(* IEC 61131-3 sources: ml2plc/benchmarks/st (part 25) *)

    bias_13 : ARRAY[0..63] OF REAL := [-0.0404071435, 0.0927777886, -0.0413042903, -0.0902542397, -0.0367607661, 0.0712136403, -0.00892876834, -0.0667051747, 0.00637631165, 0.0437391289, -0.0124141583, 0.0894438922, -0.0595212504, 0.0899347588, 0.0368472114, -0.000366137043, -0.0369593501, 0.0098438086, -0.00942459609, 0.0903767124, -0.0075942101, 0.046375595, -0.0592727698, 0.0528409891, -0.0216910169, -0.00787346996, 0.0314517543, 0.0737932697, -0.0810395479, 0.0906123891, 0.0820333436, 0.0979426578, -0.0194323044, -0.0938704684, -0.0664548054, 0.0229378678, -0.0287175067, 0.0409495458, -0.0543716773, 0.0378184244, -0.0231971722, -0.0583018064, -0.064960219, 0.00983823184, -0.0784399733, 0.0101949805, -0.0290268082, 0.0763350129, -0.0110898362, -0.00504951039, 0.0234738979, -0.0619560853, 3.6623473e-07, -0.0102051999, -0.0874569118, 0.0950193256, 0.011268124, 0.0887499079, 0.0580152497, 0.0789389834, -0.0176048651, -0.00555823185, -0.0167076774, -0.0683557615];

    weights_16 : ARRAY[0..191] OF REAL := [-0.204218104, 0.0100585446, 0.124642573, 0.249767885, 0.192972004, -0.114489801, 0.0213469081, -0.192255303, 0.0687296614, -0.116273321, -0.168248311, 0.100407079, -0.0835328773, 0.238771692, -0.1582672, -0.20680669, 0.199099779, -0.355317205, -0.275946528, 0.259559304, -0.152421042, -0.193678349, -0.0476079546, 0.168583572, 0.137155071, -0.424926966, 0.0668462142, 0.121788457, 0.166179895, 0.155418351, -0.239607006, 0.159718022, 0.181392595, 0.012098941, 0.29212448, -0.30051899, -0.042393513, -0.302967817, 0.0276647583, -0.0162179675, -0.0362443365, -0.131818026, 0.0652571768, -0.251479208, -0.163796052, 0.246231601, -0.0993305817, -0.214045271, -0.259664625, 0.121991962, 0.328099579, -0.36496222, 0.286016166, 0.174832657, -0.115100093, 0.240771398, -0.219685465, -0.0312652551, 0.361102194, -0.322652519, 0.172960237, -0.0672435984, -0.196433365, -0.310510099, 0.180873245, -0.229489714, -0.0438734591, -0.0316266902, 0.106365554, -0.354469597, 0.104236148, 0.0969249979, 0.0453101136, 0.189823419, -0.119062148, 0.0151938582, 0.05480076, -0.137107879, 0.231374756, -0.184149876, -0.152093366, 0.298650056, -0.120534711, -0.440170765, -0.291449726, -0.185382351, 0.240590215, 0.0743931085, 0.00839448255, -0.324791044, 0.0127115622, 0.201346219, -0.129334167, 0.217511401, 0.249150231, -0.227794915, -0.152671486, 0.225536987, -0.10112305, -0.260705948, -0.309738696, 0.234022498, 0.247884244, -0.138457581, 0.287121534, 0.107613027, 0.369097799, 0.20829244, -0.189594626, -0.168206543, 0.127910152, 0.117524289, -0.267760575, -0.273475945, -0.0782620981, -0.369871527, 0.318286926, 0.380977005, -0.372844636, -0.159075871, -0.35559544, -0.15261285, 0.021852307, -0.177226037, -0.057486631, 0.270852298, 0.160473123, -0.251653463, 0.100419275, -0.136632696, -0.287902951, -0.344732016, 0.126178026, -0.177843302, 0.339493781, -0.099222295, 0.0892207772, 0.163005397, 0.215954706, -0.0692603961, 0.0789305717, 0.37051788, 0.124587342, -0.095472239, 0.128479376, -0.0207961947, -0.257337809, 0.0661524683, 0.132446691, -0.221712723, -0.32083869, 0.195067048, 0.161428511, -0.336975783, -0.0876864642, 0.283737957, 0.175905675, -0.186329022, -0.0834812075, -0.0544198342, -0.247233495, -0.240931347, -0.316858917, -0.324440151, 0.33110112, 0.302384734, 0.294178426, 0.0780448988, -0.218289346, 0.095910117, 0.0984309539, -0.335624874, 0.34094283, -0.192400947, -0.337153077, 0.305544972, -0.302600533, -0.0743493959, 0.340184033, -0.0958573595, -0.265512377, 0.0674359873, 0.0557227954, -0.208096027, 0.112970375, -0.241400406, -0.123275287, -0.175267965, 0.0384325348, 0.0348930582, -0.135870203, -0.0273135975];
    bias_16 : ARRAY[0..2] OF REAL := [0.0433644801, 0.055319678, -0.0903941169];

END_VAR

VAR
    (* Merged variables from all regions *)
    buffer_0 : ARRAY[0..63] OF REAL;
    buffer_1 : ARRAY[0..63] OF REAL;
    buffer_2 : ARRAY[0..63] OF REAL;

    (* Temporary computation variables *)
    i : DINT;
    j : DINT;
    t : DINT;
    sum : REAL;
    (* Computation helpers *)
    max_val : REAL;
    exp_val : REAL;
    exp_sum : REAL;
    (* Spatial loop variables *)
    oc : DINT;
    oh : DINT;
    ow : DINT;
    ic : DINT;
    kh : DINT;
    kw : DINT;
    ih : DINT;
    iw : DINT;
END_VAR

(* Forward pass execution *)

(* Region: r0 [ACYCLIC] *)
(* Acyclic Region r0 *)
(* Layer 0: Fused Linear + RELU *)
FOR j := 0 TO 63 DO
    sum := 0.0;
    FOR i := 0 TO 0 DO
        sum := sum + input_data * weights_0[i * 64 + j];
    END_FOR;
buffer_0[j] := MAX(sum + bias_0[j], 0.0);
END_FOR;

(* Layer 1: Fused Linear + RELU *)
FOR j := 0 TO 63 DO
    sum := 0.0;
    FOR i := 0 TO 63 DO
        sum := sum + buffer_0[i] * weights_1[i * 64 + j];
    END_FOR;
buffer_2[j] := MAX(sum + bias_1[j], 0.0);
END_FOR;

(* Layer 2: MatMul *)
FOR j := 0 TO 63 DO
    sum := 0.0;
    FOR i := 0 TO 63 DO
        sum := sum + buffer_2[i] * weights_2[i * 64 + j];
    END_FOR;
buffer_1[j] := sum;
END_FOR;

(* Layer 3: Add (Bias) *)
FOR i := 0 TO 63 DO
    buffer_2[i] := buffer_1[i] + bias_3[i];
END_FOR;

(* Layer 4: Add (Element-wise) *)
FOR i := 0 TO 63 DO
    buffer_1[i] := buffer_2[i] + buffer_0[i];
END_FOR;

(* Layer 5: Activation (RELU) *)
FOR i := 0 TO 63 DO
    buffer_0[i] := MAX(buffer_1[i], 0.0);
END_FOR;

(* Layer 6: Fused Linear + RELU *)
FOR j := 0 TO 63 DO
    sum := 0.0;
    FOR i := 0 TO 63 DO
        sum := sum + buffer_0[i] * weights_6[i * 64 + j];
    END_FOR;
buffer_2[j] := MAX(sum + bias_6[j], 0.0);
END_FOR;

(* Layer 7: MatMul *)
FOR j := 0 TO 63 DO
    sum := 0.0;
    FOR i := 0 TO 63 DO
        sum := sum + buffer_2[i] * weights_7[i * 64 + j];
    END_FOR;
buffer_1[j] := sum;
END_FOR;

(* Layer 8: Add (Bias) *)
FOR i := 0 TO 63 DO
    buffer_2[i] := buffer_1[i] + bias_8[i];
END_FOR;

(* Layer 9: Add (Element-wise) *)
FOR i := 0 TO 63 DO
    buffer_1[i] := buffer_2[i] + buffer_0[i];
END_FOR;

(* Layer 10: Activation (RELU) *)
FOR i := 0 TO 63 DO
    buffer_0[i] := MAX(buffer_1[i], 0.0);
END_FOR;

(* Layer 11: Fused Linear + RELU *)
FOR j := 0 TO 63 DO
    sum := 0.0;
    FOR i := 0 TO 63 DO
        sum := sum + buffer_0[i] * weights_11[i * 64 + j];
    END_FOR;
buffer_2[j] := MAX(sum + bias_11[j], 0.0);
END_FOR;

(* Layer 12: MatMul *)
FOR j := 0 TO 63 DO
    sum := 0.0;
    FOR i := 0 TO 63 DO
        sum := sum + buffer_2[i] * weights_12[i * 64 + j];
    END_FOR;
buffer_1[j] := sum;
END_FOR;

(* Layer 13: Add (Bias) *)
FOR i := 0 TO 63 DO
    buffer_2[i] := buffer_1[i] + bias_13[i];
END_FOR;

(* Layer 14: Add (Element-wise) *)
FOR i := 0 TO 63 DO
    buffer_1[i] := buffer_2[i] + buffer_0[i];
END_FOR;

(* Layer 15: Activation (RELU) *)
FOR i := 0 TO 63 DO
    buffer_0[i] := MAX(buffer_1[i], 0.0);
END_FOR;

(* Layer 16: Fused Linear + SOFTMAX *)
FOR j := 0 TO 2 DO
    sum := 0.0;
    FOR i := 0 TO 63 DO
        sum := sum + buffer_0[i] * weights_16[i * 3 + j];
    END_FOR;
output_data[j] := sum + bias_16[j];
END_FOR;

(* Softmax: find max *)
max_val := output_data[0];
FOR i := 1 TO 2 DO
    IF output_data[i] > max_val THEN
        max_val := output_data[i];
    END_IF;
END_FOR;

(* Softmax: compute exponentials and sum *)
exp_sum := 0.0;
FOR i := 0 TO 2 DO
    output_data[i] := EXP(output_data[i] - max_val);
    exp_sum := exp_sum + output_data[i];
END_FOR;

(* Softmax: normalize *)
FOR i := 0 TO 2 DO
    output_data[i] := output_data[i] / exp_sum;
END_FOR;

END_FUNCTION_BLOCK

(* ---- ResNet3_straton.st ---- *)
FUNCTION_BLOCK ResNet3_FB

    (* Model Inputs/Outputs *)
VAR_INPUT
    input_data : REAL;
END_VAR

VAR_OUTPUT
    output_data : ARRAY[0..2] OF REAL;
END_VAR

VAR
    CONSTANT weights_0 : ARRAY[0..63] OF REAL := [-0.190466672, -0.289495766, 0.36445868, 0.11001166, -0.202885658, -0.247976601, -0.217859656, 0.152941793, -0.210685372, 0.322490484, -0.300406843, -0.0737419277, 0.271309823, 0.34986949, -0.269151628, 0.101570874, -0.0975821763, -0.0239237547, -0.28141278, -0.260361493, 0.220720425, 0.342909008, -0.106619239, 0.192217126, -0.139923915, -0.00473925471, 0.256588012, 0.106521919, -0.015166074, -0.237258494, -0.295479923, 0.237283707, -0.111313865, -0.119793385, -0.189164549, 0.109231912, 0.147311017, -0.0809866935, -0.174528345, -0.015255332, 0.110069647, 0.205406636, 0.233189464, 0.175904229, 0.192441761, -0.257080823, 0.113344185, -0.222640619, 0.0253927261, -0.0698330998, 0.304976135, 0.13343668, -0.229343772, 0.317507595, -0.0133918505, 0.251467377, -0.131539866, -0.128968731, 0.204563618, -0.234828115, 0.109687969, 0.0967651531, -0.128085941, 0.0570141077];
    CONSTANT bias_0 : ARRAY[0..63] OF REAL := [0, 0, -0.0451503769, -0.000170675936, 0, 0, 0, -0.0306519736, 0, -0.043658372, 0, 0, -0.0452437028, -0.0463685207, 0, -0.0237470753, 0, 0, 0, 0, -0.0306253415, -0.0182554778, 0, -0.0286273304, 0, 0, -0.0439416394, 0.0359471515, 0, 0, 0, -0.0393987, 0, 0, 0, -0.025377661, 0.0258860644, 0, 0, 0, -0.0256011337, -0.040137399, -0.0210138671, -0.0197667424, -0.0420954861, 0, -0.0343104228, 0, -0.0101194074, 0, -0.0385119878, -0.0309600942, 0, -0.0221530851, 0.0427107885, -0.0482655875, 0, 0, -0.0332414694, 0, -0.0204843841, -0.0293239169, 0, -0.0204854961];
    CONSTANT weights_1 : ARRAY[0..4095] OF REAL := [-0.0287969261, 0.201637134, -0.193626225, -0.0838745981, -0.179824859, -0.158866256, -0.0519343764, 0.0553617924, -0.0298234671, 0.199577436, -0.0565214604, -0.135609776, 0.19474043, -0.0305772722, 0.047594741, 0.174586251, -0.131670237, -0.0606977493, -0.00999130309, 0.160562769, 0.114603773, 0.198183253, -0.0226515681, -0.174445733, 0.0844327062, -0.0653743893, 0.166338369, 0.178600982, -0.179540232, -0.104543671, -0.04106462, 0.0376635343, -0.0928359851, 0.0239627361, -0.0751802325, -0.131423861, 0.107191309, 0.0680955499, -0.134543836, 0.162752822, -0.119452722, -0.118079856, -0.111446388, 0.103158936, -0.0164598525, -0.143377468, 0.0849187821, -0.0122491121, -0.152280733, -0.120597631, -0.0606369525, -0.0807449222, 0.147399679, 0.0629173666, -0.130655468, -0.21262382, -0.169020504, 0.105712339, 0.11746116, 0.0592246503, -0.0597587526, -0.143656209, 0.0653275698, -0.0477767587, -0.154527515, 0.0485876948, -0.0317480415, -0.000382602215, -0.0967821628, 0.0423714072, -0.0512648225, 0.0312831551, -0.17014426, 0.160105124, 0.109350279, -0.0217197388, -0.0921072736, 0.0853802711, -0.0300633907, 0.135347292, -0.0391751528, -0.199345261, -0.195168182, 0.0560685545, 0.215828583, -0.0923638716, 0.192498907, 0.178375289, -0.183688045, 0.116588429, 0.0289125443, 0.0778251439, 0.0613025278, 0.0142809004, 0.0337732583, 0.0574108511, 0.189165697, 0.196946517, 0.107737496, -0.129702166, -0.107477285, -0.107738689, -0.177952528, -0.0559140593, 0.169283316, -0.0538910031, -0.104346119, -0.127213195, -0.0331750959, 0.127317414, 0.0515208095, 0.0195653588, 0.0769012719, -0.124866173, 0.177239373, 0.0280220658, 0.0963039249, -0.0652452409, 0.105720118, 0.15663074, -0.136386782, -0.123085879, 0.0827278346, 0.21160166, -0.16991207, -0.0768297166, 0.120611772, 0.134732291, -0.139711812, -0.184518486, -0.184835598, 0.00858225208, 0.113042273, -0.102391459, -0.0780269504, -0.165388852, -0.140612379, 0.223779544, 0.162238076, -0.00674940646, 0.0487292968, 0.0836367309, -0.19456315, 0.171644017, -0.0955267325, 0.0997560844, -0.0601457544, -0.198954478, -0.00482972385, -0.079228431, -0.127536789, 0.190665379, -0.0999609306, 0.0110752583, -4.10255961e-05, 0.118868679, 0.138081178, -0.0528386459, -0.114722773, 0.170001924, 0.137378082, -0.196978897, -0.15748626, 0.0825704783, -0.033234071, -0.101335384, 0.0289265234, -0.15857622, -0.0556612536, 0.213226333, 0.00719815027, 0.223965615, -0.0638628826, 0.148281991, 0.0975444093, -0.0259753708, 0.0262751374, 0.0979252607, -0.0863377675, 0.0899253041, 0.239503771, 0.289376885, -0.204818711, 0.105383582, 0.293127954, 0.203753337, -0.119700439, -0.16846402, 0.191751063, 0.0327624083, -0.0386312976, -0.264414817, 0.153028056, 0.154591411, 0.124344207, -0.107223384, -0.137165904, 0.0300747007, 0.183606654, 0.198948666, 0.0499654785, 0.144469813, -0.210293442, -0.0324280113, 0.0683567002, -0.04100243, -0.0126516968, 0.164788797, 0.237893194, -0.0847178176, 0.0626023933, 0.155760348, 0.185824335, 0.00780587131, 0.199899733, 0.035005752, -0.0749012083, 0.067025587, 0.141089186, -0.0444214866, -0.0607198402, 0.0990498737, -0.0620695017, 0.0086689936, -0.114031576, -0.111011893, -0.204213917, -0.198096737, 0.138905957, 0.159203395, 0.12167336, 0.0172255039, 0.15101482, 0.131718054, -0.0235928968, 0.200807258, 0.209497362, 0.170748204, -0.231670231, 0.143206522, 0.225486189, 0.104716703, -0.177130625, -0.133289889, -0.0483859442, 0.107198499, -0.0196592454, -0.0476846471, -0.0815907568, -0.135093376, 0.12207596, 0.00658966927, -0.0573140644, 0.0118645504, 0.226763472, 0.178059682, -0.0891532153, 0.0825275332, 0.163484469, -0.0550447851, -0.0375959724, -0.00878846645, 0.0168165267, 0.150091812, 0.084491238, 0.174592748, 0.0785937458, 0.163301513, -0.0316622555, 0.0597050637, 0.157956466, -0.0453870595, 0.101291135, -0.0735865831, 0.0523432046, 0.00310024619, -0.111143999, -0.176621795, 0.0883997232, -0.00594709814, -0.0267459899, 0.164880231, 0.0904007405, -0.00336711109, 0.025017634, -0.136061743, -0.0808758289, 0.139091626, 0.0775778443, -0.155642897, 0.0725118369, -0.0960384831, 0.135437921, -0.188861921, 0.0681308657, 0.121807054, -0.0181216151, 0.126562431, 0.0201322883, 0.0685440749, 0.0470108241, 0.206563786, 0.167886898, -0.182285488, -0.166398615, 0.200898841, 0.191317186, 0.190035328, -0.175405696, 0.124712333, 0.052170679, 0.184364364, -0.0736751109, 0.0639937371, -0.168305129, 0.00677789748, -0.148140043, 0.10284771, -0.13430731, 0.139501527, 0.0359104425, 0.0577303618, -0.188823983, -0.174651235, 0.0696652383, -0.183670074, -0.00257234275, -0.193130046, -0.203748837, -0.153786868, 0.202487156, -0.0460375547, 0.109957233, 0.00299288332, -0.162598059, 0.210710511, -0.194323435, -0.210184813, 0.0554226786, -0.142163336, -0.152110279, -0.0163246542, -0.166943565, 0.175032482, -0.215747178, 0.171988502, 0.132436678, 0.172353908, 0.121031687, 0.186095968, -0.0588158816, -0.0108129233, -0.0942323804, -0.09778703, -0.109081298, -0.106757924, 0.172346756, 0.025905624, 0.0740813166, 0.189657524, 0.148814008, 0.197771326, 0.201267496, -0.068178758, 0.1481594, 0.184583381, -0.014007479, 0.0497234613, -0.0900920182, -0.151112944, -0.154349625, 0.155235782, -0.183371142, -0.164333746, 0.110023871, 0.0927015692, 0.194937959, 0.208203807, -0.00641842186, -0.135277599, -0.0120722651, 0.0209348053, -0.163213924, 0.183399543, 0.00101952255, -0.094531931, -0.0417330861, 0.125320569, 0.140007362, -0.0551816374, -0.0750101358, -0.184187144, 0.0996663719, 0.1298704, -0.00832244754, -0.00248210132, 0.0548401624, -0.0217346549, -0.040534541, 0.0774618536, 0.0789829642, -0.213013336, 0.00969907641, 0.131764188, -0.134339929, -0.16999869, -0.150505453, -0.203993306, 0.133900389, 0.210885063, 0.0592023879, 0.119564161, 0.129766181, -0.116630182, 0.0890186876, 0.0916796774, -0.125102013, 0.144167438, 0.190863922, 0.0828631073, 0.110106811, -0.0818011016, 0.0638723224, 0.0225199312, -0.0798923373, -0.106765099, -0.103232488, -0.0746515393, 0.214082971, -0.139221311, 0.0676382631, 0.20862554, 0.185882255, -0.0279404521, 0.0581518859, -0.0932726786, -0.0684341788, -0.148790196, -0.167229846, 0.160150275, -0.125400275, -0.0166903287, -0.0369179547, 0.0845469385, -0.191490114, -0.161978155, -0.023997426, 0.040678516, 0.14639619, 0.0431083404, 0.0106931906, 0.139329195, -0.149284765, -0.0467167646, -0.0767225027, -0.0320999771, -0.23229675, -0.0372863598, 0.128295347, -0.160325885, -0.148059294, -0.00792731252, 0.0252128541, -0.0963003412, -0.0197790675, -0.0523058102, -0.0141548719, -0.168405354, 0.093509756, -0.0733992159, -0.174149796, 0.0823272243, 0.0543129146, 0.00202205591, 0.112447657, -0.189444944, 0.0949934795, 0.133855537, 0.138600275, -0.170810059, -0.0500965714, -0.186440244, 0.0285257101, -0.000778779387, -0.128126383, -0.0261946935, -0.201500729, 0.11489366, 0.0997269675, -0.138657212, -0.256732196, 0.0291550159, -0.302546233, -0.178278208, -0.234763011, -0.0388856418, 0.0533248745, -0.146624878, -0.0823597312, -0.230229869, 0.0182416849, -0.118736058, 0.0481926613, 0.133541629, -0.114781246, 0.10070549, 0.109701976, 0.0569074266, 0.26510939, 0.00950349867, 0.0546200871, 0.151336238, 0.0048430115, 0.0378029197, 0.144169971, 0.0863773972, 0.200766638, 0.212797061, 0.138086304, -0.182377681, 0.213811055, 0.161403164, 0.124502376, 0.0246564448, -0.196184307, -0.196561068, 0.0875730366, 0.0948206931, -0.149286091, 0.0323978215, 0.0455216914, 0.151648596, -0.127112329, -0.111039624, 0.0246137083, 0.016291365, -0.00267861784, 0.0558695644, 0.201473311, -0.178703129, -0.103530645, 0.173463836, 0.157130465, 0.182277635, 0.0760518163, 0.215445682, -0.106563114, -0.196684077, -0.094135493, 0.10404627, 0.0962792784, -0.0124557465, -0.15429759, -0.0716400295, 0.11189805, 0.0764795393, 0.0549422354, -0.0472201556, -0.00484439731, 0.0528673977, 0.190446272, 0.0174336433, -0.0469030589, -0.0549324602, 0.102302983, -4.00096178e-05, 0.147421315, 0.193782583, -0.0265746713, 0.0705426186, 0.0295248479, -0.134114474, 0.0562623292, 0.172508165, 0.175126389, -0.161904559, -0.0162163712, 0.208393365, -0.100752503, 0.0273437109, -0.153811902, -0.193232462, -0.16940017, 0.188474581, -0.0369768888, 0.0354307853, -0.0991368741, -0.196591377, -0.233054638, -0.118758805, -0.0622535497, 0.0394661725, 0.267733514, 0.107220888, -0.252435923, 0.112368457, 0.166412622, 0.192772374, -0.218732044, 0.126407787, 0.0919501036, 0.00824039057, -0.0796734989, 0.182596043, 0.131103203, -0.109326825, 0.125145733, 0.122357175, 0.0696524829, -0.0965674892, 0.0579061955, -0.200026214, -0.185237691, -0.189040273, -0.224097118, 0.103700139, 0.109744169, 0.283211142, -0.108721465, 0.126635522, -0.0494364649, -0.224469841, 0.151249424, -0.162036136, 0.030354334, -0.00598688424, -0.143472508, -0.047887668, 0.0439753979, 0.0527719408, -0.152598977, 0.110804304, 0.257972151, -0.138091505, -0.110594928, 0.100734361, -0.0214415565, 0.0449742526, 0.22822006, -0.240381643, -0.128085867, -0.0693219751, -0.0846015364, -0.17030485, 0.130928531, 0.00229240954, -0.194736332, -0.0391959101, 0.0145413131, -0.144774944, -0.181710035, 0.032208994, -0.206829414, -0.0198655725, 0.0611966401, 0.00840911269, 0.158986792, 0.126695439, -0.157956257, -0.20029664, -0.104722835, -0.144183606, 0.00487022102, 0.0939430147, -0.0584943891, 0.0557004064, 0.00045491755, 0.114710584, 0.0546646267, 0.20419623, 0.0921241492, 0.0991390496, 0.176430956, -0.158750683, -0.0890071839, -0.179640472, 0.162403598, -0.0909959227, 0.0409451872, -0.0232819319, 0.165903732, 0.069598332, 0.175637826, -0.179648638, -0.00545862317, 0.00749818981, 0.0323755145, -0.158800021, 0.180631563, -0.053162545, -0.014888972, -0.188607126, -0.0488055795, 0.20547007, -0.0377693027, 0.0997820646, -0.124526724, -0.0918210968, -0.167447731, -0.188922942, 0.0540182441, 0.122466967, -0.0612903982, 0.173171565, 0.187880501, 0.0320709199, -0.0716537684, -0.146939963, 0.00549939275, 0.0170418024, -0.156284317, -0.158158392, -0.0161726922, -0.117838174, 0.0458692163, 0.0690316111, -0.102591947, -0.0113369077, -0.0506339818, 0.186475053, 0.10736011, -0.0328097939, -0.13072902, -0.14560762, 0.0873160809, 0.204848334, 0.079661116, -0.018868804, -0.018476963, 0.148941293, 0.0539769381, -0.00221420825, -0.108419128, -0.0766489506, -0.189365566, 0.0919391662, -0.212484032, -0.172094896, 0.0239589214, -0.211048037, 0.189641103, 0.0730664879, 0.206356838, -0.135675371, -0.000756576657, 0.0285059959, 0.209358588, 0.192232445, 0.11306645, -0.115133278, 0.175952092, 0.0211753547, 0.0506318063, -0.19809112, 0.0197272301, 0.054157868, 0.0254253149, -0.155184671, -0.0454918444, -0.196502686, -0.0158347338, -0.135656744, -0.211595923, -0.020885095, -0.00690788031, 0.0370714217, -0.172456279, -0.185076281, 0.160629585, 0.0181837529, -0.0211855043, 0.120963901, -0.00527728582, -0.0352699608, -0.19402647, 0.132209137, 0.0396415927, -0.118135475, 0.00657442212, -0.208759815, -0.0303688291, -0.00777827017, -0.0915059149, 0.11210835, 0.294361055, -0.142053381, -0.0571834072, -0.0146589978, -0.0864291564, -0.101504333, 0.12920031, 0.182926923, 0.192566365, 0.106406614, 0.214629248, 0.06889496, -0.11516425, -0.259321928, 0.184162751, -0.272702873, -0.117973782, 0.0606180206, 0.0292263925, 0.0766455382, -0.120667271, -0.201999113, -0.0266232025, -0.00732299685, -0.0519965291, 0.156876504, 0.123033859, 0.267217845, -0.0109749781, -0.272964209, -0.129237577, 0.053774897, 0.141416252, -0.199857935, 0.0538020581, -0.230259433, -0.0451727808, 0.258897543, 0.148216307, -0.053409934, 0.31615606, 0.0147380829, -0.202499956, 0.110624768, 0.1696845, -0.0922751948, 0.0798982531, 0.0207011886, -0.142718717, 0.0519616678, -0.127546012, 0.126492023, 0.0723542273, 0.147747502, 0.126169741, 0.0813353807, -0.1203655, -0.153749913, -0.0919978395, -0.139003664, 0.0844179541, 0.054092221, 0.110275611, -0.200139761, 0.110008813, -0.126036033, -0.166970596, -0.233972371, 0.0890860558, -0.20025298, -0.230093077, 0.0173213258, 0.275560528, 0.151483357, 0.276097506, 0.00718977815, -0.0111169517, 0.168895632, 0.10235633, -0.240326077, -0.0821303874, -0.00890312064, -0.171553358, -0.00546233356, 0.101003714, 0.0433369204, -0.187788144, -0.103547342, 0.00432489906, -0.109544538, 0.012347714, 0.0869178474, -0.257481515, -0.0600075051, -0.264836371, -0.171154037, 0.0307734851, -0.129194021, -0.199388355, 0.0987441167, -0.0623329841, 0.249395654, -0.034193743, 0.0902072638, 0.203402102, -0.0227374583, 0.0134097785, -0.0912396759, 0.0864051133, 0.0865284353, 0.228083283, 0.126239121, -0.109470509, -0.188946784, 0.00514312088, 0.181860104, 0.0482862443, 0.0316015482, 0.208089277, 0.175173715, 0.157937661, -0.175959155, -0.15175122, 0.0449968129, -0.0724449754, 0.131373897, 0.081098035, 0.0556937009, -0.127380341, 0.131804869, -0.182943538, -0.163977832, -0.00456343591, 0.0986122638, -0.0509269685, 0.144946262, 0.152006164, -0.195760101, -0.158920705, -0.0407915562, 0.0382466763, 0.120302364, 0.163731501, 0.0790192336, 0.0871210247, -0.0502094626, -0.193163037, 0.0618805438, -0.0852957666, 0.124724433, 0.0312432498, 0.114015713, 0.150832668, 0.00696192682, -0.020202592, 0.0919532925, 0.0599388927, -0.155759037, -0.0923569575, -0.0696199685, -0.127464831, -0.187969327, -0.187459841, 0.143950805, -0.0970960557, 0.154307649, -0.05652605, 0.156533435, -0.183348998, 0.139695272, 0.124307856, -0.0476845652, 0.0955802649, -0.0311176628, 0.163419768, 0.113613471, 0.182277307, -0.202524781, 0.0122317718, 0.186174095, -0.113051899, 0.208240613, -0.158425584, 0.0850085169, -0.0775510222, -0.0645689219, -0.0517540723, -0.17061533, 0.0819323882, 0.121917769, -0.119305968, -0.0747042894, 0.0523318127, -0.152910829, 0.100246899, 0.0908019319, 0.066256009, -0.0805988908, 0.0907654166, 0.0451934189, -0.0514816083, 0.192991301, 0.180941716, -0.197929591, -0.0896847397, -0.218640536, 0.058635354, -0.112284772, -0.0678162426, -0.0591657534, 0.190862313, -0.0746522695, -0.0959051773, -0.0859087706, 0.0146463895, 0.127395496, 0.0643470958, 0.222248226, -0.222716317, -0.0038960767, 0.0420699306, -0.189540833, 0.151158154, 0.174533531, 0.0537843928, 0.0724432617, -0.0636890829, -0.0554191582, 0.0796529651, 0.220607117, -0.152003556, 0.0678689852, 0.189509705, 0.196022376, 0.112115934, -0.103596382, 0.0718052611, -0.139615148, 0.17220287, -0.108806856, -0.0700540841, -0.126261801, -0.0981526002, -0.0755177587, 0.112252161, 0.196778193, -0.00826221704, -0.185675785, -0.057513833, -0.101335384, 0.0925282687, -0.0817712694, -0.131041422, -0.0185560435, -0.125542641, 0.191311106, 0.183952644, 0.13196452, -0.153428495, -0.117309444, -0.0829459131, -0.110064179, 0.198635712, -0.171391279, 0.111330763, -0.148759633, 0.0993963033, 0.0926398188, 0.208881006, 0.106514856, 0.205308661, 0.0648586303, 0.000817343593, -0.0404887646, 0.129113868, -0.0304635465, 0.057734862, -0.0244514644, 0.102735177, 0.120236859, -0.138929337, 0.0624369532, -0.155432343, -0.15313834, 0.0859217495, -0.00519438088, 0.126614913, -0.21491994, 0.0207336992, 0.175207987, 0.109249786, -0.054661721, 0.0479473621, 0.00943541527, -0.142473519, 0.116482362, 0.0937203616, -0.0977497622, 0.183454707, 0.126636133, 0.132889017, -0.179818153, -0.00318422914, -0.114538781, 0.190620884, -0.0922307968, 0.171573177, -0.113899581, 0.0264129937, -0.117907241, 0.0159941912, 0.056949541, -0.165546909, -0.079548344, 0.155183807, 0.167912915, -0.12471018, -0.0227756053, 0.195206597, 0.155959591, -0.113060772, 0.0471404046, -0.0937578529, -0.0744760931, 0.0718369633, -0.194636658, 0.0701943189, 0.00457412004, -0.0688510537, -0.159001023, 0.119077131, 0.0420625359, -0.101866595, -0.0260792822, -0.213209078, -0.0761060715, 0.0378767401, -0.0494340956, 0.0950354189, -0.119263433, -0.187393367, -0.19390738, -0.115837008, -0.11679624, 0.0311641246, -0.0763715953, 0.00562612712, 0.104230031, -0.0938740447, -0.158894032, -0.186505824, 0.123571053, 0.0021596998, -0.124141335, 0.0726272911, 0.0728365034, 0.048231259, 0.167245731, 0.173797145, -0.133879036, 0.123410001, 0.0136341602, 0.211613938, 0.0339705497, -0.0568555892, -0.0638442487, -0.165108442, 0.113140717, -0.114156596, 0.0502677411, 0.105490163, 0.154489145, 0.0633081943, 0.0605547279, -0.168472469, -0.174018279, -0.178102687, -0.0923157632, 0.0868086368, 0.142751232, 0.0472065359, -0.0355895907, -0.070602119, 0.0226132125, 0.111900166, 0.072677359, 0.126415685, -0.147081137, -0.145128071, 0.119609222, -0.149196088, -0.0602950752, 0.198493585, 0.137908891, 0.0641960949, 0.200968578, -0.0566390008, -0.1688862, 0.172993645, -0.144077167, -0.197343826, -0.0247414112, 0.199622199, -0.1655339, -0.0133733898, 0.134934023, 0.0719420165, 0.000706866384, 0.149509206, -0.156804532, -0.0837745517, -0.037465632, -0.157091066, 0.107307032, -0.00644093752, 0.0704480559, -0.183203697, -0.196138009, -0.117853299, -0.12040215, -0.11014574, -0.116727851, 0.026737988, -0.0404386818, 0.0639270395, 0.104571596, 0.0609508008, -0.0830935389, -0.20587337, 0.0998597592, 0.0920080096, -0.113937676, -0.0127168447, 0.130367443, -0.162072524, 0.206473872, -0.0470631719, 0.202682182, -0.0224076658, -0.0183282048, -0.0392407626, 0.13104786, 0.0124193132, -0.155867845, 0.187796101, 0.12736474, 0.183426574, 0.0451046377, 0.0507078916, 0.122980073, -0.21496205, 0.0355659574, -0.0358312726, -0.136690676, -0.167069823, 0.0553592891, 0.212405875, 0.186634675, 0.140052691, 0.0532232374, -0.132964134, 0.199990019, 0.129920498, -0.0277204067, 0.162883624, 0.197279349, -0.0547595471, -0.169750974, -0.0363512784, -0.0266377479, 0.122363672, 0.0337654799, -0.199149102, 0.207519457, 0.142926887, 0.215468749, -0.0605023801, -0.0568595082, 0.0636674613, 0.106427982, -0.139160648, -0.11427062, 0.189653918, 0.135131165, -0.0713291317, 0.103454813, 0.115515873, 0.0241415501, -0.141884476, 0.0647414476, 0.1221935, 0.187437966, -0.0765461177, 0.130906656, 0.209548905, 0.198075101, -0.0151947271, 0.106877655, 0.122374028, 0.0876808092, -0.0646020845, 0.179015324, 0.137440547, -0.111645944, -0.0637109131, 0.264909327, -0.00986942649, 0.19460775, -0.215875, -0.216673881, -0.195247158, 0.0369132459, 0.22958532, -0.0758189484, 0.161118656, -0.0532057211, -0.111272402, 0.0191001799, 0.154950529, 0.184459001, -0.0586241372, 0.211076126, 0.0385005176, 0.0375854224, 0.185866401, -0.0925790668, 0.0594946295, -0.199379593, 0.160706773, -0.0215413142, 0.0920865387, -0.0727619678, -0.0503336526, 0.144037127, 0.0390647538, -0.176736578, 0.218084648, 0.282077163, 0.0684015825, -0.0997406542, 0.0936136246, -0.0177756548, -0.116294734, -0.21881853, 0.0861533135, -0.144913971, -0.116913833, -0.228465006, 0.243279889, 0.289645553, -0.157389015, 0.0694431514, -0.0845005885, -0.169205248, 0.0732500702, -0.140289873, 0.217532694, -0.153820172, 0.165036872, -0.0370052084, -0.0649239048, 0.00705603603, 0.00300642545, -0.147408083, -0.0400309153, -0.0219824761, 0.021092033, -0.0739108026, 0.0152327912, 0.16345866, -0.169258162, -0.171906739, -0.0344251506, 0.0626144186, 0.0827743858, 0.0153012248, 0.214705959, 0.149533838, -0.0852295235, 0.108769022, -0.125927284, 0.0506657287, -0.0685000271, 0.132542357, 0.189130142, -0.107204311, 0.208437741, -0.0613691844, -0.15225552, 0.0756992996, -0.0966535062, -0.198031753, 0.0743363649, 0.0633449629, -0.129061252, 0.122365281, -0.130634353, 0.0883900598, 0.0156343877, -0.135135397, 0.198845685, 0.2392952, -0.145629406, 0.188295275, -0.13789998, 0.132967234, 0.132922307, -0.17668727, 0.245915323, -0.141065955, 0.192191795, -0.157576233, -0.085805878, -0.0276803467, -0.095566079, 0.219359696, 0.202878788, -0.0802682042, -0.176504254, 0.023325054, 0.0037062054, -0.138832927, 0.053536851, 0.127934501, -0.168392971, 0.0300281346, 0.0400527865, -0.206524342, -0.081766516, 0.104110494, 0.00106944144, -0.120554268, -0.0580964088, 0.109146222, -0.000105708838, 0.182546988, -0.148469537, -0.148119092, 0.149815395, 0.205082461, -0.0108131766, 0.179644182, -0.192448467, -0.0218183249, 0.112928316, 0.173357442, 0.0719634742, 0.20145084, 0.0719409138, -0.164568782, -0.130916566, -0.202400431, 0.0947056264, -0.192789838, 0.0868111402, -0.00978286564, 0.196489051, -0.0734990388, -0.146960199, -0.000552743673, 0.0167299211, -0.199335337, -0.158682853, 0.0911645144, 0.180834278, -0.122386955, 0.00548417866, -0.187905684, -0.107697234, -0.084947437, 0.0716611892, 0.132587507, 0.13105391, 0.0321043134, 0.0708666295, 0.136131003, 0.0918786675, 0.0526147634, 0.14389886, -0.0311155468, -0.188370556, -0.212843508, 0.0522523373, 0.167048857, -0.206337899, 0.072918728, 0.120494351, -0.190175474, -0.154683962, -0.000773754495, -0.186758995, 0.25392881, 0.165069968, -0.174278378, -0.0480074361, 0.0444551259, -0.0307127461, 0.197782025, 0.127323076, -0.19140029, -0.17637898, -0.0651647598, -0.0631855875, -0.170364678, 0.128072217, 0.142127141, 0.0896252617, -0.168872684, 0.0608825311, -0.199593708, 0.0163794793, -0.111544512, -0.0925613791, 0.0456584245, 0.273554981, 0.0908730105, -0.121767685, 0.133312061, -0.0430089869, 0.048706051, -0.106118105, 0.156891361, 0.199550763, 0.0661296993, 0.190545216, 0.0400548801, 0.0303085539, -0.0425427854, 0.0662297159, 0.266184568, 0.028025724, -0.122740746, 0.0264457632, 0.00358478306, 0.129521757, 0.162871301, 0.26886633, -0.0782814473, -0.0386863798, -0.0817479417, 0.0508834422, 0.212506562, -0.104619637, 0.0130023751, 0.0292652808, -0.08503066, 0.158758327, 0.0168799069, -0.0856374726, -0.150301456, -0.0860033929, -0.118447781, -0.179989219, -0.0929494426, -0.0466621518, -0.0659421533, 0.121023342, 0.105154112, -0.0455614179, -0.203972697, 0.173838392, -0.0386415124, -0.0278328806, 0.178764507, 0.104911312, 0.108715996, -0.0253986865, -0.168122798, -0.114805967, -0.0621888191, -0.0132009238, 0.0253832936, -0.0265160799, 0.0423865467, -0.100953348, 0.172172591, 0.201425806, 0.141991392, 0.0940631181, 0.194293097, 0.0401813537, 0.12128751, 0.196684197, -0.0543928444, 0.0463825911, 0.0403407067, -0.21529898, 0.00518736243, -0.0455965251, 0.0162204355, -0.183138445, -0.193831608, 0.187192395, 0.00752931833, 0.157815233, 0.141796991, -0.0405156463, 0.198203638, 0.00560341775, -0.0508095473, -0.0763344318, -0.0735320747, -0.0695720166, 0.148685709, 0.0700013191, 0.182473376, -0.1108841, -0.0968367755, 0.0362190455, 0.036774829, 0.0170685947, -0.0752303004, -0.0852943808, -0.206426427, -0.149846435, -0.155158252, 0.119575307, 0.0180834234, 0.146422639, -0.101406202, 0.0536810011, 0.0994656831, -0.0630992353, 0.0158559978, -0.0455258042, -0.21185334, -0.118426792, 0.159210399, -0.116417825, 0.0386347026, 0.159501418, 0.033601746, -0.0757299215, 0.00185963511, 0.085397765, 0.083639726, 0.178043649, 0.190545216, -0.0945898443, 0.0499521047, 0.0201606303, 0.106833711, -0.0188183188, 0.177461788, -0.100810207, -0.0469589531, -0.0987466872, 0.177121416, 0.1593398, 0.0223871171, -0.208162114, 0.062356934, -0.125736207, 0.096315518, 0.0971169025, 0.0245347768, -0.020675838, -0.111754142, 0.212888882, -0.170801476, 0.0786470622, -0.0122303218, 0.162038699, -0.199096397, 0.170362726, 0.0747093409, 0.111208364, -0.0473197848, -0.0435504466, -0.0453317761, -0.110917084, -0.0126232058, -0.177978754, -0.0992414504, 0.130278543, 0.018110469, -0.0700823665, -0.114136361, 0.0361899287, -0.18268013, 0.0165710393, 0.0793500915, -0.00841967668, 0.125138253, 0.0887469351, -0.107942894, -0.239920467, 0.201740548, 0.149393812, 0.203771755, 0.0577221662, -0.00337263942, -0.146427289, -0.257600576, 0.119674787, 0.194880754, 0.245413616, 0.0804518312, -0.166380689, -0.000451727072, 0.0460289009, 0.132229939, -0.1964733, 0.187092066, -0.0433319323, -0.0352629423, 0.137847543, 0.182559997, 0.0790997595, 0.114835717, -0.0771531537, -0.0737332329, 0.0758020729, -0.0452585854, 0.145568117, -0.1918246, -0.0583546832, -0.0145606585, 0.129812345, -0.0127620762, -0.0558166765, 0.16816707, -0.0112826349, -0.0819175765, -0.239855021, 0.103059068, -0.215481281, 0.116379917, 0.0303741544, -0.0232816786, -0.142835721, -0.178205758, 0.208591044, 0.288504571, 0.160375908, -0.10488455, -0.0112059414, 0.149956122, 0.0636754483, -0.195255071, 0.108991124, 0.206127957, 0.259172261, -0.150578156, -0.0045624678, -0.199588045, -0.115991615, 0.0703731775, -0.22166048, 0.115133122, 0.07192339, -0.00083938241, 0.0757085681, 0.160763949, -0.0662796795, -0.172549099, 0.0753220916, 0.121819116, -0.186484084, -0.165406242, -0.0917130634, -0.127552748, 0.209713519, 0.00541543402, 0.108752683, -0.048205357, 0.210129693, 0.0972502008, 0.211364299, 0.0602482185, 0.123633213, -0.154390544, -0.117387019, 0.105454966, -0.0183485299, 0.154096812, -0.168688595, 0.0630255491, -0.190940425, 0.13162984, 0.201842621, -0.189648613, -0.0979222134, 0.0130105121, 0.00230050553, -0.157333851, 0.13677448, 0.0410381854, 0.0108493455, -0.126054719, 0.0934812054, -0.0121305455, 0.150938109, -0.197522938, -0.216986924, 0.12068636, 0.100021429, -0.0908799618, 0.168728262, 0.0442929193, 0.139804959, 0.00512484135, -0.041490376, 0.163413405, 0.122350357, 0.0158086959, -0.161861941, -0.0287991706, -0.0309194028, 0.180298939, -0.0883494616, 0.163443282, 0.213652179, -0.0104613453, -0.0396695137, 0.153360203, -0.148807853, 0.00914561749, -0.165651739, -0.1075399, 0.120668754, 0.15019466, -0.168916598, -0.159659475, 0.134091392, 0.13391538, 0.0127349049, -0.148728609, 9.60677862e-05, 0.0587041825, -0.114760749, 0.076023981, -0.198310554, -0.122234218, -0.00825509429, -0.196786553, -0.111470282, 0.0473584384, 0.0859691352, -0.0197229534, -0.139441609, -0.195919603, 0.214953706, -0.211334214, 0.0864942521, 0.149090514, -0.0995983481, 0.14995639, -0.211273924, -0.128281027, 0.134673044, 0.206308767, 0.173526242, 0.00177001953, 0.178798303, -0.186740786, -0.125183105, 0.190860763, -0.15597181, 0.104340389, 0.0919784755, -0.109020695, 0.123255745, 0.160754845, -0.0181522816, 0.00826106966, -0.108122781, -0.118333563, 0.0240668505, 0.0728541166, -0.0888753533, 0.0701249689, -0.0911424607, -0.035492748, -0.0625108778, -0.201834172, -0.00986467302, -0.171905458, -0.198220938, -0.125818759, -0.0823892057, 0.124080285, 0.133759275, -0.0294942409, -0.023840189, -0.166492149, 0.0786484629, -0.0805669874, -0.202838793, -0.0324053615, 0.161780253, 0.125890866, 0.162339553, -0.184726253, 0.0838932842, -0.0687282532, 0.192603484, -0.0388252288, -0.127744973, -0.213563338, -0.101094738, -0.00717841089, -0.0166087151, -0.203627214, 0.183910921, 0.00717809796, 0.12827535, 0.0516086072, -0.162369341, 0.120600984, 0.186384007, 0.0617960542, 0.115706041, 0.115686163, -0.0111425072, 0.120042011, -0.0624903291, 0.010419935, -0.0645890683, 0.128529057, -0.0571770221, -0.175542116, -0.0534045845, 0.154075637, 0.0780510157, 0.0838643163, -0.127966419, -0.0523578525, -0.163016126, 0.00269818306, -0.0729043931, 0.213392332, -0.0667243898, -0.00207157433, -0.0347132534, 0.0671278983, 0.0825990885, -0.176288694, 0.115147576, 0.144309029, -0.0388330817, 0.0370965153, -0.145275503, 0.115442678, 0.137224212, -0.0672999918, -0.0209041983, -0.0843738467, -0.076107353, -0.13899076, 0.0134440958, -0.106940709, -0.0790602267, -0.100989997, -0.0825085938, -0.0422780812, 0.216143265, 0.0434457213, 0.171689466, 0.0899863094, -0.00309301913, -0.0964013189, 0.0696323663, 0.11887081, -0.0692265779, -0.194193363, 0.121454194, -0.191472918, -0.110765375, 0.0960554034, -0.101598121, 0.114441469, 0.0659235865, 0.130200818, 0.121813938, -0.0578708351, -0.086437434, -0.108647905, -0.0607499927, 0.0430828184, -0.193046167, 0.0327921957, 0.0684836358, -0.186204255, -0.183985829, 0.110593989, 0.0532316118, -0.177710846, -0.163656503, -0.173432246, -0.0314968079, -0.151612878, 0.143427029, -0.165966004, -0.0755198747, -0.208826602, -0.17920956, -0.0773960352, 0.0872260183, -0.0976994857, 0.114518069, 0.110299453, -0.0676979423, 0.206201911, 0.056230519, 0.158488706, 0.0116583984, 0.152704671, 0.0783563405, 0.197553605, -0.184350356, 0.189391062, 0.0166197326, -0.0901755169, -0.191783831, -0.118035868, -0.0449252799, -0.0107128965, -0.0816708133, -0.0544931963, -0.204584405, -0.0387687087, -0.0949772447, 0.0460221358, -0.000431137101, -0.173131198, 0.0689009875, -0.0812623948, -0.190199226, -0.160632268, -0.150214508, -0.0479303226, -0.133730575, 0.12269488, 0.132861421, 0.116756126, -0.0625272542, 0.0453324765, -0.212504029, -0.180632263, 0.229810223, 0.0990021825, -0.195593789, 0.235955507, -0.249435619, -0.192426175, -0.0116430558, -0.22546199, -0.0619180687, -0.0813810825, 0.178630605, 0.0092575727, 0.176159397, 0.298030823, 0.185510695, -0.137530193, -0.0452765115, -0.207549289, 0.146510646, -0.171670303, 0.265041798, -0.0187018663, 0.135485336, -0.129769668, -0.193181783, -0.213981807, 0.192192391, 0.147625938, 0.156314656, 0.05699341, -0.142236948, -0.119077913, 0.179841056, -0.0629975945, -0.104762428, -0.125211447, -0.14266631, -0.0601936877, -0.0364018083, -0.0799863786, 0.0712708384, -0.181263745, 0.128054276, 0.0881264061, 0.0278715938, -0.0938142166, 0.108250186, -0.0280871093, -0.173671246, 0.154439613, -0.199859276, -0.207510322, 0.113391146, 0.0949654132, -0.157867059, 0.0300325751, 0.0347745866, -0.0836828798, -0.109618604, -0.0289660841, -0.202263281, 0.21372427, -0.105892681, 0.191544786, -0.170336902, -0.150212094, 0.197368309, -0.186274111, -0.170028225, -0.00803947449, 0.194047078, -0.0991749167, -0.119580686, 0.0488605946, 0.0256551802, -0.125362441, -0.0738906264, 0.206044659, 0.00442288816, -0.175227448, -0.152266279, -0.199678972, 0.0752449185, 0.0161459446, 0.208508387, -0.198326081, 0.0312630236, 0.174753115, 0.153398082, 0.140059993, 0.0729063898, 0.174086884, -0.0703520328, -0.195192233, -0.157076001, -0.036226362, -0.205104709, -0.174567297, 0.0171607882, -0.116198495, -0.0708719939, 0.044384256, -0.159294024, -0.13956818, -0.147202596, -0.172137842, 0.0154579133, -0.0588126779, 0.155877337, -0.0972540677, -0.0985946134, 0.108118966, -0.0442180336, -0.0142957121, -0.113704823, 0.0837571472, 0.0825636238, 0.100469217, -0.193166032, -0.189904317, 0.110404596, 0.111059561, -0.0263882726, 0.0777775496, -0.194304436, -0.132153511, 0.118601069, 0.0515244752, -0.0868103802, -0.092175208, 0.182618186, 0.0733394772, -0.110395521, -0.153526604, -0.0347853154, 0.129671916, -0.140404195, 0.10624896, -0.198270962, -0.146404207, -0.206243992, 0.176455781, -0.125557557, -0.192070216, -0.0227239877, 0.213343993, 0.128212437, -0.0822850317, -0.155388311, -0.0103898495, -0.119988322, -0.00629195571, 0.0263843983, -0.0645047724, -0.131128609, -0.0325913876, 0.135626957, -0.072056964, 0.0038716346, 0.195447132, -0.211576611, 0.000806346536, 0.142347768, 0.193100467, -0.204855338, 0.00235620141, 0.0648757964, 0.205600873, 0.13106589, -0.0140479952, -0.196146876, -0.132513404, 0.145923689, -0.13448292, -0.00566205382, 0.185168788, -0.09505447, 0.0785790831, 0.0351739079, 0.205144569, 0.137520716, 0.16661109, 0.196318254, -0.213474959, -0.0414532572, 0.103707328, 0.0494590253, 0.0121845901, -0.14195092, 0.168113038, 0.106775209, 0.00271753967, 0.0252564102, 0.122725263, -0.0311934501, -0.200210854, 0.131448641, 0.205436215, -0.14131099, 0.0286722034, 0.168602541, -0.047244519, 0.0403911918, 0.13908349, 0.0185234249, -0.117879212, 0.0941817015, 0.170137122, 0.0652392656, -0.0828565061, -0.0910385549, 0.177681938, 0.102450922, 0.0477524549, -0.163797021, -0.101946861, -0.214260817, 0.0238904785, 0.225524053, 0.208094507, 0.0252908356, -0.174766853, 0.010269451, -0.0447409302, -0.0171606299, 0.0435046591, -0.211344436, 0.137196705, -0.00548750954, 0.106041424, -0.03372702, -0.0689889714, 0.176017016, 0.0693399906, -0.0631261542, 0.0570853353, 0.110590167, 0.158552811, -0.218137234, 0.227292344, 0.228224993, 0.104598656, 0.191354856, -0.0603202321, 0.0390501469, 0.160037979, -0.0421753563, -0.012174543, -0.0599781871, 0.0374898314, -0.16964066, -0.0145777613, -0.150289029, -0.222676113, -0.130118147, -0.0851336271, 0.0560929105, 0.124441281, -0.0389688611, 0.211753815, -0.3047176, -0.195135519, 0.0575269051, 0.118676692, 0.254068643, -0.0964110196, 0.103781089, -0.0195431523, -0.00197520107, -0.0391661637, -0.0210434217, -0.0949213803, 0.0830372572, -0.200275943, 0.184665754, -0.0754128322, -0.108697027, -0.194729984, -0.0860964432, 0.163379699, 0.195537135, -0.220752254, 0.183663502, 0.0367836021, -0.193053201, -0.213411212, 0.169405296, -0.210496545, 0.089611128, -0.0914427266, -0.146663666, 0.112126216, -0.190471187, -0.151629761, -0.118191868, -0.161780074, 0.0700828135, -0.023731539, 0.0662216842, 0.0570927225, 0.151051804, -0.0581127815, 0.187727496, 0.164582342, 0.108500071, 0.0806025043, 0.132105574, 0.171909839, 0.151336297, 0.0216216911, -0.19720386, -0.0865775421, 0.0918769985, 0.0651388541, 0.101763561, -0.165228412, 0.0967422575, -0.197852328, 0.0326667093, 0.149067357, -0.202845722, -0.0753694028, 0.185080975, 0.112593286, -0.0308894385, 0.146897539, 0.139629066, -0.0057492801, 0.196031645, -0.0433132499, 0.0949817896, -0.22793296, 0.140323445, 0.20535101, 0.00654665194, 0.0543287173, 0.082761243, -0.0949113667, -0.19657506, 0.0682489723, 0.184988469, -0.0549624749, -0.155943945, -0.159202754, -0.000955834985, -0.0745041221, 0.0357825309, -0.0457972139, -0.0863496214, -0.068731755, 0.156966105, 0.102031305, 0.0772381872, 0.0516668707, -0.069934696, -0.171752036, 0.0247167349, 0.197206363, 0.000397771597, 0.0669030994, -0.0112306774, 0.121345595, -0.181874871, -0.102461353, 0.130182162, -0.0321843177, 0.0372402221, -0.0465781689, -0.18494001, -0.0399046838, -0.0770143121, 0.134995177, 0.189494893, 0.148261294, -0.061371848, 0.119698837, -0.20221296, 2.30669975e-05, -0.205027491, 0.0951066166, -0.168831587, -0.0747900307, -0.121398196, 0.178700998, 0.0287471116, -0.0423051268, -0.106853776, 0.205980286, 0.215550825, -0.0599444807, 0.188939258, -0.098034136, 0.0424312502, 0.113852099, 0.00394080579, 0.0708767325, 0.0387572497, 0.193161801, -0.105255395, -0.149511009, -0.183171943, 0.0543221086, 0.000958368182, -0.0319679826, 0.089403823, -0.011545077, -0.0130462199, 0.00551834702, -0.00398561358, -0.0225462615, 0.157178923, -0.204262495, 0.022420153, 0.00691081583, 0.202832952, 0.103284314, 0.0576447994, -0.168464258, -0.160268232, -0.16031602, 0.13101922, -0.102683522, -0.0796382576, 0.0150442421, 0.057686463, -0.00462538004, -0.0570764691, -0.112117276, -0.202424645, 0.177651122, -0.060906291, 0.14917542, -0.0663579404, 0.207064077, -0.0621602237, -0.0727250576, -0.0505298674, 0.166853115, 0.131181166, 0.0528817028, 0.182591543, -0.131295085, -0.214916736, -0.167643577, -0.171931058, -0.0976076052, 0.0673984438, -0.192280039, 0.160496429, -0.096597679, 0.0677601844, -0.0665755719, -0.0466447473, -0.134645581, 0.0446114689, -0.188451454, 0.065866366, 0.0944281369, -0.0774573982, -0.128453493, 0.084732458, -0.0828902125, -0.0460760146, 0.0562799424, 0.0572096854, -0.120285958, -0.0611797273, -0.0863713622, -0.0313139707, -0.158191442, -0.0913565308, -0.0547137558, -0.0715128481, 0.148597136, 0.0647662133, 0.0948180407, 0.1016884, -0.107101806, 0.112274364, 0.130645767, -0.132742882, 0.063240245, -0.0239790529, 0.214894965, 0.039905265, -0.166711584, -0.164006442, 0.00362469256, -0.0177395344, -0.142894775, -0.0920766145, 0.0557132512, -0.105091035, -0.0341222584, -0.126966149, 0.0203460455, 0.194955453, -0.0237233341, -0.049101457, 0.0987512916, -0.188197687, -0.00309565663, -0.0618091077, 0.121471658, 0.114097014, 0.0614005476, -0.0874201059, 0.118369386, 0.0488611311, -0.0974244624, 0.060956791, 0.09975712, -0.0146490484, -0.213436767, -0.116138719, -0.0667345077, -0.209338829, -0.196749538, 0.202766106, -0.122498922, -0.212087691, 0.21396865, 0.0765298456, -0.0631021708, -0.114263915, 0.137899652, -0.0875501335, 0.0651765019, -0.172441825, 0.0399881452, 0.0264455229, -0.148256093, -0.208674431, 0.0328289419, 0.0215819627, 0.0447034687, 0.0569855124, 0.0466875732, -0.154296696, 0.0557099953, 0.099412255, 0.0885903686, -0.138083339, -0.215496168, 0.0766443089, -0.029674679, -0.159911841, -0.193334565, 0.129661992, -0.209483698, 0.0277790427, 0.0214523505, 0.125006989, 0.206167772, -0.247479483, 0.110709831, -0.0240806229, -0.106150419, -0.0156477932, 0.23906444, 0.0239258539, 0.0397250541, 0.159573585, 0.0976805016, 0.028400287, -0.184984565, -0.135613933, -0.235051349, 0.158971772, -0.100035571, 0.098122105, -0.0841649026, 0.181454465, -0.190613255, 0.126531929, -0.0978783965, -0.0936749801, 0.0890369713, -0.0226638466, 0.0344321169, -0.231752813, 0.125484258, 0.0367094986, -0.177370921, 0.217156366, 0.190573201, 0.178353146, 0.0782344341, 0.197666898, -0.0849834532, -0.117577732, 0.130946651, 0.117060021, -0.171168283, -0.0270178616, 0.169972658, 0.210708454, -0.176258653, 0.241882116, -0.0276549459, 0.0397499725, -0.12462277, 0.0972123072, 0.289701581, -0.09509027, -0.195481196, -0.0970052183, -0.0570235103, -0.230527118, 0.168534026, 0.0795216113, -0.0857440829, -0.104283124, 0.0783484355, 0.0913527161, -0.175007626, -0.0441816524, -0.101990119, -0.0751975626, 0.0174092911, 0.0910891965, -0.072370857, 0.0863547698, 0.030440174, 0.0699474886, -0.069681555, 0.244500011, 0.132901147, -6.72638416e-05, -0.011448239, 0.0668040514, 0.0330525972, 0.0399980098, -0.0805684775, -0.0893881321, 0.00371935964, -0.089494504, -0.135875374, -0.00690581929, -0.0437228978, -0.139606163, 0.138900653, -0.189150035, 0.0839610398, 0.064339444, -0.219201058, 0.10751234, -0.138615251, 0.25648123, 0.193666056, -0.195941389, -0.0475867949, 0.170852602, 0.0483538099, -0.23815763, -0.215300962, -0.0604494624, 0.157071248, -0.198099524, 0.1605075, 0.187679827, -0.110149607, 0.260497242, 0.0667465031, 0.0740663335, -0.0811945647, -0.0274696928, 0.256537765, 0.112993523, -0.176565573, -0.211348012, -0.174424976, -0.0731801093, 0.107577667, 0.137092873, -0.183942825, 0.161429822, -0.234576806, 0.153691486, -0.0336565897, -0.0619529299, 0.1576882, -0.00832078699, 0.144546583, -0.0621412583, 0.0572977401, 0.0700711533, 0.107443564, 0.247199208, -0.107651167, 0.257766634, 0.212229684, 0.0449296683, -0.0885326862, -0.01169773, 0.0446972661, 0.132320687, 0.146239325, -0.125418752, -0.0602291077, -0.145199999, -0.0226940326, -0.042851422, -0.200135052, -0.0707998723, -0.0483647697, -0.0434840582, 0.0195474084, -0.0806870908, -0.066419743, -0.0243462902, 0.187009096, 0.266266257, 0.0210534781, -0.190431267, 0.0193590894, 0.0430474356, 0.0968303457, -0.0600356534, 0.212457985, 0.0733742341, 0.0564355701, 0.00829766691, -0.0975096449, -0.0297273509, 0.0435266942, 0.232403845, 0.175813645, -0.0605938882, 0.075977318, -0.102545507, 0.159124359, -0.0323878899, -0.11937844, -0.210411832, -0.0369421095, -0.0605836548, 0.0146844471, -0.162964344, -0.180745065, -0.138387382, 0.191610858, -0.0805439204, -0.0106778275, 0.195784792, 0.140448511, -0.108700931, 0.154517576, -0.139445692, -0.0971742496, -0.156008646, 0.0350373723, -0.00932324678, -0.0389326066, 0.157756582, 0.0591719672, 0.191582471, -0.109771289, -0.205349728, -0.123457506, -0.113767751, -0.199369431, -0.0199184865, -0.0721435249, 0.0268921331, 0.17901054, -0.0615942702, -0.196627244, -0.0978841856, -0.0243181754, -0.252508283, -0.171970218, -0.00553819537, 0.138990164, 0.176095605, 0.0951418132, 0.00899968576, -0.21385926, -0.197060034, 0.193683833, 0.233065248, 0.06070612, 0.0120316064, 0.0260351393, -0.0639142916, 0.173514277, 0.204962239, -0.202115402, 0.188184857, 0.059859708, -0.160158709, 0.194068417, 0.03272672, 0.0373210721, -0.154273242, 0.192293808, -0.200334892, 0.123418614, 0.0633706972, -0.0923486948, 0.114942677, 0.198776662, -0.215897352, 0.0565530509, 0.0895846412, -0.13462013, -0.0126579404, -0.177565232, 0.158671334, 0.233714014, -0.193006068, -0.281954676, 0.156786814, 0.144733921, 0.151347488, 0.173282146, 0.276410073, -0.19197917, 0.292017668, -0.151239187, -0.149175525, 0.0274241325, 0.188164338, -0.293288738, 0.0220334232, -0.273543179, 0.0642050654, 0.08832784, 0.134583443, 0.0807607248, -0.000400550896, 0.0918587297, 0.07559672, 0.314674675, 0.0490694642, 0.101967268, -0.241429016, 0.0202955063, -0.209007189, -0.106268622, -0.0069014011, 0.10103409, 0.0636226386, 0.0471041873, 0.000416273368, 0.26530841, -0.10846144, 0.142565444, 0.216730133, -0.137502536, -0.120941207, 0.180886477, 0.118575349, -0.0189697742, 0.239887834, -0.142993346, 0.146749064, 0.187433407, 0.0744013041, -0.0447228253, 0.205760106, -0.0467358679, 0.0100782812, 0.180402741, 0.0978421122, 0.068239525, 0.164465442, 0.00975632668, 0.195215091, -0.0487101376, 0.0192688555, 0.031739369, 0.199693933, -0.0508198142, 0.123593971, 0.0872715563, 0.148543522, -0.150334686, 0.0227344036, 0.115462556, -0.0487159789, -0.016429022, 0.0369556397, 0.0111047179, -0.0476019233, -0.118862145, -0.0377347171, 0.0323484689, 0.0822030753, 0.0403838307, -0.0443079621, 0.0296327919, 0.104416624, -0.03586936, -0.162577927, 0.140675917, 0.0654677302, -0.155557871, 0.0191291273, 0.213035539, -0.174402893, -0.124022201, 0.169056132, 0.158662096, -0.163972616, -0.0827359259, -0.00124819577, 0.010516569, 0.212345287, 0.0464865416, 0.110000417, -0.154047757, -0.0204191953, -0.08001028, 0.064174667, -0.212888524, 0.0529602021, 0.211512908, -0.190684035, -0.0921802148, -0.151814789, -0.00803656224, -0.00784375705, -0.141917571, -0.00132001087, 0.0526149124, -0.136854231, 0.0130218118, 0.0680401698, 0.0399013944, -0.186063141, 0.0169487298, -0.0813166797, 0.116694055, 0.042951867, 0.0821733102, 0.134713322, 0.184491575, -0.191935867, 0.0131632471, -0.100137152, 0.182891071, 0.000961091835, 0.12456546, 0.145593375, 0.00720275845, -0.105598301, 0.207914561, 0.00380734471, -0.0248022173, -0.160123363, 0.0381194986, 0.129718468, 0.123341523, -0.0176308304, -0.175096646, 0.110144205, 0.0652518645, 0.094259724, -0.0674603283, 0.224985868, -0.048998557, 0.00546664651, 0.0410965495, 0.107289985, 0.00302270707, 0.0922987014, -0.0397922322, 0.0962653086, -0.093549408, 0.048931852, -0.0534424298, 0.0138503471, -0.0754063874, 0.065585278, -0.0900662616, 0.139983714, 0.128798306, -0.0214835256, -0.0355337039, -0.00254588644, -0.0779585242, -0.10749051, 0.0774092972, -0.195456222, 0.203156188, 0.103489295, -0.0295414776, -0.0359847844, -0.132312894, 0.139603063, -0.0406532735, -0.114045464, -0.155046389, -0.111411333, 0.0317999125, -0.166794747, -0.167081028, 0.0591999739, 0.129730806, -0.175916776, -0.0256558955, -0.0691830069, -0.0288138986, 0.0313598067, 0.0193842202, 0.0408626944, -0.172637001, 0.0734120756, -0.202827275, 0.190578565, 0.153090999, -0.0792387873, -0.00259576738, -0.0505202115, -0.212944731, -0.159402311, -0.0976085365, -0.0191448629, 0.130320415, -0.0283066481, -0.0278123319, 0.00982235372, -0.0937846899, -0.162156463, -0.143455982, -0.00604511797, 0.0269212872, -0.194088265, 0.10351716, 0.00833112001, -0.0464727581, 0.129887775, 0.046137765, -0.183257371, 0.0989542454, 0.0501036495, -0.156223819, 0.0834358186, 0.128036156, 0.00859726965, -0.0364925116, -0.197799727, 0.164447352, -0.122780189, 0.000409752131, -0.0851694047, -0.127068669, 0.124540463, -0.0155066447, 0.220182613, 0.0643692538, 0.0083350027, 0.208433077, -0.083687149, 0.139471397, 0.0637006313, -0.166873068, -0.044224903, -0.152341023, -0.0996580869, -0.00282181404, 0.0116580725, 0.0610121377, 0.153579026, -0.151627228, 0.0830854848, -0.0748153627, -0.00402663695, 0.196929038, 0.199087873, 0.162471503, 0.103831865, 0.0201131664, -0.0360102542, 0.155990794, 0.104891919, -0.0791717842, -0.173016161, 0.0897792131, -0.0222959071, 0.011724811, -0.0878165364, -0.0617964715, 0.103893965, 0.117816001, 0.046961911, -0.0394895524, -0.172319263, 0.0261968896, 0.128624946, 0.000213261112, 0.096357584, 0.183724195, 0.0663415045, 0.128639147, 0.257106632, -0.126175031, -0.166864216, 0.0406238586, -0.0439073667, 0.234832495, 0.110920966, 0.147819847, -0.0325478055, -0.145270362, 0.123860314, 0.0187417157, -0.133771777, 0.0191091448, -0.018727826, -0.212830409, 0.0778542906, -0.13378343, -0.0403149575, 0.176398948, -0.00964029133, 0.123386756, -0.0300345421, -0.187632725, -0.0620219409, -0.188461006, -0.139842436, -0.100581177, 0.0265599042, -0.110380962, 0.191845462, 0.00141653419, -0.11816033, 0.208042368, 0.213605359, -0.129850671, -0.0933597088, 0.122598633, 0.00595799088, -0.018640548, 0.0378848463, 0.181395903, 0.173377052, 0.0876867622, 0.192007706, -0.209600434, -0.012859717, 0.00600273907, 0.127768829, -0.130987272, 0.134607062, 0.155363366, 0.0808825344, -0.0882706791, -0.076367721, -0.0793054253, -0.00586630404, 0.142082587, -0.206148043, 0.0407580584, -0.049249351, 0.0129451007, -0.116375081, 0.164335236, -0.105530523, 0.13251628, -0.0697510839, -0.0777705759, -0.117720746, 0.0540670604, 0.164986417, 0.103021309, 0.0867776424, -0.0438529849, -0.00377820432, 0.162118211, -0.128094852, -0.0133839697, -0.0300400108, 0.191699013, -0.114906885, -0.128097042, -0.125449896, 0.0672464222, 0.181721359, -0.0279202759, -0.0308043379, 0.012561053, -0.0228079483, 0.117388152, -0.0491030663, -0.152897894, -0.0109380297, -0.141598642, 0.12240307, -0.196314692, -0.139708713, 0.0969985127, -0.166283533, -0.261718482, -0.10953261, 0.0718631297, -0.213036582, -0.144475102, -0.00279817055, 0.0964064673, 0.0178181678, 0.110280976, -0.175311595, -0.251570255, 0.141161755, -0.188831225, -0.0564760268, -0.2272598, -0.152180851, 0.152426973, -0.00386719452, -0.0721517727, -0.012255799, -0.198725522, 0.105782107, 0.280836701, 0.0152221853, 0.275105059, -0.209379539, -0.224154338, -0.104977705, 0.0988008901, 0.0514465943, -0.0128156841, 0.157611817, 0.170334578, 0.0869703367, 0.285808533, -0.0728926361, -0.0931104496, 0.0235334337, -0.110741422, 0.125828728, -0.117568605, 0.155986264, 0.104506925, -0.0337914713, 0.0296717696, -0.235040098, -0.0135234362, -0.141636685, -0.100419141, -0.134680957, -0.186574012, -0.0766067058, 0.146882966, 0.154049531, -0.0364503711, 0.0356544703, 0.0556236356, 0.0494298339, -0.277094424, 0.073460117, -0.193379238, 0.134578362, -0.102159671, -0.239353925, -0.215223923, 0.194666088, -0.0964104012, 0.0814671591, 0.0992431194, 0.0468135215, -0.162915677, 0.162857607, 0.209440842, -0.187548369, -0.0020732081, -0.0355331898, 0.0981004983, -0.182766274, 0.0926911905, -0.0237608105, -0.102904551, 0.122693948, -0.236414105, -0.211930677, 0.115730271, 0.207284644, -0.0510552563, -0.157497108, -0.115445964, -0.173785508, -0.217097312, 0.103066951, 0.00525379414, 0.076337561, 0.12234731, -0.0626737922, -0.185681343, -0.0525672026, -0.0714665577, -0.215600729, 0.125220552, 0.0981240124, -0.178441167, 0.0892993957, 0.0875188187, 0.235276952, 0.0606884509, -0.0568252951, -0.242791384, -0.0947935879, 0.141819909, 0.204088584, 0.11860837, -0.0103346705, 0.143899903, -0.109179169, 0.103566274, 0.0646427423, -0.186479658, 0.200688288, 0.173446015, 0.191234097, 0.131643906, -0.0541896075, 0.17311503, -0.0397259891, 0.179010823, -0.160451055, -0.0738938302, 0.0460077673, -0.188182101, -0.167358577, 0.0334474444, 0.0105334073, -0.123536415, -0.0196802616, 0.15479432, -0.0144007057, 0.116810068, -0.208570942, 0.100825295, -0.19967401, -0.212417796, 0.0673297793, -0.215567753, 0.052130118, -0.151904643, 0.197143808, -0.0339394808, 0.206757233, -0.0573075712, 0.136985973, 0.108611509, -0.0870095193, -0.122860461, -0.1796031, -0.0982395262, -0.101981603, -0.107995287, 0.140654042, 0.170272157, -0.124455385, 0.119262144, 0.163930461, -0.185422182, -0.21241951, -0.121740013, -0.172264829, 0.0637018234, 0.051629886, -0.14822641, -0.112850063, 0.0174066424, -0.0829333961, 0.0977343246, -0.071891427, 0.0561515987, 0.109630719, 0.0105861574, -0.0270061102, -0.190160096, -0.119579576, 0.197185382, -0.0970397443, 0.0522243232, 0.000522117305, 0.0153891267, 0.146401003, 0.159108639, 0.25341928, 0.00318193459, 0.0668381304, 0.0247753933, -0.115337625, 0.0172942206, 0.0831532627, -0.0902798697, -0.105036713, -0.213386223, -0.121249683, 0.0464711972, -0.141757503, -0.113185756, 0.193994313, -0.187768489, -0.15975529, 0.0177620109, 0.0166279227, -0.193038374, -0.0627801642, 0.0224070493, 0.105940476, -0.137638792, -0.11995957, 0.0115957642, -0.128734171, 0.138942927, -0.108310811, 0.0426762067, -0.234138444, 0.0704599395, 0.113127954, 0.180509791, 0.169870883, 0.0833347514, 0.112489417, 0.11732848, -0.0221389327, -0.110925816, 0.117433928, -0.214904755, 0.054917559, -0.0237672813, 0.148916826, -0.017192632, 0.0826454312, 0.164108485, -0.0137663055, -0.0730242953, 0.234863907, -0.178744644, 0.0621348992, -0.00839559734, -0.10974963, -0.0248806775, 0.055587817, -0.0795170292, 0.18179898, -0.149376124, 0.0317146517, -0.0143466592, -0.0674705505, 0.17889294, 0.0754329786, -0.150365472, 0.0464622527, -0.00969791599, -0.200375721, 0.0205095354, 0.154160127, -0.00569080515, 0.155038372, -0.0677913055, -0.147895366, 0.0321660787, -0.056184493, 0.0394759253, -0.157382205, 0.233074352, -0.0469223112, 0.116115957, -0.203592524, -0.123089239, -0.164869681, 0.0379196517, 0.0770090148, 0.0427877568, -0.169947818, 0.0919543505, -0.0403930247, 0.175416812, 0.21293062, 0.210629076, -0.111974031, -0.14331843, 0.0128842229, 0.0350685567, 0.0866905451, 0.13432996, -0.202785864, 0.0997599959, 0.207019001, 0.138129339, 0.0494085439, -0.108375512, -0.127402216, 0.0275171027, -0.0740583614, -0.00576845882, 0.193134576, -0.0666644946, 0.0633924752, -0.089058876, -0.0918698311, 0.0843076035, 0.202469081, 0.0892445296, -0.1374605, 0.0150794983, 0.0531005375, 0.161458567, 0.210192963, 0.04205136, 0.107358694, -0.0251380932, 0.0682467371, 0.186786473, 0.0294182803, 0.0918548927, -0.197670788, -0.144377872, -0.191045746, -0.20302172, -0.0703191012, 0.26318568, 0.183188379, -0.206453308, 0.217197284, 0.148158118, 0.0516163856, -0.0405543372, 0.0482969098, -0.0797786266, 0.0162452161, -0.142858282, -0.0700473189, -0.165941894, 0.0412169918, -0.200823486, -0.21580334, 0.0719728321, 0.0922091603, 0.149025053, -0.023213055, 0.265344322, -0.150436535, -0.021344753, -0.140235752, -0.255674452, 0.15332745, -0.00951609015, 0.165915266, 0.0167089067, 0.124824308, 0.0771664828, -0.253194153, 0.0453373007, -0.0910207182, 0.0636530071, -0.19644013, -0.231708229, 0.178851888, 0.18904604, 0.0673967227, -0.253504723, -0.004631266, 0.0158821791, -0.0782575011, 0.112024978, 0.0643248707, 0.0634058863, 0.00650183856, 0.0145138055, 0.0211943984, -0.186126992, 0.153037265, -0.0982570276, 0.117266491, -0.0641367286, 0.0506336838, 0.177407131, 0.027125746, 0.08834593, -0.170427591, -0.156710893, -0.180125281, 0.18578954, 0.132006899, 0.0475857705, 0.0842403024, -0.0162469745, 0.103354886, 0.208519891, 0.194094405, -0.0861671567, 0.138932332, 0.201304033, -0.193600982, 0.175816432, 0.107227907, 0.169770226, 0.0631686598, 0.0528858155, -0.0414999276, -0.104278192, -0.17777279, 0.107138261, -0.0946334153, 0.0493052155, 0.195973918, -0.0339171737, 0.167163864, 0.062439546, 0.191270575, -0.204546601, 0.204385087, -0.0609797537, 0.102811083, -0.0426427275, -0.144036323, -0.215613484, -0.149330556, 0.186492875, -0.112123109, -0.129927844, -0.153668568, 0.0724345893, -0.147795394, 0.195619091, -0.168710485, -0.0126553029, -0.0127404332, -0.116737291, 0.168202505, -0.139484406, 0.0554534048, 0.0361851305, -0.113191009, -0.174208596, 0.0114807189, -0.195487082, 0.134786084, 0.144725397, 0.207942024, -0.0374336243, -0.0180579275, 0.1983376, -0.0727393627, 0.0687315911, -0.0218542069, 0.0489843339, 0.160994157, 0.0465723425, -0.0552227646, -0.160425812, 0.118589506, -0.173039734, 0.094873175, 0.0973959714, -0.0334962308, 0.131362393, 0.192723766, -0.085611105, 0.186923936, 0.173444375, 0.195655927, 0.0500997752, -0.0955151692, 0.0853087157, 0.109827921, -0.0743474066, -0.135200426, -0.0115245879, -0.024191156, -0.0558120608, -0.160451472, 0.0763798505, -0.16293782, -0.1017408, -0.15939261, 0.0827288479, -0.215683803, -0.0368343294, 0.0422128886, -0.176073387, -0.105860367, 0.0477225035, -0.115710489, -0.193383917, -0.188803807, -0.170165524, 0.0757941753, 0.16839464, 0.0277366079, -0.123203889, 0.094133839, 0.195007026, -0.202828094, -0.105727762, 0.0652255863, -0.166010231, -0.126647398, -0.0466658585, -0.120006435, 0.0939842612, -0.0244721789, -0.194358811, -0.0313170701, 0.109878041, 0.194994539, -0.148321584, -0.154995516, -0.0752039999, -0.0561695024, -0.0345148742, 0.0120506845, -0.145251185, 0.276574999, -0.183512345, 0.246295869, 0.175020978, -0.134096593, -0.171224758, -0.178246081, -0.0637267604, 0.0260362774, -0.0426347815, -0.0999041423, -0.133127928, -0.217847079, -0.195832476, -0.108974583, -0.00344945025, 0.247975796, -0.0544710569, 0.0776171461, -0.0458349697, -0.232248828, 0.0165108331, -0.16456145, -0.118792772, 0.135833904, 0.191254571, 0.152048305, -0.0461367741, 0.116522327, 0.00936230551, 0.0552281439, -0.00196163752, 0.229142398, -0.142573804, -0.0892553627, -0.120750993, 0.256958574, 0.0426204354, 0.0873946771, -0.226227716, 0.141678169, -0.042470932, 0.124623254, -0.179483652, -0.116647683, -0.116587028, 0.103890166, 0.123260602, 0.0605796427, -0.0168686211, -0.00929376483, -0.0128240585, 0.172887877, -0.0799608827, -0.0303717256, -0.127870053, 0.17608051, -0.0424753278, -0.0972225741, 0.0391885191, 0.200019762, -0.0154580772, -0.186458692, 0.134563908, -0.0995464176, 0.0737005621, 0.176864192, 0.0450127572, -0.188842878, 0.0309933126, 0.0700256974, -0.0154144019, -0.0797051638, 0.187247232, -0.0477865189, -0.0276180953, 0.180766746, -0.199228138, 0.207444504, -0.16353789, 0.156251594, 0.165612713, 0.11059694, 0.209873334, -0.140326887, 0.175071821, 0.0395414978, 0.156043813, 0.0787585527, 0.199952558, -0.0327560008, 0.0251382589, -0.199105844, 0.0476279408, -0.0291632563, 0.0443746597, 0.173739001, 0.00965835154, -0.117652602, 0.0828595608, -0.164778814, 0.156857237, -0.130015075, -0.107045695, -0.222709522, -0.0534569211, -0.146377668, 0.143743783, -0.223435938, 0.0202661306, 0.0298079774, 0.130296096, -0.169427738, 0.0867685452, -0.189785749, -0.214855, 0.138201609, 0.0175307598, -0.00683422387, -0.0721608624, -0.148823351, 0.0987624824, 0.163937375, -0.221082836, 0.097356841, -0.10563866, -0.174024582, 0.231104016, -0.167891935, -0.0109430226, -0.0339421071, -0.015225037, -0.0966599807, -0.0566251948, -0.038483344, -0.0632045045, -0.173830792, 0.234540999, -0.0372984409, -0.11684528, -0.0237086806, 0.177134946, -0.135995328, 0.143075436, 0.0284443703, 0.0957668871, -0.203221127, -0.138940528, -0.170615286, -0.04803662, -0.0227327403, 0.156518131, -0.120296806, 0.116717979, -0.0278942138, -0.180543825, -0.120960377, 0.0104260044, -0.125010282, 0.105188407, -0.0110195624, 0.0892315656, -0.200755909, 0.205126464, 0.168077156, -0.118845731, -0.142220959, -0.0858293474, 0.0769720748, 0.00681600207, -0.0523019433, -0.109635837, -0.0064796377, 0.0102793276, -0.130109623, 0.150559291, 0.0784872174, -0.0432755277, 0.188085303, 0.00808112323, -0.181910425, 0.0972780362, 0.138851807, -0.165652379, -0.167549655, 0.123791538, -0.212279394, 0.103910975, -0.124968246, -0.0679621696, -0.150251463, -0.0412153937, 0.18648304, 0.171684593, 0.00163652177, -0.138664946, -0.0801473856, 0.176220953, -0.181696028, -0.00872888416, 0.181269154, 0.0954500809, 0.0857712477, -0.137488693, -0.0543198027, -0.168690518, -0.210396335, -0.211841181, 0.111533284, 0.0498711616, 0.131123632, 0.171156824, 0.0636221096, 0.0163842924, 0.00664749416, -0.193607077, 0.104148954, 0.0818801969, -0.126201361, 0.107612975, 0.109677412, -0.132316753, -0.0396888182, -0.00945395418, 0.0487647355, 0.0377194248, 0.178009942, -0.135111406, 0.137946114, -0.0810011625, -0.0691107288, -0.182944283, -0.0679595321, 0.0203998834, 0.174737379, 0.0201928318, 0.0889042467, 0.0805583745, -0.204121158, 0.00436645746, 0.0794607848, 0.0822678357, 0.00139918923, -0.0264118016, 0.0835606307, -0.00963528454, -0.0870883018, -0.12715739, 0.145659909, 0.0546541363, 0.187282696, 0.0855048746, -0.0967017934, 0.0764478296, -0.208491907, -0.0981765538, -0.017935276, 0.127355561, -0.124414347, 0.0346565694, -0.108974963, -0.0984654129, 0.125999585, 0.0118691027, 0.0898878127, -0.0464704335, -0.00716736913, -0.0696949661, -0.00315192342, -0.172756493, -0.034152925, 0.0687169284, -0.0139536262, 0.0157241225, 0.0378018171, -0.0701506585, -0.00593361259, 0.16699715, -0.0711576492, -0.043457225, 0.127052858, -0.0215502083, 0.177768037, -0.0212931484, 0.12964575, -0.196589366, 0.0531259924, 0.023148343, 0.15855442, -0.0950687155, -0.0336764306, -0.0928969979, 0.197106078, -0.0703088194, -0.0125174373, 0.104199722, 0.0937243253, -0.0498488285, -0.0790696591, 0.0754235014, 0.159118399, 0.175383911, 0.00834533945, -0.132660657, -0.115502544, -0.0156698935, -0.142873257, -0.172217071, 0.00926896464, -0.0980520546, -0.186849445, 0.104777038, 0.141713575, -0.116373293, -0.177874327, -0.0812455565, -0.180731073, 0.157215104, -0.0100824358, 0.13991484, -0.165303022, 0.129494235, 0.102651075, 0.0760747492, 0.0534787029, -0.201117173, -0.148061618, 0.158403665, 0.170118049, -0.184529886, 0.00612172484, 0.18630074, 0.0668295771, 0.203014389, 0.0470853746, 0.120209262, -0.0326153599, 0.178558037, 0.130264938, -0.158517003, -0.236181453, -0.077458322, 0.0907330364, 0.0622364357, 0.118951038, 0.0970379859, 0.157590434, 0.0286808833, -0.103834197, 0.0967250317, 0.052686438, 0.0817455575, 0.121504307, -0.154424161, -0.16611585, -0.130731776, 0.194687054, 0.186306313, 0.00081812439, 0.0815480202];
    CONSTANT bias_1 : ARRAY[0..63] OF REAL := [-0.00991463661, -0.000165412683, 0.0380159281, -0.0313414298, -0.00776600698, 0, 0.0327618271, 0, 0.0053440691, -0.012447658, -0.00528640207, 0, 0.00980756432, 0.0239994954, 0, -0.00600226782, -0.0427969247, -0.0124991806, 0.0102020688, 0.0347996801, -0.0137349106, -0.00922023784, 0.060131371, -0.043544095, -0.0354361534, -0.00553967617, -0.0374039412, -0.030632956, -0.00583763421, 0.00989670772, -0.00822056364, 0.0306522157, 0, 0.0557479262, 0, 0, -0.00697317952, 0.0160537008, 0.0252484679, -0.0129459258, -0.0292139072, -0.038203638, 0.0335591063, -0.0462469868, 0.0442246161, 0.0594434552, 0.0479242764, 0.0381261297, -0.0195034202, 0, -0.00470581418, -0.00563494209, -0.0306187645, -0.0391318202, 0.0379941873, 0.0250570383, -0.0389060415, -0.00584178604, 0, 0.00260822545, -0.0485509746, -0.0251302961, -0.00867041945, 0.0280207619];
    CONSTANT weights_2 : ARRAY[0..4095] OF REAL := [-0.141680449, 0.288066953, -0.150528222, 0.0983807966, 0.0682033002, -0.0383133292, -0.0808929056, 0.143694162, -0.143791497, 0.173556536, 0.0320169441, -0.121532038, 0.0184226483, -0.0103868982, -0.0746624023, -0.135166839, 0.113171645, -0.126689032, -0.0239767376, 0.0532080457, -0.10377644, 0.104337208, 0.0625005439, -0.119132705, 0.202529803, -0.086342141, -0.205905676, -0.150743365, 0.0873293057, 2.73770947e-05, 0.064553991, -0.0785556436, -0.157094628, 0.00396119431, 0.0939819738, -0.0202242639, -0.150879264, 0.125680909, -0.0767421126, 0.107631303, 0.0793541521, 0.0918624699, -0.0373493209, -0.227653801, 0.16160652, -0.210584804, -0.000720652053, -0.13250798, -0.103983767, -0.123876065, 0.029696513, 0.177454278, -0.053838402, -0.105550319, 0.115103669, -0.0959799588, 0.18597813, 0.231739312, 0.135426775, -0.046401687, -0.100035861, 0.0408016182, 0.0825353414, 0.136485547, 0.00270199776, 0.0867017061, 0.195101574, 0.126894072, -0.132388622, -0.0208239406, 0.00692871585, 0.128494516, -0.13354221, -0.0511906333, 0.0144319832, -0.171571314, -0.125738502, 0.13592577, -0.137273088, 0.1709162, 0.0410082564, -0.183967724, 0.0714212805, -0.0134086907, -0.0914759263, -0.111280508, 0.182648227, -0.0738228038, 0.0616786629, -0.21075432, 0.203339309, 0.0925859734, 0.115103915, 0.0693822652, -0.188044399, -0.108215593, 0.164470464, 0.153212592, 0.0917293802, -0.179572374, -0.143311441, 0.115444198, 0.0727809519, -0.00865674019, 0.127544686, -0.0877099037, 0.103159383, -0.078883104, -0.100927807, -0.0344764031, -0.12042328, 0.0344114751, 0.131927297, -0.146454126, 0.0510100611, -0.0590627939, -0.0506405383, 0.0810800865, -0.090818353, 0.0528705269, -0.201525137, -0.0838072225, 0.110697366, 0.0740895495, 0.172959939, 0.189559668, -0.065729633, -0.0720220059, 0.105840042, -0.058448758, -0.107932165, 0.216511503, 0.00461578369, -0.107524514, 0.058490552, -0.175286993, 0.0249149054, 0.0852858871, -0.157516927, -0.0535053015, -0.0676146448, 0.0599285662, -0.0855296031, 0.140303031, 0.149562418, -0.0901874602, -0.0450080633, 0.0728893131, 0.00284661353, -0.0671322271, -0.105737545, -0.0900957286, -0.198729545, 0.162473515, 0.147394195, 0.145424545, -0.0517513901, -0.0669851601, -0.164583072, 0.110631853, -0.215715826, -0.170075879, 0.0506092906, 0.00326168933, -0.0199967101, -0.0183630344, -0.0711533353, -0.148096681, 0.114399835, 0.0869136602, -0.115128055, 0.156051964, 0.14734675, -0.148528323, 0.104175396, 0.282105029, -0.235148892, -0.208776742, -0.088167496, 0.198368117, -0.205772802, 0.00897102989, 0.0128333028, -0.0552920029, -0.166966945, 0.147610545, 0.0774816051, 0.0655531734, 0.146716073, -0.00372734619, -0.214626014, -0.0576679409, 0.00339318812, -0.0645904765, 0.129015684, 0.0367895626, 0.00563158561, -0.150251627, 0.14424403, 0.219185576, -0.015582785, -0.0557845123, 0.229870901, -0.136385068, 0.193651333, 0.0781679228, 0.10057772, 0.0421372652, -0.078148827, 0.111039303, -0.0640359819, 0.213664457, 0.239976257, 0.134989008, -0.121206947, 0.158595756, -0.170423076, -0.138676971, -0.0604084283, 0.129199952, 0.163071141, -0.221609473, -0.0275269188, 0.186735034, 0.13408266, 0.0231132358, 0.196531892, 0.0723142847, -0.184686705, -0.0832601115, 0.130843252, -0.0489593074, 0.182337478, -0.0457641892, -0.00743399095, -0.126927346, 0.0406110212, 0.0973830223, 0.188993767, -0.0883924365, 0.263101488, -0.0826768279, 0.15883705, 0.172388598, 0.123626038, 0.10255266, -0.252580434, 0.211067945, -0.0147316307, 0.00241988176, 0.156785056, -0.112871908, 0.0347109661, 0.0922119021, 0.00649048388, 0.153683811, 0.138896421, 0.0972352177, -0.208112851, -0.202854082, 0.0617144667, 0.0563855022, -0.0516398437, -0.0742861032, 0.0109137893, -0.117585734, -0.0220603198, -0.0585992336, -0.0475497693, -0.0259862747, 0.119525358, 0.189453453, 0.172370642, -0.0726865008, -0.0956337899, 0.0137653798, -0.150756568, 0.118895762, -0.083567664, -0.165870577, 0.130793914, -0.133739084, 0.198176801, 0.184771329, -0.209565952, -0.183116794, -0.0640594736, -0.203715086, 0.0997374058, -0.070866093, -0.171968624, -0.122551396, 0.0937422961, 0.19882901, 0.120841727, -0.00538546452, 0.199771121, 0.121376611, 0.141540334, 0.159105301, -0.0297715347, -0.196540907, -0.124991439, -0.145521253, 0.205668867, -0.0768398345, -0.035737481, -0.0238609333, -0.124907829, -0.0484834574, 0.124906845, 0.124305926, -0.0377987772, -0.191355884, -0.159768522, 0.183061063, 0.184881866, -0.212566867, -0.0531422645, 0.0976230353, 0.00577385724, 0.130427197, 0.211715534, -0.0860495567, 0.0888584703, 0.121544942, -0.180683181, -0.0218638033, -0.0905238539, 0.0180363953, -0.02386415, -0.13335371, -0.00121800601, -0.094210498, 0.112201318, -0.216103971, -0.0530306548, -0.158522308, 0.152102396, -0.15442571, -0.134984136, -0.0138640255, 0.0654296428, -0.158441991, -0.134703487, 0.190590188, -0.176293343, -0.178531021, 0.0348580927, -0.00753350556, -0.213596776, 0.109840617, -0.103785381, -0.0846005082, -0.082864821, 0.108093217, 0.132263497, -0.156487495, 0.149631396, -0.0340299606, -0.0305996239, 0.107479975, 0.0321970284, 0.0810965151, -0.169963852, -0.0118091106, 0.173262879, 0.134186372, -0.20041047, -0.000686064363, -0.0538731366, -0.0124969929, 0.0516002327, 0.0954418629, 0.0455744714, 0.0564913601, 0.133059844, 0.110250726, 0.180289343, -0.000993043184, 0.186119303, -0.0665116161, -0.0792722255, 0.202967927, 0.205843329, 0.21862179, 0.0488890447, 0.0133959213, -0.00834459066, 0.00461511314, 0.0836300105, -0.121354386, 0.117611662, -0.234934494, 0.0287881922, -0.0978208929, 0.136924744, 0.0765881464, 0.148768306, -0.168677807, 0.0451220796, -0.0645759478, 0.182842463, 0.139968216, 0.0730862394, 0.0406570174, 0.0715097487, -0.159143537, -0.122275874, 0.147242293, -0.146196708, 0.0239535533, 0.10290198, 0.0115962736, -0.0944432169, -0.0756312534, 0.0423654877, -0.168181121, -0.0449682809, -0.0617624037, 0.152064502, -0.0231318604, -0.0633203983, -0.00436079642, -0.110454418, -0.246325403, 0.188381672, 0.122344673, 0.123941295, 0.201515913, 0.24498114, 0.182052374, -0.163516134, -0.156467408, -0.00582023244, -0.112946808, -0.127423167, -0.0515909754, 0.155103877, -0.173389852, -0.199556112, 0.115317613, -0.162211671, -0.191533402, -0.0836257115, -0.0725069493, 0.06501095, 0.035802599, -0.176167637, -0.0298467577, 0.155019239, 0.169515267, -0.000437632203, -0.0261323899, 0.199166045, 0.172561631, -0.193425417, 0.175140068, -0.0974695757, -0.142100155, 0.194233581, -0.0656768829, -0.120199233, -0.162119597, 0.169042096, -0.214600414, 0.0662081391, 0.0520145446, 0.107069895, 0.175651714, 0.131947085, 0.143850192, -0.00955465436, 0.0627427548, 0.210242525, 0.0844678432, -0.129487574, -0.0942333117, -0.0245972425, -0.090298906, -0.0466166288, -0.107186824, 0.111454025, -0.137471825, 0.136128113, -0.0861810446, -0.186852902, -0.0583910942, -0.0535676479, 0.0353205353, 0.0871732086, -0.146667257, -0.121421315, -0.143794656, 0.147011802, 0.170059487, 0.0102381408, 0.153043762, -0.00729104877, 0.0746920556, -0.0543518513, -0.0595977008, -0.0225165188, 0.0500841886, -0.182219625, 0.0947217196, -0.205081433, 0.12140505, -0.201528907, -0.0524655879, 0.155590281, -0.129846334, 0.0906220675, 0.151344299, 0.186176911, 0.0421557426, -0.207316592, -0.131616503, 0.133107722, -0.160803005, 0.143145278, -0.161467314, -0.0657405034, 0.135806978, 0.166633621, -0.200071856, -0.207391843, -0.215113148, 0.148792446, -0.0100589618, 0.0714959651, -0.0805551559, -0.0614150316, -0.174764574, 0.207058311, 0.122847259, -0.196977898, -0.1559522, 0.0978694558, -0.185000882, -0.140967488, -0.16737549, -0.106714033, 0.164967701, 0.0964245871, 0.140171438, 0.207501814, -0.0379861556, -0.0579505898, 0.225760758, 0.111228764, -0.146074057, 0.0667390376, -0.169152468, 0.938151181, 0.17469056, -0.175612152, -0.123244651, -0.126487702, -0.0329091251, 0.138695627, 0.0742424577, 0.098279722, 0.119007275, -0.172866449, 0.0933431759, 0.0521263108, -0.131282881, 0.0761865526, -0.0664989054, 0.164532125, 0.0566500686, 0.200022459, -0.0600383841, 0.182312235, 0.194255427, -0.0288380273, -0.122255489, -0.0914943814, -0.0893590152, -0.0746954307, 0.146213099, 0.184557945, -0.118034557, -0.174534202, 0.0035078912, -0.0207415409, 0.105583005, 0.0245418437, 0.184224337, -0.0410954989, 0.113560788, -0.0217513908, 0.0455570407, 0.0366436318, -0.159584582, 0.0670233443, 0.21683304, -0.128995791, 0.275691748, -0.0195934419, 0.177997693, -0.1972785, -0.0668776929, -0.216343522, 0.163236275, 0.205884218, 0.216626123, 0.147940427, -0.0883644, 0.092634283, 0.207626119, 0.171906605, -0.167044088, 0.204324439, -0.109410673, 0.0193916559, -0.119002052, 0.0720684603, 0.141300142, -0.088518776, 0.0176712964, 0.161592081, 0.126937598, -0.0751166046, -0.133596882, -0.115226425, 0.24855116, 0.122299738, -0.095500432, -0.119029626, 0.152431637, 0.00319294631, 0.21932444, -0.0965302214, 0.134576872, -0.015701618, -0.0857832581, -0.216072649, -0.137355849, -0.196437761, -0.126480833, 0.0231357962, -0.134333387, 0.171409652, -0.113697752, 0.0360458046, 0.163777098, -0.0132845491, -0.153503746, -0.213196114, 0.0580244511, 0.152173683, 0.0331603885, 0.211798117, -0.199593693, 0.129404142, 0.113514826, 0.0272548497, -0.214540333, -0.193730131, 0.215466887, 0.0018462775, 0.013003692, 0.195035413, -0.0590138286, 0.0399461836, 0.0308904201, 0.179027125, 0.0488234572, 0.0415520221, 0.137228593, 0.200982258, -0.156045571, -0.105913378, 0.133550122, 0.0291233379, -0.081467703, -0.145602509, 0.171516255, 0.0566335171, -0.00745478272, -0.167673349, -0.118719235, -0.00841763616, -0.167444021, 0.0689675286, -0.200617492, -0.121176332, 0.0399130136, -0.194600999, -0.107290849, 0.201394126, -0.0595335364, 0.197396234, -0.0294916183, -0.0975661054, -0.0199405309, -0.0464265756, 0.0777761638, -0.184141561, -0.0692353547, 0.203581437, -0.0510522276, 0.00841990113, -0.0510387868, -0.209235489, -0.0786187798, 0.0127682984, -0.0585706383, -0.149550289, 0.0406086594, -0.15494749, -0.0766567886, 0.192089304, -0.174240753, 0.168413922, -0.184974745, 0.129347548, -0.0480398685, 0.102323428, -0.00398623943, -0.0793017, 0.186511293, -0.01932621, 0.140939757, -0.008235991, 0.135236308, 0.0234718472, -0.0376885831, 0.0408930033, -0.0838549286, 0.105532184, -0.169196993, 0.00895322859, -0.0224669725, 0.214271948, 0.187380776, -0.168133691, -0.171357155, -0.0451917201, -0.090357855, 0.126548275, 0.102986887, -0.133371353, -0.0108436346, -0.0374744087, -0.17570509, -0.132929906, 0.00220645964, 0.127038345, 0.0997535139, 0.210657284, -0.137902528, -0.125172943, -0.21302484, 0.10058029, -0.0661100745, -0.00623327494, 0.0631183833, -0.103329279, -0.185445309, -0.0871112198, 0.0991731733, -0.194505647, -0.200181127, -0.0255591124, -0.205262512, -0.204970762, 0.0392911546, -0.20052886, -0.0514694117, 0.0394407958, 0.0124119818, 0.130332097, -0.101388983, 0.137814477, 0.0253826454, 0.190587938, -0.161746755, -0.198715627, -0.077888988, -0.0540392175, -0.096387893, 0.00343954773, 0.113467187, 0.166445121, 0.0665265769, 0.115969144, 0.16848965, -0.114840552, 0.164357632, -0.0157545805, 0.191388026, -0.175001413, -0.131909996, -0.0113435686, 0.147116452, -0.0923970491, -0.0562144518, -0.176853389, 0.0598261133, 0.190945908, -0.0372008011, -0.0430109315, 0.11451865, 0.0371341594, -0.0761518031, 0.110607252, 0.00426071882, -0.146474242, 0.0800529569, -0.11710421, 0.0366946682, 0.269265682, 0.191883326, -0.0611798316, 0.00541722775, 0.232036233, -0.202542618, -0.14030695, -0.0281257648, 0.230240002, 0.0162147321, -0.164047837, -0.124143533, -0.121437646, -0.17262505, -0.0583858602, -0.0723832101, -0.19505994, 0.0283917375, -0.131140262, 0.0902625024, -0.115805745, -0.117771566, -0.116753951, -0.0244481117, 0.154554754, 0.0925760716, -0.177714929, -0.0415367521, 0.0639798269, -0.128405958, 0.0617773086, 0.12867713, -0.220567599, 0.155001327, -0.164517075, -0.10119269, -0.0264345706, 0.193819627, 0.00867548306, -0.131352246, 0.168402314, -0.0690761581, 0.0819703862, -0.124435671, 0.12688598, 0.113567822, 0.0819837376, 0.236767009, -0.196865633, -0.0627399534, -0.167267427, 0.0447263867, 0.211083233, 0.127811357, 0.144808367, -0.108109578, -0.0729895085, 0.103431262, -0.130963951, -0.0642541945, 0.0399866477, -0.0517324097, 0.106077358, 0.0571983159, -0.137635872, 0.172099277, 0.171573251, 0.0966628045, 0.0747942552, 0.0563847944, -0.0897115842, -0.182717025, 0.0567689948, -0.0702779293, -0.0933412313, 0.165129632, -0.0129972473, -0.0846574679, 0.128517389, 0.12487001, 0.170890465, 0.18792893, 0.111724451, 0.177234873, 0.160684839, 0.0530777425, -0.0586484224, -0.160080284, -0.144362509, -0.159860179, -0.181875899, 0.154358193, -0.0374765694, -0.083326295, 0.181780145, -0.121391997, -0.0691839457, -0.0742421448, 0.0691870898, 0.14754726, -0.069750309, 0.0740958601, 0.198498741, -0.154731348, 0.0730743259, -0.00451502204, 0.0863774866, -0.092950426, 0.131180331, -0.18926172, 0.148594961, 0.0665854961, -0.0706014037, -0.0448699296, -0.0694603622, 0.0639980286, 0.0166171342, 0.196238205, 0.016624555, 0.0550233275, -0.180780441, -0.161480352, 0.0111390948, -0.0118472576, -0.0242867023, 0.0894839317, -0.214834765, 0.165922478, -0.146362454, -0.205421194, -0.146823198, 0.0966032892, 0.148615941, -0.0852327496, 0.163918838, 0.102714762, -0.208166033, 0.0172590613, -0.0552005172, 0.0110155195, 0.179708347, 0.0191160589, -0.133684993, -0.0525586009, 0.205576107, 0.210995749, -0.138825268, -0.142582893, -0.141632929, 0.0855522454, 0.198174328, 0.00804278255, -0.0469306856, 0.0574738979, -0.144030869, -0.165960878, -0.108321778, -0.197332725, -0.0156382918, 0.0518989488, 0.0718663186, -0.0900121629, -0.0854760781, -0.216951966, 0.180414304, 0.0896183103, -0.0315984115, -0.038237486, 0.16515182, -0.0816439539, -0.0227444768, -0.0454315543, -0.185322598, 0.0210614055, -0.194109529, 0.0599969067, 0.0527030006, 0.0741187185, 0.156095579, -0.0249356292, -0.164651155, 0.123715535, 0.172677234, -0.0501076728, 0.0449018963, -0.0228640102, -0.0200645179, -0.084004961, 0.0933688506, -0.12003617, 0.146246135, 0.114758648, 0.0661290213, 0.126682028, 0.161090702, 0.140608266, -0.148477748, -0.0640800446, 0.133195326, -0.0674081072, -0.181248829, -0.0289781466, -0.0194690824, -0.0494243838, 0.106817186, 0.195835143, -0.0803123191, 0.161425516, -0.0493547022, -0.05296278, -0.196740344, -0.17108798, -0.0269036777, -0.257117361, 0.0609735921, 0.126235262, 0.234910175, 0.298613906, 0.110691503, 0.163770065, 0.164086029, -0.102102607, 0.269784272, 0.298873127, -0.141947195, 0.00401810464, 0.160247535, 0.199671581, 0.102458611, -0.171934664, 0.211893931, -0.109412298, 0.0464521386, 0.174394637, 0.0244902223, -0.0639190525, -0.0315829515, -0.0628100634, -0.145441294, -0.248165399, -0.096565783, 0.0521190837, 0.171565145, -0.0265039522, 0.113324709, -0.0879507959, -0.022442922, -0.175112098, 0.194249406, 0.0624903068, -0.174791113, 0.0232726112, -0.254210442, -0.126247719, 0.245405003, 0.154142827, -0.183761641, 0.124047622, 0.143147632, -0.11987894, 0.0924994051, 0.238024503, -0.0995406434, 0.127400458, -0.118362844, 0.0286737774, 0.0726793855, 0.0532515496, -0.00276745413, 0.147954509, 0.175074711, 0.263851762, 0.0354693085, -0.0399195738, -0.0167579949, -0.0360376686, 0.119187571, -0.175929293, 0.179050192, -0.209990561, 0.0303346924, -0.0304141119, -0.168580458, 0.0159338806, -0.143411383, -0.14976643, 0.0935455635, -0.0950493068, 0.0929078311, 0.0551954135, 0.0518541336, 0.176312774, -0.183571264, -0.102172591, 0.174365237, -0.10537722, -0.041147884, 0.0739963651, -0.111693986, -0.0890176594, 0.0285699144, -0.157434717, -0.14237228, -0.00719396165, 0.0457479246, -0.146615341, -0.07867226, 0.00846140739, -0.130273566, -0.117995292, 0.0493791625, 0.183448762, 0.148034781, -0.191158175, 0.15299876, -0.0805099756, -0.0233456288, -0.168751732, 0.00436502555, 0.139199287, 0.193048775, -0.143146724, -0.197523668, 0.112838462, 0.0882283896, -0.176614121, 0.0627285391, 0.115050167, -0.203107342, -0.130106881, -0.0552822948, -0.10732834, -0.131432489, 0.0808235332, 0.217252836, 0.0871307775, -0.0174604356, -0.165878817, -0.172403678, 0.254087269, -0.162096322, 0.323802054, -0.012599051, 0.151775375, 0.153595924, 0.00913618691, -0.182565987, 0.114645109, 0.0815113634, 0.121357247, 0.126867056, 0.0927122906, -0.136515841, 0.106271967, 0.209716767, -0.152262896, -0.0599813312, -0.0153267533, 0.0652863383, 0.219464377, 0.196837217, -0.223917902, -0.143790111, 0.138385013, 0.113471806, 0.367199123, -0.137293875, -0.0288341846, -0.0667795986, 0.038723208, 0.102534734, -0.138440862, -0.0140577843, -0.0820909142, 0.329797894, 0.0938638672, 0.0398048386, -0.20963259, 0.154240653, -0.0378240161, 0.134357706, -0.0533082113, -0.0598759018, 0.0404425971, 0.21940358, -0.00829724967, -0.120814763, 0.0788223594, 0.11621587, -0.20682922, 0.00859716535, -0.00990748219, 0.0331411287, 0.114033349, -0.151647523, -0.158313036, 0.0926335678, 0.0706593469, 0.351727486, 0.166647702, -0.0461413115, 0.216942608, -0.138307035, 0.144426495, -0.169870242, 0.200646102, -0.16545783, 0.181138262, 0.11609225, 0.077415742, -0.182514325, -0.15969798, -0.21806176, -0.160868764, 0.104007304, -0.160312831, 0.0297145694, 0.0499397293, 0.0594710223, -0.0964953378, -0.177800402, -0.0670034215, -0.19343999, 0.180497482, -0.0837211534, -0.128186598, -0.13259843, -0.089160189, 0.0347441472, 0.128377378, 0.105255894, 0.11304494, -0.158335477, -0.183520451, -0.132612199, 0.195470482, 0.171718106, -0.21191743, 0.176613376, -0.0911389291, 0.0547690429, -0.122613512, 0.0449908227, -0.0874788165, -0.0113770878, -0.102273077, 0.125744522, 0.0171495155, 0.103814244, 0.185875043, -0.0773060992, -0.207971171, 0.0723132193, -0.0591497123, -0.174698785, -0.0662334561, 0.0624778345, 0.181660056, 0.0352354199, -0.144429192, -0.0237713046, 0.1413863, -0.055128105, 0.107294582, -0.0923522636, 0.10639482, 0.0696970969, -0.104372099, 0.0329963788, -0.142583638, 0.197051004, 0.039161697, -0.0938943475, -0.0997598544, -0.0650602877, -0.0785568804, -0.0371245071, -0.13516289, 0.00734080002, 0.0694661215, 0.0717197061, -0.038889166, -0.0539452471, 0.213663176, -0.0399716944, 0.015419662, 0.0576197021, -0.211071417, -0.00350436778, 0.15874508, -0.0291592199, -0.0852676928, -0.186650351, -0.143953145, 0.160483733, 0.23401615, -0.174104869, -0.0815619752, 0.178066641, 0.206289992, -0.13791053, -0.162200421, -0.111578882, -0.0799070597, 0.137941718, -0.109797254, -0.0264309049, -0.0568498187, 0.0664690062, 0.0718042403, 0.0974657089, 0.0933575481, -0.0164596867, 0.210323125, -0.142812029, -0.149296373, -0.180004731, -0.0265571047, 0.128158346, 0.0553876162, -0.122902334, -0.0440571681, -0.112295315, -0.138417289, 0.039254874, -0.193141863, 0.0195326358, -0.201830551, 0.150758162, 0.115440972, 0.202520981, 0.106997013, 0.0990103036, -0.129501849, 0.0595938414, 0.090642944, -0.112931691, 0.0857426375, -0.152478904, 0.144109204, 0.0355113298, -0.107244223, -0.0304977745, 0.113781944, 0.12506713, -0.207027107, -0.182988301, -0.0227130949, 0.0429330915, -0.17101869, 0.116467908, 0.116578884, 0.0260287896, -0.0962790847, 0.036279276, -0.0381992906, 0.212093785, 0.158137083, -0.112858787, -0.131867021, -0.191359714, -0.146997213, -0.000313639641, -0.003441751, -0.0417472273, -0.0491207764, -0.178802773, -0.0664816052, -0.0104046613, -0.0142799169, -0.188737929, -0.0185466558, -0.0352328829, 0.0682502836, 0.0788259357, -0.195347801, 0.203497171, -0.154879391, -0.18561314, -0.17881757, -0.117247216, 0.0698423609, 0.0224083364, -0.0493452102, -0.140239567, -0.183991462, -0.113582537, 0.0816551074, -0.203832656, 0.148944646, 0.166977555, -0.168197036, -0.0038562566, 0.0320169367, -0.17292963, -0.15642412, -0.165192544, 0.182672083, -0.15258047, 0.101091012, 0.174555406, 0.0823695511, 0.157132462, -0.129125595, 0.0654330179, -0.166881204, 0.0782062784, -0.0887168273, 0.00821068604, 0.0453969091, 0.220597595, -0.196104899, -0.0166419595, -0.0927555114, -0.107461981, 0.221482277, 0.223973781, -0.0611179322, -0.0668021888, -0.0858261585, 0.0375918262, 0.267744839, -0.0345278829, 0.254966795, -0.00994786248, 0.022099562, -0.127365038, 0.18192032, 0.0513121448, -0.110994041, 0.25041303, 0.196979046, 0.135527775, -0.0681474656, -0.0267207474, -0.199583828, -0.0502842888, 0.00327560958, -0.0646822006, 0.19758679, 0.261831164, 0.0999355987, 0.0594527014, -0.154063612, 0.0252208039, 0.221329957, 0.131121457, 0.00249284413, -0.0733978972, 0.100284182, 0.0556562096, -0.0429260246, 0.0306841414, 0.219935, 0.13371262, -0.00598191097, -0.132255256, 0.221873939, -0.163495034, -0.0360863805, 0.0824131444, -0.239943579, 0.172781795, -0.212151602, 0.236218229, -0.0616496243, -0.0723682791, -0.0943582132, -0.173591569, -0.158820465, -0.0388342962, 0.209313601, 0.105139598, -0.0127423787, 0.23334001, 0.105608903, 0.189134374, 0.161174685, -0.0848595649, -0.13802968, -0.00375816296, 0.102438428, 0.0600083843, -0.197466984, -0.15549612, -0.0712063238, 0.154483199, -0.0873283222, 0.15228495, -0.0364889465, 0.179233074, 0.14827925, 0.185523212, 0.27177012, -0.0103518441, 0.156902194, -0.0411169007, 0.0607469641, -0.0220632553, -0.0432856232, 0.142093897, -0.147602007, 0.18813391, 0.0621521808, -0.181282967, 0.0722836629, 0.179992348, 0.0792825669, 0.247705981, 0.228616223, -0.0473009236, 0.00126909569, 0.0863893405, 0.155630812, -0.100628406, -0.123317964, -0.11671751, 0.0799793229, -0.16633673, 0.0691096857, -0.0983060077, 0.161242321, 0.171100721, 0.143575251, 0.182359606, 0.00890773162, 0.110979609, 0.0892734379, -0.105653889, 0.227419034, -0.03998366, -0.124580286, 0.130855098, -0.0131535288, 0.272792101, 0.179608643, -0.210909322, 0.00432928372, 0.21848838, 0.253688663, 0.106119879, 0.0625382364, -0.143925086, -0.0632008985, 0.0975730494, -0.141114861, 0.0668569505, -0.0672182292, 0.162051871, -0.122773834, -0.0107828472, 0.0403296016, -0.0795900598, 0.277176142, 0.00853289384, 0.173946515, 0.117141366, 0.183931693, -0.0793479383, -0.0215559229, 0.187337711, 0.061015863, 0.0663154572, 0.169271708, -0.201445878, -0.0256252605, 0.244238496, -0.231323823, 0.0469608344, -0.0628846064, -0.14439863, 0.113650277, 0.163789138, 0.021281559, -0.103731513, -0.192868605, 0.147293687, 0.0449895933, -0.160115749, 0.0899030939, -0.165846884, 0.198117554, -0.167129472, 0.218909174, -0.171495542, -0.161191314, 0.129484773, 0.0846461579, 0.169623926, 0.0230460148, -0.112478353, -0.0921991095, 0.211257413, -0.0030605495, 0.0351988226, -0.0332586169, 0.139157876, 0.0921685547, 0.122303888, 0.0700193793, 0.179862246, 0.0254115313, 0.204242676, 0.0813357979, -0.0274808407, 0.200144112, -0.119426139, 0.161797479, 0.0829108208, -0.153130651, -0.0846347809, 0.0271065533, 0.140034661, -0.130517483, -0.186353624, -0.0104580438, -0.201147348, 0.075118795, -0.045870319, 0.156480566, 0.0903002545, -0.00378783746, 0.192498252, -0.038612958, -0.131505221, -0.0437254906, -0.101072744, -0.0389576852, -0.164237425, -0.175792545, 0.0373107754, -0.119521856, -0.156602532, -0.113795958, 0.112055942, 0.113850042, 0.00677617686, -0.0850653872, -0.0733917803, 0.187380284, 0.182089031, -0.0248251855, 0.163996622, 0.132685319, 0.142668948, 0.0152747529, -0.0172108244, 0.216359109, 0.118470624, 0.123126626, -0.100131035, -0.054644499, -0.133699596, -0.0788406134, 0.115421988, 0.143789545, 0.187183872, 0.167815328, 0.202092215, -0.0217228085, 0.144933701, 0.106362499, 0.259433448, 0.15671441, -0.0946840271, -0.186438739, 0.0081841452, -0.14182502, -0.00946078729, -0.0603948757, -0.00157379068, -0.18708539, -0.0983730108, 0.0651348308, 0.00732422806, -0.0354584157, 0.0694651306, -0.170068949, -0.146637738, -0.0188922025, 0.130627021, 0.253977299, 0.161411852, 0.247188866, 0.203512952, 0.0883074552, 0.113822445, -0.046621304, 0.175482243, -0.0289865751, -0.15941821, 0.178795829, -0.277471334, -0.199458614, -0.00665188488, -0.127981231, -0.209003299, -0.148039356, 0.137913957, 0.0634118468, 0.166315272, 0.170956552, -0.215199739, -0.110592142, 0.0109336888, -0.026153028, 0.0884291679, -0.0187547766, -0.0606251135, 0.185180321, 0.139575243, 0.104148917, -0.216128081, -0.0651518703, 0.100283109, -0.0865191743, -0.0341802686, 0.0216208063, 0.072604768, -0.122850962, -0.0247077513, -0.147178918, 0.12824367, 0.182407543, -0.000500810798, -0.184659287, -0.0473984033, 0.0934755877, -0.0367431417, -0.15300943, 0.24329026, -0.151669785, -0.114891134, -0.186268806, -0.0633910894, -0.166982651, -0.107574888, -0.0891585425, -0.139917731, -0.0927230418, -0.175722167, -0.0773153529, -0.115566179, -0.145081356, -0.147527725, -0.138250202, 0.217643395, 0.224325195, 0.150407761, 0.0212292019, 0.0613440573, -0.188086301, 0.23438555, -0.0300599616, 0.206930742, 0.0815451145, -0.375011235, -0.0562498868, 0.00639961939, -0.0058033783, 0.168399513, -0.0654805675, -0.0274477936, -0.109949432, -0.0414189361, -0.0130247008, -0.200141788, -0.163074657, -0.170476168, 0.193809062, -0.111856036, 0.152590171, 0.0143048586, 0.185440674, -0.169017375, -0.158529475, 0.00929309428, -0.0942657292, -0.148064896, -0.134354785, -0.206875667, 0.202413216, -0.0598236918, -0.166547075, 0.152515814, -0.163616508, -0.202204078, 0.114426211, -0.182107091, 0.0707437545, -0.0522488952, 0.0869736522, 0.0402545184, -0.0945940241, 0.185991451, -0.124674715, -0.03174752, 0.162187114, -0.137566179, 0.184869885, 0.0221520253, -0.197971106, -0.170951381, 0.0330120921, 0.0279635787, -0.139334649, 0.0697774142, -0.197592616, 0.17985791, -0.0284902453, 0.115595266, -0.201338783, 0.0367098935, 0.07913436, 0.127372906, -0.124858603, -0.0313890874, -0.181075796, 0.0527459234, -0.135128409, 0.0876705199, -0.184465155, -0.0735049844, 0.0535863489, 0.00994851347, 0.137904853, 0.0959903747, -0.186176807, -0.0812415555, -0.112533055, 0.174689725, -0.096371375, 0.122750133, -0.0395515561, -0.0953361019, -0.142940253, 0.0410725772, 0.111044452, 0.0270516891, 0.161732242, 0.0858138651, 0.0895572454, 0.037848372, 0.162806571, -0.0460997261, 0.0349680036, 0.160732448, -0.129507929, 0.113114722, -0.0166504215, 0.120835945, -0.0622817799, -0.133667618, -0.0202337652, -0.0207774434, 0.170200497, 0.00774796167, -0.0592490025, 0.230593592, -0.00738770561, -0.0436120033, -0.0423453487, -0.0329519622, 0.206478819, 0.0155085847, -0.0256422833, 0.0234079231, 0.0186074525, -0.1795073, -0.180009589, -0.00913083926, 0.196808264, -0.21870546, -0.179154739, -0.0917448699, 0.14978005, -0.061042279, 0.012972462, -0.0826573893, -0.0671150908, -0.138860673, 0.00231725769, -0.166636378, -0.0871414915, -0.0446091257, 0.192121252, -0.109329425, 0.0788124055, 0.152980164, -0.129419059, -0.0276356209, -0.0259925574, -0.0593720526, 0.179485679, 0.0266083553, 0.0747748911, 0.101830587, -0.0766663998, 0.0163841695, -0.161232248, 0.0171750262, -0.279156268, 0.221496373, -0.186395198, -0.0143639594, -0.143523067, -0.0878556073, -0.0815294832, -0.067358315, -0.16824618, 0.111157678, -0.160450444, -0.161506832, -0.0405490361, 0.102888331, 0.0339654423, 0.118124977, -0.00176335871, 0.165163413, -0.0700196028, -0.00438803434, 0.175777838, 0.186697081, -0.121123411, 0.122397795, -0.0532331169, 0.0590221882, -0.105305605, -0.204723135, -0.175872728, -0.0677143931, -0.161616057, 0.0188506059, -0.210944623, -0.148904279, -0.113570303, 0.221049219, 0.0313297138, 0.107811853, -0.180402234, 0.109366827, 0.0825608298, -0.15245305, 0.205485806, 0.0317764021, 0.0504349619, 0.00149199367, 0.00595451333, -0.174039871, -0.0160308499, 0.194607705, 0.179732472, 0.0789086595, 0.197504297, 0.0629399493, -0.116470531, -0.186572343, -0.0899397954, 0.19567205, -0.00335924979, -0.208514586, 0.0973969102, 0.0326924175, -0.206587866, -0.0218385514, 0.0725486577, 0.155927837, -0.188840836, 0.0960423201, -0.165740326, 0.1604902, 0.267009914, 0.0818572193, 0.260096461, -0.186999142, -0.0683261901, 0.0665122792, 0.0479869246, -0.101161063, -0.0638602898, -0.218564659, -0.0387957096, 0.0902684554, -0.16147168, -0.0608646087, 0.062403813, 0.0504773445, 0.0787408352, -0.0066665113, -0.0551999062, -0.200761631, 0.00933836773, 0.297097772, 0.16794759, -0.185238838, -0.0823579729, 0.0469955355, 0.3021909, -0.134364396, 0.196597978, 0.0334144868, 0.0336058177, -0.10905616, 0.0721478015, 0.0315832756, 0.189071074, 0.0691891909, 0.34283489, 0.150725141, 0.00169667602, -0.117639907, 0.121499099, 0.194060832, 0.0223687626, 0.161883071, 0.516069353, 0.384240836, -0.0662594065, -0.219141394, 0.113189861, 0.174268171, -0.0602926537, 0.023207292, -0.0562035777, 0.223606259, 0.17101483, 0.15739201, -0.0148757435, 0.195277646, 0.0899973437, 0.48358345, -0.0253587756, -0.00797794759, -0.0891540423, 0.092290625, -0.185479164, 0.0852196366, 0.213107035, 0.0252361298, 0.200780615, -0.189653561, -0.182161033, 0.021594137, 0.145947233, -0.112602293, 0.0719485134, 0.073290661, -0.068946287, 0.146695599, -0.164526656, -0.0765778124, -0.171564609, -0.0508742183, 0.214564845, -0.203749716, -0.138006911, -0.0141354799, -0.206376866, -0.174090385, -0.0728472918, -0.0598603934, 0.0906234831, -0.216011941, 0.122935966, 0.127648816, -0.192449927, 0.0749056488, 0.138052747, 0.105709121, 0.0347812921, 0.110028967, -0.135962948, -0.144907042, 0.154864535, 0.0592765659, 0.0534629077, 0.0385289937, -0.156602025, -0.0317876786, 0.208689615, 0.177388117, 0.00780889392, 0.0349562615, -0.0682702363, -0.0363424569, -0.0553218275, 0.133666351, 0.00441069901, 0.096022442, -0.133351326, -0.00378321111, -0.136954084, 0.0019338131, -0.181480229, -0.155208886, 0.203421369, -0.125472635, -0.171183765, -0.165254846, -0.133507237, -0.0173198301, 0.21947293, 0.143755376, -0.0401268005, 0.0731849745, 0.0850220844, 0.0371454805, -0.0326308534, -0.0790177658, 0.0200932287, -0.121129356, -0.126217842, 0.0199649576, -0.169905156, 0.237343252, 0.177157223, 0.165131941, -0.183802426, -0.125728503, -0.134026647, 0.102495909, 0.0696081296, -0.167917982, -0.166213095, 0.0101573337, 0.134656668, 0.0390270464, 0.147898167, -0.0125229191, -0.171897367, 0.18344982, -0.0810840577, -0.00678340718, 0.122303508, 0.0799789727, -0.0815866068, 0.0310235824, 0.154979914, 0.0764822215, -0.128525659, 0.152218923, 0.0648555607, 0.10429927, 0.165912151, -0.00706859026, -0.0883911997, 0.165610254, -0.205627054, 0.172161713, 0.206336021, 0.121359043, 0.0919625983, 0.223842055, -0.209351197, 0.0634121448, 0.227562383, 0.0355994329, 0.00256789825, 0.237201974, 0.037827909, -0.177561209, 0.222521156, -0.202093512, -0.0229218453, -0.118946023, 0.0302829295, -0.0116465688, 0.022469908, -0.211659819, 0.0230853111, 0.193522528, -0.0245168656, -0.201854825, -0.0753775686, -0.0310619175, -0.200594962, -0.0756556392, -0.128971279, 0.156894669, -0.179421097, 0.0251898766, 0.023289308, 0.0580800325, 0.140855506, -0.0611620098, -0.0153288692, -0.00615723431, -0.21604234, -0.084130466, -0.15956971, -0.0087262094, 0.0838872939, -0.0140172839, -0.186466902, -0.0742408633, 0.134943053, 0.0629239827, -0.158630103, -0.111521803, 0.00854839385, -0.152197734, -0.187499329, -0.146150753, -0.0487617552, -0.12666437, 0.148413315, 0.00076122582, -0.0748235434, 0.210751161, 0.0419287831, 0.0125453025, -0.0107841194, -0.07289505, -0.126931146, 0.140740082, 0.129911378, -0.0123122483, -0.202497944, 0.214250848, -0.119241752, -0.205320999, -0.152010053, 0.159491345, -0.165408313, -0.185733244, 0.0348138064, 0.191792235, 0.200777933, 0.161115959, 0.115620837, -0.125909343, -0.0419274867, -0.0674549639, -0.164896861, 0.200165018, -0.163343281, 0.133848891, 0.066679135, 0.0242425203, -0.215839475, -0.177766964, -0.178671584, 0.179792449, 0.210112378, 0.118905827, 0.180896834, -0.202173829, 0.175342038, -0.0985738114, 0.193638191, 0.0229219347, -0.0222909003, -0.0943710357, -0.024797678, -0.16884923, 0.0664104372, -0.0999937505, 0.0858398229, 0.203513905, 0.182638362, -0.0276584178, 0.143701836, -0.159802675, 0.138917372, -0.0687357336, -0.118034951, 0.165999964, -0.0323487371, 0.123346254, 0.0527410358, 0.137795433, 0.01838772, 0.0875368267, 0.173462018, -0.0463278592, 0.129204765, 0.150611833, 0.107375845, -0.0264342129, 0.169134393, -0.0467272401, 0.199903682, -0.0980908126, -0.190550029, -0.0762602538, -0.0315628797, -0.0798259974, 0.160073265, -0.00462961197, -0.183606789, -0.0188505352, 0.0691810995, -0.197972029, -0.15645048, 0.116300687, -0.124517485, 0.173053637, 0.0755809918, 0.081306681, 0.161437288, -0.0970465466, -0.130220771, -0.0481538028, 0.180401117, -0.0649009943, -0.165097132, -0.130503684, -0.00572030758, 0.0470085293, 0.00363709033, 0.00171510922, 0.0857786089, -0.0651379302, -0.066770114, -0.157249182, -0.17459558, 0.108071186, 0.18482846, -0.0944221914, 0.0439717509, 0.0515320636, -0.101472825, -0.191481218, -0.157240301, -0.0539558493, -0.125500441, -0.157671779, 0.217446938, -0.153299645, -0.0213545188, 0.169633135, -0.202749312, 0.15830192, 0.123832054, 0.202120841, 0.178851813, 0.0410678647, 0.00611580582, -0.053331662, 0.0464291424, -0.0324332118, -0.106219634, -0.216207579, 0.228908926, -0.0941737071, -0.134803563, -0.202760994, -0.00565075129, 0.168043837, 0.0981038436, 0.0794638395, 0.167057589, 0.128910467, -0.0112976059, 0.170332775, 0.0585579872, -0.22341539, 0.0355694294, -0.154355466, 0.0759388655, 0.105432287, -0.0729613379, -0.0318719745, -0.0295223258, -0.100262426, -0.100136787, -0.0460873507, -0.0712981075, -0.0222990401, 0.0588900596, -0.113420017, 0.17419365, -0.10283038, -0.144499213, 0.124155849, 0.0594922118, 0.0716532618, 0.129410103, 0.0517303199, 0.148354009, 0.0255827624, 0.0190704111, -0.149046123, 0.136326805, 0.105247073, -0.0295574721, -0.238865554, 0.0468696915, 0.0912098587, 0.0714069828, 0.0229250956, 0.110962324, 0.131823346, -0.165668309, -0.00778792799, -0.185458347, 0.20212841, -0.0874781683, 0.0586535111, 0.143871352, 0.275070757, -0.044842042, -0.0718936771, -0.072808072, 0.0834283978, 0.133895293, 0.198372915, -0.0804026723, 0.188191667, 0.0981120318, 0.206251636, 0.177413091, -0.102985151, 0.196867242, -0.013884523, -0.188111216, -0.130392522, 0.0190863628, -0.148793653, -0.0467367023, -0.192909583, -0.0972905159, -0.137692288, 0.211145386, 0.140261218, -0.142052516, -0.194741502, 0.192499146, -0.049346976, 0.0810934156, 0.0646863505, 0.125058278, -0.0799507052, 0.132487938, -0.0906506926, -0.0655713826, 0.0928521007, 0.183620468, 0.138887301, 0.162195206, 0.155351385, -0.058083415, -0.0219758153, 0.0991288573, 0.0169533193, 0.103431225, -0.130349159, 0.0779341757, -0.241531909, -0.178271845, -0.138706401, -0.0624510534, 0.111244112, 0.111007653, -0.0359138511, 0.0459302366, 0.0223376025, 0.165935397, 0.0252500176, -0.147416338, -0.110299625, 0.00361161027, 0.167947292, 0.132642567, -0.0257409364, 0.250626832, 0.08315216, 0.0183384717, 0.0648797005, 0.108391851, -0.218746424, 0.223503336, 0.0558422469, 0.081787914, -0.0234055668, 0.0559378527, 0.0436194129, 0.0106922649, -0.0692483187, -0.0691979155, -0.0494184643, 0.0244371723, -0.167693228, 0.158963591, -0.115475364, -0.173542932, 0.0758400708, 0.0158745944, 0.176581964, -0.032615751, 0.140387014, -0.0867669731, -0.0148333311, 0.0844656676, 0.191718534, -0.194510147, -0.0462476611, -0.142200023, -0.127892822, -0.0507825464, 0.0212071091, 0.0735275894, 0.101716116, 0.074662827, -0.197910756, -0.133237764, -0.187822059, 0.145099476, 0.0327065587, -0.146056384, -0.0505298674, 0.108181708, 0.107639544, -0.138911337, 0.122266933, 0.115411207, 0.144105688, 0.0382299572, -0.148832917, 0.139190271, 0.167309538, -0.144928098, -0.0563678443, -0.043597877, -0.1119316, -0.12973395, 0.0584410578, -0.0437880307, -0.0104946736, -0.165186569, -0.0112327933, 0.118900821, 0.182406887, 0.192648664, -0.00062443316, -0.184834018, 0.199227616, -0.121603794, -0.167943582, -0.00912922435, -0.0713112056, 0.171490803, -0.0891723186, -0.0559416711, 0.174898937, -0.070852831, 0.0793064982, -0.212293357, 0.0701971725, -0.0021967846, 0.0451571047, 0.0195722282, 0.0461180322, -0.00641624769, 0.0517838448, 0.137161285, -0.0997539088, -0.118641637, 0.234035909, 0.150188163, 0.0618825108, 0.0109362891, 0.0320615731, -0.1136159, 0.0582003295, -0.195525587, 0.137793392, -0.0844204947, 0.0396005958, 0.207778886, 0.199851304, -0.0735878795, 0.106541574, -0.0736700818, 0.13129513, -0.0877129585, -0.0679071546, -0.0147504732, 0.202523276, 0.194757164, 0.0617246218, -0.123547576, -0.248862714, 0.104788274, -0.100657925, 0.000960324774, 0.188817993, -0.108579315, -0.204805076, -0.244371086, -0.0309919175, -0.00391102675, 0.070959501, -0.016308561, 0.146207169, -0.172038585, -0.13708587, 0.14507246, -0.0678439513, -0.154684559, -0.240108371, 0.138188958, -0.206409857, -0.159489393, -0.214073613, 0.107187405, -0.204427004, 0.0283892639, 0.172533706, -0.206037849, -0.11586225, -0.24410139, 0.109407388, -0.0316474549, 0.158885717, -0.0667252243, 0.118405201, 0.289276123, -0.165092245, 0.108930469, 0.070623219, 0.179036945, 0.108090542, 0.182895318, -0.156233117, -0.117184833, 0.142791912, -0.0148069672, -0.0239627529, -0.214217961, 0.137310907, -0.188492745, -0.246256724, 0.147092804, 0.176855475, -0.0857564658, 0.0680939779, -0.0448941737, 0.0981446952, -0.172164232, 0.304895014, 0.0906158388, 0.297383636, 0.0652368665, -0.0184425749, 0.28164503, -0.173171684, -0.238063306, 0.186662257, -0.00241088937, 0.125462785, 0.304029018, -0.342890888, -0.0287288111, 0.17390269, -0.066968292, -0.177149415, -0.0643516853, 0.122750431, -0.0577152073, 0.0959472433, -0.0236832555, 0.116106987, -0.160913095, -0.0329174101, -0.014049178, 0.123443589, -0.0367398858, -0.110727645, 0.15123257, -0.144489914, 0.0620885342, -0.191643208, -0.0555331744, -0.0333120152, 0.0111381225, 0.200533777, 0.188959613, -0.155872673, 0.0341290683, -0.192276001, -0.171046734, -0.0678890795, 0.0327494256, -0.123621963, -0.123488769, 0.00637859805, -0.0630104989, 0.205584362, 0.169972613, 0.0232409332, -0.0955383033, -0.102426589, -0.0347150117, -0.141734734, 0.128293246, -0.0925778523, -0.0108686425, -0.13012214, 0.0815413147, -0.0893505439, 0.0880092233, 0.02950003, 0.23860997, 0.183169857, -0.0187763385, -0.13275674, 0.234897241, 0.110683218, -0.18547368, 0.144646749, -0.074404262, -0.10398934, -0.135641322, -0.157735169, -0.124934033, 0.137574792, -0.0147348205, -0.139187038, -0.221444562, 0.107474491, -0.156930476, 0.0779651478, 0.0951431543, 0.0451893285, 0.0516319498, -0.191372216, 0.0186820943, 0.126253679, 0.042005375, -0.0644702911, 0.114736617, 0.16525045, 0.116882309, 0.070220463, 0.188503683, 0.102188125, -0.0785993859, -0.15001981, -0.0465400182, 0.231806532, 0.0954680666, -0.184053317, -0.0501416922, 0.167674035, 0.191605791, -0.0193787068, 0.0830391496, -0.107822374, 0.207061484, 0.0861738399, -0.00507401815, -0.00288677309, 0.00758164329, 0.121445261, 0.092905201, -0.163787112, -0.0633125082, -0.123845324, 0.0347361527, 0.0725645497, 0.254036367, -0.0882892832, 0.199529752, -0.203118846, 0.0343604796, 0.198467344, -0.235339314, 0.237031609, 0.0543105453, 0.153027922, -0.00393469399, 0.10333398, -0.0708734468, 0.0561602749, -0.239301354, 0.0680253059, 0.183111206, 0.0810918957, 0.24312824, -0.160712034, -0.137365401, 0.21149838, -0.208581164, 0.0860498995, -0.222985104, 0.195945591, 0.0468437523, 0.0805253461, 0.301470578, 0.110695809, -0.153531685, -0.107340924, -0.115410239, 0.0342867225, 0.195745423, 0.0319843628, -0.207723111, -0.0392347164, 0.231147945, -0.129315481, -0.176766947, 0.177469, 0.192669258, -0.226546422, 0.0189814288, 0.0556515306, 0.107801184, -0.265750676, 0.168204769, -0.0855395198, -0.059515968, 0.0842674077, -0.0828177929, -0.130357698, -0.184084356, 0.137147471, 0.0251989067, 0.190306425, -0.209870204, -0.0716328025, 0.0316385627, 0.153478116, 0.396686941, 0.147947639, 0.192033961, -0.0293983817, -0.206629544, 0.275531769, 0.46042946, 0.140281811, 0.24135609, 0.0912894011, -0.17723383, -0.0607077032, 0.0781214163, 0.374888659, 0.137123927, 0.672217488, 0.276213497, 0.175734013, 0.0280658901, 0.0311749578, 0.0746272653, 0.349832982, 0.218783423, -0.185958922, 0.68218708, 0.800624728, 0.210476741, -0.00437949831, 0.130500868, 0.0502584949, 0.0294641983, -0.0176065117, 0.108612187, 0.358226597, -0.121234097, 0.108403966, 0.231736287, 0.210347712, -0.0159039721, 0.554084659, -0.167776093, -0.0969910622, 0.255162835, -0.0156714115, 0.26939097, 0.0617705248, -0.0752833113, -0.0614468567, 0.0244390815, -0.091742225, -0.137374878, 0.0531701297, -0.174850404, 0.141812295, -0.150860801, -0.187058046, -0.0874524713, -0.0264754221, 0.140813321, 0.182697207, -0.153970152, -0.177734926, -0.141945884, 0.0117159495, -0.00985656679, -0.00101221201, -0.0196746346, -0.174091488, -0.052107349, -0.22018443, 0.14820832, 0.0818826631, 0.233457372, 0.0977712348, -0.115955748, -0.0530783907, -0.140831947, 0.122053191, 0.121684685, 0.264127553, 0.0270333346, -0.0565839447, 0.019359095, -0.194519073, -0.00262582256, 0.0962572768, 0.0432850756, 0.113889135, -0.0236177016, 0.236521289, 0.183020383, 0.123297013, -0.167065337, 0.191284567, 0.14299646, 0.0509699844, -0.0904205814, 0.110933594, -0.0448181033, -0.187609032, -0.0712240487, 0.176699147, -0.118739776, 0.271520019, -0.166733369, -0.165289536, -0.0146756694, -0.00527196797, -0.0271551386, 0.00151156972, 0.228332981, -0.0739963129, -0.15750289, -0.0617005788, 0.00474839332, -0.154549867, -0.106653541, 0.176194146, -0.126685426, -0.0473142527, -0.0840078592, -0.00723607512, -0.212898895, 0.168081641, -0.185128301, -0.0536887795, 0.0943454057, 0.182923332, -0.0643337741, 0.196476832, -0.151796073, -0.0726564005, -0.0456830412, -0.0407369286, 0.192159489, -0.025926657, 0.0753762797, 0.0520100966, -0.0740965158, -0.0278436802, -0.0877467319, -0.213060349, 0.0216137562, 0.013314412, 0.175274462, 0.137478024, 0.0799314231, -0.00686348975, -0.124030545, -0.0374336392, 0.0357716046, -0.103798419, -0.0145825977, 0.123516023, 0.147583932, -0.0383550748, 0.0558126122, 0.107982129, 0.20239383, -0.106662877, -0.186953425, -0.145417884, -0.153639495, 0.027993679, 0.190795079, 0.0476124473, -0.12085294, -0.109654099, 0.167916715, 0.200663969, -0.00801608246, 0.0825436339, -0.0943990722, 0.113534227, 0.17334342, 0.111058161, -0.124200851, -0.0368134826, -0.00652719568, -0.141232178, -0.0518599898, -0.0585245639, 0.0653005391, -0.235346124, -0.148109958, -0.133401841, -0.114027344, -0.0275279973, 0.0593129881, 0.0982646197, 0.0619096607, 0.0287333895, -0.0120723862, 0.217594147, -0.139917493, 0.167802855, -0.168642655, 0.0747052282, 0.269419819, -0.116047248, -0.00862775743, -0.221282467, -0.118697263, -0.205058426, 0.093385309, -0.101342008, -0.183804184, -0.0605899505, 0.121015184, 0.0115664136, -0.208521381, 0.170277372, -0.0868665427, 0.248344138, -0.0432597287, 0.0541927218, 0.174610093, 0.181111693, 0.0449905209, 0.108599983, -0.130895346, 0.00717880577, -0.129434913, -0.042265553, 0.144251227, 0.259774655, 0.186873987, -0.0417911112, -0.048804868, -0.0295425355, 0.191073224, 0.0611833222, -0.0762384161, 0.140305713, 0.123962991, -0.0918691456, 0.218360201, -0.117257692, -0.127649173, -0.0255799256, 0.0222741216, 0.104327299, -0.0732962042, 0.0868302435, 0.228259474, 0.213780165, -0.0154352821, 0.131837606, 0.23168534, -0.214955419, -0.172440171, -0.0347957499, 0.128808409, -0.126937971, 0.061891485, -0.0297385268, -0.111321308, -0.0260849223, 0.120274864, 0.109222718, 0.0718200356, -0.235081047, 0.149947703, 0.0434079766, 0.0383607633, 0.116888225, 0.140750632, -0.0997844785, 0.174422219, -0.138142154, -0.0749339536, 0.0785625502, 0.120397143, -0.160959065, 0.0388336182, -0.167576253, 0.28271389, -0.191148162, -0.0925715864, 0.183668092, 0.0161793791, -0.0543912798, -0.0963794515, -0.102523632, 0.0610520095, 0.219306812, 0.0398645885, -0.0823789462, -0.102402054, 0.0275531858, 0.0220897496, 0.00813651085, 0.224854186, 0.173899412, -0.0672621354, -0.160013005, 0.224919304, 0.156423524, 0.0298209954, 0.127081707, 0.0212131441, 0.0445396155, 0.0335416645, 0.108812883, 0.111677632, 0.198874697, 0.0437096506, -0.165222168, 0.146299198, -0.0258866847, 0.206391677, 0.21082823, -0.125449836, 0.212311164, 0.166904435, -0.0247623175, -0.0211795866, 0.0768647045, 0.200587884, -0.0911418498, -0.169951767, -0.160309315, -0.0806967169, -0.158640265, 0.113370135, -0.00294652581, 0.0389382094, -0.216152698, -0.0083335489, 0.0735277981, 0.0742935687, 0.128101602, -0.00542548299, -0.115529254, 0.113532469, -0.160332292, 0.0508067459, 0.0624400526, 0.209660366, -0.214744583, -0.092242986, -0.160066396, 0.153950915, -0.212624639, -0.136968851, -0.135505289, 0.121049806, 0.0121994615, 0.151701763, -0.11071489, -0.171668932, -0.0537894666, -0.0878971219, -0.205776945, 0.099695608, -0.190786853, 0.0116519928, -0.144893363, 0.0865933746, 0.123252288, -0.182795584, -0.187821805, -0.18338947, -0.205582917, -0.0606609881, 0.0743346661, -0.0960690454, -0.211429507, -0.0481314957, 0.135181442, -0.216266423, -0.0187025368, 0.0537178665, -0.108392335, 0.0977317542, 0.129478082, 0.0895232707, 0.0533473045, -0.0970297307, -0.206168756, -0.139258206, -0.0563539565, -0.131601334, -0.0870515406, -0.0619503707, 0.20224908, 0.189971015, 0.208698735, -0.0417911559, -0.0538787693, -0.0976427495, -0.00286698341, -0.0744511336, 0.0304896683, 0.0333309472, 0.0902835578, -0.0216697603, 0.0137269134, 0.150900915, -0.182306468, -0.20932512, 0.0233798623, 0.136948779, 0.0849334449, -0.092384629, 0.188453048, -0.0954338461, 0.0955692083, -0.00602588151, -0.182517394, 0.0109124696, 0.106711015, -0.203821674, -0.108474381, 0.118665077, 0.153626904, 0.0262012091, 0.0375920273, 0.154369608, 0.0770949274, -0.117124625, -0.0335433446, 0.0450399965, -0.128809497, -0.00421985984, -0.0802144259, -0.139152095, -0.153811246, -0.120795593, 0.143708199, 0.185526088, -0.142273381, -0.195421949, 0.152865365, 0.0122631425, -0.000951811671, 0.0673113987, 0.136099085, -0.0278965831, -0.0474108718, 0.213819981, 0.142901793, 0.00495843589, 0.0418358333, -0.00355575676, -0.0105182827, 0.16393365, 0.101665772, -0.169067964, -0.195942327, -0.0434645265, 0.0727494806, -0.198469073, 0.132359818, 0.0526619218, 0.0468863398, 0.134476244, 0.0864710659, -0.16446723, 0.0303983875, 0.0437866561, 0.16037491, 0.161007166, 0.0387010314, -0.202730685, 0.044473853, -0.129946947, -0.05610618, 0.164238542, 0.137609839, -0.208719894, 0.153201148, 0.13046816, 0.180548891, 0.156915024, 0.205377564, 0.0167820454, -0.11153812, -0.0215259828, -0.126827091, 0.162156314, -0.0532439612, 0.0574748926, 0.0771525949, -0.0153041324, -0.0292977095, 0.191961616, -0.0606812425, 0.0860238746, -0.146850556, -0.0733355656, -0.149648055, -0.0798214898, 0.0446455069, -0.170179084, 0.0201480612, -0.0888226479, -0.103910781, 0.119667917, 0.153799519, 0.054285761, -0.148660555, 0.035269402, 0.109882556, 0.204186887, 0.0496170707, 0.161113545, -0.135843858, 0.253733486, -0.0944817513, 0.0327358693, 0.230729103, 0.108584575, -0.221280649, -0.11051406, -0.145698979, -0.132175505, 0.178192541, -0.156799883, -0.137536705, -0.0399425589, -0.134871528, 0.18148458, 0.11162968, 0.092132248, -0.171199903, -0.0500270128, -0.191958666, 0.122761637, 0.114319079, -0.13137719, -0.0537062585, 0.113184899, -0.263052046, 0.141020328, 0.239564508, 0.170219958, 0.102902547, -0.101794772, 0.158655852, 0.161232308, 0.257718861, 0.234837502, 0.0273188651, 0.121293917, 0.120111875, 0.256624699, -0.0763987452, 0.0835199878, -0.0190323666, -0.103317492, 0.0232522283, 0.10880886, -0.0914563537, 0.109213397, -0.0964482874, -0.169531703, 0.281256527, 0.0533225201, -0.00718479324, -0.117911838, 0.0900024846, 0.135364503, -0.0926576406, -0.165947258, 0.212630153, -0.199972525, 0.206199676, 0.18481414, -0.179684758, 0.0156940166, 0.11673253, 0.173709407, 0.145675406, -0.00235269964, 0.186596662, 0.211974829, 0.000806359749, 0.0446996912, 0.0769063011, 0.0293873399, -0.0577886961, -0.0997519717, 0.115017757, 0.0576308221, 0.0125924861, 0.225485265, -0.00981596857, 0.139237881, -0.0530043356, 0.260116875, -0.22942251, 0.0249016378, -0.0571197607, 0.153768301, -0.206047684, 0.0895582587, -0.279679924, -0.0219289549, 0.10167665, 0.0845968127, 0.00727231754, -0.0432331599, 0.225695342, -0.0686216056, 0.28638041, 0.272146463, 0.140005305, -0.0245791562, 0.0761088356, 0.201061755, 0.00954514742, 0.218374774, -0.168220788, 0.103706576, -0.20218125, 0.0332696922, -0.0424223542, 0.108355887, 0.1041262, -0.00260003889, 0.0343024097, -0.102693766, -0.100874119, -0.0986998156, -0.235685483, -0.0899084508, 0.0854150206, 0.0691602379, -0.185052946, 0.0787002891, -0.165196121, -0.0326854065, 0.0315757096, -0.149115399, 0.0719742849, 0.0407750756, -0.0767336041, -0.187577948, -0.048541002, 0.0360414013, 0.249366537, -0.192914456, 0.190689608, 0.0374177843, -0.0437144637, 0.213710159, 0.096700497, 0.00223939074, -0.0764921829, -0.0575337037, -0.145044506, -0.0802579448, 0.064725399, 0.0837969631, 0.0941284671, 0.0538992845, -0.0705573037, -0.115551233, 0.0803196281, 0.0834578872, 0.0238675773, 0.136617467, -0.186541721, -0.0417114496, 0.245139882, -0.00578208687, 0.0275053699, -0.0501771569, -0.179348543, 0.173432946, -0.0807827562, -0.179962143, 0.110388212, -0.146068901, 0.213116661, 0.144476965, 0.0446254946, 0.146554768, 0.093346484, 0.16855067, -0.192628831, -0.028239293, 0.160450786, 0.203553155, -0.11479301, -0.107505403, -0.0260372236, -0.144633308, 0.114200078, -0.127950758, -0.214850038, 0.207950816, -0.0725203902, 0.0758482069, -0.046793025, 0.0461012349, 0.0468173474, 0.00463971123, 0.0375378318, -0.0815252587, -0.0458168387, 0.10962835, 0.0194397829, 0.0926095471, 0.073319912, 0.0239949729, -0.0836053863, -0.137725636, 0.0898624137, 0.253191203, -0.192230299, 0.223583639, 0.214670718, 0.12229877, 0.229018718, -0.0431688577, 0.110472642, 0.139069289, -0.0282006748, 0.101184413, 0.0894554704, -0.0786872953, -0.0111689866, 0.0286502857, -0.0633932576, 0.171827883, -0.0444677696, -0.0850014165, -0.169253916, 0.120693155, 0.0252687819, -0.170735449, -0.123299576, 0.220411927, -0.217961624, -0.149791226, -0.171596184, 0.0943251699, -0.100113608, 0.087037079, 0.0855410993, 0.0791215971, 0.11918585, -0.0505308397, -0.117827907, 0.063941285, 0.00416628085, 0.0839637816, 0.267723888, -0.227810621, -0.0777227134, 0.0388324112, 0.256261855, 0.245122582, -0.138452694, 0.0876130164, 0.0878035948, 0.129902616, 0.102416001, 0.264991552, 0.139974669, -0.013653418, -0.065480873, 0.0472233519, -0.193420827, -0.0574077927, -0.100826748, 0.0330015197, 0.15693666, 0.109514177, 0.00890431553, 0.031340763, -0.0226426851, -0.170719773, 0.0925062895, -0.228847221, 0.130559415, -0.0788129494, 0.128267556, 0.176107913, -0.0924457237, 0.0958436653, 0.144238055, 0.0475376062, -0.100932501, -0.115049355, -0.207394749, 0.26449883, -0.0507705212, -0.0272947475, -0.00600530533, -0.106777452, -0.117991619, -0.234071791, 0.0523665883, -0.204911649, 0.043802131, 0.1575744, -0.220566079, 0.0123432605, 0.0531032309, 0.103713386, -0.205086485, 0.223250866, -0.0471659116, 0.00876451191, 0.214768395, 0.246275902, 0.0651466101, -0.197602212, 0.205826506, -0.0679371729, -0.000915050507, -0.105748199, -0.145877063, -0.201368526, 0.0879625231, -0.0965842009, 0.198548451, 0.161472961, 0.0642927736, -0.0918231159, 0.182744697, 0.0693864375, -0.188803703, 0.00650767982, 0.172555879, -0.0635101199, 0.00677795708, 0.202838168, 0.040710941, -0.209036991, -0.144217819, 0.188803896, -0.00212830305, -0.148173034, -0.20080778, -0.192079917, -0.0633593947, -0.16399309, 0.153926134, 0.203168228, 0.0955855399, -0.137954876, -0.19007811, 0.123448029, 0.21018137, -0.0810624957, -0.111288175, 0.021730572, 0.146542504, -0.157430366, 0.181623116, 0.126291782, 0.207365617, 0.165423319, -0.0239322782, -0.0631945282, 0.12825425, 0.200958624, -0.052633673, -0.0713848397, -0.185413659, -0.101239368, 0.182738468, 0.165163174, 0.0180790871, -0.15865013, -0.0937678143, 0.19551906, -0.0590572059, -0.0486637354, 0.0733446032, -0.0732812583, -0.0904489607, -0.0468690395, -0.124550417, -0.0455771685, -0.104021177, -0.185393631, 0.0408243984, 0.105959103, 0.119070217, -0.215867609, -0.12802428, 0.069313094, 0.0940398425, -0.179975063, -0.0170270354, -0.16964227, 0.0537156612, -0.0739964396, -0.210699499, -0.169508368, -0.114205375, 0.20856382, -0.0094743818, 0.023435086, 0.0358004421, 0.044800505, 0.186260834, 0.149650797, -0.101585321, -0.194993809, -0.0581209809, -0.189571068, 0.00125160813, 0.174607709, 0.0704791695, 0.140320167, -0.0318251103, -0.0955716968, 0.16221489, -0.177237138, -0.00738732517, -0.0435195267, -0.00547859073, -0.215163887, -0.00860790908, -0.00653317571, 0.126314595, -0.103846706, -0.0728396028, 0.0168418288, -0.0725217909, 0.109986708, 0.0920121819, -0.171025246, -0.0454324782, 0.0630950481, -0.0997218713, -0.0783640891, -0.00420938432, -0.18078503, 0.172304526, 0.125460967, -0.0567836761, 0.113854423, -0.00121866679, -0.0124422107, 0.037865255, 0.0818271786, -0.159302071, 0.0689702779, 0.16112043, 0.000206770215, 0.0466447026, -0.219438955, -5.96225691e-05, -0.000440880656, -0.174127713, 0.066909574, 0.0277200025, -0.213515118, 0.060687568, -0.0385784097, -0.109999962, 0.0165164806, -0.188594639, -0.0643988177, -0.0376132242, -0.113160878, -0.177742392, 0.20572792, 0.197053879, 0.178338304, 0.0188686363, -0.0623674206, 0.0213672761, 0.165976256, -0.0983577296, 0.201859236, 0.278185248, 0.16634202, 0.0324927792, 0.185975701, -0.162036508, 0.214893028, 0.144453928, 0.18897824, -0.02271723, 0.173502356, 0.0860304534, 0.157381833, -0.109898388, 0.0889903679, -0.00139595452, -0.0246559381, 0.0552617051, -0.0490884259, 0.0221240669, -0.00970905647, 0.271192163, 0.0836053491, 0.136748031, 0.0590723492, 0.131660268, -0.0782020912, 0.233400002, 0.020858407, -0.199875951, -0.10958828, -0.0476728119, -0.112283461, 0.0634761229, -0.11828354, -0.206033915, 0.193904743, 0.208372578, -0.0133872097, 0.128678188, -0.0611923672, -0.0264214631, -0.0343179964, 0.120693304, 0.242108658, -0.123052984, 0.00721185189, 0.0428376906, 0.185159311, 0.189356312, -0.121340357, -0.0659567639, 0.0139191207, -0.172991693, 0.231255203, -0.0546388291, -0.12772809, -0.186477616, -0.0920270532, -0.131607428, -0.115861528, 0.102707088, 0.152410567, 0.159929469, 0.0160477627, -0.0876519978, 0.0969803855, -0.213091269, 0.196864411, 0.273380667, -0.188008323, -0.0920328945, 0.289578468, -0.0528584607, -0.0977249518, -0.00144148862, -0.179536566, -0.0322223529, -0.212180287, 0.231571823, -0.193322748, 0.215044737, -0.0583524294, -0.148938805, -0.104199901, 0.0954470932, -0.0519888364, -0.120300457, 0.0400745571, -0.208074585, 0.16796045, -0.126946077, 0.105555303, -0.179807782, -0.139423996, -0.110121422, -0.143779054, 0.0281973183, -0.213963971, -0.00856938958, -0.181462109, 0.209135398, 0.0444553941, 0.212432578, -0.152585238, 0.0589921027, -0.0956718326, -0.202689767, 0.189238891, -0.00226314366, 0.00328245759, -0.07723362, 0.0444654375, -0.110938296, 0.11733903, 0.118250266, 0.0411194339, -0.0846743733, -0.214066923, 0.13189514, -0.14326416, -0.171151295, 0.00388705614, 0.208343133, 0.0269903056, 0.059002623, 0.0961068422, 0.100626692, 0.0702101141, 0.020035034, -0.0141857117, 0.0257037412, -0.0787355751, 0.149851128, -0.0874555111, 0.0847222954, -0.203368247, 0.0913478732, -0.190981388, 0.0381076187, -0.0793296993, -0.0151991285, 0.0998160616, -0.113543928, 0.0162660182, 0.103863224, 0.0264875349, 0.0567879528, -0.0818504989, -0.174385443, -0.00410155952, 0.0188013464, -0.0961839706, -0.133884028, -0.0904380009, -0.123644434, -0.132027194, -0.0969853327, 0.178106606, -0.164912462, -0.129356861, 0.254577816, -0.244255126, 0.085457325, -0.20408611, -0.0806175619, 0.049568817, -0.0337973684, 0.0333623476, 0.147425145, 0.115208894, -0.0453046039, 0.300857335, 0.0715077147, 0.0815929845, 0.217304617, 0.174860537, -0.217734858, -0.0545187891, -0.110197, 0.0350490846, -0.187146857, -0.0842425302, -0.155964121, 0.00266452134, -0.0114788301, -0.0303328782, -0.183492959, 0.043718189, 0.119714215, -0.0836073384, 0.194770262, 0.176857576, -0.0258767977, 0.260465145, 0.108764701, -0.0949423462, 0.0376914777, 0.063421309, 0.0491331071, 0.185503632, -0.00521813333, -0.195495903, -0.131301835, 0.135766819, -0.212390468, 0.0454258732, 0.116974734, -0.0042796433, -0.0877883956, -0.0176164117, 0.116867885, 0.084963426, -0.145454615, -0.00281196297, 0.158816293, 0.261381388, -0.103646547, -0.0409106165, 0.119343556, 0.0541383289, -0.179490834, -0.226963773, 0.0730867088, -0.0670445934, -0.146837354, -0.100336365, -0.206874445, -0.147349969, -0.0639766306, -0.0242820475, -0.0191500783, 0.0574500002, -0.118401602, -0.0355735309, -0.0470449142, 0.0599663332, -0.176558927, 0.00412532967, 0.213447168, -0.010397274, -0.0719934478, -0.0328418612, -0.00671752123, -0.0474058241, 0.162177995, -0.0395350344, 0.200220659, -0.0697177351, -0.161850125, 0.107072055, 0.178566739, 0.209856763, -0.148664251, 0.0821418315, -0.125930011, -0.173101038, 0.0771152675, 0.0780660436, -0.134412229, 0.186319694, 0.0190821849, -0.23414728, -0.104899429, 0.19066, -0.0627585649, -0.169341192, -0.178378239, -0.0991300195, -0.0998610705, 0.131659567, -0.00676505361, 0.211450562, 0.0258109439, 0.220644847, -0.207787529, 0.0453971066, 0.0513934791, 0.0972999409, 0.0140249133, 0.185306981, 0.132868722, -0.124948919, -0.0208617114, -0.0660538822, -0.103338204, 0.0198297929];
    CONSTANT bias_3 : ARRAY[0..63] OF REAL := [-0.00983189233, 0.0739286318, -0.03035645, 0.0550533831, -0.011248054, 0, -0.0295825377, -0.0090773385, 0, -0.0277472436, -0.00766381249, -0.00870534033, -0.0367787257, -0.0242641736, -0.00147182879, -0.00894620363, 0.0173237566, 0.00239057303, -0.00620334735, -0.00517789647, -0.0133990953, 0.0294917747, 0.0401097015, -0.0258607231, -0.00522571057, 0, -0.0150696058, 0.0860590115, -0.0117668696, 0.065539062, -0.00745888008, -0.0186666064, -0.010953215, -0.0240848884, -0.0448102988, -0.0404310934, 0.0785407722, 0.0790930837, -0.0278634299, -0.0265457965, 0, -0.0240220856, 0.00635804934, 0.0217319299, -0.02775204, 0.00820828322, 0.0399322994, 0.0746404901, -0.0329935588, 0, 0.00812079571, -0.0131024169, -0.0233938117, 0.0117759928, 0.0732261613, -0.0248215012, 0, 0.000535005063, 0.0062644016, 0.0363470353, 0.0787089318, -0.0285863206, 0, 0.0387545452];
    CONSTANT weights_6 : ARRAY[0..4095] OF REAL := [-0.0211104695, 0.157233626, 0.0721651465, -0.0791621804, -0.145463645, 0.0476885587, 0.103807047, -0.217098057, 0.15736191, -0.173330665, -0.128692865, -0.0421262085, 0.0980989784, 0.155999586, 0.0207046866, 0.184844807, -0.00715442142, 0.172988996, -0.206348658, 0.157887205, -0.037524119, -0.140499547, 0.187242225, 0.152909175, -0.145436138, -0.0675008371, 0.169665024, 0.210023656, 0.206236467, 0.208556831, 0.0959817022, -0.148986042, 0.0728623122, 0.026120171, 0.211910024, -0.0622561015, 0.0902522206, 0.0471122339, 0.0779013783, 0.0172086973, -0.039685376, -0.0467820168, 0.0570690036, 0.0242511332, -0.209991112, 0.00939850137, 0.112361535, 0.116925567, -0.153550565, 0.212469026, 0.14040117, -0.0208477583, 0.182546362, 0.0197014436, 0.186374202, -0.168809876, 0.196177915, -0.00232131779, 0.137093261, 0.162052512, 0.199661002, 0.0766961128, 0.211054429, 0.125300422, 0.00426613819, 0.288283914, -0.159290671, -0.0769464672, 0.0940423161, -0.0546351485, 0.0653043687, 0.0303289033, 0.0641354099, -0.192860484, 0.04200764, 0.0343205296, 0.155289501, -0.180832982, -0.12778616, 0.262020022, 0.0602597371, 0.10863255, -0.237889618, -0.095524922, -0.272757202, -0.0731869787, -0.0907882899, -0.147379801, -0.169592246, 0.178864881, -0.101507559, -0.0397703201, 0.016668126, 0.0635820627, 0.0767925531, -0.102012202, 0.0477126874, 0.0524956584, 0.111083403, -0.0878348276, 0.011967063, -0.0565153994, 0.170608982, 0.309960365, -0.105272628, 0.211850211, -0.0994742885, -0.153632715, 0.267046332, -0.203152657, -0.160044357, 0.0353948474, -0.0975862592, -0.0403899029, 0.07099244, 0.0249471422, -0.0422067828, -0.220276818, -0.185284197, -0.0370966718, 0.148172244, -0.120848358, -0.0141801946, -0.0953512639, -0.253198028, 0.104871087, 0.0740961581, -0.182465032, 0.0539166033, -0.159959942, -0.161966518, 0.0288212746, -0.135103494, -0.112145692, -0.0749802366, -0.0615305528, 0.157502532, 0.0857658535, -0.0273212269, 0.141590878, -0.0330497138, 0.176339731, -0.0418806784, 0.0999175385, -0.0713153332, 0.263013691, -0.115717605, 0.204661101, -0.11504811, -0.0947428197, 0.153199002, 0.335939616, -0.00631709397, 0.100122802, -0.209013268, 0.0137379616, -0.204656497, 0.0605559498, -0.175298169, -0.123451911, -0.0473049544, 0.0416926257, 0.156591177, -0.101554133, 0.115582488, -0.0190878287, -0.0975746512, 0.155756831, 0.108877532, 0.171931863, 0.235213891, 0.00560221262, -0.151249588, 0.00370491436, -0.0536345989, -0.181572989, -0.117012545, -0.106260225, 0.242837548, 0.223648071, 0.0628157556, 0.295081288, -0.0346996188, 0.15143846, 0.187727511, 0.290291816, 0.0033030943, -0.161266476, 0.00898908544, 0.244648784, -0.134097993, 0.0367004983, 0.0216495004, 0.180981815, -0.0798874199, 0.13122049, 0.0334438831, 0.0200074967, 0.103910699, -0.102675296, -0.207296401, 0.0869636759, -0.20655781, -0.0956464559, -0.203777537, -0.105265148, 0.0783180222, -0.0458374731, 0.204411358, 0.118474796, 0.122315288, -0.0419053994, -0.340604126, 0.135242134, -0.129586041, -0.0497838371, -0.0099619776, -0.0477824807, 0.281962305, 0.00426848233, -0.181631833, -0.170377254, 0.104996637, 0.114299156, -0.163810551, 0.249239355, -0.0833768472, 0.0697716847, 0.014485863, 0.157567188, 0.110193223, 0.230861947, -0.110680073, -0.0243154187, -0.0779362693, -0.0843363702, -0.049658794, -0.00124949845, -0.0668900907, 0.086151801, 0.179528475, 0.0938131064, -0.204934552, 0.0532739088, -0.120318048, -0.151893049, -0.146782264, 0.312886775, 0.0673337728, -0.1004811, -0.171645507, 0.268849701, -0.229744852, -0.134535402, -0.119718812, 0.0152729712, -0.196205392, -0.123321056, 0.00104016194, 0.114403293, -0.109209985, -0.116009399, -0.00587476185, -0.100333177, 0.104191698, 0.0102303922, -0.134384453, -0.204718813, 0.0862976313, 0.140776381, 0.0467067696, 0.094970122, -0.189605281, -0.0276639797, -0.0749640316, 0.0723377988, 0.00538966572, 0.0190833975, -0.0198820475, -0.00954220816, 0.0676214248, 0.104344197, -0.200903356, -0.206617773, 0.084322378, -0.0795044377, -0.0956577435, 0.191447124, -0.0795495212, -0.00805467833, 0.205130324, 0.179273605, -0.0990068316, -0.0614028908, 0.148120746, 0.132912666, -0.189888284, 0.200087667, -0.164052576, -0.0751432627, 0.0476862341, 0.0292347074, -0.052457124, -0.0892619789, 0.0716815516, 0.0529787801, 0.213911965, 0.209351331, -0.129100218, 0.0809682086, 0.176059052, 0.149538949, -0.126543701, -0.188590631, -0.183877945, 0.117343932, -0.167362183, -0.0124702444, -0.152586102, -0.18852441, 0.0780072361, -0.153538495, 0.0840239376, -0.148158073, 0.0951781124, -0.0676086247, -0.202492416, -0.0601291209, 0.0147494972, -0.148133397, -0.00998263061, -0.096799612, -0.00623972714, -0.0822741985, 0.134943768, 0.196010545, 0.0348980874, 0.194250599, 0.00896206498, -0.170046642, 0.0372118801, 0.0163984746, 0.179545149, 0.112079129, -0.104169428, -0.0681873262, -0.14190802, -0.167659834, 0.171136335, 0.176123098, 0.15911971, -0.0608612299, -0.0210849196, -0.132437974, 0.0952331275, -0.0566280484, -0.179609761, -0.202228233, 0.160658821, -0.127846152, -0.169803977, 0.0259776413, -0.175173402, 0.108989462, -0.174509123, 0.163906083, -0.0123733133, -0.192176595, 0.168579057, 0.167967841, -0.0916754827, -0.00778664649, -0.041722253, -0.215875, 0.107255802, 0.09431611, 0.110112235, 0.155124173, -0.0552193671, -0.00624886155, -0.116997302, 0.125487968, 0.149071887, 0.0814684778, -0.0264531672, -0.202291474, -0.107270196, 0.208046228, 0.198929116, 0.124986812, -0.116254002, 0.106430285, 0.0689994991, 0.123037621, -0.144080907, 0.0291826203, -0.0867067724, -0.122828558, -0.193552107, 0.180794746, -0.151306659, -0.108268835, 0.0360157453, -0.162983239, 0.180829659, 0.123341292, -0.143707618, -0.0218093451, 0.100755021, 0.048000399, 0.0416897722, -0.030838713, -0.10653317, 0.0873832777, -0.188493058, -0.0422797352, 0.0743354112, -0.125618383, 0.163786501, -0.184897706, 0.0689249486, 0.216842949, -0.173285306, 0.185100108, -0.117793359, -0.19082053, -0.106456965, -0.0742470324, -0.0494265445, 0.165998891, -0.185700104, -0.121370681, -0.174497947, -0.0514864251, 0.10049998, -0.107571743, 0.159631327, 0.187085122, 0.0653448254, -0.120375261, 0.275558501, 0.182469591, -0.175698802, -0.0759939849, 0.065009132, 0.259765774, -0.086910978, 0.0502287, -0.0737552643, -0.0215020366, 0.161072969, 0.123396195, -0.175406262, 0.0518808141, -0.0351930261, 0.0470791981, 0.262363374, 0.1363094, 0.180866018, 0.132682219, 0.165143073, 0.126118854, 0.0938046128, -0.254130632, 0.0568571538, -0.0724096671, 0.0160691887, -0.0521572456, 0.22484374, -0.0792442709, -0.00761091337, 0.276181072, -0.086371094, -0.129833862, -0.0362726077, -0.0417017639, 0.0206526667, 0.239292666, -0.0601968914, 0.0359402746, 0.308184862, 0.0270620137, -0.208643079, 0.131217003, 0.0645703152, 0.118619733, 0.0201364737, -0.165239125, 0.162001967, 0.177479923, -0.111770749, 0.135645315, 0.0129162921, -0.202752113, -0.0295399278, 0.022838518, -0.0796107128, 0.0467211269, -0.051113341, 0.160861671, 0.00665348954, -0.104955673, -0.0838543624, -0.236661151, 0.214804575, -0.0623946115, 0.140443742, -0.0886547342, 0.0746734887, 0.276039749, -0.199886113, 0.121124074, 0.0216602683, -0.167079479, -0.138646215, -0.0189068019, -0.0126770437, 0.0390007943, 0.0360741764, -0.141568631, -0.0118533075, 0.178898349, -0.0807059556, 0.0550475866, 0.178213313, -0.0915158764, -0.109646633, -0.066618517, -0.00931756198, -0.201538652, 0.0959077924, -0.019727543, 0.00191234052, 0.180038348, 0.112552777, 0.101054952, 0.215217724, -0.185405463, 0.122277573, -0.0108845085, -0.0374378562, -0.0693836063, 0.206913039, -0.193783402, -0.0592647493, -0.198673338, -0.00192482769, -0.00480589271, 0.0151784569, -0.11449635, 0.150387093, -0.0220891237, -0.0531173348, 0.0558237582, -0.0155561566, 0.110152856, -0.10219758, 0.125887617, 0.187418178, -0.00413711369, 0.199766979, -0.0751423836, -0.196204484, -0.163247168, 0.0657932907, 0.179478303, -0.0909180194, -0.0187031627, -0.0687615424, -0.125233293, -0.00715054572, 0.191343263, -0.140845746, -0.101612061, 0.028948009, 0.00607836246, 0.0241835825, -0.0792405158, 0.170693278, 0.121472552, -0.159257323, 0.15754503, -0.139394745, -0.044453688, -0.0742065012, 0.176449284, 0.226904213, -0.0162550025, 0.281962007, 0.141561612, -0.179304242, -0.22687985, 0.0888308734, 0.1368251, -0.215948135, 0.232278898, 0.14440532, -0.210397243, 0.0025057646, 0.257558495, 0.069859311, -0.0588960908, -0.178999975, -0.00917844474, 0.0827753693, -0.0334500261, 0.0289534777, -0.147056982, 0.18982479, -0.0401569977, -0.00673311763, 0.117641859, 0.0199112538, -0.110949092, -0.10525246, -0.110742055, -0.149034083, 0.176191643, 0.164675817, -0.152210981, 0.111859016, -0.0424617529, 0.070398286, 0.0940225571, 0.160483241, -0.166004077, -0.0361319557, 0.156162739, 0.255399585, -0.0411905348, 0.0899951607, -0.214364231, -0.0514262058, 0.136874646, -0.0144281425, 0.0158658996, 0.173274562, -0.0837578475, -0.021164313, 0.189715445, 0.0227939058, 0.0768007636, 0.0420344919, 0.13114506, 0.0212835968, 0.125271335, -0.0908199325, -0.2127489, 0.223346874, -0.168397516, -0.143092021, 0.0855721906, 0.217426375, -0.010913834, 0.161978483, -0.0237388425, -0.0148029672, -0.0206773132, 0.163911536, -0.115519904, -0.0708635896, 0.160120934, 0.21680361, -0.0919932425, -0.106572457, 0.186694637, -0.0864723846, -0.0672358871, -0.0620637983, -0.0492999963, -0.031213671, -0.214064613, -0.0040052929, -0.177249506, 0.198898122, 0.029973764, 0.0648880824, -0.0722419471, 0.0583239459, -0.161417127, 0.118529066, 0.0775398463, 0.0136581725, -0.019831283, 0.0340036228, -0.069475472, -0.141518444, -0.0155703966, 0.0465259701, -0.13712129, 0.215217024, 0.153940856, 0.233599231, 0.069659397, 0.0283375084, 0.136588395, 0.114837028, 0.00435284665, -0.0815577209, 0.0850224197, 0.0896461308, 0.0839098245, 0.12630628, 0.102898523, -0.0242574364, 0.0395214707, 0.179158911, 0.140869483, -0.0315961689, -0.211324051, -0.101073779, 0.164895773, 0.0432892777, -0.0961784273, 0.187965691, -0.0886578932, -0.143109977, -0.200058162, 0.128884479, -0.150142565, -0.0212808698, -0.0118450765, 0.0831215233, -0.0732853338, -0.0489297211, 0.000687902851, 0.0266030431, -0.201587737, -0.185360029, -0.00679598097, 0.108024552, 0.102891639, -0.178852096, -0.173995063, 0.0813450366, -0.0506051332, -0.0515105948, 0.0880956501, 0.173789188, 0.00271931873, -0.181898132, -0.0750331804, -0.0916771367, 0.0279746372, -0.0858160108, 0.0492289215, -0.0897664428, 0.118924871, -0.00673155487, 0.0254511833, -0.0507416576, -0.131477594, 0.0658444315, -0.176156193, 0.00369836204, 0.209861919, -0.144315973, 0.0758810192, -0.126617879, 0.0478404015, 0.0629696399, -0.181336939, -0.070628196, 0.0589700602, 0.0671523064, 0.0530530922, 0.148497984, 0.199353352, -0.2551274, -0.155184016, -0.00421486888, 0.212831467, -0.0586378425, 0.147449061, -0.201066777, -0.0765811056, 0.0298376996, -0.028335914, -0.0145538365, 0.120011285, 0.263296843, -0.0805929601, 0.196454912, -0.194894016, 0.0144730853, 0.00976360589, 0.105623856, -0.128629684, 0.224141806, -0.244979411, 0.214529052, -0.0382702313, 0.156628206, 0.0189788435, 0.127576098, -0.204321966, -0.106341101, 0.309783638, -0.0312428474, -0.136540458, 0.271282047, -0.320485145, -0.130114317, 0.0987244472, -0.0768140033, 0.292481333, 0.028581921, 0.0651605949, 0.0565245636, -0.207960293, -0.105757877, -0.0665429085, -0.00274416106, 0.0682443231, -0.106524602, -0.163970143, 0.0532483347, -0.200977892, 0.0309002809, -0.0602365695, 0.202884033, -0.04036038, -0.0263917297, -0.138741806, 0.261350095, 0.0551347472, 0.181741431, -0.147500739, 0.178088039, 0.114219822, 0.046044156, 0.0941443816, 0.0813267976, 0.0595558062, -0.197245672, -0.0100678066, -0.211604849, -0.148000121, -0.198542699, 0.196343526, 0.138460979, 0.107107386, 0.0907673761, -0.121037595, 0.252360672, -0.0970465541, 0.0558764599, -0.0847656652, -0.209763199, 0.167329192, -0.237716049, -0.0499278046, 0.249167144, 0.0408127345, -0.165352255, 0.176838875, 0.00782003999, 0.176427022, -0.0851962119, -0.192636058, 0.187963501, 0.170646742, 0.0470952839, 0.00458228588, 0.141556203, 0.0644658133, 0.0417393818, 0.0441780165, 0.039651297, 0.0833919719, -0.172924563, 0.0634429529, -0.0965564921, 0.0724875107, 0.21937269, -0.0974312797, -0.130002752, -0.121189877, 0.0671949536, 0.0867445171, -0.00312029221, 0.126738116, 0.0653212741, 0.252740234, 0.287628323, 0.167519346, 0.139367387, -0.0309090856, 0.263746917, 0.0875785947, 0.0128881168, -0.0565036125, 0.120908678, 0.240472659, -0.201509178, 0.293792278, -0.131671205, 0.0896654353, 0.0370695144, 0.135521129, 0.20480074, -0.175205469, -0.171041086, -0.0579688512, -0.156582564, -0.0778886229, 0.0664458051, 0.130356193, 0.0996769667, -0.153313071, -0.192398816, -0.106274486, -0.0162558295, 0.0870158821, -0.192340657, 0.048169598, -0.171457037, -0.136983603, -0.064907901, 0.145346314, 0.190712199, 0.0360278338, 0.0434320495, -0.211738184, 0.160129383, -0.105414405, -0.171388596, -0.0388856754, 0.142384306, 0.137329713, -0.130360201, -0.0619715676, 0.00965698808, -0.0439127162, 0.170497492, 0.212079838, -0.142104536, 0.0586519986, -0.115233481, -0.0224351734, -0.16999881, 0.0918107182, -0.167155147, 0.195335492, -0.0757286102, -0.172540411, 0.103915311, -0.141615734, -0.00377908791, -0.0657154992, -0.148804039, 0.022908235, -0.168834493, 0.152186722, 0.0506493412, -0.112933271, 0.00049599976, 0.100557655, 0.112081513, 0.142245606, 0.0271094441, 0.0381551534, 0.20742555, -0.110420324, -0.100627325, 0.145201087, -0.202350944, 0.120480955, 0.0444104783, 0.211891606, 0.19280535, 0.0655445755, 0.189393878, 0.196804807, -0.0521670766, 0.0503715128, 0.214662924, -0.0492795333, -0.0675857663, 0.178876325, 0.0826835707, -0.169171751, 0.0269653201, 0.211806223, 0.130338058, -0.000949479057, 0.196632594, 0.186210766, 0.0524837524, -0.0555000752, -0.131404147, 0.146059439, -0.0972863659, -0.0147773847, 0.105667993, -0.00656548562, -0.144193918, 0.0886233747, 0.215485469, -0.0223604683, 0.165627271, 0.117518991, 0.000273500162, -0.196279138, 0.0528765172, 0.137227044, 0.0115529299, -0.0449971259, -0.0784725025, -0.172097519, -0.0769113824, -0.144809157, 0.087641567, 0.0567293391, -0.165308416, 0.0845244378, -0.0673978627, 0.191283584, -0.0394614935, 0.203768536, -0.202162296, -0.138682559, -0.109796427, 0.112647042, 0.0804700181, -0.0721322224, -0.102790877, -0.0195402578, 0.00424019992, -0.117378324, 0.205446005, 0.203034252, 0.101452544, -0.0454550199, 0.157199964, 0.0115054222, -0.0943236724, -0.0565667748, -0.107933104, -0.0655731708, 0.157481402, 0.128197148, 0.00223283307, -0.00375899929, -0.1018316, -0.173439905, -0.15236567, 0.212863877, -0.152796358, 0.162461266, -0.0564482771, -0.120488144, -0.13375029, 0.025584979, -0.205807254, -0.192222401, 0.214670464, -0.0954632461, 0.183467418, 0.183182776, -0.00882993639, 0.169890597, -0.197005555, -0.106948674, -0.00395756867, 0.0120129455, 0.0223759171, 0.149836347, 0.228335664, -0.0534032434, 0.132094547, -0.0133346152, 0.183536708, -0.190487862, -0.00259809522, 0.000128543412, 0.127965212, -0.0134203611, -0.129633933, 0.229406625, 0.0699569285, 0.198570237, -0.0478203781, 0.181146488, 0.0680752471, 0.00578152016, -0.110974222, -0.088077426, 0.117438272, -0.202719942, -0.0765619129, 0.0070055034, 0.00518807769, 0.0908474326, -0.210115537, -0.259739071, 0.0877127647, 0.178909853, 0.0252563711, 0.161810607, 0.14697203, 0.0207887739, 0.192217827, 0.0119345486, 0.111504808, -0.138566241, 0.0183499251, 0.178135261, 0.10215006, 0.11800538, 0.0883670896, 0.0227976646, -0.122666731, 0.0188208688, 0.0996467769, -0.100148812, 0.117532745, 0.237992808, -0.130577683, -0.15731205, 0.271030456, -0.23369348, -0.0929943994, 0.0971348509, -0.104811274, -0.120445482, -0.0412788987, 0.0163263902, 0.138564199, -0.144116297, 0.125310749, -0.172860175, -0.224062487, 0.13113521, -0.0350915194, 0.102414116, 0.00754255336, -0.0123361535, -0.0915403515, 0.0783033222, 0.109218769, 0.00511339353, 0.059927389, 0.0361303464, -0.121367157, -0.0622647256, 0.0529602021, -0.149987593, 0.0344639942, 0.244372755, -0.129179358, -0.0458081402, -0.141225874, -0.00293263793, 0.152275071, -0.0406294242, 0.139919147, 0.187548757, -0.178822875, -0.0349252298, -0.0637998432, -0.192398965, 0.0176388826, 0.0132232755, 0.081162639, 0.00220011175, -0.148068249, 0.189775273, -0.21044074, -0.193314359, -0.0609930158, -0.191583186, 0.169178709, 0.170702919, 0.149429336, 0.0734934062, -0.0319855362, 0.0536946096, 0.0498708934, -0.117750682, 0.0036894232, 0.0974819437, 0.162416473, 0.036212638, -0.152097091, 0.0102473954, -0.175146922, -0.109410793, 0.0510285608, -0.102032453, -0.0270780027, 0.112112477, 0.179075554, -0.174917683, -0.115047842, -0.104785867, 0.0759669393, -0.185626954, -0.114752382, 0.0533825904, -0.104991615, -0.0954450741, -0.0869510844, -0.132044673, -0.191752613, 0.00513811922, 0.0554652661, -0.133202344, 0.148236826, -0.174548671, 0.101005033, -0.147775263, 0.151600003, 0.195948124, 0.146968648, -0.181632847, -0.126265585, 0.0861280486, 0.0299651623, 0.0794558972, 0.0533921868, 0.0195937455, 0.0455982238, 0.150372431, 0.139378235, -0.101709567, -0.0294380337, 0.0811925083, -0.0342354178, 0.0327691734, 0.0400085896, -0.1412265, 0.0617004111, 0.0421027988, -0.104852192, 0.00592757761, -0.180350497, 0.0525539964, -0.111471675, -0.0811403841, -0.0120081007, 0.15921399, -0.188091248, 0.184693262, -0.0228968561, 0.115342319, -0.0535733849, -0.114198565, 0.0240756273, 0.147423342, 0.15892826, 0.00908050407, -0.213146105, 0.152774766, -0.00141887786, -0.0586975515, -0.114548035, 0.0891831964, -0.0406573191, 0.0181619823, -0.049714718, -0.200603843, -0.135449693, 0.129440948, -0.212808505, -0.0500480942, -0.0812454671, -0.180212289, 0.0619920045, 0.0307168979, -0.0518378466, 0.0701079816, -0.190243214, -0.138796121, -0.193981051, -0.0390182026, -0.117929213, -0.204903558, -0.202367961, -0.155948266, -0.171265543, -0.129201606, -0.0976203829, 0.221453071, 0.138735101, -0.158441961, -0.225554422, -0.0675398037, -0.132319763, -0.0978091806, 0.210110873, 0.178208128, 0.101490974, 0.0418321043, 0.160106704, -0.187610939, -0.192003295, 0.0196090881, 0.0968832597, -0.175496653, -0.0902556181, -0.155951157, 0.107045144, 0.0573832281, -0.0581211299, 0.0521087125, 0.171671689, 0.158271715, -0.212730348, -0.0388053134, -0.172507182, -0.125131086, 0.156479985, -0.335062623, -0.0702413097, 0.223254368, 0.0645823479, 0.219279632, -0.196573928, 0.0732722208, 0.263311893, -0.159265086, 0.0834448114, 0.13835384, -0.136304572, 0.106453225, -0.0613590926, 0.138230368, 0.174712658, 0.094565548, 0.0211733319, 0.102425985, 0.0467876047, 0.111685343, 0.147267804, -0.258844495, 0.145146266, 0.14244695, -0.22259891, 0.0884163454, -0.207033977, 0.202475429, 0.0740721077, -0.0818101689, -0.125599563, 0.048894804, 0.139541343, 0.0525139496, -0.179559693, -0.0716978014, 0.0090209581, 0.113008924, 0.172887772, -0.0844542906, -0.0717213899, 0.188895106, 0.00843533594, -0.161318779, -0.00458678044, 0.0416456424, 0.0458753034, -0.117116317, 0.134884998, -0.0610275529, -0.0735569224, 0.220500335, -0.0618452467, 0.0568264462, 0.0672242194, 0.0536397211, -0.0376431644, 0.156504616, -0.207624599, -0.0204942245, -0.208658844, -0.179129675, -0.100364596, -0.150991708, -0.186092764, 0.17417559, 0.134831354, -0.095172435, -0.0442455336, 0.256724715, 0.21277459, 0.17345655, 0.216043293, -0.0360164866, -0.0652590916, 0.0154270008, -0.0202574134, -0.175363034, 0.0316524692, -0.0490601547, -0.0729391202, 0.13120921, -0.115910649, 0.162211448, -0.200046033, 0.113587596, -0.098146148, -0.062560007, -0.212389871, 0.212651432, -0.207820579, 0.16756323, -0.120097443, 0.245886236, 0.0261694063, 0.250802189, 0.213231578, -0.110681944, -0.0259542018, 0.0393911712, 0.141605258, 0.0951679051, -0.0903783441, 0.0266120266, 0.130146444, -0.202337459, 0.0765965804, -0.010533765, -0.0858198181, -0.00901217386, -0.0870363861, -0.011424928, -0.090558961, 0.0835403949, -0.256125689, 0.0130133061, -0.127759323, -0.238343403, 0.161234543, -0.192689836, 0.27777794, -0.0743051767, -0.0246492773, -0.264801741, 0.13777788, 0.039771352, -0.199020803, 0.278468162, -0.208027422, -0.0828270987, -0.00967502873, -0.0816069394, -0.0424416326, 0.0527059995, -0.163091287, 0.00891038775, -0.224737093, -0.0790355057, 0.0459024347, -0.0678463578, 0.174242303, 0.00127267418, -0.0481367819, -0.149950892, -0.261374563, 0.152924955, 0.115787119, -0.151344597, -0.208144918, 0.193755448, 0.148202732, -0.200177088, -0.14347811, 0.0296298023, 0.120643049, 0.0740528107, 0.0289400071, -0.219525307, -0.0684371665, 0.170777753, 0.0165751912, 0.161401957, 0.09001939, 0.137214094, -0.0132981138, -0.075612478, 0.223878801, -0.129973829, 0.163486749, 0.025689736, -0.02602401, -0.176745981, -0.096706301, -0.229914978, -0.208292037, 0.115179032, 0.131318823, 0.12323276, 0.0363375023, -0.18000105, 0.0444394164, 0.292281061, -0.209439784, -0.0804421529, -0.241354913, 0.0492477566, 0.115014032, 0.113993555, 0.0711855739, -0.105379127, 0.116060019, -0.230782375, -0.071728304, 0.166753724, 0.141988203, 0.203238681, 0.135525316, -0.0675361156, 0.258204639, 0.0555558056, -0.0669079423, -0.0546362698, -0.0095171025, -0.112937562, -0.112366028, 0.196951315, -0.190239713, 0.100786179, 0.27030012, 0.0785356015, 0.0146926921, 0.0336835608, -0.0475944877, -0.25933221, 0.114190906, 0.159268126, -0.0437385812, -0.259978563, 0.119038261, 0.196310908, 0.126920417, 0.1142755, 0.0501057506, 0.134804621, -0.0957523063, 0.14846307, -0.0672448725, -0.16493322, -0.21647732, -0.138321653, -0.0105587812, -0.105590709, -0.183317751, -0.0017683208, 0.0214145966, 0.0840778798, 0.1456929, -0.141866982, -0.177974984, -0.183813006, 0.0323574543, 0.216028988, -0.174554035, 0.0929575935, -0.0752552748, 0.0173932761, 0.00922764838, -0.194893017, 0.129454538, 0.132133171, 0.13402985, -0.0701206028, 0.176784858, -0.0571110547, -0.0514186881, -0.08907713, -0.0646748692, -0.194243208, 0.129443407, 0.00619410118, -0.00450532138, -0.207810163, 0.0717498884, -0.0734594464, 0.124055974, 0.075352475, -0.150470659, -0.187533662, -0.0271674097, 0.153355226, -0.0271843374, 0.0681567341, -0.0659090728, -0.0516456589, -0.198433399, -0.0102793267, 0.0921462923, -0.107441001, -0.0820229352, 0.0697086006, -0.121913351, -0.0349813551, -0.0305808745, -0.0559222177, -0.0764169097, 0.170531899, -0.119125612, 0.0380934328, -0.0192875862, 0.0188238919, -0.0392661095, -0.202440292, -0.115953766, -0.132373601, 0.210289285, -0.207067996, -0.074820444, 0.171109334, -0.0611716658, -0.187234789, -0.178964883, -0.0744869262, 0.042780444, 0.0340865999, 0.0349340886, -0.0808666945, 0.200756922, -0.0821405053, -0.177407742, -0.0506182462, 0.0319291204, 0.111412361, -0.119748138, 0.0575083643, 0.148518518, -0.0711778849, 0.0900242478, -0.166702032, 0.0707694143, -0.0672384202, -0.148692697, 0.0733167678, -0.0461998433, 0.0212943405, -0.105709076, 0.0511011332, -0.0303771347, 0.0363206118, 0.0554131418, -0.191839933, 0.0704303831, -0.014075771, -0.192795038, 0.0864057988, 0.0957165509, 0.0517887622, -0.207105055, -0.0549096018, -0.197128266, -0.0435425937, -0.00281360745, -0.0405648947, 0.0581579953, 0.131218538, -0.16994527, 0.199992672, 0.115575358, -0.18995063, -0.156800047, -0.0196557939, 0.076645188, -0.163925126, -0.123550206, -0.00278422958, 0.0024073571, -0.075328432, 0.0587575585, 0.194733024, -0.112012841, -0.17458263, 0.0873643756, -0.171549991, -0.150170997, 0.145191774, 0.0886108205, -0.191762626, -0.102553405, -0.103013307, -0.116796724, 0.200971395, -0.162655994, 0.0177573599, 0.0770139471, 0.135249302, -0.149339631, 0.0532134771, 0.125556737, -0.111500844, 0.13430278, 0.116502553, -0.133535191, 0.0993374139, 0.0131562548, 0.141030326, -0.215099677, -0.0540164895, 0.0587758832, 0.133371785, 0.128054485, 0.181748942, 0.186617449, 0.140814275, 0.158420652, 0.117290303, -0.0828610957, 0.181842074, 0.0536724478, -0.156423688, -0.0572760254, -0.0758121386, 0.0171979927, 0.0617454574, -0.123269998, -0.0501214638, 0.210173443, -0.0469620526, -0.0736155212, -0.0198381282, 0.159689367, -0.164338425, -0.148481369, -0.0429480225, -0.0946798697, 0.200503424, -0.101595551, 0.201301143, -0.0489229187, -0.162824064, -0.0438856035, -0.21362631, 0.244266868, 0.274435222, 0.169392526, -0.185727969, -0.0522047542, 0.00556242652, 0.0991317555, -0.132557571, 0.172653839, 0.0851856023, 0.190462366, -0.117255479, 0.117573619, -0.132007942, -0.0157813504, -0.00529545965, 0.0486687161, 0.209120095, 0.188496932, -0.197368637, 0.0993192643, -0.154122457, -0.135731071, 0.0958589017, -0.109322362, 0.0503121465, 0.0242886506, -0.151156679, -0.141134143, 0.0115236547, -0.248438224, -0.112202108, -0.0897251442, 0.253748894, -0.000320830557, -0.138551369, -0.0638582781, -0.0156727377, -0.10645014, -0.000941439182, -0.117576726, 0.0970672369, 0.159923315, 0.136554152, -0.0385889336, -0.103830874, 0.0358882025, -0.187269032, -0.206554636, 0.0885479078, -0.0132518057, 0.214956224, -0.12615642, 0.275876939, -0.0640837476, 0.144479454, 0.205591425, -0.0275788121, -0.140130028, 0.203447714, -0.107345656, 0.177566424, -0.112334542, 0.135879055, -0.141970098, 0.109072447, 0.110946029, 0.10664539, -0.176637948, -0.212433696, 0.0630291849, 0.150753275, -0.124068864, 0.0347972997, -0.203520656, -0.162690356, 0.0804221854, -0.183624178, -0.168030873, -0.0466670021, 0.201229915, 0.0762459859, 0.0738973469, -0.107046053, -0.0266148597, 0.140076771, 0.0768975466, -0.0661414787, 0.205275372, 0.117615834, 0.162698045, 0.0471834056, 0.066787824, 0.0462587886, -0.0657628477, 0.150616497, 0.180957869, 0.0334356651, 0.0815333351, 0.182552829, 0.0747729093, -0.0848053396, -0.192697644, 0.000992957503, 0.0669444054, -0.0864309072, -0.208967999, -0.163346067, 0.0919444114, -0.11361666, 0.0901513845, 0.121801101, 0.18307288, -0.129042506, -0.0295936447, 0.133450344, -0.149377078, 0.0841869488, -0.167957082, -0.156804591, 0.111636445, 0.122521162, 0.0814686567, 0.0948956907, -0.142786413, -0.16495119, -0.0619355738, -0.151000232, 0.235567585, 0.242622092, 0.0626911446, 0.158189178, -0.130945265, -0.0510335267, -0.193246707, 0.181436405, 0.039453797, 0.0719453469, 0.000969689456, -0.204767287, -0.0541508645, -0.0104957288, -0.165310189, 0.228289202, -0.133238673, -0.173104972, -0.197261706, -0.160179675, 0.207100019, -0.20425573, 0.0656981021, -0.064999491, -0.0689243972, -0.0135737462, -0.114986956, -0.148001194, -0.156635731, 0.136174291, -0.0735397115, 0.024009943, 0.18861106, -0.0555349216, 0.167080164, -0.0663658902, 0.156313211, -0.137416631, 0.219937623, -0.0101457722, -0.192980722, -0.00603267178, -0.00608571619, 0.156647861, -0.213914216, -0.00686631678, -0.18698661, 0.137742862, 0.107735321, 0.0747293308, 0.135365367, -0.0309074614, -0.103391051, 0.253569245, -0.167082265, -0.155858532, -0.0525114238, -0.182957605, 0.192761794, -0.103556834, -0.0391536839, -0.0144170625, 0.179714397, 0.0125448611, 0.164514452, 0.108714201, 0.228309497, -0.086764805, -0.134017855, -0.0286707878, 0.0568587519, 0.081173256, -0.0287004691, -0.0670309067, -0.064888604, 0.114137292, -0.0725059435, -0.174008653, -0.0875643715, -0.127273753, 0.131509304, 0.225763783, -0.0839330703, -0.136040702, -0.189437702, -0.202584773, 0.0523217767, 0.263796657, 0.136124715, -0.175133616, 0.0481774323, 0.0252242032, 0.180632174, 0.14017573, 0.0722272471, -0.141429991, -0.14743869, 0.172693461, 0.250584245, -0.0508589484, 0.149392784, -0.0614273623, -0.188037321, 0.136032209, -0.115289845, -0.215180367, 0.175799161, -0.142253354, 0.0276352465, -0.149539113, -0.0436008498, 0.214859545, 0.134571746, -0.0436521098, 0.222684115, -0.109537765, -0.0431752317, -0.0141235311, -0.0353392698, 0.182102561, -0.152115494, 0.237127289, -0.166017041, -0.0662677586, -0.123375967, 0.0391481966, -0.0662866086, -0.032407172, -0.226494104, -0.163152546, 0.00762933912, -0.171422973, 0.25206548, -0.0176769458, 0.277596235, 0.00642719865, -0.0545174591, 0.0522982441, -0.0763136446, 0.245492265, -0.0421209559, -0.140477717, 0.123090878, -0.069406189, -0.00897048693, 0.0338697173, -0.145748019, -0.143358067, -0.170915663, 0.179273531, 0.0158482641, 0.0439317264, -0.164723992, -0.163618878, 0.129824698, -0.307914853, 0.00500768237, -0.177501172, -0.196434334, 0.159178451, 0.193265259, -0.0784411952, -0.0199198276, -0.136541232, -0.0581868403, -0.0336628743, -0.163134873, 0.0191420875, 0.00514668226, -0.136096939, 0.169880554, 0.146405965, 0.12389233, -0.157588914, 0.135902241, 0.020170236, -0.197500393, -0.211237401, 0.183388785, 0.173877329, 0.0596420616, -0.0495417826, -0.00247370661, 0.196426719, 0.119838014, 0.030950062, 0.0507870428, -0.0551843941, 0.080456607, 0.13434732, -0.188290507, -0.0291505717, 0.0936101824, -0.0743033737, 0.238530099, 0.0853732973, 0.0866866857, -0.0472731218, 0.101936914, -0.161955655, -0.103445411, -0.115826197, -0.185676217, 0.144468918, 0.0192127451, 0.243185744, 0.213160887, -0.0700132027, 0.132710531, -0.0866566449, -0.126810819, 0.239814758, -0.0543582328, -0.0970630199, 0.151953116, 0.247111589, -0.157347828, 0.137009367, 0.0681802928, -0.325023025, 0.0898184255, 0.0172431283, -0.0638230145, -0.00389597355, 0.201046601, -0.10115499, 0.215875402, 0.148981452, 0.156407848, 0.0929401219, -0.116457552, -0.0533874482, -0.0953917503, 0.0635540038, -0.174071953, -0.014446131, 0.174123392, -0.0109589575, -0.06459672, -0.00470030122, -0.210424423, -0.214112669, 0.073211208, -0.116393417, -0.215505868, 0.165930703, -0.111611903, 0.0542642213, 0.02777946, 0.254414827, -0.237083703, -0.106226139, 0.135093778, 0.188917518, -0.088959381, -0.153844506, -0.0671698377, -0.253456146, 0.211136952, -0.0188651383, 0.00893640518, -0.0500897728, -0.103367783, -0.209297687, 0.185887992, -0.0478939153, -0.121324107, 0.19026418, -0.0403532162, 0.206234485, 0.206992447, -0.200000763, 0.156136796, 0.0766848624, -0.213080689, 0.129118517, -0.0300498139, 0.0841510743, -0.0039588213, -0.053927239, 0.0600163192, 0.118532047, 0.125032127, -0.141252995, -0.134606391, -0.149302527, 0.181654245, -0.0525682978, -0.0095063895, -0.0866127312, 0.0237378366, -0.0967183784, 0.133381084, -0.0180076975, 0.0250853039, -0.159199923, 0.179142401, 0.146943107, -0.0130850719, -0.208270669, -0.122804597, 0.086103417, -0.0587755069, 0.140682414, -0.192945361, 0.0519251116, 0.232186466, 0.0842411444, 0.0156072173, -0.0367138796, -0.129091635, 0.286088198, -0.050661698, -0.0959331617, 0.196171507, -0.166134045, 0.110787347, 0.0763130635, -0.195894212, -0.016266359, 0.0650015101, -0.000705195009, -0.0798940808, -0.157687202, 0.0367488489, 0.0635683686, -0.00835195277, 0.147954598, 0.00347357406, -0.0717437714, 0.0263384692, -0.0868112966, -0.1464587, 0.183965608, 0.154775858, 0.0563162044, 0.119879685, -0.0458873212, 0.0146314949, 0.01340455, -0.127139658, -0.0805401057, 0.010805428, -0.0598547757, 0.140515849, -0.0332521386, -0.139405355, -0.00381903304, -0.119757995, 0.0642717928, -0.00595461437, 0.00971299782, 0.0181997381, 0.14657104, 0.236595348, 0.133447409, 0.165538937, -0.171264574, -0.17734462, -0.118777111, -0.0742687881, 0.163928539, 0.158281639, -0.0200940482, 0.00364433066, 0.110924534, 0.204607725, -0.056781482, 0.00452534854, 0.161825106, 0.231086031, -0.114858396, -0.00962379854, 0.207619533, 0.090628311, -0.0552490801, -0.168093532, 0.12639004, -0.0469605736, -0.124545485, 0.103754275, 0.116334625, -0.200652197, 0.122327343, -0.24620837, 0.150227144, 0.124391578, -0.149749219, 0.0835158229, -0.15222469, -0.0924759209, 0.121347412, 0.103715703, -0.179746136, 0.0542897433, -0.121789955, -0.0700749233, 0.0558092073, 0.159794122, 0.125659496, -0.0444125459, 0.0128017385, -0.172242373, 0.17140238, 0.0414437614, 0.0733803064, 0.0441474169, 0.0272179805, 0.0157027543, 0.0845738202, 0.19979848, -0.103852771, 0.145444691, 0.1565492, -0.183115691, 0.0272264779, 0.00203362154, -0.176931471, -0.136718005, -0.0667834654, 0.160385624, -0.0971334875, -0.0346084386, -0.00125173316, 0.214042053, 0.100500204, -0.181512147, -0.207882851, 0.18568328, 0.205129042, -0.012027801, 0.136106357, 0.0456399471, 0.181273654, 0.0196859818, 0.0653820038, 0.0663783401, -0.0337033458, -0.0586933829, 0.108097129, 0.091456309, -0.134444326, -0.027708875, -0.145242408, -0.00287574693, 0.0847207606, -0.181775391, 0.183636069, 0.0688786507, 0.263257593, -0.00427195895, 0.123155445, 0.158885136, 0.170019612, -0.181566104, -0.0179279, -0.184301853, -0.0013938545, 0.177570879, -0.121418886, 0.0150488978, -0.000610802672, -0.218872413, 0.133591279, 0.112349041, 0.202252939, -0.194210395, -0.0492385663, 0.199029937, -0.0331471264, -0.189999968, 0.15875043, -0.0649037361, -0.0359622762, -0.101073802, 0.178152233, 0.0650028139, 0.0732081607, -0.0311551392, -0.00686773099, -0.112522438, 0.281459391, -0.150038421, -0.154241458, 0.0597723648, -0.0180041976, 0.095261544, 0.196119681, -0.0852496773, -0.220084459, -0.141354889, -0.00177710166, 0.115805745, 0.211524799, -0.146760225, 0.130397364, -0.200928628, -0.082532011, -0.0342374705, 0.0937826261, 0.204201654, 0.259379774, 0.143860042, -0.022885045, -0.0885771513, 0.225629315, 0.203129902, -0.0972949266, -0.167454958, 0.209564671, -0.0261494219, -0.121619433, 0.170461625, -0.0545143932, 0.0480193757, 0.184107944, -0.127340436, 0.183212698, 0.121917456, 0.189465776, -0.198853567, 0.176508516, 0.0776296109, 0.071349591, -0.163570002, 0.121416613, 0.0280675068, -0.0353203863, 0.0381100923, -0.0884888694, -0.00105153024, 0.197435677, -0.0372472778, 0.199374154, -0.0266889483, 0.0552413613, 0.16077064, 0.0775329843, -0.056018278, -0.0785094425, -0.111316718, -0.0708481371, -0.219346598, -0.0713492781, 0.0917782038, -0.111492112, 0.0235726535, 0.113839343, -0.0846240744, 0.186591521, 0.107423566, -0.0425455049, 0.133113995, 0.112909913, 0.155081719, 0.12983717, -0.0908117145, -0.0424004309, 0.123853929, 0.161590233, 0.0740211159, 0.220889717, 0.0111323493, 0.0138287498, -0.108956374, 0.218805134, 0.116877005, 0.0139654735, 0.0478446335, 0.00290354271, -0.135019958, 0.100197278, 0.202663228, -0.0565481894, 0.0516312271, 0.164359331, 0.027229758, -0.161545083, -0.0841104686, -0.132132292, 0.0750347823, 0.126185328, -0.0328487605, 0.121280387, 0.17534402, 0.142205924, -0.222641334, -0.0284508038, 0.0550886728, 0.0873866901, -0.098779656, 0.108810529, 0.222481266, -0.133257478, -0.0171785951, 0.23207663, -0.16922313, 0.0166405141, 0.149411425, 0.244119301, -0.0342978686, 0.0424096137, 0.0300826505, -0.302469999, 0.12808831, 0.202303231, -0.128145292, 0.254153311, -0.0533468723, -0.00429165037, 0.00639062561, -0.0596186407, 0.106781147, 0.116036557, 0.164889902, 0.118450627, -0.11772456, -0.212542042, -0.0230301227, 0.15320763, -0.102894507, 0.164426908, 0.137734249, 0.0360440724, 0.053503558, -0.19689019, -0.089921236, 0.255165786, -0.121091068, -0.186938509, -0.199636534, 0.228079587, 0.0136816055, 0.137275338, 0.147264242, -0.157951266, -0.133595556, 0.198956296, 0.0500613302, -0.104482673, 0.153554499, 0.186254889, 0.0757497177, -0.146393776, 0.136819497, -0.161653802, 0.202596903, -0.184190035, -0.143676028, 0.129627481, -0.0586775057, -0.181300387, -0.0238430016, -0.189769417, -0.0744324401, -0.197278708, 0.164129451, 0.0219707415, 0.0293897092, 0.0587765612, 0.0964035615, 0.15167059, -0.125168294, -0.190928459, -0.112992272, 0.0658306628, -0.0772390664, -0.199625686, 0.125136733, 0.016112512, 0.0507222563, -0.0624214858, -0.16135475, 0.0569047816, -0.0239417739, -0.0304762162, -0.194920689, -0.12425144, 0.00409839163, 0.107493088, -0.208759293, -0.066616863, -0.172572762, -0.0572636537, -0.0250401981, -0.186279193, 0.0375845768, 0.201264232, 0.04939197, 0.123899333, -0.155704662, 0.0954312757, -0.150194436, -0.055589918, -0.14039661, 0.131468296, 0.194920346, -0.212645948, 0.0513700098, -0.117145963, -0.108924069, -0.186193109, -0.0858286917, -0.074252367, -0.052907601, -0.174557745, 0.0896119028, -0.119890451, -0.0677545518, 0.141775265, 0.183063552, -0.098954916, -0.143848076, -0.180254698, 0.0703581721, -0.000212103128, -0.0897746533, 0.183473036, -0.0284350216, 0.0284716189, -0.0381336361, -0.20608604, 0.169497326, -0.0935021788, -0.162120327, 0.0298986882, -0.152690023, -0.0220084935, 0.0699769109, 0.09413068, -0.161180288, 0.107032284, 0.170551285, 0.0715923756, 0.0323232859, 0.098411873, 0.14979668, 0.1879002, -0.0492424816, 0.119373843, 0.0076083988, -0.0622389913, 0.184939489, 0.085078761, -0.205675215, 0.0704781264, -0.108920917, 0.160283193, -0.135330096, -0.0439995378, -0.0609262735, -0.146751195, -0.0557816476, 0.187445238, 0.112474993, 0.108281776, -0.1571922, -0.0101753175, 0.032023266, 0.0926543921, -0.0471730232, 0.121487752, -0.0342903174, -0.0375407673, -0.0172177386, 0.241554603, 0.127430961, -0.0501674153, -0.136261061, 0.0438360311, 0.275473982, -0.0898060501, -0.00404814957, 0.150418699, 0.26817739, 0.0120358318, 0.0627415776, -0.217566565, 0.0120521989, 0.231260166, 0.174179092, 0.20312205, -0.099578023, 0.131383866, 0.0526953712, -0.0166083407, -0.179985553, -0.0176230427, -0.16833955, 0.055621013, 0.16548951, -0.078905493, -0.102710724, -0.144292682, 0.193504497, -0.167036876, 0.143709898, -0.106144384, -0.158193961, 0.180407584, 0.134830743, 0.0780916661, 0.21605663, -0.203453779, 0.153617635, -0.0991857052, -0.259447694, -0.157837898, -0.0765701681, -0.166750148, 0.0323081128, 0.0766944364, 0.231664136, 0.099929817, 0.225088254, 0.0904840156, -0.0980547816, -0.139175221, -0.0406756736, -0.0503455848, 0.013110226, -0.236767709, 0.108082667, 0.0616400279, 0.12457861, -0.0175604355, 0.0778381824, 0.0382082202, 0.210355639, 0.0954632461, 0.211079672, -0.10271854, 0.0311335325, -0.0154708745, -0.20266667, -0.0589585006, -0.15951401, -0.0808824971, -0.206491053, -0.0773185492, 0.0643220842, 0.269766062, -0.0534514859, -0.0768430829, -0.181922227, -0.12921229, 0.0590348989, -0.0676625296, -0.163617879, -0.210261837, -0.108614251, 0.141992033, 0.292766303, -0.00388330221, -0.0342260152, -0.278354913, 0.202880338, 0.114471421, -0.0569821373, 0.209743157, -0.197622269, 0.11517106, -0.282697707, -0.177471429, -0.0363213867, 0.0715632513, 0.0966505781, 0.156586885, 0.00711535243, 0.193091586, 0.319586277, -0.077367425, 0.194643721, 0.133760348, 0.162715733, -0.213925645, 0.0577851124, -0.115082778, 0.0244967844, -0.233547971, 0.16115953, 0.116338134, -0.0176728424, 0.103588142, -0.0136159752, -0.0320229046, 0.0752808824, -0.0454647131, 0.141926035, -0.157470793, 0.0646567643, 0.116127677, -0.0982909575, 0.0018835736, -0.206134573, 0.0186304394, 0.119598277, -0.114110075, -0.196623132, -0.202344328, -0.0913590342, -0.201012149, -0.0851496235, -0.0685937256, -0.235107616, -0.12301024, 0.124149792, 0.0983350128, 0.0774306282, 0.0723523647, -0.215187356, 0.111336991, 0.127059489, -0.112067282, -0.00816392899, 0.126290902, 0.0156315081, 0.0512061268, -0.210605562, -0.0202413108, -0.145583779, 0.00709361816, -0.124394178, 0.180435747, 0.104641557, 0.0187026784, 0.0350805745, -0.163335904, 0.194162667, -0.0241593253, 0.117580511, -0.171764538, 0.225402132, -0.0720629022, 0.0310874283, 0.0749795213, -0.205305517, 0.124029838, 0.0928468481, 0.104787186, 0.122945972, 0.0687557608, 0.197842777, -0.038209822, 0.209728137, 0.148183659, -0.0895242766, 0.102743544, 0.158801213, -0.0225127339, 0.176194936, 0.0220577177, -0.0678962469, -0.0967836902, -0.167863473, 0.179799557, 0.148632124, 0.0381179079, 0.208649412, 0.0900598094, 0.143464074, -0.0833160579, 0.129522786, -0.0478451103, -0.0691998526, 0.0784664005, -0.0541049801, -0.142444491, 0.157873392, -0.0442984365, -0.0314130932, -0.0341217779, -0.190294713, -0.0624290369, -0.0108193904, -0.0722554624, 0.0450399257, 0.184874624, 0.0353574604, 0.250395238, -0.211719662, -0.0713019222, -0.0945236161, 0.0628559738, 0.113878533, -0.166120961, 0.0611039735, -0.0665954202, -0.190605044, 0.104317546, -0.00670157606, 0.197475791, -0.157059222, 0.0666453913, 0.190627366, 0.00203674077, -0.0640138537, 0.169015393, 0.158805847, 0.00249635987, 0.175454721, -0.11453028, -0.0718963668, 0.0581686459, 0.0863645673, 0.254797548, -0.0167599767, 0.0753724277, -0.191692099, -0.037594419, 0.0371002257, -0.0114472676, -0.129038393, 0.135102063, -0.0811199322, -0.0868073627, -0.140736476, 0.270534247, 0.211350933, -0.0777289495, 0.0280433893, 0.0301295258, -0.138493523, -0.226183578, -0.00809103157, -0.048917044, 0.134023279, -0.111272015, -0.131809756, 0.167289764, -0.0939597264, -0.0454141498, -0.199593216, -0.0715295821, 0.16763784, 0.155164659, 0.0330340266, -0.0935863256, 0.074379988, -0.055489637, 0.0121996375, 0.216600537, 0.0732028931, 0.106504105, -0.179512233, -0.0358368456, -0.192034081, -0.0353995189, -0.0244174004, 0.0996022075, -0.0177846104, 0.219992995, -0.101739459, -0.0576194376, -0.169102862, -0.0963000655, 0.0924205929, 0.0396039449, 0.0483620577, -0.0561504178, -0.0868818238, 0.0164745953, 0.0548049062, 0.114303872, 0.013754636, -0.0567086786, 0.102405623, -0.0438192934, -0.0643145293, -0.0401981324, 0.00962526165, 0.195387542, -0.162058115, -0.118062168, 0.0846031681, 0.0343922898, 0.0729532316, 0.186529264, 0.0633441284, -0.0136433439, -0.0180960745, -0.022626821, 0.130006075, 0.141576752, 0.0769681633, 0.0622897595, -0.126342788, 0.0708925575, 0.0250345729, 0.00250566704, 0.137845576, -0.0369660184, -0.186658204, 0.0200903825, -0.0130848829, -0.10494981, -0.0606996045, 0.169031233, 0.125592455, -0.081215255, -0.0654265434, 0.0523951836, -0.142207876, 0.254872948, -0.153936654, -0.188501954, -0.160121426, -0.134948, 0.205956161, 0.190052256, 0.16584532, 0.151236117, 0.0718697757, -0.080587402, 0.110667244, 0.0943986848, 0.181700706, -0.00617637718, -0.208006665, 0.14149186, 0.0434235521, -0.0528380871, 0.0149466833, -0.00435288716, 0.181254312, 0.10414812, 0.132486179, -0.0475688763, -0.139805526, 0.061016947, 0.088329263, 0.104247503, 0.237457544, 0.22448419, -0.0426649414, -0.0163636543, -0.204058439, 0.163758263, 0.243123114, 0.234052137, 0.0471326299, -0.117478944, -0.0863664374, 0.0787322223, -0.159595221, -0.173156038, -0.0570174493, 0.086930953, -0.141002566, 0.124750815, 0.191485867, -0.202254176, 0.205454722, 0.166258335, 0.0726499707, 0.0952544957, 0.100071169, -0.202629045, -0.172590211, -0.13892965, 0.0231076777, 0.111921228, 0.274842918, 0.0941486955, 0.0641628727, -0.142406732, 0.0568496808, -0.0287323724, 0.0187774654, -0.0521207936, -0.164493352, 0.131963298, -0.0280933343, -0.212045416, -0.104063354, -0.0864547491, -0.204800725, -0.0237307753, 0.0920451134, -0.0136097614, -0.11391791, -0.264806271, -0.201454163, 0.147936925, -0.146814078, 0.171959713, -0.124607295, 0.129478768, -0.204661041, -0.0736282244, 0.190738454, 0.0476327986, -0.0412670225, 0.103763528, -0.215454429, -0.0301665645, 0.00799800269, 0.193996519, 0.155501172, 0.0539092608, 0.0650432557, 0.226527035, 0.180688441, -0.182288006, 0.0930174738, 0.260853142, 0.016753193, -0.214730203, 0.0154327303, -0.0481189452, 0.0598105043, 0.0232905801, 0.130197376, 0.17757155, 0.0245893449, 0.151050985, -0.107956119, -0.240185767, 0.00206723274, -0.0504090339, 0.212470889, -0.160272613, 0.239395365, 0.203135297, 0.189087495, 0.0853048265, 0.171777859, -0.029955145, 0.11319828, 0.0216485877, 0.00814698357, -0.110079348, 0.0574759692, -0.0117787374, 0.0587957054, -0.0188551173, 0.187958941, 0.201361075, -0.212008983, -0.150154889, -0.0777181834, -0.0097771734, 0.262629092, -0.0380698293, 0.043783132, 0.22858268, -0.0257687774, -0.0354431905, -0.0717736334, -0.0261267014, 0.238806605, -0.0407217331, 0.00614640862, -0.00211061444, -0.158218428, -0.0143331885, 0.0456409603, -0.0461011529, -0.145143121, -0.0836481154, 0.0455304757, -0.164061174, 0.137408197, 0.160984814, -0.05268538, 0.0676740408, 0.082190454, 0.213888645, 0.108864151, -0.229466036, -0.00585621083, 0.220650971, 0.128265545, -0.0412900858, -0.21077244, 0.15473862, -0.119168244, 0.1800441, 0.207246855, -0.11915756, -0.0156303793, -0.198259041, 0.0665771812, 0.108989105, -0.00986023247, 0.165291443, 0.0965227336, 0.00951856375, 0.0554960519, 0.0457220227, 0.196098253, 0.128513381, 0.0316233784, 0.00890362263, 0.166757986, -0.0175813287, -0.158623844, -0.20614323, -0.167428017, 0.00473146141, -0.106193721, 0.15801324, 0.00607329607, -0.00859092176, -0.154501185, 0.0736638755, -0.172929317, 0.178296432, -0.204777554, -0.0184551328, 0.0859390348, -0.0314055979, -0.110383652, 0.024170354, 0.0688661188, 0.103539482, 0.1746995, -0.0174282789, -0.188645795, 0.130957142, 0.161050007, -0.171988711, -0.124570034, 0.18495886, -0.173855573, -0.0370936096, -0.142793447, -0.145858899, 0.182163581, -0.183721334, 0.0315484852, -0.0502992272, -0.0749663711, -0.187164277, -0.0742956847, -0.130046368, 0.0317636281, 0.142129526, 0.0862586349, 0.0828672573, 0.0140935238, -0.079975754, 0.173597023, 0.141604081, -0.0771767423, 0.118548639, 0.0442024469, 0.0727466717, 0.266035914, -0.00593646383, 0.260059625, 0.144515678, -0.0130532747, 0.188891038, -0.0634195805, -0.0261913594, -0.0180802289, 0.237168074, 0.171025172, -0.130810335, 0.208993554, -0.030096842, 0.0740133673, 0.241876543, -0.184140071, -0.0688809901, -0.146465331, 0.16539228, 0.190757021, 0.17606993, 0.196502313, 0.136242479, -0.0804710537, -0.00782729965, 0.188913107, -0.0548046194, -0.0303347055, 0.142485619, 0.151637778, -0.158051103, -0.0266635474, 0.0728768855, 0.137775302, 0.125231311, 0.0346932858, 0.163109958, -0.205083966, 0.0756561756, -0.116977692, 0.0437464379, 0.231042966, 0.193829939, -0.18651934, 0.149564371, 0.154574603, -0.0290720891, -0.0690897927, 0.179843798, -0.0955478922, -0.0206622425, 0.190791145, -0.122945897, 0.125592127, 0.00321447477, -0.195028916, 0.0442178249, -0.104046471, 0.0260952171, -0.0816862285, -0.110913567, 0.091348283, -0.115662403, 0.251517475, -0.21434246, 0.175582513, -0.14993903, -0.0990529507, 0.0514201038, 0.150468886, 0.228353143, -0.173500925, -0.00461063208, -0.0714868903, 0.143813297, 0.217226163, 0.114283666, -0.197505504, 0.0496195182, 0.0727943853, -0.0745235234, -0.0619089901, 0.0918129012, -0.117093414, 0.0321687013, 0.236869738, 0.126950324, -0.162127212, -0.119039662, 0.161647394, 0.231011108, 0.177849144, 0.147918016, 0.133619756, 0.190788567, 0.0492400676, -0.00180678465, 0.0893449634, -0.148697823, 0.177664801, -0.0726399198, -0.0793330893, -0.225488186, 0.131051272, -0.113395549, -0.14153862, 0.0294948965, 0.191074476, -0.00509508047, -0.0429674871, 0.0682959855, -0.122674003, -0.110053435, -0.0392141566, 0.0516043007, -0.0405695885, 0.278859168, 0.146024361, 0.223367631, 0.179515615, 0.182836056, 0.0309408158, 0.0159752686, 0.00173792825, 0.11343246, -0.10914018, -0.056721732, 0.0177230816, 0.175182432, -0.036981035, -0.131743401, 0.207399696, -0.0125906104, 0.192897528, 0.10380502, -0.128706738, 0.141425639, -0.141085252, 0.0864470005, -0.00618862314, -0.00134076655, 0.00479231775, -0.11014533, -0.135056555, 0.00566653907, -0.179885507, 0.197231576, -0.0278437734, 0.132824823, 0.150243133, 0.151170567, -0.0333556682, -0.0339126848, 0.0283680595, -0.025435755, -0.0908457041, 0.0670256168, 0.119782694, -0.048878938, 0.0382228903, -0.106433287, -0.129820496, 0.0346301049, 0.0843395144, 0.0345586091, 0.151655838, -0.0818703771, -0.081794247, 0.115935832, -0.0413574092, -0.00304169138, 0.0973383635, -0.00981269684, 0.0169961806, -0.168726087, 0.124752775, 0.0624595955, -0.166663989, 0.134228542, -0.133986801, -0.117507249, -0.183109924, -0.0409472734, 0.190115988, 0.0337236971, 0.117162749, -0.076600574, 0.129812434, 0.134825528, 0.0260062516, 0.0371112674, 0.177381799, 0.183222786, 0.216518879, 0.015962854, 0.0845715106, 0.108023062, 0.135057315, 0.000637001474, -0.203383252, 0.196280256, 0.0818561018, -0.100496322, 0.158635378, 0.179170743, -0.0156604201, 0.093567811, -0.101123378, 0.00368472934, 0.0540641397, 0.180312157, -0.201012507, -0.00493814051, 0.0403486565, 0.10555122, -0.219209358, -0.0529356785, -0.0400650203, 0.158233479, 0.10751909, 0.123106666, -0.0264859833, 0.143902779, -0.155771375, -0.109103367, -0.0625805184, -0.0451420695, 0.210679486, -0.194820687, 0.07988628, -0.162504762, 0.208094731, -0.150656149, -0.078792125, -0.12391606, 0.0141808093, 0.172131687, -0.108649395, -0.0934482217, -0.219430164, 0.193088472, 0.0839586705, -0.0547866635, 0.0759218782, -0.0979883671, -0.0717851892, -0.133541152, -0.214100048, -0.147924244, -0.00851948559, -0.0822613388, 0.111076437, 0.204227194, -0.0590670258, -0.0866161436, -0.0972947702, 0.0178795159, 0.0895289332, -0.0690636188, -0.0857937858, 0.16783753, -0.0259044375, 0.00509806909, -0.225554511, 0.154907301, -0.146912664, 0.268833876, 0.140848532, -0.159942165, 0.204923227, -0.16968435, -0.0109424917, -0.140655488, 0.00905802846, 0.0975849852, -0.113203347, -0.00286432612, -0.00585176935, -0.163264215, 0.177411392, -0.200985014, 0.00323767564, 0.0647737458, 0.0477584526, 0.103176244, -0.0821804181, 0.0348460563, -0.110611327, 0.148955032, 0.269896477, 0.0960517451, -0.103157543, -0.162139267, -0.149393424, 0.125260234, 0.070246011, -0.225312755, 0.25742054, -0.0397864655, 0.177335784, -0.0546780899, 0.248964921, -0.166126356, 0.192700773, -0.00790695101, -0.0664229989, -0.153038487, -0.129117221, -0.0757997856, 0.0386017896, -0.135388434, -0.158859819, -0.104986891, 0.146457687, 0.199433178, 0.066154249, -0.27667287, -0.118511088, -0.0179567039, 0.222479478, 0.0455367491, 0.243386254, -0.120252974, 0.132388383, 0.00776485447, -0.194177583, -0.0780516565, 0.00999934599, 0.11524263, 0.142233551, -0.0642258972, 0.186899021, -0.103108883, 0.099964574, 0.237639084, 0.121256396, 0.0142423958, 0.202542499, 0.20030944, 0.180703923, -0.214075804, 0.0230388809, -0.299164712, -0.128671005, -0.189861313, -0.167792231, 0.0813844353, 0.00933712721, 0.0428303629, -0.1023985, 0.174391836, 0.253679901, -0.0937102586, 0.0857886672, -0.158551842, -0.167360649, -0.0763060898, -0.0540213883, 0.133122638, 0.148575723, 0.0668005571, 0.152676195, -0.0732476413, 0.0157247335, -0.270311266, -0.0190660674, 0.212057456, 0.182492748, -0.241901889, -0.0313768871, 0.228386506, 0.0656861812, 0.192671508, -0.157984391, 0.0745935887, -0.0429898053, -0.122312985, 0.124423012, 0.0292300582, 0.181159899, -0.110646807, 0.205835596, -0.127989545, 0.139688984, 0.0181228518, -0.0549869686, -0.161712885, -0.0697539151, -0.0804900229, -0.0285761952, 0.123424694, -0.207021698, 0.0395707637, -0.211159229, -0.045374617, -0.150724575, 0.179440662, 0.103816822, 0.015124768, 0.0048571527, -0.185660616, 0.0693678111, 0.0240155458, 0.0238517523, -0.130017757, -0.210529521, 0.112137035, 0.178406164, 0.19203876, 0.21485664, 0.191359922, 0.0654983968, 0.166367605, -0.0858131945, 0.0867324322, -0.141689003, -0.137133151, -0.210735589, 0.216141865, 0.00645007193, -0.170115247, 0.0192143917, 0.156424567, -0.12158598, -0.170511737, 0.118564084, -0.203893989, -0.100373045, 0.206237301, 0.0579547733, -0.109020285, -0.159191296, -0.196344331, -0.10288664, -0.0650167316, 0.0364720076, 0.210455045, -0.198279276, 0.0561158136, -0.191313118, 0.021069834, -0.0339165032, -0.191652551, 0.198695317, -0.120528094, -0.0548847243, 0.0808626562, -0.00428579329, -0.102671824, 0.117770836, 0.140487507, 0.134317502, 0.156712055, -0.212678373, 0.115886249, -0.0798269957, 0.215774462, -0.161133751, 0.178629026, 0.0955588222, 0.155450925, 0.0492355675, 0.135866612, 0.202169314, 0.0468329042, -0.150953293, -0.0446973443, 0.103053465, 0.0478212684, 0.214107037, 0.135672152, 0.200946644, -0.174147338, 0.12126869, -0.139116272, -0.0563006103, 0.0277512744, 0.246417493, 0.0611405782, -0.0119189397, 0.208439246, -0.0356294885, -0.170967788, -0.115360253, -0.129960269, 0.144377574, 0.0454087257, 0.259763271, -0.105527014, 0.055321455, -0.0526598319, 0.159842834, -0.0482077226, 0.236779749, -0.132585362, 0.189681903, -0.0961048529, 0.0563793406, 0.18519479, -0.127709776, -0.0987681523, -0.0303634182, -0.0687099472, 0.0578852296, -0.0381461047, -0.18619667, 0.12401966, -0.121132657, 0.225062236, -0.205080852, 0.0551929399, -0.0777834952, -0.053174451, -0.199143633, 0.159538761, -0.238657549, 0.220129281, -0.114376858, 0.221257493, -0.255461693, 0.0300092585, -0.0607489645, 0.126692057, -0.112293094, -0.0986434072, 0.0438456684, -0.130739585, 0.0128232781, 0.166859791, 0.0306993425, -0.0176246464, -0.130978495, -0.0725799501, -0.00697065098, 0.149285182, 0.0522971042, 0.0522838607, 0.132519081, 0.192778155, -0.0416352339, 0.109511234, 0.202514991, -0.189964101, 0.0592628978, -0.133078381, 0.249684885, 0.151773691, -0.0527177453, -0.100954384, 0.124180362, -0.203475311, -0.118713893, -0.0816718787, -0.0157442, 0.100288361, 0.124790654, -0.027971575, 0.0515414514, -0.152316317, -0.139562219, -0.135580957, -0.084609136, 0.167367682, -0.169176459, -0.128676862, 0.160356179, 0.167749211, 0.208847791, 0.059897989, 0.161345467, 0.195118994, 0.11026185, -0.0473038405, -0.162515476, -0.140200004, -0.138756335, -0.189846769, 0.20646067, 0.0327555984, -0.222942144, -0.0198731795, 0.0467148684, 0.0791418999, 0.0614629388, -0.126075357, 0.108883843, 0.00917934161, 0.0830445662, 0.080400981, 0.113189146, -0.147388667, 0.200981006, 0.09387137, 0.0662245005, -0.127312094, 0.101593748, 0.146900043, 0.230416954, -0.221930906, -0.0331053957, 0.17240724, -0.0221072081, -0.0760479346, -0.20360899, 0.112684511, -0.138931423, -0.162155733, -0.119198255, -0.126619726, 0.012630037, -0.109421387, -0.166782975, -0.182280928, -0.172797754, -0.0645593479, 0.0926890373, 0.0646796972, -0.123785369, 0.259334207, -0.0265048742, 0.0963960364, 0.0207417514, -0.0640984923, -0.0827390105, -0.134210065, -0.0423009247, -0.0835836828, 0.077250883, 0.0914835781, -0.000481657393, 0.0296047516, 0.176210508, 0.155236304, -0.120164134, -0.0224553142, 0.136641458, 0.0316355117, -0.099346526, 0.0761687532, -0.172814578, -0.228517711, 0.158629566, 0.0357749611, 0.00243570539, -0.0157305691, 0.0191846807, 0.00691910414, 0.0227921773, -0.0236533042, -0.18064791, 0.00115233322, -0.156837761, 0.111577243, -0.148221925, 0.230223015, 0.0173706133, 0.206947878, -0.0331011862, -0.160140678, -0.0975864902, -0.116723441, -0.13038072, -0.0243134685, 0.12657474, -0.0980337113, 0.175942108, 0.00192179182, 0.0473435558, 0.205429345, -0.0407878272, -0.213827103, 0.10833922, -0.0446451604, 0.0655935183, -0.188038319, -0.00301687419, 0.0675255656, -0.143765509, 0.00169246364, -0.0247743782, 0.065864265, -0.127450123, 0.186487421, -0.184591785, 0.0808997974, 0.0317924172, 0.00249277428, 0.0951853916, 0.276850134, 0.122914597, 0.0458479226, -0.112578034, 0.171549395, -0.214462727, -0.219333857, 0.215502247, 0.0376836024, -0.101821326, 0.23026073, 0.149181589, -0.116133168, -0.0090032015, -0.116861179, 0.256513149, -0.162931934, -0.112243503, 0.00128614902, 0.0244441722, -0.213078201, -0.0275032464, 0.0797179267, 0.111045495, 0.246224776, 0.0375076756, -0.0120324278, 0.122870028, 0.260363281, -0.0590779483, 0.0948166922, 0.153928548, -0.166328102, -0.198541239, 0.0432137474, 0.0723608881, 0.0856808871, -0.0166272782, 0.121594638, -0.196286201, 0.0552772507, -0.0785965696, -0.0785046741, -0.0733379275, 0.0284803696, 0.183244765, -0.0545121506, 0.183057174, 0.0930560529, -0.0827762261, -0.214541987, 0.0781526715, 0.0538695231, 0.179998606, 0.187902153, 0.0758102015, -0.117636815, 0.0950077325, 0.158064738, 0.0105737597, 0.0903970301, 0.108313836, 0.15097709, -0.0819445699, 0.0761458278, -0.140456557, 0.131802991, 0.0474786013, 0.155419514, 0.0239446163, -0.0219119042, -0.135106996, -0.144528925, 0.202310726, 0.0346909016, -0.190453961, 0.0817741007, -0.110087767, 0.0702924579, -0.0885792077, 0.0543277413, -0.0371818244, 0.1415499, 0.0944445878, 0.0789010972, -0.0174358636, -0.187914088, -0.0285935998, 0.206651524, 0.162923053, -0.0869459808, -0.17593582, -0.0593883246, 0.12480326, -0.130898282, -0.130268216, 0.0238823146, -0.129311413, -0.167941093, 0.0979045182, 0.115539357, -0.0248285532, -0.0738229454, -0.0171255767, 0.214699998, -0.214020938, 0.140577748, -0.122401878, -0.0789570361, -0.0618365258, -0.0654320568, 0.0157889575, -0.0293144584, -0.185034052, 0.036581561, 0.194275334, 0.1666383, 0.215620413, -0.100140139, -0.0502271801, 0.148168072, 0.105212435, 0.172577128, -0.205824286, 0.108652189, 0.156266138, 0.0341610163, -0.207641378, 0.0638252646, -0.162136316, 0.0771442205, -0.136415035, -0.0285003185, -0.0351519659, 0.0870053843, -0.13288036, 0.0186352301, 0.0405196398, -0.0903854445, 0.0850627348, -0.0760384947, -0.237707302, 0.177195832, 0.128395244, 0.0780189186, -0.200771526, -0.0849047601, 0.0701752678, 0.260807902, 0.156773731, 0.19866395, 0.0359680429, 0.0136158485, -0.113989539, 0.0786288232, 0.202783525, -0.145905748, 0.0732347518, -0.0434487239, 0.204440325, -0.00198599696, -0.118598729, 0.0120036881, 0.201528028, 0.209207103, -0.0491646491, 0.15841648, 0.136860237, 0.0266900212, 0.0796270967, -0.100128114, -0.114517465, -0.0816531703, 0.195008367, -0.0176160038, 0.113583505, -0.074151665, 0.154809341, -0.0299604684, -0.128933713, -0.00159797072, -0.211855963, -0.238786757, 0.0815278813, 0.179436997, 0.165538907, -0.105617143, 0.0446293801, -0.116550677, 0.212327167, -0.186529025, 0.178048402, -0.152893737, 0.211425483, -0.0932270586, 0.134178355, -0.082460545];
    CONSTANT bias_6 : ARRAY[0..63] OF REAL := [0.0747542903, 0.0747530833, -0.00429329416, -0.0110996887, 0, -0.0352521576, 0.0479723401, 0.0685250089, -0.0227601323, -0.00580839999, 0.0100521399, -0.0113847172, -0.0245158654, 0, -0.0200175196, 0.0475497283, 0.0741227865, -0.0268050022, -0.053697817, -0.00196474558, -0.0566426925, 0.0682095364, -0.00484778127, -0.00283427443, 0, -0.0188507643, 0.0644902736, 0, 0, 0.00199445919, 0, -0.00884012785, -0.00463645626, 0.0127481027, -0.0124424472, -0.047869388, -0.0151582286, -0.0145472726, -0.0152692702, 0.107757747, -0.032102257, -0.00659875572, -0.0174676776, -0.0266960394, 0.0917816684, -0.00874918327, 0, -0.0106172459, -0.0176149886, -0.026105281, 0.0043185926, -0.0422325172, 0.00292709749, 0.00419008406, 0, 0.0809127167, 0.0434060618, -0.00947956275, -0.00768119283, 0.0844815671, -0.00330898049, -0.0406921245, 0, 0.0103572262];
    CONSTANT weights_7 : ARRAY[0..4095] OF REAL := [0.0985890701, 0.261478722, -0.0590967536, 0.0771033317, -0.00640187413, -0.0827855617, -0.230103448, 0.0237006657, 0.211521849, -0.133053824, 0.144778341, 0.0126608955, -0.264563471, -0.0297934134, -0.171915665, -0.144233555, 0.184128761, -0.199485853, -0.128364205, -0.10924013, -0.0942144915, 0.12244907, -0.134638637, 0.159754649, 0.102856718, 0.193186775, 0.0345768109, 0.0443875194, -0.0223890841, -0.0877400488, -0.224890769, -0.0661405474, -0.0205741599, -0.132689729, -0.134608626, 0.0912717804, -0.0320888869, 0.207671627, 0.0316983312, -0.263397604, -0.159447983, -0.123716153, -0.0258523077, 0.231007561, -0.107568942, 0.228946403, 0.115262851, 0.202499971, -0.222295597, -0.0375091396, -0.23364678, -0.123035237, -0.0525233448, -0.0821483433, -0.12599954, -0.358725101, -0.0378492288, 0.14551425, -0.117850862, 0.0302092116, 0.136658132, 0.0596454889, 0.0601940267, -0.115125708, 0.190094337, -0.0647920668, -0.120055743, 0.00146726007, -0.178027615, 0.0304296073, 0.155361906, -0.165448382, -0.0763782412, -0.227639481, -0.156574205, 0.134376928, -0.335413128, -0.213705391, -0.0161788668, 0.176306963, -0.0786898807, 0.0378909893, -0.156903595, 0.0734621733, 0.145642534, -0.0653213263, 0.00195453106, -0.167763978, -0.112661101, 0.116725579, 0.228570595, 0.185373247, -0.0674858838, 0.123988092, 0.114007965, -0.0454010144, -0.077554442, -0.0201824624, -0.275262088, -0.114391603, -0.0663379133, 0.280113071, -0.112193778, 0.0486323275, -0.137166336, -0.0401128717, 0.0894181207, 0.00908427685, 0.179754227, -0.0671511367, -0.120330289, 0.114102527, -0.226583004, -0.0849781409, -0.0418890789, 0.17914106, 0.204921558, 0.0455944687, -0.0450889394, -0.0856394097, -0.113558985, 0.166775107, 0.0186151415, 0.211812183, 0.186384693, -0.132189557, -0.156687155, 0.191395983, 0.110498078, 0.139661208, -0.0920242742, 0.222033158, -0.00120364304, 0.00128853915, -0.0888353512, 0.211148933, 0.0156825483, 0.197753608, -0.181704342, -0.159737736, -0.0235950705, -0.0353642218, -0.00933676027, 0.126852483, 0.171151608, -0.0931896344, -0.0475037992, 0.138531879, -0.194260553, 0.0657681227, 0.136853874, 0.0619690791, 0.100470409, 0.0687212795, 0.0456814691, -0.0741193444, 0.143832967, -0.0251761973, -0.0440490879, -0.197995454, -0.100512169, 0.0636347532, 0.194363266, 0.14988251, 0.117436595, 0.0813431665, -0.0845726654, 0.041465167, -0.143196225, -0.13916254, 0.0370236412, 0.106373869, 0.133378014, -0.0168813877, 0.0678688437, -0.0221709907, -0.178990752, -0.0615577288, 0.208223164, 0.117776372, 0.0550451688, -0.11717312, -0.106960475, -0.132753909, 0.0749269575, 0.0704251528, -0.121250421, -0.182553753, 0.0348108932, -0.169337317, -0.0431644917, -0.06188545, -0.044683557, 0.0603879951, -0.086644128, -0.0278274007, 0.146163434, -0.0545757636, 0.0299487282, 0.174511701, -0.0916855708, -0.153672263, -0.0549600422, 0.0154589014, 0.00445316266, -0.102152765, 0.0601579957, 0.166933239, 0.040345829, 0.268830568, 0.154072955, 0.10402365, 0.0998772457, 0.0329706669, -0.18961744, 0.16987507, 0.083305344, -0.127246037, -0.209014222, -0.192148447, -0.160925955, 0.114261568, -0.133135706, 0.0742198899, 0.115098283, 0.229157656, 0.0866794065, -0.141607061, -0.00846149493, 0.1364851, 0.165410504, 0.177613571, -0.198162705, 0.204134092, -0.171739325, -0.204839557, 0.274487436, -0.0561079755, -0.183752149, -0.0607956015, 0.128661469, 0.0149638271, 0.00135228958, 0.187765002, 0.0477933511, -0.146877944, 0.164612621, 0.104129799, 0.0751872286, 0.09320952, 0.17067422, -0.122773752, -0.0966985524, 0.148433819, 0.166774407, -0.050018996, 0.107592955, 0.17758055, -0.0572009236, -0.115987271, 0.10496451, 0.0970115513, -0.0402181149, 0.143645063, -0.114797451, -0.0233546644, -0.0524974316, -0.180076912, 0.134013399, -0.138859093, 0.0046711117, 0.0682574362, -0.11045447, 0.101280972, -0.141288802, 0.131182745, -0.104055196, 0.1359476, -0.105594479, -0.199489638, -0.100357562, -0.184324607, 0.0823699385, 0.111964449, -0.0532657355, 0.0663902014, 0.177432373, 0.210205242, -0.210125804, -0.0332980007, 0.096206829, -0.0193504691, 0.167757437, 0.0213211328, -0.105646975, -0.073984772, 0.203198329, 0.0314622223, -0.175412863, -0.122094072, 0.0986203104, -0.122762077, 0.19236134, 0.135295138, 0.182322904, -0.103380427, 0.144614473, 0.0554241389, -0.175479814, -0.0391083062, 0.191711053, 0.121323869, 0.115582779, 0.181385979, -0.192489818, -0.173019394, -0.173292458, 0.0201414824, -0.0125766397, -0.0790846944, 0.0685555041, 0.167224765, 0.189211607, 0.210358679, -0.0415095538, 0.126387641, -0.0842779204, 0.0439397581, 0.00644816831, -0.152137846, -0.152992308, 0.0245475248, 0.192403287, 0.163964272, 0.116401248, 0.0257411487, -0.142266706, -0.146128058, 0.0102699744, -0.0180726349, 0.197232619, 0.193206668, -0.0754495487, 0.134801105, -0.00232620165, 0.225295782, 0.0273058284, -0.154496655, -0.201236218, -0.157684937, 0.187730253, 0.115707032, 0.131131858, -0.167114601, 0.047023993, -0.0567260347, -0.0668960586, -0.083985351, 0.0849857107, 0.0702214763, -0.179636031, -0.0277230721, 0.162856936, -0.20755665, 0.160055265, -0.182279021, -0.235589236, -0.151465133, 0.0571531281, -0.148302287, 0.248307049, -0.12540251, 0.115537778, -0.190976933, -0.0118816132, -0.0110264076, 0.138518065, -0.122859232, -0.0116230948, -0.185463518, -0.193349451, -0.160361007, 0.130532175, 0.209439963, 0.0375103466, 0.285149574, -0.158949748, -0.277013332, 0.153673515, -0.260961682, -0.172621742, 0.167940751, 0.207475811, -0.175017715, 0.145652935, -0.026749935, -0.0299806502, -0.266049534, -0.196326286, 0.033781562, -0.0726778582, -0.262074381, -0.0483580381, -0.143439263, 0.141321659, -0.00700642727, 0.292194456, 0.185188755, -0.0455660783, 0.101106308, -0.0083050346, 0.150430575, 0.15473111, 0.277323723, 0.112545229, -0.0247835293, -0.176015452, -0.04111927, -0.0102430824, 0.111235037, 0.142509177, 0.131318763, -0.15878965, -0.124645673, 0.191819474, -0.0986970142, 0.120010592, 0.279321134, 0.121246748, 0.170530006, 0.0124538634, 0.146209851, -0.0564521439, -0.453932881, -0.115464613, 0.0486782379, -0.212593615, 0.0844182074, 0.152913198, -0.0890955701, -0.014261798, 0.0763275549, 0.094609946, 0.16527921, 0.152573839, 0.215471298, -0.189632729, 0.0542746969, 0.0475845337, 0.165836349, -0.248436794, -0.139802009, -0.117795072, 0.0680505931, 0.127019078, 0.141767994, 0.108608454, 0.0795560554, 0.215438023, 0.253515422, 0.0968242809, 0.0465329401, -0.0367862582, 0.205732152, 0.0410595387, 0.14549467, 0.0515940823, -0.204010546, 0.097479187, 0.136549056, -0.0882421583, -0.231916368, 0.0916896313, -0.097374104, 0.108968385, 0.064018704, 0.0505693108, 0.151754782, 0.0724061951, 0.0685940981, -0.0536143109, -0.00958465319, -0.0650544614, -0.118865497, 0.0617310181, 0.164938733, -0.125389904, -0.0580696389, 0.076752767, -0.0623037033, -0.0602061898, 0.14020063, -0.0644329116, 0.185091019, 0.00150486734, -0.0492826067, -0.230618313, -0.0963186398, -0.0396718048, 0.0157787632, 0.147863075, 0.136901587, -0.0209644865, -0.0838856548, -0.0987434536, -0.0661321655, 0.0437461026, -0.125251681, 0.245231941, -0.142143026, 0.178793207, -0.120658711, -0.252990127, -0.0960166603, -0.148348227, 0.217699945, -0.152953058, 0.0320299491, 0.0397147648, 0.20091784, -0.297417134, 0.043796204, 0.0147441905, 0.0458022691, -0.151441351, 0.0129484637, 0.0644230098, -0.122672424, 0.11798434, 0.212057024, -0.0869171694, -0.126012012, -0.04658252, -0.0954014957, -0.244200468, 0.145332858, 0.0195005015, 0.189192265, -0.230275482, -0.0202685073, -0.150195628, 0.13925834, -0.0658622757, 0.158107281, -0.0311671887, 0.00751672499, -0.177279904, -0.0161855966, -0.106229313, -0.159273162, -0.194914743, -0.1878708, 0.0287032183, 0.288048238, -0.0252802446, -0.0553182103, 0.14248237, -0.203866616, -0.238840014, -0.207598493, 0.112077221, -0.100770809, -0.0132202683, 0.131064698, -0.162306666, 0.10710378, -0.166209847, -0.00958471466, -0.105003767, 0.24485141, 0.152514249, 0.208566174, 0.162460268, 0.00807126984, -0.141904116, 0.108676672, 0.125443801, 0.036231447, 0.135343865, -0.187444642, 0.0880331844, 0.023205962, 0.00651972136, -0.00225225091, 0.183123365, -0.118129879, 0.130323112, 0.107369676, 0.211500779, -0.0843634605, -0.156388134, 0.207216874, -0.0687728524, 0.0857001096, 0.0248294771, -0.100912109, -0.157147497, 0.0598580688, 0.0957521722, 0.153322056, 0.0638879687, 0.0558222681, 0.13312462, 0.0504909046, 0.184043959, -0.147291183, -0.0967333466, -0.0938999057, 0.0367397517, 0.0814364702, -0.111346483, -0.120195106, -0.137015536, 0.00596247334, -0.127521366, -0.168997496, -0.0679924712, 0.0334541053, 0.0365803689, -0.0112984832, -0.0791522115, 0.165152445, -0.0490483344, 0.145707756, -0.203866005, -0.0773670673, 0.187672272, -0.124051414, 0.118377551, -0.152038693, 0.187986448, -0.178593695, -0.0927914903, 0.08069361, 0.205642715, -0.054671783, -0.0563890673, 0.062154606, 0.0556793362, -0.077488631, -0.237223327, -0.00743269641, 0.0303223412, 0.1891305, 0.115924723, 0.243285507, 0.128094137, 0.0924103409, -0.173196748, 0.186365053, -0.102543443, 0.0903031752, -0.0225095805, -0.0684509724, -0.0492378138, -0.142380729, 0.273817688, 0.162142336, 0.0942962393, -0.196417257, 0.0544637963, 0.0642177686, -0.0781479776, -0.00544341793, 0.0882533863, 0.135036305, 0.153385952, 0.060867317, 0.0675654262, -0.190924585, -0.0308644846, 0.209309757, 0.23535271, -0.114015281, 0.211691156, 0.103498377, 0.175216466, -0.0897360072, -0.178171828, 0.188865781, 0.184034958, 0.143535584, -0.0759150386, -0.144946337, 0.123703592, 0.072421141, -0.073435992, -0.120332345, -0.207936838, 0.0859730244, 0.089198038, 0.21525383, 0.042071078, -0.188023686, -0.222388178, 0.173431069, -0.0430555344, 0.15827693, 0.0902394876, 0.192961678, 0.073467873, -0.000299184467, -0.143207088, 0.194787577, -0.0937701017, 0.147017911, -0.167207763, 0.0221077409, -0.148127094, -0.0726192892, 0.0140165687, -0.131738737, -0.107379422, -0.0532393269, -0.183383986, -0.132864356, 0.14306511, 0.166543275, 0.0633267611, -0.00475004269, 0.159882694, 0.0209031757, 0.193773642, 0.0460488647, 0.00657480629, 0.135696039, -0.122650474, -0.0921338946, -0.0184501112, 0.197395191, 0.149274558, -0.212168857, -0.0961322784, -0.0972493216, 0.061156068, 0.0288367011, -0.129334092, -0.0287208185, -0.12547949, -0.109855622, 0.0713636428, -0.202687904, -0.0736791939, -0.170345217, 0.00483758748, -0.0566800907, -0.0133493776, 0.177170977, -0.16139634, 0.0383036919, 0.18136698, -0.0358033031, -0.158096969, 0.122688517, 0.081486389, 0.160581172, 0.210082605, 0.139138475, -0.0031660106, 0.0011371508, 0.153799191, -0.0630362555, -0.0959898457, -0.0677730069, 0.0763605982, -0.0591884851, -0.103758797, 0.0877787992, -0.203684002, -0.213626981, 0.216784999, 0.0821806788, 0.0854039118, -0.0622716844, 0.178851873, 0.0519754291, -0.102133691, -0.0585566014, 0.0188398492, 0.202151239, -0.104732491, 0.27045393, -0.0917108878, -0.208633393, 0.156232789, 0.231986329, 0.132011876, 0.000424101949, -0.220415235, 0.295938492, 0.0743808001, 0.14029865, 0.242455915, 0.23396118, -0.245414257, -0.195483923, -0.114712641, -0.0220132805, 0.322085798, -0.021815693, 0.282940984, 0.12972188, 0.131338835, 0.25256893, -0.182917267, -0.158058509, -0.129873797, 0.0281693563, -0.139118776, -0.060282778, -0.288214117, 0.18269442, 0.0694092885, 0.122847252, -0.0459760986, -0.18629986, -0.000292814599, 0.19988957, 0.157423139, 0.132337287, 0.124669015, 0.156890973, -0.164955139, -0.0223253407, 0.294166148, 0.301510572, 0.13682279, 0.0792005882, -0.100755952, 0.0107995598, 0.122480787, 0.0160061363, 0.146093562, 0.0933857411, -0.00256964564, 0.0729778558, -0.193990499, 0.00561368465, 0.168780282, -0.0343219191, -0.16398114, 0.19884105, -0.170096159, 0.0851236135, 0.046119079, 0.149938866, 0.106523618, 0.0622120649, 0.194288179, 0.153273478, 0.0731689781, 0.00548323989, 0.150967196, 0.0232321769, -0.163167983, 0.0613376349, 0.199462637, -0.0988652036, -0.202331737, -0.201972619, -0.0975645036, -0.103157334, -0.0671368837, 0.0251828581, -0.12365777, -0.0824821144, -0.0295259356, -0.200477883, 0.213229522, -0.126918197, -0.0524763167, -0.0709132403, 0.13771455, 0.182151392, 0.0844053477, 0.192415133, -0.0920736194, -0.0465842038, -0.146784067, -0.0747133791, 0.186533436, -0.201628059, 0.102212504, 0.176582918, 0.0926011056, -0.0415422022, -0.173487782, -0.145804495, 0.138758883, 0.215857342, 0.118435606, -0.183083788, -0.206599399, 0.0207605958, 0.0811169297, -0.150482222, -0.0474843644, 0.148732826, -0.0435940437, 0.168024451, -0.111467153, 0.138727993, 0.0159117766, -0.0708138347, -0.0325546637, -0.187760904, -0.0735307932, -0.0522092022, 0.207347527, -0.0800161883, 0.0155367013, -0.171100616, -0.15568769, 0.0280985534, 0.155661479, -0.0907097906, -0.0465506762, 0.0450913496, -0.167255431, 0.0276872609, -0.0394791812, -0.20365721, -0.135010064, -0.065793246, -0.15259999, -0.24566929, -0.254977822, -0.261519402, -0.123870581, -0.197444856, -0.12559481, 0.179250687, -0.00984245725, -0.0307493377, -0.0284540262, 0.0870079026, -0.101884559, 0.167557895, 0.16733788, 0.0386115685, -0.186165556, -0.0420892499, 0.132793337, -0.0517253689, 0.0506563708, 0.181324065, -0.230184272, 0.172225639, 0.0384657383, 0.201920986, 0.227207035, -0.140594408, 0.0149281584, 0.0272123087, 0.0511507243, 0.157599419, -0.12310376, 0.0275888201, -0.119697392, -0.133497775, 0.177538306, 0.287879407, -0.332083166, 0.174466282, -0.0631491616, -0.0642071292, 0.0698080435, -0.194340572, 0.174546167, 0.112725794, -0.130530342, 0.0916617587, -0.0443805419, -0.242965654, -0.259136677, 0.200497359, -0.16344808, -0.0397210233, 0.0303804427, 0.146784887, 0.15142341, 0.138190344, 0.246435046, 0.077768594, -0.080286853, -0.204465911, -0.0890383646, 0.0499912277, 0.106659219, 0.261487067, 0.16590409, 0.179442301, 0.140036687, 0.0401791185, 0.00325127738, 0.013187293, 0.0925546288, 0.07011462, 0.165935919, -0.256534755, 0.0718082935, 0.0792537257, 0.030161446, 0.242915824, -0.0511688851, -0.0652604699, -0.0842846036, 0.108259201, -0.128864169, -0.00321713765, -0.184777811, 0.0591468774, -0.107330173, -0.0423216075, 0.19637309, -0.107558452, -0.200378031, 0.0274944436, 0.047395166, -0.194123879, 0.188412562, 0.199617177, -0.141710162, 0.221462101, 0.209144309, -0.0284675043, -0.244087934, -0.183096975, -0.0241368171, -0.148103431, 0.177265957, 0.186891973, 0.0422130674, -0.344164699, -0.0773528889, 0.141355872, -0.373026252, 0.0433265753, -0.210413083, -0.148437619, -0.0495266616, -0.17753464, -0.1127683, -0.113730326, -0.156939805, -0.224368513, -0.104205146, -0.0880409703, -0.173214465, 0.0337923206, 0.300643057, 0.00617149146, 0.155847415, 0.126247868, -0.133445188, 0.015533735, -0.183959901, 0.0210792925, -0.192985684, -0.0331071578, 0.135724992, 0.211360231, 0.133701399, 0.0228303764, -0.05452976, 0.110739149, 0.183961943, 0.0661156029, -0.00822394434, -0.11427819, 0.245802104, 0.14801845, -0.0657031313, -0.236966819, -0.207826287, 0.0913634151, 0.0438724905, -0.18313092, 0.00411039777, -0.126928151, -0.211722925, 0.214022741, -0.128302187, 0.0836230144, 0.164736882, -0.112882853, -0.11854811, 0.19892104, -0.207083598, 0.0527174808, -0.0543283299, 0.103308566, -0.142663166, 0.112300202, -0.14731279, 0.0822475776, 0.0341244563, 0.0138530098, 0.073856324, -0.196735963, 0.154973254, 0.233334199, 0.0869767517, 0.116376385, -0.0416299328, 0.0994379148, 0.166396573, 0.16971387, -0.173807308, 0.213895455, -0.0528170429, 0.0617500283, 0.259949446, -0.0118162651, -0.234531507, 0.0625089556, 0.0717810541, -0.13730064, 0.239427283, 0.0305171944, 0.23850891, 0.2220653, 0.25341624, 0.171295524, -0.0135789579, -0.209433094, -0.0696900189, 0.0471944325, -0.138306618, 0.157414973, -0.149076745, -0.149825826, 0.0214383248, -0.118996307, 0.119986966, -0.0147008747, -0.237432435, -0.076058656, -0.0901724845, -0.132154062, 0.0539183468, -0.0170942433, 0.0179768484, 0.22421883, 0.0985278562, 0.228690475, 0.0216967724, -0.131215245, 0.135511026, 0.258222163, -0.0243793726, 0.123374104, 0.129674554, -0.0193014108, -0.143381625, -0.161064699, -0.172403276, -0.158084139, 0.0584857427, 0.0655151159, -0.160059884, -0.204120889, -0.0126833543, -0.0621461421, 0.142932773, -0.0626193658, 0.16576916, -0.15621151, 0.00211782986, 0.103418313, 0.0376950353, 0.0308611691, 0.0366130322, -0.139915824, -0.104231551, -0.207542226, -0.064083159, -0.145862356, 0.146586224, -0.0424620397, 0.186795101, -0.158907622, -0.110902712, 0.142597273, 0.0426524207, -0.011229001, 0.210712969, -0.0741818473, 0.086176455, 0.252430946, -0.123034984, 0.0468166359, -0.134075209, 0.0980751961, -0.0789282247, 0.148234606, 0.105269954, -0.168516472, -0.161657631, 0.0963762105, 0.163820669, 0.135545686, -0.079741396, -0.195735767, -0.077804029, 0.171317056, 0.126934454, -0.0572446063, -0.21873033, 0.21519053, 0.170210302, 0.124228232, -0.073779501, 0.176543459, -0.0158718117, 0.00454410026, -0.118912876, 0.162831694, -0.174594507, 0.0981904119, 0.188442662, 0.0812480599, -0.0692835823, -0.0890745521, 0.0326154418, 0.167388737, -0.03485322, 0.0143670244, 0.0791173428, 0.134169146, 0.0797807947, 0.14800404, -0.141179651, -0.016895188, 0.154919192, 0.00256294012, -0.192573935, 0.118427344, 0.107221924, 0.151232108, 0.210011765, 0.0565974601, 0.00145513611, 0.0219323114, -0.189139843, 0.06658151, 0.21069631, -0.0141648222, 0.0961672589, 0.19676432, 0.11270266, -0.092723079, 0.039994482, -0.0988364965, 0.186328426, 0.0684169978, 0.0352716595, 0.0923228562, -0.247896671, 0.0594582744, 0.215583935, 0.0443359576, 0.106910646, -0.09841194, 0.0154830469, 0.186022297, 0.122082792, 0.109951109, 0.178713337, 0.185618713, -0.00407085847, 0.14384532, 0.237962916, 0.0404084362, -0.162489235, 0.0169203728, 0.0621280223, -0.159193203, 0.120504037, 0.243941158, -0.153041452, -0.133457929, 0.290807456, -0.0554177649, -0.162622347, 0.186095059, 0.0159069337, 0.226315305, 0.192118213, 0.279498637, -0.1455594, -0.360007048, 0.156156048, 0.0351749025, 0.309243917, -0.00659387093, -0.0777715594, 0.212203711, 0.107820228, -0.191825479, -0.215385392, 0.145686373, 0.250261635, 0.132179976, 0.0784063116, 0.141661942, 0.0102276588, -0.28464517, -0.0189468563, -0.153701648, -0.150468856, -0.016683815, 0.133815899, 0.334772259, 0.0575955845, 0.042229306, -0.224532291, -0.0747981966, 0.0232652463, 0.25478974, -0.157321453, 0.133630514, 0.0333518349, -0.266530663, -0.0646840036, -0.172265172, -0.189026609, 0.0687507093, 0.00638828939, 0.319402933, 0.122809738, -0.0131080216, 0.135142997, 0.102929942, -0.202861682, 0.0329007581, 0.00744347926, -0.21400103, -0.316629291, -0.374617159, -0.319015384, 0.384847909, -0.186712921, 0.0658086613, 0.032412149, 0.0714035854, -0.255016744, 0.0262498483, 0.0766730756, 0.138087109, -0.0706778392, 0.0776452422, 0.0143215396, 0.00803621765, 0.152218983, -0.0326965526, -0.233084202, -0.0957412347, -0.182263479, 0.161254615, -0.130365536, 0.0748982504, -0.149099216, -0.215250716, -0.117837511, 0.0308287051, -0.167285755, 0.142437562, -0.0721527189, -0.0916155428, 0.218848243, 0.0761095062, -0.175035179, 0.103456758, 0.20379065, 0.225135043, 0.158203647, -0.142868116, -0.173013821, -0.00321286987, -0.0699528158, 0.107067905, 0.197857693, 0.181346416, -0.133046284, 0.0340469182, -0.0929345265, 0.0420503095, 0.0250554103, 0.184311718, 0.174113616, 0.220722213, 0.00232743588, -0.150735736, 0.0382508636, -0.129761532, -0.130726188, 0.119928777, 0.0578796864, 0.0282058474, 0.0902101099, 0.0399041548, -0.155804977, -0.120978624, 0.249803692, 0.0158650391, 0.0688268542, 0.134503469, -0.288924664, 0.176216707, 0.00563906645, 0.102420114, -0.0788406879, 0.213966206, -0.154680684, 0.0656312183, 0.0721544251, 0.173323125, -0.147119582, 0.0787703097, 0.0888866857, -0.0924119502, -0.0353752673, -0.0151055222, 0.0759745687, 0.280328214, -0.129063725, -0.0747397095, -0.203125596, 0.227080092, -0.206261814, 0.119735092, 0.0916555002, -0.0724879056, -0.155287698, 0.0132731264, 0.212116286, 0.0839198157, 0.114934556, 0.160972327, 0.185490161, 0.182898089, -0.15434128, -0.0223024506, 0.0369399376, -0.242618233, -0.04812406, 0.124690734, 0.0266579203, 0.0357043222, -0.0241595097, -0.170285985, 0.198587388, 0.153542444, -0.0928277895, -0.0493879616, 0.0720407665, -0.0875376537, 0.0800556913, -0.106703565, -0.188763604, 0.1804066, 0.190824226, 0.139410958, 0.134015784, 0.0551224127, -0.0588871315, -0.172435537, 0.120842956, 0.102679841, -0.0483263209, -0.0404443517, -0.0905011818, 0.00734967226, -0.175017715, 0.253821075, 0.107986726, -0.0605778471, -0.127831027, -0.0520662367, -0.15249005, 0.0787140727, 0.177878886, 0.0623937584, -0.0510694347, 0.162456274, 0.0961652696, 0.156488523, -0.0103794681, 0.298527658, 0.117508285, 0.00845222175, 0.00402975967, 0.244920164, -0.262802303, 0.239384681, 0.194349378, -0.0255465209, -0.0071021365, 0.0496552289, 0.189110205, -0.0734819695, -0.0138057666, 0.22511366, -0.024540307, 0.0501983725, -0.130734563, 0.261949658, -0.129572645, 0.0852468386, -0.195301205, -0.128256202, -0.146074802, 0.114428394, -0.109575629, -0.171998858, 0.1805114, -0.0983749181, 0.168353647, 0.00222684909, 0.107877977, -0.133522928, 0.0821961313, 0.055921942, -0.189155638, -0.211974889, 0.035456989, -0.03801715, 0.151340604, 0.0116558271, 0.0453454293, -0.138027087, 0.165734008, 0.0903293639, -0.17851457, -0.181823134, 0.105536416, -0.00437751412, -0.0242398828, -0.197221443, -0.169698417, 0.00265513361, 0.119570628, -0.0556186885, -0.179043248, 0.0923377424, 0.0260195583, 0.142739668, -0.0102109313, -0.0621111393, 0.207488343, 0.0741483122, 0.158786342, -0.101714008, -0.185144261, 0.16310133, 0.0921799093, 0.0151199698, 0.0675591677, 0.0690498203, 0.0627175122, -0.156824663, -0.0990713686, 0.0945287794, -0.0230718404, -0.0956377164, -0.203232855, 0.193041012, -0.171600953, 0.00985047221, -0.0484160632, 0.0128556937, -0.0141810179, 0.199574545, 0.0574304312, -0.0120507926, -0.10293258, 0.171099111, 0.0624095947, 0.127719328, 0.0310608298, -0.127090856, -0.135603577, -0.0402774811, -0.00777311623, -0.0236091018, 0.115270123, -0.0440471768, -0.0969943702, -0.0702738315, 0.00185018778, -0.135444164, 0.138630465, 0.206673846, 0.0269248039, -0.194600731, -0.108348511, 0.100241527, 0.204216614, 0.0310706943, 0.0207177736, 0.0246665124, -0.0369903184, 0.189978585, 0.18308571, 0.0601348951, 0.165929869, -0.0339035504, -0.0099209277, 0.190639094, -0.13286522, -0.00495153386, -0.0395436101, -0.138987705, 0.176830545, 0.00814937707, 0.252283871, 0.218431175, -0.0865562707, 0.0898508579, -0.0586666316, 0.155118331, 0.0155698694, 0.178617969, 0.0938429683, 0.0607920587, -0.209286168, -0.142663464, -0.104432322, -0.207258865, 0.128569424, -0.0403374508, 0.0755493268, -0.123791821, 0.166542724, 0.103759401, -0.260609299, 0.0588776469, 0.163806662, 0.00261614448, -0.00516588986, 0.0550476126, -0.34296912, -0.12214759, 0.163169816, 0.0452847183, 0.178035349, -0.0292446893, 0.00157334586, -0.143873423, 0.129343823, 0.214960068, -0.062136814, -0.0185418073, 0.185974956, 0.050098747, 0.20793201, 0.228919804, -0.174892411, 0.0396745056, -0.129953608, 0.206800371, -0.000112072892, -0.138918951, 0.0954689011, 0.255405635, -0.118499793, -0.175630018, 0.123674139, 0.0513064191, 0.236296624, 0.0593134351, 0.0739371106, -0.0461705178, -0.106488623, 0.128243804, -0.229913831, 0.103818499, -0.208989188, 0.0269889422, -0.0170714278, 0.172011673, -0.00835058093, 0.083449766, -0.153386265, -0.206975192, -0.0904331207, -0.100907929, 0.0201056469, 0.0092816418, 0.138591155, 0.123229094, -0.204459578, 0.125524312, -0.198420554, 0.136316523, 0.0642325506, -0.111182407, -0.292572588, -0.0476938225, 0.25313285, 0.0092351269, -0.0328827761, -0.112535074, -0.0818377212, 0.143190131, 0.162059993, 0.0104096029, -0.0401865542, 0.072995171, 0.204331324, 0.0964775011, 0.0549218319, -0.26574558, -0.149334505, -0.219716296, 0.0813605562, -0.102174677, 0.165653527, -0.23237288, 0.0617746599, 0.219712645, -0.245772511, 0.0843116418, -0.0313958414, -0.0511075445, -0.202375591, -0.0243414436, 0.0134311467, -0.184688628, 0.0857788771, -0.0375306755, -0.212528273, 0.0812165588, -0.14801389, 0.103163257, 0.124996766, -0.112198733, -0.214695185, 0.196181044, 0.0699417144, -0.214553803, -0.158492222, -0.173867494, -0.040612489, -0.0375947803, 0.060765788, -0.0616895109, -0.0461635143, 0.215136424, -0.158336386, 0.0892048329, 0.0994321257, 0.113832906, 0.20994629, 0.0749067515, 0.0561294109, -0.0114479363, -0.117390744, -0.0267652422, -0.152938411, 0.13877742, 0.104254767, -0.169561014, 0.180426642, 0.111701086, -0.00645264983, 0.125381544, -0.147052184, 0.153655097, -0.0217939615, -0.0914004594, -0.178690523, 0.178770587, -0.0424079597, 0.024468869, 0.0716981441, -0.119676486, -0.0311208218, -0.0731271207, -0.103556246, 0.0954664797, 0.0873899013, -0.0905441493, -0.144235373, -0.0789919347, -0.10910587, -0.0982930511, -0.0370353907, 0.189428493, 0.00647680461, -0.0638864785, 0.212589487, -0.161814377, 0.0216575265, -0.0850141943, 0.194710687, -0.178992704, 0.125666514, -0.192258149, -0.193372041, 0.20426394, 0.118718341, 0.100960627, 0.0680707842, 0.0463458747, 0.165338323, -0.0671609789, 0.168787971, -0.0070540607, -0.202503204, -0.0853080601, 0.211600348, -0.122439608, -0.147218913, 0.199023679, 0.120119318, -0.0956019461, -0.122479819, 0.0545401126, 0.214297399, 0.0260116011, 0.117337689, -0.182416037, -0.0304358751, -0.194916844, -0.0680961162, 0.0540857166, 0.176674083, -0.0712954253, -0.00287421048, 0.0383953899, 0.0185558945, 0.112168685, -0.180515826, -0.112304345, -0.0206410438, 0.0596600622, 0.0638618618, -0.148700684, -0.181752264, -0.206867248, 0.142111555, -0.0103422552, 0.16394259, 0.199925497, 0.208245948, -0.125069648, 0.0724749714, 0.132800862, 0.131532744, 0.122560248, 0.0359630138, 0.0514701158, -0.00991392136, 0.16258727, -0.102539249, 0.131538868, 0.000688975444, 0.210872754, -0.0939219445, -0.155480877, -0.0926667899, 0.150634632, -0.125974014, -0.0297515579, 0.0463272557, 0.0345584452, -0.159411788, -0.00879441015, 0.0906654373, -0.222819507, 0.300452858, 0.24445796, -0.220637038, -0.073617816, 0.0579014607, 0.160616696, -0.179756835, -0.0254850835, -0.136787683, 0.0766259208, 0.120203525, 0.149309546, 0.168427154, -0.0670610815, -0.104210295, -0.112162739, -0.101194017, 0.124157779, 0.121481434, 0.176228672, 0.172684014, -0.166508585, 0.0264002513, 0.0834020749, -0.182705998, 0.112678163, -0.0141648045, 0.00864631962, -0.135217071, 0.139958009, -0.111488022, -0.0717050955, -0.21887809, -0.0830352902, 0.106444001, 0.194088787, 0.0767873973, -0.150106505, -0.0719411075, 0.0724190921, 0.292881131, -0.0399664752, 0.243576974, 0.117913261, 0.246021658, 0.0811332464, -0.0399341844, -0.0816165209, 0.171891883, 0.082011655, 0.0575862974, -0.109388068, -0.163562402, 0.170695201, -0.162173331, -0.134208307, 0.158017829, 0.163954869, -0.198981807, 0.133076355, 0.174984023, 0.0209734291, -0.135800138, 0.167734668, 0.190667316, 0.203086928, 0.146870956, 0.0645530969, 0.113435879, -0.187958598, 0.147743359, 0.0670311004, -0.187562466, -0.0608942211, -0.0351307988, -0.058291018, -0.129617661, -0.0873317271, 0.0594988018, -0.211554736, -0.0564201325, -0.128696471, -0.0596370399, -0.181903094, -0.153074175, 0.0677614063, -0.08287628, 0.113757566, -0.153864205, -0.00586368144, -0.216033623, 0.0404614061, -0.214554414, 0.100273564, 0.139342979, 0.0685483068, 0.129975602, -0.173656166, -0.0469692796, 0.135614976, 0.188055262, 0.127508983, 0.0973801762, 0.116156682, 0.0537556559, -0.0190902501, 0.0643442422, -0.176481023, -0.0268422067, 0.170466408, -0.0452373028, 0.0346771628, -0.0764650702, -0.161790356, -0.169284806, -0.160289347, -0.0043374598, 0.0272316784, -0.0586752929, 0.0605526119, -0.175261557, 0.159667954, -0.139275417, 0.187538177, 0.0448392779, 0.0851275474, -0.0254395697, -0.168208286, 0.205435231, 0.0792442113, -0.167214826, -0.162651837, 0.0390271097, -0.0277169496, -0.0349142514, 0.122520849, -0.129117578, 0.116114929, -0.0394956619, -0.131158963, 0.0104077011, -0.183592737, -0.0942491591, 0.0787120685, 0.0059645921, 0.083924517, -0.00701065361, -0.118871383, 0.140056029, 0.211868882, 0.0615758449, 0.00838501751, -0.000891566277, 0.0594077855, 0.146011487, -0.0805511698, -0.193798214, -0.186887994, -0.089735806, -0.180153847, -0.0625011772, -0.123947091, 0.194204822, 0.00806425512, -0.116187446, 0.0269125104, -0.0904725119, 0.011333555, -0.0565276444, -0.166684598, -0.17863436, -0.184847683, 0.206926495, 0.199473783, 0.028638497, 0.0610053949, -0.209566385, -0.149408638, 0.0373195261, 0.06447687, -0.126612946, 0.28914547, -0.0355662853, 0.0583788455, -0.2373074, 0.221651822, 0.175030649, -0.0361175053, 0.154063821, 0.242598936, 0.178581849, 0.13535817, 0.0564856976, -0.0409523547, 0.106473468, -0.0620523989, 0.146483317, 0.0771263912, -0.165507808, -0.0569170639, 0.214328185, -0.0147469528, 0.146464691, -0.0852415189, -0.0795736313, 0.0171650928, 0.262713403, -0.0182778351, -0.125869542, 0.218170211, 0.08039435, 0.166997373, -0.0870893747, -0.104434751, 0.135473803, 0.0149303246, -0.0789194182, 0.279207557, -0.232716322, 0.0479517728, 0.111858115, -0.0409652069, 0.120025121, 0.0328806192, -0.234696463, 0.109781213, 0.242693588, 0.263724536, -0.209186554, -0.0229675435, -0.177582771, -0.134655267, 0.301631212, 0.173010796, 0.277582735, 0.0801606327, 0.115403861, 0.258175075, -0.203490555, -0.169273093, 0.197581336, 0.233946189, 0.188818827, -0.110022955, -0.0721238554, -0.127027333, -0.0361180678, -0.182209134, -0.0469776765, 0.0636565313, -0.125594214, 0.112164833, -0.153257549, -0.0699059218, 0.0906096771, -0.156303734, 0.163650781, -0.120070562, -0.187784672, -0.110630184, -0.0369865112, -0.221759483, 0.265062481, -0.0200742166, -0.0210180636, -0.0318562686, 0.289968342, 0.209271714, -0.163250521, -0.033234816, -0.158912554, -0.15139316, -0.161861673, -0.182225049, 0.0245842095, 0.0447209552, -0.133103281, 0.0522985011, -0.140202329, -0.0881955624, 0.0748139471, 0.14398168, 0.229476035, -0.100793242, -0.0547418669, 0.254428893, -0.0232664496, -0.0325468257, -0.118670925, 0.167250693, -0.220140129, -0.0891620591, -0.0795891732, 0.125988051, 0.360238761, -0.187357172, 0.164008111, -0.184598282, -0.250819564, -0.0614155643, -0.213410959, 0.0295955334, -0.188740283, 0.165933087, 0.14575623, -0.169412017, 0.0403924398, 0.0863903165, 0.125428617, -0.122938238, 0.203624532, 0.0290758889, -0.194397897, -0.0813511461, 0.136541203, -0.168952912, -0.118765511, 0.07683599, -0.129231229, -0.0414971858, -0.0406129733, 0.101526216, -0.0764528364, 0.131897673, 0.0560044497, -0.0730934143, 0.0276858192, 0.173554912, 0.00495803775, -0.0322014466, -0.0102797113, 0.213982448, -0.0208447874, -0.107821919, -0.0264427457, 0.0145503255, 0.019508658, 0.0594968982, -0.0592152774, 0.121941999, 0.122733139, -0.140440956, -0.176466525, -0.0972242281, 0.0811412483, -0.212435484, -0.107308395, -0.0842584148, 0.0197450221, 0.215222329, 0.17154865, -0.0421809405, -0.0426143073, 0.156440645, -0.123030953, -0.0165297743, 0.086967513, 0.130930915, 0.192302629, 0.108801588, 0.189616874, 0.134053215, -0.100600176, -0.105523147, 0.0837425441, 0.176915631, -0.0862870663, -0.128423661, -0.185953289, 0.162213311, 0.238823578, -0.0322427824, -0.172987208, 0.0383077003, -0.168837801, -0.0999560133, -0.140007496, -0.13302283, 0.0654487237, -0.054558441, 0.00409579836, -0.0385583751, 0.0616787598, 0.0229705647, 0.174310103, 0.220073834, -0.228525922, 0.20903562, -0.12730284, 0.266811848, -0.0645477623, 0.12383756, -0.11437133, -0.110793918, -0.0366560929, -0.113584034, 0.0970615298, -0.0828079358, 0.186074406, 0.16188024, -0.0919989794, -0.0214854963, 0.209291995, 0.132674858, -0.158335567, 0.129601404, -0.043703422, -0.0580179356, -0.122194469, 0.0626526251, 0.0995965749, 0.125470623, -0.173571438, -7.04564809e-05, 0.0105728703, -0.142664522, -0.0462249145, 0.0775359049, -0.0809029341, -0.13692227, -0.0882295668, 0.0266289487, 0.0734391138, 0.0406049676, 0.192088261, -0.0451808535, -0.0661438555, 0.120225728, 0.151128128, -0.10713999, -0.0322566256, -0.134458154, 0.0705581233, -0.200856641, -0.113959946, 0.161113799, -0.181794733, 0.15956901, 0.160805613, -0.186158001, -0.0237688925, 0.127835721, -0.0186184216, 0.101857841, 0.197322085, 0.125265792, -0.01271844, -0.171266645, 0.0350334905, -0.108482718, -0.214593604, 0.172298625, -0.182126477, 0.161291301, 0.146099284, 0.103996262, 0.0945375413, -0.212611616, -0.150450736, 0.155232683, -0.0679181367, -0.155561522, -0.0921959952, 0.0946691111, -0.127165928, -0.122972131, -0.186263174, -0.139322162, 0.242685571, 0.0045821243, 0.011791165, -0.0878160745, -0.159043938, 0.0593511797, -0.167231545, 0.23195985, -2.63589227e-05, -0.150773689, 0.0332254022, -0.115814731, -0.191897079, 0.104204178, -0.0777447969, 0.17065756, -0.217323199, 0.114431463, 0.069135122, -0.0210048091, 0.00420680922, -0.0845233724, 0.0959770456, 0.0833298042, 0.0301761869, 0.0593393333, -0.158845872, 0.0165265705, 0.0481217168, -0.00209004036, 0.138400525, 0.1577003, -0.206650645, -0.140175536, 0.139429837, 0.0434673727, -0.00637131557, -0.150466055, 0.0634823367, -0.122112915, -0.115015678, 0.0883953124, 0.213094011, -0.128786102, 0.10067419, 0.269909352, -0.0107553555, -0.135354757, -0.217162892, 0.0356924273, -0.0991727114, 0.132911071, -0.0588454865, 0.243446231, -0.254837215, -0.0441369563, 0.0588260442, 0.174045861, 0.0421890616, -0.0813888386, 0.280730367, 0.255607665, 0.208496362, 0.256909579, 0.0790268704, -0.118365906, -0.21108976, -0.135365918, -0.191761851, 0.147386804, -0.238638878, 0.0442762636, -0.106006496, 0.0480982736, -0.262756944, -0.083258003, -0.210455641, 0.221321031, 0.214391738, 0.140733302, 0.168415472, 0.177380338, -0.0998223275, 0.0802876726, 0.024429664, 0.23944816, -0.0581545308, 0.213931069, 0.196635291, -0.0161537938, -0.0103867967, -0.126716629, -0.083251968, -0.0781524554, -0.0834515467, 0.0193810612, -0.186825454, -0.128707543, 0.204980001, -0.00399512053, -0.101887874, 0.0210454538, -0.0412895195, -0.0971676558, -0.048628062, -0.20430325, -0.197556436, -0.190492779, 0.0837618262, 0.125030011, -0.0541782528, 0.146718219, -0.150529712, 0.113789588, 0.159004748, -0.00630572857, -0.206578702, 0.167073652, -0.0800563917, -0.0184968971, -0.132193252, 0.15642193, -0.146631718, -0.0564464815, 0.0205936134, 0.215904519, -0.170073912, 0.0835290179, 0.00320865051, 0.0229984596, -0.114689462, 0.171532705, -0.0459926128, 0.057841301, -0.0879666209, -0.0287654698, -0.144966319, 0.105421446, -0.0273225829, 0.0585521348, -0.101430416, 0.131310791, -0.0334190056, 0.184861079, 0.0362242311, 0.205380991, 0.0049544517, -0.0775810778, -0.21244362, 0.0842021108, 0.0351231582, -0.181801394, -0.0861293525, 0.0863052607, -0.0654114634, 0.0168641414, -0.0446151756, 0.247980848, -0.122818522, 0.182896554, 0.0511074699, 0.0474656112, -0.133897036, -0.157300696, 0.131089389, 0.00570026645, 0.156846672, 0.0670417845, -0.074737817, 0.179072648, 0.139402583, 0.209800005, 0.0514971539, -0.157501861, -0.137726873, 0.0395912975, 0.0381566659, -0.0413452275, 0.046529077, 0.195759162, -0.0611983314, 0.0869912729, 0.16404058, 0.197312593, -0.185774952, 0.172979549, 0.269182414, 0.0887734294, 0.205442265, 0.01246008, -0.211092308, 0.227946341, -0.0107464157, 0.245333567, -0.048793897, -0.0402365625, 0.0947469473, 0.0884542614, -0.0422119237, 0.165364295, 0.0160138234, -0.0176507104, -0.178265303, 0.0195886772, -0.0455894843, -0.0993135348, 0.0292526782, -0.0872291252, -0.194193006, -0.204600781, 0.144727439, -0.265376478, 0.262558103, 0.0440654457, 0.00297656655, 0.124401599, 0.256192356, 0.140282795, 0.181511864, 0.127582431, -0.0810992941, 0.00457523856, 0.194761962, -0.0414959528, 0.0110664666, -0.0478526093, 0.218107626, -0.097522147, 0.0221662484, 0.0307420697, 0.00897521432, 0.0723016262, 0.156312093, 0.0830891505, -0.102879122, -0.220429748, 0.111000456, 0.0493231416, -0.167957768, -0.200361371, -0.220628932, 0.0213064477, -0.13790077, 0.16264008, 0.0366902873, 0.0662807301, 0.0843776241, -0.00975239743, -0.187409461, -0.00850835908, 0.214093223, -0.0262640547, -0.0037057586, 0.261299968, -0.0119852293, 0.0840612352, -0.140529484, 0.086045213, -0.178673238, -0.101949222, -0.0606811792, 0.2623505, -0.159947217, -0.152141213, -0.0400353037, 0.0315761305, 0.1173632, 0.117560208, -0.0394015647, 0.194363236, 0.0334627554, 0.122356705, 0.0350546427, 0.0978516936, -0.236527696, 0.205010638, 0.248273745, -0.0951982066, 0.0346223675, 0.07659439, 0.0673788562, -0.0866984576, 0.0852876976, -0.069079563, 0.019739734, -0.0612785369, -0.103156194, -0.131891444, 0.194864705, -0.194438815, -0.132523477, -0.202051356, 0.0380129889, 0.137692869, -0.100640491, -0.0755962133, -0.12461704, 0.0515572987, 0.132496744, -0.0181591716, -0.146472231, -0.118328683, -0.168681785, 0.0452108234, -0.196983844, -0.133911699, -0.107775599, 0.0720314309, 0.139389187, -0.127528727, -0.114843562, 0.140681937, -0.208352178, 0.0613223463, -0.0877515376, 0.0889104754, -0.122407876, 0.0725748539, 0.0339392349, 0.0478396267, -0.198128894, 0.0607758276, -0.0642398596, 0.119521871, 0.206692919, -0.0587804914, 0.205643147, 0.108449683, -0.100034304, -0.158070832, 0.116327606, 0.0159044266, -0.102844685, -0.0278574713, 0.160228476, -0.175503105, 0.194432482, -0.192663267, -0.0688776821, 0.20138903, 0.11521215, 0.0320747495, 0.0258750096, 0.182264447, 0.0569877252, -0.0823236406, -0.0462619513, 0.106567733, -0.0499362051, 0.0560031161, -0.00147831102, 0.215228215, 0.102208264, 0.22965087, -0.0239753295, 0.095687367, -0.0616672896, 0.0587593913, 0.151922241, 0.0286311377, 0.0363215096, 0.115954399, -0.0627551451, -0.0331935957, -0.0891616046, 0.0451479107, 0.0505939499, -0.201272562, -0.0867501497, 0.152432233, -0.234590366, 0.142962754, -0.0309544504, 0.0265288632, -0.107768282, 0.0372548141, -0.185375005, 0.0994121656, 0.146933943, -0.0775678679, 0.136601061, 0.116011761, 0.162975177, -0.133521244, 0.0610307641, -0.172060072, -0.175027579, -0.0902606323, -0.119711854, 0.00174348196, -0.080424875, -0.0717453212, 0.0530059896, 0.142690092, -0.2024865, 0.0607569851, 0.0632190183, -0.0805430338, 0.0256457161, 0.202368066, -0.182796001, -0.22332494, -0.173913211, -0.0483726896, 0.130500004, 0.14105849, -0.0087418789, 0.0575943477, -0.0352024697, -0.0449910536, 0.0370082781, 0.0126874121, -0.143768162, 0.0430835038, 0.0192103907, 0.214269981, 0.121653453, -0.171620205, -0.115121514, 0.0637972057, -0.150997698, 0.138255328, 0.0768500865, 0.0764330328, 0.205035627, -0.203529269, 0.144700333, -0.134389654, 0.208693668, 0.0657688901, -0.068395406, -0.0664896816, -0.113522142, -0.0315324329, -0.0550373867, -0.0346781798, -0.145656422, 0.0172823854, -0.0111174863, -0.157122552, -0.190427795, -0.0916103199, -0.00143183256, 0.0899138302, 0.136021599, -0.198203564, 0.174707979, -0.0790932477, 0.134556785, 0.0119398087, -0.0647746325, -0.0214638021, -0.0843484104, -0.112631276, -0.0474717468, 0.0715068504, -0.0579168312, -0.0775391087, -0.0880511031, 0.0911753923, 0.0051047653, -0.150063142, -0.0598085932, 0.0396242812, -0.0492532253, -0.091608271, 0.150526419, -0.0564503483, 0.0292801782, -0.0795698985, 0.0905861259, 0.154940531, -0.0895984471, -0.158532158, -0.0644570738, -0.0941605195, 0.0961572528, 0.27700609, 0.0923415422, 0.157652989, 0.0674565509, -0.0285261758, 0.0780545026, -0.150813326, -0.078189984, 0.0764895827, 0.140417024, 0.176455826, -0.0467667431, -0.0611154847, -0.135509744, 0.0651874691, 0.00128756708, -0.13219206, 0.0725255162, 0.0488932282, -0.211957008, -0.241675302, -0.0976792723, 0.079120189, -0.0794882551, 0.0674599707, 0.306206286, 0.167326748, -0.0135372728, 0.256001234, -0.222973049, -0.0457991101, 0.0760016367, 0.174197108, -0.0268575419, 0.0531892926, -0.0637947321, 0.199966535, 0.0592058152, -0.166631758, -0.0820748508, 0.044286795, -0.0869615451, -0.0670766756, -0.0154077159, 0.168325067, 0.0498711281, -0.0202831142, 0.178866312, -0.253515154, 0.122428641, -0.0470641106, -0.180592746, -0.193016753, 0.198658079, -0.0529388189, 0.108853698, 0.0329008251, -0.172148854, 0.155390486, 0.223928601, -0.105937399, -0.109959118, 0.256064564, -0.107306272, -0.119646482, 0.0797421783, 0.0929884836, 0.0979342908, 0.133596629, -0.0257349536, -0.198378071, -0.109671965, -0.140990347, 0.0564259849, -0.00328065758, 0.0223205835, -0.111956462, 0.100838266, -0.118380174, -0.106406175, 0.13367115, 0.140827075, 0.149365082, -0.034094438, -0.0994511619, -0.202903464, -0.102243468, 0.216089889, -0.167881742, -0.185640097, -0.163032368, 0.0955848545, 0.196899727, 0.198177576, 0.189767465, -0.125597715, -0.0851550102, -0.012896874, -0.0585481524, -0.12292812, 0.161586598, -0.10934332, 0.0761391968, 0.00712056924, 0.0470088422, -0.0579094887, -0.00209463271, 0.0494624302, -0.00159580936, 0.126086533, -0.029434476, -0.0511376858, 0.0322339237, 0.0604848899, 0.217367649, -0.157550901, -0.1742405, 0.00597815914, -0.181396201, -0.0200733002, 0.0123654017, 0.212862641, -0.0284591522, -0.0449727364, 0.168478563, -0.0509453565, 0.112934813, -0.0566788465, 0.176471725, 0.0360399634, -0.0752981752, -0.146713302, 0.115039334, -0.128386751, -0.0662233233, -0.046212554, -0.0662843436, -0.126971036, 0.116823152, 0.191384241, -0.0919323936, -0.0727686882, -0.173104316, -0.0298395753, -0.131576031, 0.145610556, -0.016514197, 0.089529559, -0.1694635, 0.0887180716, 0.0909219533, 0.206983224, -0.128153592, -0.175801769, 0.156361684, -0.141585872, -0.0933236778, -0.0274668038, 0.200519279, 0.16725488, 0.0719681829, -0.0101237446, -0.189104065, 0.203866377, -0.140116215, 0.168043867, -0.0233105272, -0.202382937, 0.13448818, -0.0404603183, 0.0488183945, -0.0125396252, 0.0655785948, -0.0455810428, -0.131461859, 0.0987256318, -0.0785749108, 0.0762815624, 0.0706483275, -0.182909623, 0.204016224, -0.0563442409, -0.161886901, -0.204789057, -0.0380925536, 0.149280533, 0.186354056, -0.142447859, -0.190923437, 0.0317074656, -0.195126057, 0.0115836412, -0.0849219933, -0.00952991843, 0.0764236376, 0.0596605688, 0.120444655, 0.184710845, 0.0115267038, 0.127696022, -0.146930456, 0.169530034, 0.0189637188, -0.021946907, -0.0109692765, 0.0416838974, -0.00754594803, 0.0580874756, 0.0444080979, 0.184013709, 0.104757175, -0.0313890278, -0.100590184, 0.128223568, -0.20617266, -0.132255659, -0.0874492675, -0.143805087, -0.0500562638, -0.205596805, 0.148389444, 0.00172358123, -0.106911823, 0.0452977568, -0.21107322, 0.0668992624, 0.122114658, 0.0477002077, 0.120604172, -0.188552618, -0.138453364, -0.0456057191, 0.115633465, 0.165090904, 0.0320103727, 0.0575927421, 0.177304104, 0.0367988423, -0.212701097, 0.195212469, -0.194699734, 0.0594319105, 0.0195149295, -0.210422724, 0.18505533, 0.156053185, -0.0448524803, 0.123860724, 0.0762408525, -0.191941276, 0.113714948, 0.0830711722, -0.162165016, -0.0373560488, -0.118707739, -0.10479752, -0.182017535, -0.151235938, 0.0206096731, 0.145007297, -0.0153894899, 0.218414783, -0.000869259238, 0.0154756503, -0.200680226, 0.170030713, 0.0636367649, -0.172657162, 0.0794806182, 0.150627524, -0.102580756, -0.0683144256, -0.0945177898, 0.102912441, 0.169210717, -0.120361015, 0.194299057, -0.188841209, 0.146587253, -0.188844159, -0.0558344238, 0.0359239876, 0.053900253, 0.0142748058, -0.0113670798, -0.111485705, 0.0116025666, -0.215477005, -0.0928430185, 0.115675338, -0.102832057, 0.168732792, -0.126997501, -0.221014336, 0.182971597, -0.152135015, -0.0638246462, 0.180992663, -0.0825914219, -0.200327739, 0.186104283, -0.0761064738, 0.0455469042, 0.175332025, -0.0451734737, -0.172262177, 0.0572228953, -0.168096662, 0.204400107, 0.00175916846, -0.05636115, -0.163206309, 0.0695815533, 0.0637750551, 0.179285645, 0.018083917, -0.0526664667, 0.0717682764, -0.16865924, -0.150882706, -0.0112172551, -0.11952614, 0.0920963809, -0.115396291, -0.150909141, -0.179976657, -0.0421908833, -0.163812667, 0.122877382, -0.0942356437, 0.0453507863, -0.11259599, -0.0999261439, -0.100916177, -0.182669953, 0.154555917, -0.184113041, 0.0896566585, 0.145971134, 0.197596744, -0.0454761721, -0.150642499, 0.159919247, -0.143244132, 0.0210799035, -0.0441629775, -0.0810907111, -0.163442492, 0.045595862, 0.16091612, 0.106087513, 0.0664898232, -0.135403961, -0.0642762035, -0.174812168, -0.0309586972, -0.0548433885, -0.207458809, 0.172602981, 0.0843047872, 0.00955646299, 0.190302178, -0.0120949578, -0.152737558, 0.231507719, -0.0443149954, 0.0997370183, 0.133509561, -0.15396592, -0.129581988, -0.182943463, -0.169034809, 0.0301441699, 0.0955079123, -0.255378693, 0.0398402438, -0.0638692528, 0.154308721, 0.0580761209, -0.0793571323, -0.0826579779, 0.0314475968, 0.219111726, 0.0478798449, 0.0276127569, -0.00546862464, 0.0695564821, -0.131611675, 0.202782288, 0.183789968, -0.0195452888, -0.13255091, -0.0230764579, 0.111142918, -0.0910572112, 0.056702368, 0.14888303, -0.0929223374, -0.178360641, 0.164307311, -0.0853743032, -0.0649680644, 0.0779206306, -0.119389273, 0.230036467, -0.0436925627, 0.137377337, 0.0679846555, 0.0158325471, -0.0744110644, -0.222410843, -0.168998629, 0.0108635696, 0.183892742, 0.160881788, -0.0410534963, 0.05518483, -0.0880163535, -0.0370547585, -0.00287609058, -0.0478597283, -0.199008241, 0.146402642, 0.171959668, 0.290840656, -0.112652093, 0.105188161, -0.0585999079, -0.0022179212, -0.270577133, -0.0842458159, 0.184451506, -0.133775994, 0.244962484, -0.0110368654, -0.202473283, 0.0172045603, 0.145742238, 0.0488118939, -0.0988596231, 0.151816502, 0.0309539363, -0.0803498104, 0.237187728, 0.137721777, 0.0540012866, -0.00746989995, 0.0480698049, 0.150505424, 0.183417454, 0.0880424529, -0.0611262359, 0.0990205705, 0.155396596, 0.0898856223, -0.0296041518, -0.034501303, -0.0609594285, -0.104777358, -0.0443655364, -0.159524351, -0.0758568123, -0.149849355, -0.107333899, 0.0991479903, -0.122835763, -0.109809339, -0.114645869, 0.194594607, 0.0984508544, 0.23515442, -0.000617691898, -0.128364742, 0.199048966, -0.0401824042, -0.0760140866, -0.11002256, 0.0939248428, -0.05619229, 0.122873552, 0.268885493, 0.103352867, -0.105801336, 0.0070370757, 0.106131047, -0.0532236435, 0.0677729547, -0.123542935, 0.222401768, 0.124410555, 0.181627676, -0.0229594037, -0.138093278, 0.107260153, 0.0116578275, -0.0297462214, 0.1843528, 0.051715672, 0.109194115, -0.0787402317, -0.00220843637, -0.0251405481, -0.121136881, -0.0643095151, 0.203086615, -0.0400864892, 0.0907601193, -0.144587412, -0.0898020267, -0.098853603, -0.0770658627, -0.287551373, -0.0851627141, 0.0827269629, -0.0861964077, 0.0113888374, -0.0776093453, 0.0809763595, 0.0635781661, 0.00109870185, 0.216651306, 0.0141436849, -0.12719737, 0.0942884311, 0.303492576, 0.0959326848, 0.17719087, -0.0954696015, 0.323434025, -0.166302964, -0.0378812701, 0.119964503, 0.222246632, 0.0803848058, 0.0778280646, 0.274888039, -0.1463819, 0.16310896, -0.139771625, -0.180156469, 0.164859727, 0.305645019, 0.25364998, -0.0705485269, 0.135831848, -0.0893951431, 0.28743431, 0.070728071, 0.0838205442, -0.0445251912, -0.0326616764, -0.120599262, 0.139440745, -0.270022005, -0.108915411, -0.0532744862, -0.245501712, -0.0115316864, -0.127213374, 0.149182394, 0.173800245, 0.0761279762, 0.238401845, -0.062345773, 0.0435865968, 0.0119816968, -0.113206729, 0.142904684, 0.0389598235, 0.236816138, -0.058863014, -0.140110746, 0.274992466, -0.14359425, 0.10345877, -0.0460031852, -0.167516112, -0.00952434354, 0.247703657, -0.0753713027, 0.121685714, 0.0823878422, 0.23488979, -0.0619931184, -0.0766328648, -0.0780418068, -0.0143457921, -0.133595392, 0.280221343, -0.123221971, 0.0499226376, -0.0771679506, -0.0386132747, 0.050129544, -0.0213634074, 0.0406502597, 0.29187867, 0.00179839157, -0.128595933, 0.0654454753, 0.0833715722, -0.0237372257, -0.160019487, -0.0706409961, 0.13007459, 0.193477109, 0.12929526, 0.194544196, -0.0337707773, 0.153220907, 0.208017707, -0.112889752, -0.0212976448, -0.110117443, -0.0935627148, 0.201002955, -0.0485042818, 0.135973632, 0.127661034, 0.11343646, -0.1885878, -0.0211448614, -0.126879215, -0.183075756, -0.0898045972, 0.000568327669, 0.00911092758, 0.0558643304, -0.18213293, 0.0719175339, 0.152180195, -0.0481474549, 0.258260578, 0.199615657, 0.148173228, 0.0394268632, 0.10337054, 0.106657632, 0.193686217, -0.113603137, -0.137724444, 0.0699722022, 0.063817814, -0.0267793834, 0.0403312594, 0.0746018738, -0.0369499028, 0.111911014, -0.209794521, 0.124978349, -0.0450591743, 0.114969119, -0.207217485, 0.0647557825, 0.15988557, -0.0394030064, -0.00352300704, 0.07973288, -0.183837622, 0.143634632, 0.0214877576, -0.0452758223, 0.207906798, 0.0875673741, -0.133096695, -0.0591884553, -0.171955109, 0.0771896988, 0.0395951718, -0.0173865706, -0.100543596, 0.202937528, 0.206836805, -0.154319584, 0.027785033, -0.0755964369, 0.0502325445, -0.0981198698, -0.204409614, -0.200881124, -0.0966312289, 0.1947162, -0.205129281, -0.0549425334, -0.13413088, -0.00894080102, -0.132092237, -0.01263915, 0.102246657, 0.183655664, 0.0780696124, 0.147488251, 0.0796844512, -0.206366494, 0.105821297, -0.0866758525, 0.117468521, 0.0730968863, -0.0894768089, -0.197888821, 0.123780325, 0.0636071116, 0.182967439, -0.048382435, 0.309802204, -0.250160158, -0.167235941, -0.203475639, 0.0432632677, 0.175398722, -0.0192775838, 0.100834183, -0.152954876, 0.0144183151, 0.232581377, -0.321812779, 0.167421177, -0.191333041, -0.117632791, -0.214048147, 0.0570586398, -0.0707548633, -0.0965818316, 0.0956328809, -0.211586624, 0.159526497, -0.122753829, 0.0936640054, 0.038983807, -0.0090486221, 0.134821489, 0.167622879, 0.156822473, 0.0900678411, 0.153534383, -0.226792514, 0.0524546355, -0.174388677, -0.115811922, 0.00570448162, 0.27308467, -0.106389359, -0.136367708, -0.222481415, 0.0649660677, 0.231387734, 0.199437037, -0.0451859161, 0.00607657246, 0.122315645, -0.0604027137, 0.126780376, 0.144564077, 0.0225306693, 0.0650955886, 0.0242205709, -0.118545949, 0.268948376, -0.0256855562, 0.0343104936, -0.069202207, -0.0779325366, -0.102411069, 0.179498464, -0.101506397, 0.0488925502, -0.0689219609, -0.0659783483, -0.136400327, 0.133670032, 0.243812606, -0.00633601891, -0.148582682, -0.00797831547, -0.126626313, -0.0936052874, -0.197196543, 0.182358727, 0.116384923, 0.0608248077, -0.114480652, 0.0227467716, -0.0658283457, 0.155729368, 0.239702567, 0.197265238, -0.109269656, 0.048140429, -0.113062605, -0.164667413, 0.109318092, 0.117424659, 0.226807907, 0.242188722, 0.244667873, 0.0913275629, -0.0497324169, 0.133244559, 0.139072567, -0.0962307155, 0.156236574, 0.0416714326, 0.0171999503, -0.115829073, 0.193360731, -0.0875519365, 0.0553654693, 0.15870443, 0.112140588, 0.0085960133, 0.115142487, 0.0321300998, 0.0831481293, 0.0826298743, 0.16946727, 0.1216354, 0.0426968448, 0.0600113608, 0.00731581124, -0.0923310071, -0.0970181897, -0.110141873, -0.0211779475, 0.180789977, 0.214999735, 0.143563792, -0.0888314769, -0.0837424845, 0.19645004, -0.0607952587, 0.0226881709, -0.334903687, -0.0999383703, 0.218144059, 0.213849559, 0.163884476, 0.0333319828, -0.0647564679, 0.138918817, -0.190249652, -0.186543033, 0.214060068, -0.139762402, 0.118343443, 0.200249881, 0.195759326, 0.0673449859, 0.0379764214, 0.226978466, -0.205298588, -0.20902957, 0.153362259, 0.01173349, 0.078916654, -0.100195095, 0.151100561, -0.0188093036, -0.0797100887, -0.233888417, 0.117763057, -0.0822941959, 0.0278804805, 0.143493846, 0.160960034, -0.0659005791, -0.108755261, 0.187783971, 0.0706701577, -0.188152313, 0.0074400031, 0.202091694, 0.112989739, 0.283432066, -0.0650387108, -0.154812038, -0.070825696, 0.0947837383, 0.0300658494, 0.147857964, -0.0216534138, 0.149756923, 0.0929859504, 0.0209971983, -0.00134888815, 0.0633148849, -0.0827424526, -0.000136449045, 0.19020921, -0.099270843, -0.0141247753, 0.0675853714, 0.0370295681, 0.183386773, -0.220024183, -0.0877708718, -0.214005783, -0.0824217796, -0.206398562, -0.221563339, -0.198710755, -0.119112119, -0.179287687, -0.00589003647, -0.145204052, 0.188346729, -0.233802795, 0.0376543291, -0.0215257984, -0.0865447745, 0.0118213641, 0.0664706305, -0.114263661, 0.0727500916, 0.0725146085, 0.189405486, 0.0885372013, -0.118517295, 0.0957777277, 0.113105021, -0.129922196, 0.0589649342, -0.0539315492, -0.0531233847, 0.0959037095, 0.159117237, 0.149913475, -0.0260760263, -0.0374908708, 0.105810463, 0.0345708914, 0.145390734, -0.0901318491, -0.0717779323, -0.0579015464, 0.0103023499, 0.205496356, 0.0216532797, -0.0160493869, 0.0679177195, -0.101879142, -0.0618111826, -0.0948672071, -0.0378079861, -0.0649976283, 0.0622105785, -0.0198299233, 0.117059089, 0.152212754, -0.112169929, 0.181148887, -0.168585852, 0.159860879, -0.0673378035, 0.0107045667, -0.0135089708, -0.0416479558, 0.0822456405, -0.127546847, -0.19231008, 0.173437029, 0.316009939, -0.185705617, -0.200298309, -0.158173889, 0.109854989, 0.152270272, 0.0278286487, 0.131128207, -0.071521163, 0.0525241606, 0.190306738, -0.124342375, 0.167207927, -0.0263414159, 0.0591874644, -0.0529713295, 0.0697124153, 0.054551594, -0.0173513144, -0.057966955, 0.0469674952, 0.178930059, -0.167295069, 0.0556705557, -0.217425913, 0.233187571, -0.0404247306, -0.173242241, 0.184321582, 0.102461167, -0.117671609, 0.0971307158, -0.212536231, -0.0653044954, -0.0705413967, 0.0569576286, 0.0243945643, 0.130107, -0.167852372, 0.0545675196, -0.238953099, 0.0423130803, 0.210260853, -0.0551566482, 0.26816833, 0.22665599, 0.225868911, -0.0444056578, -0.160370082, 0.0105681, -0.122951277, -0.115540609, -0.146256328, 0.188854426, 0.0384555124, -0.208536968, 0.277146548, 0.121490255, -0.0306008048, 0.0699297115, -0.22213009, 0.125744939, 0.205969438, 0.0161051843, -0.0934454426, 0.066526264, -0.123336747, 0.0589029752, 0.0126853334, 0.0986614898, -0.161116496, 0.0941702724, 0.0936794654, 0.196723357, 0.115641594, -0.157700956, 0.189485446, 0.114763916, -0.0271968227, 0.113643214, 0.195243552, 0.0987473726, 0.0990002304, -0.103220224, -0.150364637, 0.103585221, 0.107007116, 0.135821953, 0.181942925, -0.0627690554, -0.144740254, -0.109147213, -0.197329372, 0.0922926366, -0.163006827, 0.176730946, -0.122540452, -0.0845109373, 0.0133600179, 0.192756966, 0.1442388, 0.0578771867, -0.193552926, -0.110479511, -0.139845818, -0.165370867, -0.193599299, 0.20830974, 0.0628420413, 0.0663306862, 0.0201054998, -0.165055826, -0.00232632901, 0.0501528941, -0.162904873, 0.0240556058, -0.224557728, -0.207684785, -0.167241246, 0.0520122238, -0.150205687, -0.0774307996, 0.11285919, -0.0143467495, -0.0623829924, -0.0121905468, 0.149959132, -0.143484727, -0.241820574, 0.0834508464, 0.260972261, -0.0260955114, 0.24016428, -0.0213887114, 0.187113076, -0.0581168793, -0.0142169902, 0.12647666, -0.12786144, 0.167034611, 0.279815257, -0.179704726, 0.0132486979, 0.306648284, 0.178435475, -0.171064615, 0.0263747424, -0.0204333719, 0.21583344, 0.0672153682, -0.00418544794, 0.273084223, 0.157282963, -0.227137044, -0.136186168, -0.110910267, -0.12844494, 0.221502915, 0.213847071, 0.13926363, 0.259363115, -0.0436799936, 0.129494667, -0.0956437588, -0.247783363, 0.0357580781, 0.190545321, 0.139593437, 0.301190645, -0.155897871, 0.211046383, 0.180168241, -0.0615664087, 0.0724108592, -0.0146866199, -0.00990192872, 0.174645156, -0.0571350642, 0.0744009539, 0.148385659, -0.0929297581, -0.0392975882, 0.173364505, 0.0863989219, -0.111795798, 0.2648094, 0.0697908551, 0.0017024983, 0.000772171537, -0.191161424, -0.189653471, -0.0896795243, -0.0889835954, 0.120452896, 0.0736927539, 0.134213611, 0.205259874, -0.130877107, 0.180374101, -0.157959193, 0.176034316, 0.0191567838, 0.0846825391, -0.108345933, 0.202308819, -0.119057111, -0.198355615, -0.106700107, -0.0142671615, -0.0904524177, -0.136138856, 0.207652286, 0.154344276, 0.0967385918, 0.0491920561, 0.0370327979, 0.113051429, -0.198209167, -0.210644111, 0.100362405, -0.00893753767, 0.160789892, 0.0860281438, 0.149556741, -0.120294005, 0.0554995388, -0.189491674, -0.216242567, 0.164922521, -0.0101215243, 0.163655207, -0.209463686, 0.153605536, 0.135718778, -0.0541202426, 0.0377530009, -0.147346109, 0.138376907, 0.214301333, 0.10419561, 0.00336061418, 0.062403366, 0.142508909, 0.1622089, 0.136284068, 0.133917317, -0.179188401, 0.166013911, -0.162876546, 0.182987556, -0.101054475, 0.207223997, -0.100585461, 0.108998492, -0.059228152, -0.289831012, -0.0246569235, -0.00949376542, 0.175843939, -0.00427034125, 0.133596122, -0.0528981984, 0.174341112, -0.323382407, -0.0103142979, 0.0814552531, -0.0453974083, 0.0312591642, -0.0158383772, 0.018919412, -0.0416506566, -0.0423595347, 0.104281411, 0.125730589, 0.167497084, 0.190087736, 0.0710149929, 0.0990974009, -0.117281586, 0.103747696, 0.119485021, -0.0836957917, -0.219795361, -0.000133946538, -0.115642637, -0.0691571683, 0.00982022285, -0.128957704, 0.252099067, 0.190815985, 0.156464547, 0.0271001942, 0.12782681, -0.18666859, -0.100569583, -0.115921304, 0.245715797, 0.0163808819, 0.113201968, 0.270258486, 0.0548837595, 0.103501529, 0.170653298, 0.106830947, 0.0374602042, 0.227922827, -0.00101049035, 0.154585198, 0.0332156345, 0.00934819411, -0.0605532117, 0.00581356371, 0.247514546, 0.257806003, 0.10757257, 0.150476232, 0.0365517661, 0.0860407799, -0.145575255];
    CONSTANT bias_8 : ARRAY[0..63] OF REAL := [-0.00346507085, 0.0794098824, -0.0815823004, -0.0197601747, -0.0118380254, 0.0312293377, -0.00609452976, 0.00358696282, 0.00419461308, -0.0723088458, 0.0482314527, 0.0938620642, -0.0692073926, 0.0194631442, -0.0589119196, 0.0299020465, -0.00631620362, 0.00955793448, -0.0159860123, 0, -0.00618809368, 0.0138237355, 0.00124220713, -0.0202849712, -0.00431400631, -0.0275725052, 0.111446135, 0.11047177, 0, 0.0995986015, 0.0175163615, 0.0613925792, -0.00830586068, 0.00282396353, -0.0744342729, -0.0211106688, 0.0866850466, 0.0997213498, -0.00675268006, -0.0535650924, -0.0118874479, -0.0482638218, 0.00823871326, 0.0484990887, -0.0278981514, 0.0414009988, 0.0608626865, 0.0968099013, -0.0129826535, -0.0369008854, 0.00364142703, -0.0370340049, -0.00600347202, -0.0126274861, 0.0921183825, -0.0980235487, 0.00168389722, 0.0823842064, 0.0339883827, 0.0445966795, 0.0921582058, -0.0254019089, -0.0172969531, 0.0778813958];
    CONSTANT weights_11 : ARRAY[0..4095] OF REAL := [0.152399674, -0.263345957, -0.224488631, -0.188193366, -0.0617991723, 0.148717895, 0.0324863903, 0.114666007, -0.289823532, 0.0125278663, -0.0137963807, -0.022444414, 0.110561207, 0.119829476, 0.334477097, -0.139504924, -0.0269849207, 0.113053806, -0.0107069612, -0.180623204, 0.0457108654, -0.214532733, 0.0401020236, 0.00631321967, -0.167630613, -0.0481288582, 0.195484549, 0.111929268, -0.0581923984, 0.0258115064, 0.238763675, 0.0641915128, -0.0806587264, -0.224124625, -0.0460969172, 0.091414094, -0.013553381, -0.043530602, -0.0263040792, 0.140525028, -0.0622836426, 0.15601474, -0.497485936, 0.129424945, -0.170885473, -0.125799641, -0.339268953, 0.0710499883, -0.116152979, -0.0266817547, 0.126233891, 0.131714255, 0.290685475, 0.165184066, 0.283396602, -0.059989959, 0.0141595677, -0.136663362, 0.20351474, 0.0463219136, 0.00223265006, 0.0316324756, 0.182196692, 0.341547728, 0.0614045113, -0.00371772563, -0.275792897, -0.193623677, -0.0266438629, -0.103982933, 0.0405711122, -0.00346332369, 0.0464573167, 0.000740021234, -0.303002685, 0.0795986727, -0.0327266343, 0.0721366256, 0.147136018, -0.105440497, 0.101954572, 0.0728471428, -0.0363206528, -0.0158560108, -0.330246508, -0.212550044, -0.093112044, -0.197731018, -0.125574902, -0.078097105, 0.034774553, -0.262974173, 0.15699707, 0.14151752, -0.0313425213, -0.0470193997, 0.19462584, -0.255247116, 0.357496887, 0.000614301243, -0.195358515, 0.0303748176, -0.175757021, -0.0335321315, -0.0249454323, 0.0811241418, 0.0762640387, 0.116933405, -0.128208607, 0.00518320873, -0.029634852, 0.11359746, 0.017268436, -0.104347244, -0.115615718, 0.202678129, 0.10678266, 0.0986468866, 0.190590888, 0.0687514096, 0.0356852412, -0.0412406325, 0.0757317245, 0.0352434814, -0.342369705, -0.0480474308, 0.266226262, 0.0569148995, 0.0286941677, -0.2472938, 0.0204578005, 0.0296292026, -0.0654909462, -0.10515099, 0.151057318, -0.0363138504, 0.00139550562, 0.0611258186, 0.0148243103, 0.227309123, -0.0798782185, -0.11899174, -0.157541484, 0.314520597, 0.170248464, 0.265226632, 0.0593360811, -0.0398373678, 0.0081351446, -0.0901603773, 0.18755962, 0.00631602108, -0.207302138, 0.103253566, -0.240270436, -0.0895837396, -0.105462186, -0.135611624, -0.0793325603, -0.0249736756, -0.13815324, -0.0941773206, -0.189351335, -0.112737559, 0.293767184, 0.0163262729, -0.175204575, -0.0996527299, 0.231760427, -0.0418962091, -0.0648548007, 0.268336385, -0.032381732, 0.245270595, 0.0585076436, -0.0289969705, 0.232107788, 0.279983878, -0.011282769, -0.121292524, -0.295017779, -0.131171674, 0.0821883231, 0.216307148, -0.0106242169, 0.00658608973, -0.21936737, -0.139937028, 0.182932571, 0.233257622, -0.286341697, 0.246410012, -0.0386230387, 0.0858042613, -0.0830237195, -0.110467531, 0.0558926836, -0.0293775387, -0.216672435, 0.134263664, -0.0869384855, -0.0198220555, -0.0998319387, 0.122479506, 0.124716364, 0.12669073, -0.165978372, -0.0657829642, 0.0525778681, 0.0783382952, 0.0370095335, 0.141239166, 0.0418702848, 0.0749414936, 0.240086794, 0.0674306303, 0.0347193331, -0.0469557568, 0.041893255, 0.090664953, 0.0798208192, -0.124962248, -0.0150589822, 0.0606806017, -0.212737143, 0.0127978772, -0.0479948185, 0.193862215, 0.18940939, 0.110280916, 0.00163242826, -0.0205761306, -0.129006281, -0.141371146, 0.147304669, 0.0262788441, 0.167370602, -0.141203105, 0.200771987, -0.234238222, -0.149722278, 0.23931098, 0.0104937805, -0.266669959, -0.164157122, -0.041039072, -0.250695556, -0.112417288, 0.193107903, 0.140542001, 0.0903390646, -0.230039254, 0.0777369738, 0.260997742, 0.0930059701, 0.138459459, 0.0424353629, 0.171048418, 0.156789139, 0.0312985368, 0.133111879, -0.120839193, 0.0985307842, -0.175964057, 0.122762412, -0.117720641, -0.129174918, -0.104449466, -0.144933715, -0.215081707, 0.0680070445, -0.129005954, 0.0603452325, -0.0575148351, -0.203575164, -0.0453374311, 0.155170351, 0.106897905, 0.0749150291, -0.144247919, -0.171046615, -0.132302389, -0.147862911, 0.00684731873, -0.0410480648, 0.15876098, -0.190579101, 0.0498549677, 0.0963715315, 0.086084798, -0.0875354186, -0.153710201, 0.145764962, 0.0200527348, -0.100025706, -0.135493338, -0.0464859232, 0.00132688298, -0.0185684748, 0.0582565144, 0.187669724, -0.0816467628, -0.0872224793, 0.157934099, 0.0402881019, -0.0318563916, -0.142950997, -0.11230398, -0.0497585908, 0.161313683, -0.1942278, -0.0826544166, -0.0122894971, 0.0872979611, 0.0720221922, 0.0849900693, -0.177533969, -0.152409315, -0.100491337, -0.0112174684, 0.106480442, -0.0379864834, 0.0722993612, 0.163500831, 0.18924883, -0.135068297, 0.0942396447, 0.0284191072, -0.0632716715, -0.138580009, 0.193715364, -0.150715292, 0.0303814765, 0.111110657, 0.117106274, -0.0263905209, 0.0506038666, 0.0267103072, 0.0400604308, 0.154954746, 0.108434454, 0.0550541244, 0.0168840457, 0.0785695761, 0.0604145676, 0.144188315, -0.206482708, 0.0983125418, -0.0374258012, -0.00447623339, 0.205374479, -0.0380841345, 0.0740306601, -0.0350800455, 0.0866823494, -0.0981449634, 0.0656447932, 0.0974652469, 0.0593180098, -0.0401085094, -0.0922544375, 0.0644713044, -0.0637705103, 0.205211937, 0.27076602, 0.0604185574, 0.245794445, -0.0236300994, -0.027567558, 0.1355685, 0.0849664137, -0.138995841, 0.159796208, 0.0539290234, -0.0213833489, 0.0917554945, -0.193392858, 0.0205196254, -0.154481247, -0.0105813192, 0.158501342, 0.01522783, -0.0629718155, -0.222794086, -0.138768524, 0.00203081919, 0.170994595, -0.0148755405, 0.0800000504, 0.194157824, -0.113540575, 0.0917406157, 0.238140926, 0.00717910752, 0.21342735, 0.0675954148, -0.0781002492, 0.179200038, -0.0140909683, 0.217517018, -0.0182730798, 0.154534876, 0.130978897, -0.15910472, -0.242845848, 0.192364007, -0.0712619573, -0.172466293, 0.153321937, 0.196527407, -0.14488329, 0.0236006379, 0.0861952752, -0.0437985249, 0.175121501, -0.0954023749, -0.114573762, 0.143516839, 0.00525142904, 0.126135498, -0.116257451, 0.109212697, 0.0145286033, 0.104307882, -0.0975407884, -0.164253727, 0.0486553423, 0.0687329695, 0.187514946, -0.049572818, 0.0788708553, -0.0701822415, -0.045390375, 0.100607939, -0.0249090847, 0.0791288838, 0.154155806, 0.232392356, 0.110889055, 0.0298407078, -0.0190417878, -0.0341505446, -0.22469382, 0.0715206563, -0.109233215, 0.0421755537, 0.0418922678, -0.0328179933, -0.161357954, 0.0284879543, 0.0438218452, 0.257945627, 0.227448493, -0.129958495, -0.392283171, 0.109769329, -0.0173306819, 0.0859658271, 0.108519241, -0.0660175383, -0.0608303361, -0.0360111594, -0.0876427889, 0.190083712, 0.0288716163, 0.238107309, 0.136543661, -0.00705705583, -0.0259979162, -0.00647293031, 0.069024533, 0.0381969362, -0.152234167, 0.295585841, -0.401145488, -0.108133636, 0.209102049, 0.0307547674, 0.147690207, 0.128031835, -0.0473762713, -0.147987187, -0.164643124, -0.059981253, -0.14839074, -0.0456473343, -0.335970312, 0.0270624142, 0.273908377, 0.0461861901, -0.221928775, 0.151594713, 0.0270567555, 0.0552504733, 0.288964689, -0.075935334, 0.270585835, 0.235102609, 0.181183606, -0.116892524, 0.0349841826, -0.0259137452, -0.310423553, -0.0737684369, -0.224190742, 0.102769867, 0.148424283, -0.00051581359, 0.109018147, 0.131758898, -0.241935253, 0.0429472104, -0.192998812, -0.156563684, -0.199549347, -0.0259795301, 0.118114009, -0.202294961, 0.00430562347, -0.0795410797, -0.186826259, -0.12402641, -0.0973436236, 0.062623024, 0.0698438436, -0.0140991006, 0.0761193931, -0.157981157, 0.054249879, -0.0833289996, -0.119116187, -0.175815642, -0.193181172, -0.0350408033, 0.0374635346, -0.148473918, -0.111192934, -0.110237554, 0.0392782576, 0.0543338954, -0.212789983, 0.214189187, 0.261465758, 0.0389742181, -0.0119669382, -0.041862458, 0.0934221447, 0.154760599, 0.104591891, 0.135659441, 0.124115832, 0.125245571, -0.0981265381, -0.173501864, -0.225834534, -0.040620435, -0.0631992593, 0.11226812, -0.151412457, 0.0888080448, 0.130535215, 0.114341483, 0.0704539269, 0.238751054, -0.0625069663, 0.183925942, 0.162767082, -0.0624889433, 0.18303372, 0.0478743874, -0.214895129, 0.150446177, -0.0400604196, 0.164489478, 0.156864062, 0.280662, 0.0744856521, -0.109412298, 0.222006962, -0.188556612, 0.257241905, 0.00763767865, -0.0429345556, 0.000701996032, -0.256307662, -0.0537884794, 0.258199453, -0.145994559, 0.0452899151, 0.0317057781, -0.0876930654, 0.08571475, -0.092731908, 0.184803054, 0.18809928, 0.0703473389, -0.00392604945, 0.142104432, 0.160575241, -0.0699259192, 0.196616039, -0.160764754, -0.202707544, 0.150236309, -0.194807246, -0.142325938, -0.240276873, -0.0591731966, -0.0514629297, 0.00134343619, -0.166902661, -0.188654795, 0.0843883976, 0.0013771971, 0.169252023, -0.161208317, 0.208919898, -0.118219167, -0.24853687, 0.147254348, -0.040950682, -0.104150467, -0.182231963, -0.162871018, 0.0433620438, 0.126293465, -0.166178107, -0.186834484, -0.22719419, -0.216035366, -0.311863422, 0.10080345, -0.10563679, -0.21303615, 0.0257087015, 0.063385427, 0.0836621374, 0.137088358, 0.0247118175, 0.157823056, -0.162809089, 0.274433285, -0.0909785628, 0.219206274, -0.150779128, -0.206102833, 0.0196267851, 0.215949804, -0.080320105, 0.0171771869, -0.126778483, -0.169971392, -0.0758564174, 0.037309479, -0.184586704, -0.176283911, -0.0172518641, -0.223967373, 0.0620737523, -0.210962385, -0.0175580438, -0.198382184, -0.133766785, -0.192560017, 0.00918835402, -0.0767401755, 0.136367351, 0.171674535, 0.183295757, 0.220561728, -0.0821217224, 0.1140071, -0.127449334, -0.151443526, 0.118891813, 0.0171878282, -0.027197564, -0.0242941491, -0.232013106, -0.109213538, -0.117022179, 0.0856248662, -0.151049286, 0.142516539, 0.125007212, -0.156722993, 0.266981691, -0.130809814, -0.0616114177, -0.0442247763, 0.0877789408, 0.0459268093, 0.225089535, 0.059550181, -0.0352692939, -0.0199252516, -0.140248358, -0.181541502, -0.0301125441, 0.114853002, -0.155363366, 0.120270431, -0.119383417, 0.15385288, -0.137697816, 0.0990949422, 0.139819413, 0.101220191, 0.0159896575, -0.0617526323, -0.0679681972, 0.113188118, -0.042417895, 0.0258083455, -0.169725969, 0.075258702, -0.0537487082, -0.149268836, 0.109437704, -0.116023861, 0.0976026133, -0.215568498, -0.257916421, -0.0836541727, 0.0753511712, 0.194070086, 0.0318242721, 0.0160240829, 0.0868645757, -0.188116699, 0.181180835, -0.207172692, 0.110726506, 0.171905503, -0.121312834, 0.00326830451, -0.134259403, -0.244052947, 0.156338409, 0.239065826, 0.0572260544, 0.22199899, 0.0920382291, -0.0747542828, 0.0250579547, -0.209005356, 0.314894259, -0.0127276182, 0.188592002, -0.105892763, -0.203456968, 0.218186542, -0.0714133903, -0.090361774, -0.0645971596, 0.0143091576, 0.298341304, 0.159289271, 0.0570015721, -0.199153751, 0.019798452, -0.0419481322, -0.128920168, 0.0999377146, -0.245023876, -0.0517567694, 0.247462109, -0.070638895, -0.0811767727, -0.128980458, 0.11074882, 0.0168372188, 0.0593690798, 0.175101206, -0.054478053, 0.022643229, -0.307910532, -0.0983424112, 0.0169419218, -0.131076947, 0.295372337, -0.176049858, -0.0388735868, 0.261773378, 0.186196834, 0.0407921039, -0.060955897, 0.0722839534, 0.1541913, 0.118314162, 0.185275882, -0.0770900249, -0.186694846, 0.118786186, -0.022491321, -0.0364597216, 0.089644663, 0.0571428053, -0.253871858, -0.0122213988, 0.204711184, 0.312439799, -0.320880443, -0.27240929, 0.122102626, -0.273709536, -0.0164961014, 0.0607479513, 0.291678041, 0.223591253, -0.198138237, -0.118850462, -0.238560677, 0.323092818, 0.0589599535, -0.194248945, 0.00573190255, -0.0346102566, 0.00809514709, -0.1437345, -0.0768056959, -0.0114840511, 0.14923422, -0.0970238969, -0.0471924804, 0.0891452581, 0.176614508, -0.150917053, 0.31215173, -0.0488434397, 0.0310474988, 0.13556391, -0.210260242, 0.265471876, 0.127534941, 0.00403250754, 0.210733801, 0.0956179649, 0.0654093474, 0.0347067229, 0.0318550393, 0.248021692, 0.0198314767, -0.115047991, 0.108949013, -0.10042078, -0.29889968, 0.0146387629, -0.141234264, 0.204530731, -0.144104674, 0.105720773, -0.23340179, 0.0790494978, 0.18509376, -0.206608996, -0.0394043922, -0.0189410113, -0.230545685, -0.198211581, 0.220677823, -0.0647635758, -0.195251271, 0.201641157, -0.177163646, -0.095896475, 0.0920335501, -0.138604224, -0.109693781, 0.236355498, 0.0536849797, 0.115611076, 0.212027684, 0.0571522713, 0.240873307, -0.0458607674, 0.310614586, 0.233346224, 0.0570905395, 0.130410984, 0.169783399, 0.0727831423, -0.0302463956, -0.30536887, 0.0152019113, 0.163850963, -0.109125808, 0.0144169629, 0.132228628, -0.0707990453, 0.193070427, 0.165563926, 0.0941457525, -0.0627072603, 0.0423249342, -0.111638814, -0.0591745116, -0.0470574982, 0.29292962, 0.0765838027, -0.142371729, -0.112034045, -0.0560461804, 0.156755283, -0.235810399, -0.201336101, -0.125491038, 0.201229259, 0.123228803, -0.238689259, 0.0129049234, 0.0961765721, 0.0151871378, 0.266222477, 0.186487585, -0.217119902, -0.0869368389, 0.124067664, -0.065676488, 0.140951827, -0.198084503, -0.178457528, 0.0855591595, 0.1007246, -0.0287072621, 0.0854200944, -0.178427383, 0.0386579223, -0.0619194172, 0.09910997, -0.129233211, -0.068861261, 0.13413316, 0.139778435, 0.0833287686, 0.0622766875, 0.235616207, 0.201298133, -0.182556123, -0.00869753398, -0.047157418, 0.268308789, -0.225152835, 0.0152922235, 0.153030574, -0.0839851871, 0.167121798, -0.0833399519, 0.093423374, -0.0923105478, 0.178122193, -0.203960165, 0.0267385971, 0.0512525626, -0.22356531, 0.056387879, -0.0550887249, 0.161965206, -0.195818886, -0.0647771284, -0.182523564, 0.17741926, -0.116015404, -0.0489375815, -0.202825278, 0.147160143, 0.191247597, 0.0707065612, -0.00766302971, 0.170157924, 0.0735885873, -0.141567349, -0.21014148, -0.129353657, 0.0956847668, 0.0227197595, 0.0941244364, -0.0791912824, 0.107957929, 0.199303105, 0.0537132025, 0.0155240446, -0.147489786, 0.0846396238, -0.0715232193, 0.182592198, 0.00312403357, 0.0118206823, 0.0933757424, 0.162187204, -0.0768953189, 0.130623519, -0.154309347, -0.0370425209, 0.225373268, -0.0371935703, -0.512049019, 0.0894301012, 0.149142876, 0.0406918228, 0.054195568, -0.222945645, 0.125597313, -0.121843651, -0.192063659, 0.022529887, -0.129418507, 0.100320496, 0.14389959, 0.100439146, 0.211798623, -0.139967546, 0.104904346, -0.0939587057, 0.127366856, 0.138831839, 0.0239571333, -0.00880390406, -0.0611199997, -0.10359811, -0.0635057986, -0.00202414393, 0.188975051, 0.18646647, -0.133227944, 0.0697101131, -0.0743370131, 0.0876726359, 0.174912781, 0.132824585, 0.00545993866, -0.000499482965, 0.169128001, 0.219260916, 0.214551806, -0.0652708858, -0.0217023604, -0.193402603, 0.00403163396, -0.117414609, -0.0933148414, 0.00748919882, 0.200135365, -0.141633987, -0.214732349, -0.091433309, 0.204348087, -0.0532101393, 0.154062733, 0.248481318, -0.13802442, 0.192950904, 0.16888696, 0.149313912, -0.222851619, 0.153076321, 0.182242945, 0.185836926, 0.141479209, -0.0413135886, -0.0169824678, -0.0272292644, 0.089787066, -0.0702687651, 0.158348948, -0.0452950932, -0.0598885454, -0.174950615, 0.291644782, -0.0561419651, 0.0800843909, -0.215036035, 0.13363564, -0.103067927, -0.0768741667, -0.0631346405, 0.0626737475, 0.15906544, -0.327983201, -0.123729207, 0.19425182, -0.14580068, -0.110915102, -0.0493397824, 0.0671491474, 0.00072730938, 0.0883379132, 0.123690397, 0.189004809, 0.0893278271, -0.114139549, 0.308739871, 0.0107161012, 0.118270479, -0.337565839, 0.261260688, -0.0494029, -0.0752659142, 0.238311097, -0.108185798, -0.12475723, -0.0681707337, 0.0807750225, 0.0104115838, -0.0831196159, -0.161203995, 0.0769510195, -0.178012058, 0.165514678, -0.0196140297, -0.0373411514, -0.0155290961, -0.161595047, -0.0622068048, -0.291716814, 0.218920842, -0.128163859, 0.044695992, -0.187777534, -0.105463572, -0.0571242459, -0.0119509697, 0.00533423526, -0.0132009489, 0.161444128, 0.190533608, 0.136306271, 0.158209473, 0.215961605, -0.0804739892, 0.117368713, 0.126664549, 0.133364782, 0.152663857, 0.136497244, -0.336019129, 0.150216475, 0.20953989, -0.0419718549, 0.00763540342, 0.0507058874, 0.0899446309, -0.0746354163, 0.126670465, 0.0997138247, -0.131774053, 0.18959567, 0.186503679, 0.0671444461, 0.107626587, 0.125563666, -0.0331348479, -0.0831428245, -0.0118116708, 0.13317202, 0.179913059, -0.00435783528, -0.103403352, -0.169043481, 0.134726152, -0.143405557, -0.143480599, 0.145388424, 0.0501072556, -0.100935332, 0.0670109838, -0.0547590144, -0.11869137, -0.164782315, 0.14261204, 0.0516628996, -0.0139837861, 0.158076271, -0.0323812068, -0.0253638402, -0.0481653959, -0.166442499, 0.0914008841, -0.126121193, 0.10642685, 0.080969587, 0.195150837, -0.0635801703, 0.0927808583, 0.0660431832, -0.113444202, 0.2108161, 0.0454176217, 0.207712188, -0.158912182, -0.149667591, 0.225732028, -0.144124746, 0.220306486, 0.187320516, -0.056225121, 0.190556765, -0.184439331, -0.128877133, -0.0283655971, 0.148606017, -0.103650376, 0.0173259694, 0.0809403509, 0.00934745371, -0.129418105, -0.0100147277, 0.0515523404, 0.00264053047, -0.133236319, 0.213405624, 0.200618967, 0.011354222, 0.0573964044, 0.0985980853, 0.00135266967, -0.129998296, 0.151727006, 0.204372659, 0.200007543, 0.21404855, 0.189805731, 0.172358885, -0.0890808403, 0.0522677153, 0.107005432, 0.113238558, 0.0461152345, 0.119334862, 0.113662854, -0.202756092, 0.122567102, 0.156569704, 0.0166884214, -0.127153099, 0.130326495, -0.162898168, 0.0981043428, 0.199507132, -0.092357628, -0.0304451138, -0.156488106, 0.0427581519, -0.213457823, 0.157986298, 0.212126359, -0.191093981, -0.0687070787, -0.155501977, 0.075762704, 0.202147499, -0.0100540668, -0.0357479602, -0.165612519, 0.0348113328, 0.0888052136, 0.0522147566, 0.00634533167, -0.000127598643, 0.0748969465, 0.0386748761, 0.0424322337, 0.212277904, -0.0906898081, -0.0402118266, -0.14763388, -0.163068712, -0.00134003162, 0.0113786161, -0.114206046, 0.0614237338, -0.143889531, -0.096885711, 0.20141612, -0.20934172, 0.159835026, 0.0288719237, 0.0186812729, 0.0141171068, 0.202441737, -0.00636282563, -0.0913520604, -0.00343427062, -0.0776682198, 0.114591286, 0.178352684, 0.072447516, 0.207320198, -0.164817482, -0.133918926, 0.0607623905, 0.133606508, 0.108131513, -0.00368179381, -0.0975685716, -0.18251574, -0.12751992, 0.217671528, -0.00256840885, 0.0633859858, 0.0459913127, -0.0114317834, 0.019155506, -0.0564544499, -0.173174202, -0.0360071398, -0.161694646, -0.201523215, 0.143933117, -0.0519516505, -0.189812288, 0.0398772061, -0.0408333391, -0.180227458, 0.141621813, -0.115172304, -0.121136017, -0.0121303732, -0.204050809, -0.0434726924, -0.046715267, -0.0699533895, 0.171459943, -0.144236326, -0.0683937967, -0.0708762109, -0.102386728, -0.0776161775, -0.193716198, 0.186093926, 0.0237003118, 0.121066563, -0.125280246, 0.0977233648, -0.0399483182, -0.0141839087, 0.145612508, 0.0374964625, 0.0779918507, -0.0435630977, 0.0875028968, 0.071565561, -0.0101307984, 0.165002391, 0.201880664, 0.00914894603, 0.186509728, 0.170419008, -0.00774519145, 0.0486198589, -0.257243395, 0.0580342449, -0.123784639, 0.13865912, -0.172557667, 0.151741877, -0.101602815, 0.110366128, -0.120282121, 0.0840358585, -0.13807863, 0.135065734, 0.152518809, -0.213707358, 0.157859072, -0.0512838028, -0.119913951, -0.0603275895, -0.0344250649, 0.0280932616, -0.113776729, 0.00914250128, 0.169182256, -0.0726605803, -0.118695714, -0.162195101, 0.109512694, 0.214561909, 0.201593056, -0.0490923934, 0.231536657, 0.000906694273, -0.0773898289, 0.229626477, 0.292316675, 0.0434411876, 0.0439935587, -0.171945095, 0.168419257, 0.138824657, 0.187337905, -0.121906206, -0.121290758, 0.0895823315, -0.205835402, -0.102580823, -0.064769879, 0.0918552354, -0.0006545863, 0.0484051257, 0.00231042434, -0.1427017, -0.00512752309, -0.118499592, 0.167649359, 0.173335105, 0.0724587515, -0.0639462695, 0.189106256, -0.0253329333, -0.167535514, 0.199837193, 0.054232005, 0.173054591, 0.208212107, 0.063709937, 0.178403363, 0.102365844, -0.145370528, -0.0627328828, 0.204421952, -0.217216507, 0.152429745, 0.177940995, 0.123621874, 0.161663517, -0.0583134182, 0.113821968, 0.147727966, -0.0192146897, 0.120329253, -0.206288442, 0.118907943, 0.0558229275, -0.119626381, 0.115259588, -0.123966016, 0.189842731, 0.304001242, -0.133949921, -0.00190896366, 0.111900635, 0.194404766, 0.129541457, -0.0793663859, 0.0952215493, -0.205361709, 0.0308174528, 0.276944697, 0.150184885, 0.0571603253, -0.0862910375, -0.209261745, -0.00469737314, -0.107266292, -0.0262841173, -0.21763204, 0.0261462647, 0.0255539753, 0.159364834, 0.0638701171, -0.133363664, 0.166979283, -0.191513494, 0.167016715, -0.201660112, 0.0460934602, -0.00581953721, 0.00407372508, -0.078385748, 0.176348567, 0.261097163, 0.0668909401, 0.0932687446, 0.268428653, 0.111295953, -0.0538752489, -0.0353972577, -0.0643084422, 0.0826371983, 0.241673946, 0.0859841257, 0.0413935967, 0.192854241, -0.0863617063, 0.102388531, 0.0939005539, 0.110310666, 0.0338847861, -0.0237080809, 0.192427814, 0.00698334165, 0.0662905425, -0.134980679, -0.00617967499, 0.190878674, -0.00159786642, 0.0727328956, -0.240946233, 0.196102977, -0.0931468382, 0.0836528018, 0.103284612, -0.239004865, 0.0113834683, -0.129806876, 0.14836894, -0.232858315, 0.089459613, -0.179351673, 0.144995049, 0.196424425, -0.0279766843, 0.132153019, -0.105318397, 0.187499374, -0.00858527701, -0.0920507312, -0.11234127, -0.0994759649, 0.175084785, -0.0811289176, -0.100668162, -0.387158185, 0.153878331, -0.178559199, -0.119826905, -0.0257519037, 0.202533126, -0.165797308, 0.1972083, 0.0326090157, 0.191457987, 0.208948106, -0.0303138606, -0.168486714, -0.212763578, -0.00552030979, -0.0189667419, 0.196747944, 0.209965065, -0.14008227, -0.356117338, 0.0720864087, 0.2261962, 0.262177914, 0.190582126, 0.125341758, 0.131352305, -0.0850886703, 0.105056457, 0.0996146277, -0.364396185, -0.1066579, -0.145678446, 0.0647635385, 0.0825714245, -0.0452001728, 0.13121967, -0.145201892, 0.102415368, 0.160855427, -0.1157851, 0.176233247, -0.106195346, -0.17459546, 0.0715932772, 0.0647462085, -0.0499108769, 0.0551721789, 0.0756226256, -0.115369171, 0.115483992, 0.182759956, 0.134363547, 0.19813326, -0.00339539489, 0.22427693, 0.0874575227, -0.0538085252, 0.0250612367, 0.194358304, 0.0420459919, -0.197343454, 0.15234834, -0.0194482468, 0.207918748, -0.370312631, -0.191926241, -0.238808528, -0.0383893885, 0.126615122, -0.0540592968, -0.207585737, -0.0226110499, 0.0861546621, 0.258043557, 0.30580011, -0.265124172, -0.172527641, -0.0776732266, 0.0940554887, -0.0529039092, 0.22364676, -0.0504839607, -0.111994199, 0.0752739981, 0.167051509, 0.231486157, 0.222942859, -0.0696845353, -0.151163772, 0.250781924, -0.146447971, -0.0967529416, 0.184217557, -0.300973266, -0.126572028, 0.215180457, 0.187338904, 0.185731187, -0.11665196, 0.000876162725, -0.0202561766, 0.125354245, 0.10827215, -0.160607785, 0.188338622, 0.0980067775, 0.0324687324, -0.219831422, -0.168211251, 0.200699002, 0.1139713, -0.216335818, -0.0309214499, 0.0763551295, 0.0451243334, 0.0868523866, -0.000636569108, 0.0952483416, -0.11416243, -0.125886872, 0.0755488724, 0.107398666, -0.0849267319, 0.0167402681, -0.368645281, -0.106054433, -0.136857152, -0.113142923, -0.140909985, -0.0106369946, -0.0734956935, -0.242627531, -0.163561374, 0.0919052735, 0.125031963, -0.043657735, 0.0146407625, 0.153221101, 0.0668651685, -0.190944195, 0.0788392946, -0.0817975849, 0.124928646, -0.361474574, 0.110909373, -0.255627602, -0.142462447, 0.0353607163, -0.252555937, 0.194031313, -0.0276524629, -0.0741961077, 0.0262450166, -0.102495871, 0.107768953, 0.141406447, -0.322431296, 0.174083382, -0.174821675, -0.395054817, -0.0608991683, -0.341402888, -0.146280155, -0.290810555, -0.0700072646, 0.0340672284, 0.114190154, 0.212211475, -0.29652983, 0.0295428969, 0.194639176, -0.0198184811, 0.133799478, 0.138498858, -0.182915777, 0.0482293516, 0.0976990163, -0.18222487, 0.0835105181, -0.106537037, -0.0591551289, -0.115260668, -0.11497248, 0.0435057431, -0.159548879, -0.105683692, -0.260151893, 0.0550674088, -0.0321849883, -0.0744472593, 0.00243522367, -0.181820303, 0.252596408, 0.270988226, 0.168165222, 0.0595975779, 0.0989734977, 0.17273213, 0.0179654639, 0.013571118, 0.0022207133, -0.0643146485, 0.14008981, -0.0777452365, 0.134650469, -0.155961126, 0.0555896498, -0.0966854021, 0.0125770848, -0.000214683023, -0.151022673, 0.196903691, -0.115989923, 0.262134969, -0.0680010691, -0.224485368, -0.199625343, -0.210131735, -0.0643070862, 0.0685092211, -0.413198173, 0.0757171661, 0.0919734463, -0.359562606, -0.201385498, 0.0115947183, 0.174798757, -0.0814683214, 0.0596277267, -0.0625551641, 0.0350604355, 0.184136912, -0.164665803, 0.0183611717, 0.250624686, 0.0125863301, 0.0112502538, -0.0108454721, -0.0688611045, 0.16646485, 0.0284723155, -0.326143622, 0.251596063, 0.0676906854, -0.111148089, -0.0604397766, -0.357566506, 0.00267260056, 0.0472641513, 0.185109943, -0.0561866984, 0.148887575, 0.102317147, -0.0849794373, -0.0614579991, 0.0326576456, 0.0126584023, -0.0629983395, 0.223311111, -0.00327185332, -0.148226351, -0.183692589, 0.00595363649, 0.178311333, -0.14655976, -0.0530309901, -0.0653009266, 0.237797007, 0.173097223, 0.200525954, 0.131583318, -0.116117708, 0.0929283351, 0.098859176, -0.101166539, 0.211423203, 0.180236056, -0.098462984, 0.0356300026, -0.055087164, 0.070975855, 0.0152753443, 0.0117747337, 0.0124992579, 0.0186377019, -0.040137589, -0.174795151, -0.0888965726, 0.216044262, 0.173421398, -0.0901128203, 0.0402170271, -0.123981677, -0.0186401308, -0.120826356, 0.106725052, -0.19337979, -0.137401208, -0.123095892, 0.124976858, 0.151482031, -0.141049087, 0.0428393334, 0.174957797, -0.14806959, -0.0215549618, 0.186499581, -0.204556108, 0.210095719, 0.0789846629, 0.029979974, -0.108856134, -0.0139944702, 0.0263781548, -0.125280932, -0.10276451, 0.0262285024, 0.0617966205, 0.0358561426, -0.181433201, 0.116816476, -0.173377424, -0.181904286, -0.178747416, -0.00100579858, -0.141323447, -0.17858167, -0.215236828, -0.124892443, -0.18321009, 0.166554824, 0.0349302441, -0.0718755722, -0.21206364, 0.202988341, -0.262059748, -0.0846684426, -0.0264383312, -0.0190072507, 0.2202245, 0.128679246, -0.126438454, -0.0482899137, -0.136346161, 0.164990321, -0.0377886444, -0.00999837369, 0.145294696, -0.206945017, 0.168252572, -0.123122193, 0.0317248851, -0.0978919715, -0.111651219, 0.074932836, -0.281826913, 0.185020849, 0.055261448, 0.00178773759, 0.0390683152, -0.246171236, -0.0958288237, 0.210186899, 0.275020272, 0.0562327988, -0.133841649, -0.161592439, -0.0814305469, 0.151387647, -0.0924248621, 0.256124526, -0.0551051423, -0.211608618, -0.0358127393, -0.104693621, 0.1162875, 0.113921165, -0.0199713167, -0.23672004, 0.17288205, -0.0616145991, -0.167591259, 0.0158987548, -0.105777226, 0.00850734301, 0.206110939, 0.220944673, 0.173485622, -0.0885103047, -0.123291343, 0.119619459, -0.0967060253, 0.162609577, -0.23304899, 0.024063224, 0.0214320533, 0.2257936, -0.116359495, -0.0210717637, -0.0603798702, 0.0435092635, -0.00730895204, 0.103644289, -0.10791108, -0.00523050129, 0.0974855199, 0.250795186, -0.0883831903, 0.211329684, -0.0763134733, 0.0505424179, -0.194253653, 0.160468459, 0.0373329632, 0.00362053118, 0.232644767, 0.0308330338, 0.161484063, -0.0271853432, -0.131138071, 0.11403884, -0.0388104171, 0.0234489087, -0.0291281473, -0.16315636, 0.238832727, -0.125655994, -0.051028531, -0.150253788, -0.0957489237, 0.161308855, -0.010553672, 0.145903602, 0.178950518, 0.206775278, -0.197363213, 0.100926705, 0.127155304, 0.0886795744, 0.0384771898, -0.0636024028, 0.136744395, -0.0296712294, 0.255500585, 0.0886330456, -0.015306036, 0.127241626, 0.0978040919, 0.00628852937, 0.0744743049, 0.213523507, -0.0189819261, -0.104008943, 0.028438326, -0.0549609102, 0.108124904, 0.0547557399, -0.0689821094, 0.282766223, -0.0776696652, -0.145231634, -0.219961882, -0.0325948037, 0.170671925, 0.238952041, -0.220119491, -0.0539352782, -0.205213696, -0.0961958393, 0.0955754817, 0.190853387, -0.106655076, -0.0676123053, 0.207522944, 0.0059924447, -0.136339933, 0.170324996, -0.0170212891, -0.186595798, -0.122996755, 0.0536680296, -0.124922357, 0.0955476314, 0.0518711582, 0.176927432, -0.112219326, 0.100288011, -0.117357753, 0.199554503, 0.0488559753, -0.0699957237, 0.228910819, 0.00692145294, -0.0817696825, -0.108787522, -0.128030986, 0.0173476879, -0.131096452, 0.236910611, 0.0257094558, 0.255908877, -0.018263232, -0.00103016174, -0.0486674346, 0.073059462, 0.244683802, 0.0431794897, 0.0152821513, 0.168885887, 0.108368844, 0.167778686, -0.213540077, -0.211735442, 0.105609275, -0.0604555644, -0.155116454, -0.196209759, -0.0379836187, -0.0647224784, 0.00641336106, -0.14297466, -0.107331365, 0.183396488, 0.184337839, -0.0531041622, 0.00186734158, 0.244511604, 0.0740732402, -0.0291328561, -0.0445070565, 0.144737765, 0.0123820817, 0.11382781, 0.197113797, 0.201976836, 0.245440185, 0.119564258, -0.146405488, 0.117127948, 0.0338072814, 0.190734386, -0.25059697, 0.199911967, 0.207614452, 0.0533561595, -0.0374337807, 0.142019153, 0.0490953773, -0.216328979, -0.10855855, 0.115646183, -0.263035089, -0.148798853, 0.124370195, -0.13782458, 0.124930479, -0.116868503, -0.0248529781, 0.0512323603, -0.0528448075, 0.0193750132, 0.192962959, -0.152398363, -0.0119206896, -0.0373266339, 0.0179096516, -0.0443546325, -0.0742346868, -0.0461954102, 0.294702619, 0.154465228, 0.0773186088, -0.310861647, -0.0707053468, 0.266035378, -0.0992082134, -0.332212776, -0.205583721, -0.196842909, -0.281396747, 0.136664137, 0.201202393, -0.139625281, -0.0458463132, 0.186710879, -0.129951373, 0.130285919, -0.235751554, -0.0895666406, 0.199424937, 0.0833966285, 0.135916606, -0.108947381, 0.00343655213, -0.116784215, -0.189424649, 0.235676333, 0.225083172, -0.0404505059, 0.0241782386, 0.138108522, 0.141151369, -0.180884242, -0.070838213, 0.0613366216, -0.134111598, 0.025904512, 0.201248944, -0.128643408, 0.12299782, -0.132246569, 0.249260843, -0.18512398, 0.17548199, -0.11300002, -0.368429303, -0.0116485134, -0.0219518971, -0.187667757, -0.0626360103, -0.028858915, 0.153726026, -0.104429685, -0.266087621, -0.209274143, -0.186508, 0.180915117, 0.156441614, 0.203999043, 0.144177482, 0.10513787, 0.0303519256, 0.133759394, 0.192577541, -0.140958086, 0.237446681, -0.237315372, 0.0912553743, 0.172334418, -0.11051251, -0.380104393, -0.185993105, -0.231100082, -0.0684015378, -0.165600955, 0.194090798, 0.0481378883, -0.139796764, 0.130825281, 0.172460839, 0.265127957, -0.112289988, -0.0345997512, -0.167480007, 0.0347576514, -0.0154025862, 0.0508864224, 0.138450637, -0.143623456, -0.216727793, 0.0870179385, 0.152233243, -0.218138441, 0.134071931, -0.105602548, 0.0766346306, -0.210313886, 0.173437417, -0.0167097338, 0.176717728, 0.260095805, 0.0725469142, -0.0281031746, -0.0118673686, -0.23178342, 0.196914256, 0.207952037, 0.0597638041, -0.0669040531, -0.202766195, 0.105974823, -0.196885899, -0.130043596, 0.0408547632, 0.051734861, 0.150090992, 0.126557499, 0.0610106736, 0.0459405072, 0.217397436, -0.178916857, -0.235516325, 0.257763088, 0.0747808293, 0.144583955, -0.205134392, 0.245919466, -0.208999187, 0.260882437, 0.132566705, 0.150488973, -0.00251174299, 0.13973631, 0.0961362347, 0.177716032, -0.0470190607, -0.0734431297, 0.0359828062, -0.00525023043, 0.102971934, 0.0987021625, -0.173347533, -0.00715078134, 0.127415687, -0.0373299271, -0.204287812, 0.178136423, 0.138002157, 0.0237582866, 0.174087659, 0.240981013, -0.116837405, 0.130510405, -0.000766741985, -0.124521762, 0.261766434, 0.236482263, 0.087483488, 0.248471096, -0.0924688652, -0.0650356933, -0.0104683442, -0.0764830336, -0.209237933, 0.0235566385, 0.124604762, 0.106890164, 0.159328818, -0.0968483388, 0.100116894, 0.12527816, -0.213597402, 0.0560539104, -0.121492833, 0.0191260874, 0.126306266, 0.0674194768, 0.0697287023, 0.0672566965, 0.0521879978, 0.053629946, 0.205602214, 0.0651868656, -0.0143089797, 0.175055593, -0.143693537, 0.184233233, 0.245637834, -0.0019021834, 0.0554781668, 0.122372709, -0.0944118276, -0.00765591115, 0.246960357, -0.0359783396, 0.013843908, 0.250939488, -0.0550113358, -0.0771496817, -0.129822791, -0.0721774176, -0.287194103, -0.0553002506, -0.0833646432, -0.0302243531, -0.209284484, 0.0714682192, 0.174552351, -0.00634080404, -0.255132675, 0.0539513268, -0.171819359, -0.130697995, 0.0328636803, -0.172556356, -0.2824184, -0.0451180376, 0.0577123426, -0.192122251, 0.0324847363, 0.00184812211, -0.140389964, 0.0564051718, 0.0673946068, -0.0826997831, -0.218807384, -0.226912007, -0.0740968361, -0.0628938675, 0.0246492196, 0.0681713596, -0.344983399, 0.0526000336, -0.31024906, -0.206341609, -0.216349587, 0.0267339684, 0.122782297, -0.178241864, -0.0923086107, 0.0223308429, 0.136397615, 0.248619109, 0.200533465, -0.293138444, 0.311404914, 0.239410847, 0.0427243561, 0.252901375, -0.0671737939, 0.0358522087, -0.101214036, -0.0909479931, 0.312909693, -0.0543796271, 0.225179315, -0.30917415, -0.0924400315, 0.233333379, 0.0843650997, -0.160150632, 0.179808214, -0.0429063886, -0.0673761442, 0.215058282, 0.171212927, -0.0550884008, 0.142365858, -0.110932022, -0.169926539, -0.0976140499, -0.0154480785, 0.0212051291, -0.0351677053, 0.020173341, 0.0828600079, 0.0684699938, -0.140169322, 0.12288864, -0.249438584, 0.161289573, 0.183076456, 0.0643565208, -0.0405365787, -0.003901063, -0.0275522638, -0.114001192, -0.344557256, -0.0885162503, -0.06081542, -0.332393795, 0.277116388, -0.0268625468, -0.190394998, 0.21460636, -0.215998247, -0.222107425, -0.255408615, -0.136359274, -0.14687404, 0.142695963, -0.140400141, -0.0201289766, 0.0542479455, -0.00637657382, 0.137159288, 0.123378307, 0.173221618, 0.0176266842, 0.0871137902, 0.314738423, -0.24674274, 0.139450938, -0.0980865434, 0.0819776729, -0.202197522, 0.0445437841, 0.0490690246, -0.248550311, -0.235274941, -0.334431201, -0.0380337983, -0.0726476014, -0.166573018, -0.0421880521, -0.231450424, 0.130716771, -0.0721551031, 0.11855723, -0.14029862, -0.0331737548, -0.018478848, -0.0687058344, -0.1540602, -0.107552357, -0.146992445, -0.246584743, 0.264962852, 0.0624919087, -0.0870190263, 0.115786649, -0.114350855, 0.212790087, -0.20117563, -0.0133681539, 0.204012766, 0.191788897, -0.0210248157, 0.115564667, 0.113092259, 0.174278691, -0.148719802, 0.190654084, 0.0438634008, -0.0724180192, 0.134725466, -0.123058394, 0.162449196, 0.204366207, 0.116563216, -0.19426021, -0.0909457207, 0.199671999, -0.118528321, 0.117968924, 0.109732315, -0.0419445187, 0.00864718016, -0.0645976812, 0.0311101824, -0.109628826, 0.111323684, 0.014768647, 0.208999589, -0.094222419, -0.179808035, -0.0267504808, 0.109660603, 0.217561051, 0.106540732, -0.00727470964, 0.0496581346, 0.134096339, 0.0660558417, 0.167213649, -0.0612058528, -0.0911486596, -0.0100888135, -0.155831024, 0.189135149, 0.156071231, -0.00602033734, 0.0703240484, 0.0744462162, 0.0984698087, 0.140996054, 0.124672696, -0.163873687, 0.0303707868, -0.199095607, -0.0432972983, 0.0943269432, 0.0672637746, -0.0916577727, 0.0945999026, 0.271431386, -0.146770418, 0.228228882, -0.088630408, -0.221145526, 0.201267377, -0.0209989715, -0.205188558, 0.0660831109, 0.165487453, -0.110452496, 0.0229095519, -0.023997318, -0.0244352669, 0.0483070128, 0.0403944179, 0.00371245272, -0.026503861, 0.00920362957, 0.130575255, 0.185562894, -0.150229856, 0.208181933, 0.066503644, -0.14963977, 0.183380142, -0.0742605925, 0.0525272898, -0.207853332, -0.150708884, 0.0244787, 0.118969277, -0.244963139, 0.108839378, 0.370168149, 0.162852734, 0.0989103541, -0.13296926, 0.045421198, 0.0944304913, 0.0636059344, 0.0407316796, -0.128235891, 0.211519986, 0.188827261, 0.0511491187, 0.00440762937, -0.0511926375, 0.0151363136, -0.112162314, -0.0530756265, -0.261404067, -0.0806499943, -0.114475191, 0.092728734, -0.112707078, -0.186766997, 0.16012606, 0.137830883, 0.170057893, 0.185820624, -0.140461251, -0.213634878, 0.125510231, -0.215242818, 0.0796449333, 0.132684961, -0.2006073, 0.0357116349, 0.198004097, -0.0991434678, 0.0635548085, -0.215833962, -0.0722895563, -0.108518705, -0.051846981, -0.137091249, 0.120727405, -0.0786514506, -0.0299482532, -0.0290962607, -0.0490365773, 0.156231463, -0.0395558923, 0.0900194496, 0.128394648, -0.0630546808, -0.0585276112, -0.205579251, 0.160481736, 0.0202968903, -0.163621709, -0.0748255625, -0.184875816, 0.125386044, -0.127115071, -0.143687502, 0.091046527, 0.0920635611, -0.0941656902, -0.173573211, -0.0986982659, 0.0191576183, 0.0842896551, -0.209140688, -0.0771613792, 0.168761611, 0.0210189521, 0.129767984, -0.0285845138, -0.202819064, -0.209608585, 0.0455416664, 0.167025864, 0.163965836, -0.132653818, 0.0619048737, -0.0682924837, 0.166164339, -0.127146959, 0.166915938, -0.199976191, 0.0883914679, 0.122442588, 0.157862335, -0.0999033526, 0.107905447, 0.271243006, -0.0405978113, 0.181895465, 0.10665185, -0.0172348171, -0.263982832, -0.0332699679, 0.253317565, 0.263973176, 0.151911378, 0.0881777182, 0.22092396, 0.1231746, -0.152555913, 0.101217501, -0.179812282, -0.047235027, 0.064411968, -0.100622997, 0.134386688, -0.197145775, -0.0489049777, 0.00595416129, -0.0711699873, 0.0988756642, -0.25260219, -0.135066882, 0.178719059, 0.0527570769, -0.217263788, 0.0104796821, 0.141307697, 0.192717046, 0.0233423207, 0.0181158278, -0.0247748066, -0.1053892, 0.0186107531, 0.0304267742, 0.247790694, 0.0885608569, -0.165538073, -0.0982961208, 0.078451246, 0.0747933313, 0.149838224, -0.294142485, 0.204276547, 0.0315016098, 0.148058638, -0.0792296454, -0.00655980362, -0.0633319467, -0.134122044, -0.0603130311, -0.228715405, -0.0372798219, -0.0637207702, -0.00131563691, 0.0267799813, 0.205451921, 0.0369303524, -0.194896266, -0.146388203, 0.0251822565, 0.10831248, -0.304889441, -0.067542769, -0.0279039573, 0.224844977, -0.0980764031, -0.177602947, -0.11175137, -0.233728245, -0.223739907, 0.0452572368, 0.0688700527, 0.0517109595, 0.0646637455, 0.0814413205, 0.185665578, 0.199086443, -0.045935303, -0.206678033, -0.110741898, -0.0746753067, 0.0203328282, -0.0121729225, -0.32386151, 0.317199111, -0.000200206137, -0.0206671208, -0.0143212825, 0.109568812, 0.127662241, 0.148976833, 0.134836257, -0.0659915805, 0.0971495807, 0.129318729, -0.261195183, 0.139618188, 0.175515547, 0.177529424, -0.0397923216, -0.171056911, -0.152844191, -0.256262839, 0.0387250036, -0.109484434, 0.348202139, 0.181829244, -0.0921679214, -0.14175418, 0.351582646, 0.0428714491, 0.109188475, 0.113643356, 0.190801248, 0.0840984732, 0.0745595545, 0.202311695, 0.110946044, 0.0192239713, -0.138841808, 0.142307326, 0.354664713, -0.0450815856, -0.107993297, -0.03863943, -0.0024780829, 0.0134169487, -0.117628835, 0.0603437982, 0.166732147, -0.118978985, -0.163896814, -0.0940616056, 0.139851525, 0.0401148871, -0.000361859042, -0.0329533368, 0.00609338423, 0.0956700072, 0.0159509256, -0.183647871, -0.0647861436, -0.0180492532, 0.126684785, 0.174701124, 0.00719110668, -0.0489515066, 0.151985407, 0.0191572756, 0.103651136, 0.0472620092, 0.0433273539, -0.0642805994, -0.117137074, -0.117250271, -0.217558905, 0.238560513, 0.156538591, -0.201861724, 0.252844602, -0.153291538, 0.0394916683, 0.131754085, -0.168700293, 0.282408744, 0.0575271547, 0.270327926, -0.210436061, 0.136073276, 0.0850231051, -0.187773168, 0.179164112, 0.0486085825, 0.131480142, -0.0669804588, -0.12845093, 0.136758476, 0.183792964, -0.0880155787, -0.0198557992, 0.0737654716, -0.150122464, -0.181854174, -0.0218842644, 0.244106069, -0.0331436694, -0.118402436, 0.112792633, 0.161135405, 0.193292305, 0.0654401034, 0.151135877, -0.105567589, 0.163530335, 0.0537123606, 0.115299411, -0.107796557, 0.144485876, 0.190182522, -0.225720987, -0.188096419, 0.0644563586, -0.219243228, 0.0506861359, 0.0646403879, -0.155654714, 0.0720595792, -0.0648836493, 0.0587573051, 0.115380988, -0.144375831, 0.193385601, -0.216615528, 0.0823164284, 0.121625237, 0.0662951022, -0.104674295, -0.0913950354, -0.0744329914, 0.0588016734, -0.0569245294, -0.123344973, -0.112728342, 0.0536800511, -0.0440075137, 0.00869007315, 0.231819123, 0.180460185, 0.112645507, -0.151289985, 0.170129269, -0.118003756, 0.0397904888, -0.0155688487, 0.000529384532, 0.16991967, -0.0197017621, 0.0159432869, -0.152901173, -0.141727105, -0.209757477, 0.0510494262, -0.206472322, -0.125095367, -0.144546479, -0.213549063, -0.0514436178, -0.0335596912, 0.141235679, -0.224663511, -0.0350644737, 0.0376378372, 0.17774488, 0.188020244, 0.0334532149, 0.155813828, 0.0600071736, -0.0559457168, -0.0678997114, 0.0960994884, -0.202544078, -0.157427654, 0.0421013534, 0.115875132, 0.152794838, -0.12245059, -0.152902767, -0.212830245, -0.124761559, -0.202095598, -0.0178206097, 0.126928881, -0.0542535968, 0.128561482, 0.212066635, -0.144553557, 0.0753035396, -0.1383304, 0.0503492504, 0.265743077, 0.227717698, 0.131189972, 0.0942342579, -0.0386557281, 0.00459791953, -0.151728719, -0.0490803644, 0.170358211, 0.107892729, 0.027722558, -0.0222314857, 0.0439844616, 0.0846926421, -0.136754051, -0.126678228, 0.0100780185, -0.00410804106, -0.0236090273, -0.235840544, 0.116327874, 0.12390665, 0.154099762, -0.0710356757, 0.0358319879, -0.00236812909, -0.056195125, 0.0473820642, 0.121515736, -0.12424425, -0.177752599, -0.165439278, 0.0420489013, 0.13842456, -0.122449316, 5.4429478e-05, 0.0483980328, -0.198470056, -0.0108445771, -0.129893675, -0.102530636, -0.0193273257, -0.14624238, 0.08766298, 0.0668683425, -0.133514196, 0.0853877515, -0.0655543208, 0.133385897, 0.00266161677, -0.10532745, -0.0290171318, -0.00419039, -0.00792111829, 0.0604869053, 0.00910193752, -0.118941627, -0.12992464, -0.172481984, -0.012415126, 0.165430143, 0.0105601074, -0.0124265226, -0.204574227, 0.0933492258, -0.0265834965, 0.0440250263, -0.120509379, -0.237719804, 0.141081452, 0.251164675, -0.00922667235, 0.0145384986, -0.23117803, 0.120755881, -0.0217975043, 0.120932087, 0.0436988175, 0.000108511711, -0.174057677, -0.0660731643, -0.0309707671, -0.133766994, 0.115545824, 0.188281238, 0.153618366, 0.0869733766, 0.126192153, 0.0268286113, -0.138225377, -0.106887072, -0.0767892227, -0.220131189, -0.119694576, 0.00380183011, -0.226367459, -0.111844957, 0.152785808, 0.242726147, 0.106298521, -0.248363763, -0.32967785, 0.105129965, -0.155959815, 0.138976559, -0.00137228239, 0.0948434696, -0.0816367492, 0.0710474625, -0.418901235, 0.135055959, -0.310039103, -0.0387624092, 0.249349698, -0.416977942, 0.0891338736, 0.00944569428, -0.237012804, 0.0804961771, -0.195645198, 0.0945587382, -0.0762844086, 0.0416320711, 0.00949457288, -0.127774417, 0.259676754, -0.40856576, 0.0794008449, 0.0908604041, 0.133119613, -0.100699835, -0.156859353, -0.162409276, 0.00788537692, -0.0637622774, -0.32110858, -0.134144261, -0.206960112, 0.0118728764, 0.0764703378, -0.394238651, 0.183452353, 0.241670236, -0.141249031, -0.16704978, 0.018816743, -0.0430508442, -0.170661062, 0.176272959, 0.16203025, 0.23600857, 0.149680734, 0.0821367577, 0.175770909, -0.126697093, -0.148051918, 0.190101504, -0.0317378193, 0.0456583053, -0.270201981, -0.0483634844, 0.319031864, 0.0222948454, 0.0767141506, -0.00711641507, -0.153200984, -0.143897697, 0.140922055, -0.0283886902, -0.113231972, 0.139692098, 0.142846361, -0.157825753, -0.100115009, -0.0507604778, 0.0704903975, -0.0313803554, 0.161187619, 0.0637935027, 0.154604718, -0.178512841, -0.108615682, -0.119129255, -0.0183542315, -0.200408816, -0.06402006, 0.0961765796, -0.183909222, 0.103326656, 0.12906833, 0.175179169, 0.075670667, 0.138392508, -0.121290363, -0.0992279351, -0.141292989, -0.0473258048, 0.130663127, -0.147083119, -0.123233199, 0.203898117, -0.204678267, 0.167588547, 0.158947214, -0.115444884, 0.0865047872, -0.162406579, 0.00433421135, 0.0109670609, 0.0494914539, -0.0845709294, -0.0436661392, -0.0943619311, -0.133204848, -0.133604929, -0.0241765436, 0.0312332567, 0.0160661489, -0.192561835, 0.170536771, 0.0699443966, 0.18987824, -0.198280796, 0.13675791, -0.128286049, 0.133142799, 0.0423047841, 0.19421573, -0.0902426615, 0.045400776, -0.0236111488, -0.0612643398, -0.0522969365, -0.185536757, -0.0624252073, 0.0719867498, -0.145684376, 0.342741668, -0.169891864, 0.189545587, -0.20563516, -0.106448837, -0.00803494453, -0.139683664, 0.239471704, 0.347251058, 0.0986964926, 0.191767052, 0.0345206708, 0.117405772, -0.0646648407, -0.0939145163, 0.0358834863, -0.14516075, 0.329907864, -0.245812029, -0.20081225, -0.128157064, -0.32458353, -0.202067211, 0.310102135, -0.259800404, -0.183582872, 0.348934501, -0.00135924411, -0.00762309879, 0.0397878811, 0.0435562618, 0.190664694, -0.219969705, 0.167273611, -0.0363034643, 0.0843212157, -0.0630743131, -0.127757251, 0.133702457, 0.241022587, -0.0452217422, 0.157935485, 0.0468397252, -0.184891075, 0.0217796862, -0.174830914, 0.0529149808, 0.0344027728, 0.0301657226, -0.0991806537, 0.0966322273, -0.0987405106, 0.0616976731, 0.037891306, 0.144457489, 0.293943793, 0.125130758, 0.279702634, 0.2190516, -0.0891123265, -0.319427043, 0.020325454, 0.198740065, 0.244544879, 0.150971532, 0.139485016, 0.155953914, 0.100290887, 0.039516408, -0.11156898, -0.239001468, 0.0233942177, -0.0897894874, -0.0399748348, 0.141847938, 0.0783665776, 0.00495733274, 0.020279035, 0.166984901, 0.280435681, -0.217270985, 0.185803846, 0.191354558, 0.0111610517, 0.1644153, 0.0352947488, 0.0664995685, -0.0161591228, 0.0244116578, 0.0823068097, 0.0366923697, 0.20036611, 0.0597134568, 0.0136301629, 0.0214036219, 0.0707080811, -0.0257597454, 0.141371503, -0.0871877447, -0.0384720117, 0.159895733, -0.271953613, 0.118647724, -0.0838832259, 0.14117156, -0.0238901209, 0.0837025568, -0.0994942114, -0.311766535, -0.0361485183, -0.173598096, -0.0820912719, -0.109803088, -0.202099934, 0.13466467, 0.298355758, 0.147975996, -0.0162965041, 0.0887476951, 0.0656182021, 0.158688262, 0.00327817141, 0.216407076, 0.0288510714, 0.0746814311, 0.0788815916, 0.183364213, 0.149168417, -0.0533465818, 0.120975912, -0.0698309764, -0.131480917, 0.0775775313, 0.190101609, -0.175806463, 0.208605766, -0.0509476848, 0.0475929938, 0.172246516, 0.128037199, 0.135146201, 0.04195638, -0.179263756, 0.191762373, 0.124527775, 0.18047376, 0.0364429019, 0.133441925, -0.0794005841, 0.152522027, 0.0759226233, -0.194360182, -0.11856693, 0.0628863648, -0.140197754, -0.118163697, 0.148727104, 0.109244518, 0.0861630365, -0.0484799929, 0.144106314, 0.0300433505, 0.159115046, -0.0456953831, 0.159014627, -0.230968624, -0.191417232, 0.079684414, -0.0845753998, -0.216385618, 0.1015696, 0.12075875, -0.195914701, 0.0704701394, 0.00612893514, -0.172618523, 0.14040117, -0.0350932516, 0.0685307756, -0.0815743059, 0.0343151689, -0.226708308, 0.0161583424, 0.00600387063, -0.0403283834, -0.200709447, -0.136831269, -0.0756262839, -0.0913945809, -0.00991040468, 0.0491666384, 0.181557953, -0.0815197825, -0.1748669, -0.105041094, -0.024442181, -0.137364954, 0.213511899, 0.114984736, 0.141203478, 0.191028729, 0.209437281, -0.117445506, -0.211069152, 0.213400275, -0.00855989754, 0.0147007108, -0.17848292, -0.160719216, -0.169281244, -0.00666991761, -0.12999402, -0.017418623, 0.0077680028, -0.096811451, 0.0399670899, -0.099848032, 0.00562751293, 0.0391903967, 0.144329935, -0.0322996452, 0.142276108, -0.0690825805, -0.215008646, 0.0819310695, -0.147535652, 0.157100156, -0.100781769, -0.191613704, -0.178416789, -0.164667308, 0.029264966, -0.00163395703, -0.157853901, -0.0132551193, 0.0478072613, -0.149802342, 0.168672904, 0.0820260644, -0.120356776, 0.0662041232, -0.183392614, -0.178459927, -0.156899661, -0.164349243, 0.209907949, -0.115875721, 0.0444762632, -0.201963484, -0.0449665599, 0.198717207, 0.198328122, 0.0849034563, -0.103813514, 0.117308304, 0.0936804041, 0.0462679416, 0.0836406723, -0.0418322682, 0.0411524326, -0.190647915, 0.0886535197, 0.211842492, -0.0770319477, -0.0116216559, 0.147017792, -0.0120076491, 0.0194121003, 0.138708234, -0.120179571, -0.0352452397, -0.028329812, 0.0094909966, -0.00187779963, -0.0943269953, -0.078908205, -0.0844167471, -0.197576553, 0.121277407, 0.210520267, 0.141214922, 0.0709877908, 0.185094103, 0.119538829, -0.0926069394, -0.0566524863, 0.17638126, -0.0237376336, -0.135814071, -0.136954382, 0.119367145, -0.203730926, 0.00643029623, 0.167091712, 0.179837942, -0.10910327, -0.0022002249, -0.169260845, -0.0575643629, 0.0475613885, 0.114217445, 0.0275517702, -0.15122728, 0.000335678458, -0.201629221, -0.191943482, 0.0599358231, 0.215006664, 0.157104149, 0.123682573, 0.199631587, -0.193868354, -0.253842771, -0.192569867, -0.450649053, -0.13617, -0.0669108927, 0.111150347, -0.00369961141, -0.191271275, -0.237755463, 0.181265593, -0.132041126, 0.157904267, -0.0143442852, -0.395011663, 0.0413822122, -0.119375452, -0.274717003, 0.0961166471, -0.392918706, 0.138946593, -0.406194896, -0.126115769, 0.103300825, -0.0749610662, 0.187398925, -0.0632039681, -0.0863866061, 0.222676188, 0.219102636, 0.28613168, -0.187663198, -0.416728288, 0.0453014523, 0.244026601, -0.129714295, 0.295904279, 0.085724242, 0.0173482616, 0.17430979, -0.268255919, 0.0690714642, 0.0642987117, 0.0120566841, -0.298500836, -0.250954837, 0.0702187121, -0.439573526, -0.121676624, 0.167861462, 0.185528114, 0.26526314, 0.27663222, 0.25443691, 0.0214734077, 0.161424711, 0.144671425, 0.157419518, 0.182189599, -0.0776689202, -0.0120218601, 0.271168381, 0.156823754, -0.127337053, 0.0545059741, 0.128410771, -0.148533046, 0.0630049855, 0.0160781369, 0.151448995, 0.101595782, 0.0654489025, -0.167899147, 0.13213931, 0.0983135328, 0.0369849391, -0.194617927, 0.0153781129, 0.270563185, 0.0342637785, 0.0746257529, 0.211298779, 0.154260978, -0.119062982, -0.0627138913, 0.259788841, 0.117369875, -0.0632641613, -0.137389138, -0.2181786, 0.174714953, -0.0711210594, -0.237840936, -0.0302677024, 0.0867897719, 0.185713023, 0.240260184, -0.186787859, 0.0108405575, 0.0771833137, -0.141014621, 0.147447675, 0.252978861, 0.0547764972, -0.0874451548, -0.31400758, 0.118284583, -0.199673429, 0.111848548, -0.214292303, -0.0464315489, 0.230785057, 0.18862094, 0.0352876596, 0.00474979123, 0.0109337727, -0.0291237906, 0.122409284, 0.128479972, -0.105726346, 0.106454507, 0.1788349, -0.0558397211, -0.0373482071, -0.0495012775, 0.0530157499, -0.163363129, 0.202189162, 0.0545998327, 0.157361299, 0.214383185, 0.107534043, -0.200028911, -0.125518799, 0.216706932, 0.230916902, 0.250411302, 0.146487787, -0.01959024, -0.140795499, -0.0633696094, 0.0885654092, 0.0913219228, 0.0871412084, -0.0358804837, 0.0180488303, -0.0806887895, -0.0637854189, -0.190897569, 0.136343226, 0.0202956051, -0.0698644817, 0.239365906, -0.306738168, 0.180551901, -0.0763572007, 0.0489863828, 0.00122147053, -0.0715313926, -0.173467308, -0.174637392, 0.170282349, 0.186628222, -0.00949032791, 0.00133445614, 0.011871323, 0.00409735739, 0.0181704815, 0.117498547, -0.129429266, 0.120077997, 0.216407701, 0.180566475, 0.232433349, -0.0555412471, 0.189128026, -0.151290759, 0.180261225, -0.321341038, -0.101906769, -0.174282476, -0.286496341, -0.0306703895, -0.115755208, 0.171560839, 0.127792448, -0.0103189619, -0.0854421407, 0.20230858, -0.135044008, 0.137085229, -0.0906790271, 0.206210405, -0.109169461, 0.221058965, -0.203725383, -0.223818555, 0.00837364979, 0.0698773786, -0.11478246, 0.0962926373, -0.0567478091, 0.194004565, -0.0646269023, -0.230514511, 0.121396624, 0.051594045, 0.0810926184, 0.11312753, 0.117401369, 0.0351090729, -0.101227865, -0.0286359861, -0.152758554, 0.195657834, -0.129182458, 0.255799025, 0.0658524111, -0.133879721, 0.135263368, -0.117422193, 0.259024024, 0.12137039, 0.0429658368, 0.161656618, -0.109413959, 0.0212555416, 0.00380118797, 0.0245974474, 0.0452777967, -0.109418437, 0.0556083173, -0.0991568714, 0.240161121, 0.131009638, 0.21446988, 0.0535303056, 0.0080528371, 0.0592104085, -0.117336079, 0.101440094, -0.180672362, 0.153361961, -0.148895979, 0.123094238, -0.20419763, -0.00546182692, 0.169995323, -0.0374472365, -0.0513039343, -0.100886956, -0.144634396, 0.226476029, -0.123933963, 0.082715638, -0.0514412038, -0.137042806, -0.0798420236, 0.295484096, 0.14945595, 0.0148293832, -0.141559213, 0.152552426, 0.110004902, 0.264642984, -0.182816103, 0.203673571, 0.0767816678, -0.0460664965, -0.0965382606, 0.00824740529, 0.00633397093, -0.0335266478, -0.00525524374, 0.0221320633, -0.144528076, -0.181572482, 0.186975211, -0.0915289372, 0.0789494962, 0.0443420336, 0.0566833429, 0.0106719388, -0.153921574, 0.0117017636, 0.0780537501, 0.172404632, -0.0487603694, -0.0259934999, -0.112953916, 0.013087403, 0.199101657, 0.0694961324, 0.099969998, -0.0189182963, 0.137308478, -0.00687692454, 0.130568698, 0.157788232, 0.0861073285, 0.195408612, 0.237710238, -0.0510148071, -0.127946258, 0.0196243692, 0.0884056464, -0.229083344, -0.0584382601, -0.0112535618, -0.056976635, 0.207119659, 0.0605573431, 0.170117199, -0.0873071477, 0.0375184156, 0.0693956614, -0.0853421167, 0.168883324, -0.246331498, -0.15294233, -0.0786210001, -0.0727810487, 0.230497375, -0.124767907, -0.0180434044, 0.152893081, -0.176393285, -0.135040537, 0.012329434, -0.066455029, 0.0633047223, -0.168565243, -0.169502109, -0.223331943, -0.168321326, -0.0599934012, -0.0564355031, 0.199666232, -0.193147793, -0.0922575146, -0.0880292282, -0.181692928, -0.200924233, -0.170735195, 0.138240859, -0.0760595798, -0.0921700075, -0.166161865, -0.0384436809, 0.0141204651, 0.130763844, 0.105647944, 0.153559715, 0.212668225, 0.0108604385, -0.019111041, -0.140727684, 0.150457844, 0.1883111, 0.221798778, 0.112573713, -0.165191919, 0.0167138427, 0.24837476, 0.165022895, 0.240100026, -0.0641816482, 0.156478882, 0.19513236, -0.0954566598, 0.0913641751, 0.0593185239, -0.123686202, 0.053503748, 0.0152200609, -0.153226435, -0.145596594, -0.0840086117, -0.179127425, 0.0691409111, -0.0299637914, 0.152311578, 0.0949365795, 0.00141828961, 0.201368794, -0.174666852, -0.0636612177, -0.171069294, -0.13758266, -0.182560191, -0.137745142, -0.127387106, 0.148039132, -0.000196392211, 0.176657051, -0.127840057, -0.0359740965, -0.0467125587, 0.00534770545, -0.0455735289, -0.177512407, -0.173216969, 0.162237197, 0.04842823, -0.178101718, -0.0483464934, -0.167974755, 0.0910376757, 0.184863344, 0.174440339, -0.133150682, -0.120608732, 0.217321798, 0.269066572, -0.138795853, -0.0962826163, 0.141585678, 0.243578151, 0.226173848, -0.0334078334, 0.0868586823, -0.236201584, 0.0429105237, -0.00714816013, -0.183364853, 0.0685243681, 0.0485652611, 0.211708516, -0.145325571, -0.0299601406, 0.0740182772, -0.17283687, -0.146753222, 0.0394501612, -0.102561951, 0.279482722, 0.234896556, 0.136510789, -0.0687329471, -0.146247506, 0.166320026, 0.088236481, 0.0455387309, 0.0368321836, 0.0928156599, 0.251261562, -0.202283695, -0.0876553059, 0.188739464, -0.1219403, 0.0595511906, -0.0864975601, -0.0519133434, -0.159869671, 0.255505502, -0.0236511845, -0.099469468, 0.146673471, 0.00879366975, 0.202414125, 0.200698897, 0.118802421, -0.0520094372, -0.194901958, -0.0494996794, -0.132057235, 0.0713604391, 0.166914493, -0.103728242, 0.173196629, -0.108285852, 0.130671516, 0.00665229931, -0.216195241, 0.00278148265, 0.150077969, 0.0377425104, -0.109352857, -0.0078518251, -0.143112957, 0.237058267, -0.24492383, -0.232783735, 0.0026126157, 0.0566774793, -0.217854828, 0.158665374, -0.141393185, 0.240377933, -0.0147471335, 0.105589516, -0.132414341, 0.269156039, -0.0360066108, -0.279901594, -0.070857726, -0.000133716909, 0.0994284675, -0.399730533, 0.0423182473, -0.0807459578, -0.364677131, -0.173550189, -0.201698035, -0.150411874, -0.104539521, 0.0632497221, 0.0475217737, 0.106961772, -0.0748255625, 0.0537245125, 0.150076792, 0.100195438, 0.160947844, 0.136155531, 0.0336693786, 0.00195461512, 0.0391892754, 0.155441701, 0.0603906885, -0.0828605369, -0.188219786, 0.01371055, -0.108915485, -0.188475981, -0.00214913161, 0.209178224, -0.0138332155, 0.106863379, 0.17023693, -0.104419991, -0.0188917425, 0.124385007, -0.112276614, -0.0786361247, -0.047841236, -0.249989852, 0.157759428, 0.0704554766, 0.0761716887, 0.124297529, 0.132825673, -0.0735627264, 0.202956781, -0.0342735052, 0.110366948, -0.150816396, 0.152661726, -0.146618992, 0.171531007, 0.0614210069, 0.077137284, 0.0930158645, -0.143225402, -0.158822253, -0.251074195, 0.135286197, -0.0735299885, 0.244000822, 0.113809302, 0.116750523, 0.051723171, 0.183311462, -0.137916028, 0.0244293083, -0.088045761, 0.0404897481, -0.0778224021, 0.131730989, -0.0429636389, 0.115714654, 0.0684564859, -0.044515267, 0.00754295383, -0.050703045, -0.129571319, -0.187777609, -0.16493459, -0.126211151, -0.0829479098, 0.0330205783, 0.243688241, 0.13541998, 0.0975747928, -0.206415966, -0.0957572684, -0.0585407391, -0.195936382, 0.123246349, 0.13101624, -0.196200132, 0.0490147881, -0.0278630313, -0.224047154, -0.20703429, -0.0990627408, -0.115552947, -0.419253439, 0.0287015885, -0.0131201446, 0.16262652, 0.122940429, -0.308744431, 0.117334351, -0.00441871164, 0.158816338, 0.171548396, 0.0269443281, -0.146471247, -0.013632034, 0.217089698, -0.228731453, 0.0371344909, -0.157528311, -0.0783996806, 0.00250388891, -0.308794379, 0.221041724, 0.121599473, -0.219423294, -0.411408722, 0.115201004, -0.142029077, -0.111949541, -0.151291326, -0.0684362724, 0.147531658, 0.108987704, 0.28183502, 0.207470536, -0.0262030065, -0.0661180243, -0.0931391194, -0.0792838484, -0.211057425, -0.32554251, -0.183445573, 0.00182158989, 0.121516146];
    CONSTANT bias_11 : ARRAY[0..63] OF REAL := [-0.00635589194, 0.0714284107, -0.0793445706, -0.0154935429, -0.0884047896, -0.00860749092, 0.015439475, -0.0443723239, 0.0648666918, 0.0137735978, -0.0558123514, -0.0234004352, -0.0720951036, -0.0323092379, -0.0251345523, -0.0864192247, 0.0349380858, -0.0508749001, -0.101302393, -0.00825020857, -0.0878332034, -0.0217018481, -0.0879978016, 0, 0, -0.0321543552, 0.0255989321, -0.0501851514, 0.0153964404, 0.0969368443, 0.0876909047, 0.0749777704, -0.00993307587, -0.0840824917, 0.107733645, 0.0926610008, 0.000463146862, 0.0615399294, -0.0173791237, -0.00302339089, -0.00108950492, -0.0433365181, 0.0978755206, -0.0621731691, 0.0341274589, -0.0879570246, 0.00440526195, 0.00455495017, -0.0902555734, -0.0262572207, -0.0154181952, 0.0162822157, 0.0986388773, 0.0995882377, 0.0237515792, 0, -0.0163629819, -0.02235475, -0.00682879193, -0.0143427243, -0.0962111577, 0.0128893042, 0.0858025402, -0.00971365813];
    CONSTANT weights_12 : ARRAY[0..4095] OF REAL := [0.106257081, 0.00435368251, -0.200017139, -0.170659184, 0.140568718, -0.121934257, 0.121075258, -0.16430898, 0.0690469891, 0.0433366559, -0.062450733, -0.20864369, 0.149895057, -0.0887060761, -0.0112437466, -0.137328371, -0.182793975, 0.00182112318, -0.192540094, -0.0729949772, 0.0874842256, -0.199801773, 0.161684632, -0.20927608, 0.18800509, 0.0292491615, 0.1377161, -0.00336401165, -0.0864470974, 0.13110055, -0.151119724, 0.182269529, 0.177959964, 0.145959258, -0.153364599, 0.208557755, 0.107231423, -0.122332707, -0.0526105985, -0.0178942829, 0.171287671, 0.0380937643, 0.210034788, 0.114255026, -0.176481709, 0.159083605, -0.0201071408, -0.0995351151, 0.158686295, -0.121905096, 0.0662830025, 0.145770177, -0.202360839, 0.108805642, -0.00403741794, 0.0131892227, -0.110621646, -0.0315053463, 0.0544626564, 0.0432279147, -0.0527887791, 0.0743454844, 0.000725448132, 0.13499485, 0.249794126, 0.201496869, -0.105599739, 0.115793243, -0.0131411431, 0.0381885171, 0.0861910731, -0.127799913, -0.0971342772, -0.12288598, 0.262936473, -0.178271964, 0.0656890273, 0.0264430493, -0.112000212, -0.0541253053, 0.0306299999, 0.030385958, 0.188352376, 0.216451868, 0.0554085672, 0.0997735932, -0.0144361956, 0.293800294, -0.2299909, -0.0211171489, 0.0223787352, 0.207233086, 0.164753318, 0.177156463, -0.0375560075, -0.0163145456, -0.0929765627, -0.104105949, -0.0902710557, 0.251464099, 0.178618342, -0.289695442, 0.0912541896, 0.120610818, -0.046938058, -0.0419063605, -0.189616457, 0.0257992372, -0.130752474, 0.205490381, -0.194339946, -0.151713759, -0.17453213, 0.178030372, 0.173221558, -0.0263473187, 0.186066285, -0.153767124, -0.00557854539, -0.177357957, 0.270246536, 0.203962401, 0.238550261, -0.148142517, 0.269313812, -0.0103741148, -0.183588952, -0.193594933, 0.162554562, -0.115353428, 0.0583416782, 0.0762180537, -0.09497796, -0.214766502, 0.139911622, 0.131524205, 0.00997098256, -0.11585062, 0.164202839, -0.320977002, -0.0759125501, -0.0785337314, 0.0255053025, 0.128980473, 0.0306141712, -0.126000479, 0.107428253, -0.118020132, 0.138766393, -0.284001321, 0.170607731, 0.102398202, 0.148915827, 0.160759792, 0.110466659, -0.252095222, 0.139449462, -0.315892965, -0.244656861, -0.123431899, 0.170097247, 0.321350873, 0.175645128, -0.206368536, 0.175698891, 0.00147240586, 0.29501459, 0.0298838075, 0.296299219, 0.187590197, 0.212566584, 0.11760661, 0.0084051853, -0.10937953, 0.149446264, 0.106912412, 0.118477888, -0.116064332, -0.0906607434, 0.0801626742, -0.060745582, 0.118430406, 0.241397575, -0.199510291, 0.1551781, -0.296400189, -0.0104944538, -0.145789325, -0.129684851, 0.0872599632, 0.0820529014, -0.00545078563, 0.218558997, -0.143248811, 0.192341313, -0.201770559, 0.0760860071, 0.106566764, -0.0349904001, -0.00749497209, -0.162278533, 0.247534171, 0.103120431, 0.123288512, 0.166345581, -0.0299496409, -0.244585529, -0.0239745378, -0.0884519145, 0.00908797327, -0.186777309, -0.0307503436, 0.0863535553, -0.029496571, 0.132126838, 0.0579786561, -0.00642398978, -0.0869056135, -0.130231008, -0.0773765892, 0.241189286, -0.0329741426, 0.00026981649, 0.196063191, -0.00166879594, 0.163482696, 0.0171640627, 0.214319944, -0.199893922, -0.0535125323, 0.118300594, -0.342376232, 0.12815164, -0.0961666852, -0.210583001, -0.26564607, 0.176150426, 0.109022953, -0.0346871875, 0.0834982768, -0.189139843, 0.0655928552, 0.091176711, 0.260871142, 0.140941069, -0.0211790819, 0.18120195, 0.180467978, 0.24436079, 0.15343453, 0.288015127, -0.0526540764, 0.196438268, -0.090705663, -0.138662577, -0.251701206, 0.137427241, -0.215658352, 0.0927336663, -0.161177158, 0.185746282, -0.143332213, -0.125291377, 0.217623547, -0.229488418, 0.0239045564, -0.12882176, -0.117315933, 0.127802238, 0.0137906745, -0.092000097, -0.113476872, 0.0914460868, -0.00983959343, 0.0662833154, -0.250207067, -0.0580342449, -0.122949809, -0.00861869287, -0.0351496413, -0.138369471, -0.120193399, -0.181908339, 0.1659161, 0.161926165, -0.243621573, 0.0815375894, -0.22421664, -0.200593099, 0.0567479655, 0.0271451306, -0.143274829, -0.200878218, -0.131388023, 0.264421344, 0.0492096022, 0.0876826793, 0.214776635, 0.0356173888, 0.108095407, 0.0600323044, -0.00878227595, 0.0185248479, 0.167779326, -0.167263448, 0.133649796, 0.0860351771, -0.0738951042, 0.167534858, 0.182380617, 0.0853289813, 0.126694575, 0.0129384911, 0.169833899, -0.119239196, 0.163785785, -0.0672808215, 0.15020664, 0.0820419118, 0.170347661, 0.100519873, 0.100219205, 0.0340493061, -0.20067209, -0.136349007, -0.114618428, -0.19835715, 0.0851126164, -0.147766441, 0.162698075, 0.192914501, 0.188429147, 0.0658050552, 0.034532465, -0.0661727563, 0.13281174, -0.0711044297, 0.0274692085, -0.19102478, 0.106214181, 0.193854347, 0.0253953449, -0.0946320966, -0.166038856, -0.0701704547, -0.203632638, 0.0977531224, 0.0993859842, -0.162032917, 0.0353222936, -0.0693225861, -0.213332132, -0.0769920498, -0.0619540252, -0.170087278, -0.0315041505, -0.0012934655, 0.152092174, -0.164900064, 0.0507530719, 0.152842164, -0.120405428, 0.077816084, 0.11334984, -0.129420042, -0.0410492569, 0.141592532, -0.118363351, 0.135873318, 0.104652397, 0.103805363, 0.20919849, -0.213056386, -0.123535939, -0.0476374961, -0.12322703, -0.0815903842, 0.043837294, -0.104243912, -0.019641865, 0.19847779, -0.0767066404, 0.0687408, -0.18236804, -0.0714362264, 0.0506636314, -0.110496551, -0.0978325754, 0.072953321, 0.00686401874, 0.0755573437, -0.123891488, 0.315234214, -0.154309481, -0.241670758, -0.320736408, -0.0229317304, 0.100737318, 0.0693938807, 0.00485423952, -0.212198153, -0.269200683, 0.111313589, -0.147343546, -0.0591220744, -0.314041585, -0.104359977, -0.196067065, -0.199609593, -0.062965855, 0.282515615, -0.0779074356, -0.0812170208, 0.237137318, -0.167712182, -0.0139279505, -0.229874283, 0.134501129, 0.0717539415, -0.0137814144, -0.207121581, 0.245981425, -0.163413405, 0.223312944, -0.112920046, 0.10596218, 0.128136829, 0.223039329, -0.0331489667, -0.155040503, 0.181968331, 0.0779197216, -0.0980575457, -0.179500878, -0.145538241, 0.112551749, 0.0494974405, -0.0378191695, -0.06296812, 0.135410845, -0.231428131, 0.027612973, -0.211544007, -0.222097173, -0.198571667, -0.042331215, 0.00269386172, 0.173073843, -0.106698252, 0.108658753, 0.231999084, -0.0199163556, 0.0840402842, -0.164054617, -0.169759646, 0.23305276, -0.097792089, 0.0453311168, 0.0280471761, 0.128820732, -0.119299456, 0.115963653, -0.0075415466, -0.112931721, 0.0670242161, 0.302933872, 0.017848229, -0.0486157276, -0.0201860815, -0.0808905512, -0.0494740121, 0.19418247, -0.223715872, 0.204738364, -0.268613338, -0.0106582586, -0.118218318, -0.109672047, -0.0247898009, -0.152243793, 0.117515177, 0.237196997, -0.170047969, -0.143073574, 0.0319675468, -0.291564047, 0.0861566067, -0.139199525, -0.128801718, 0.255365193, 0.143989652, -0.308390856, 0.00239204685, -0.0202191174, 0.121472307, -0.170474201, -0.174699128, -0.165195644, 0.310387254, -0.0541064925, 0.190462306, -0.0273283124, 0.122453421, -0.0220364239, -0.0813105553, 0.197180018, 0.104430646, -0.150599644, 0.307831496, -0.1770574, -0.1636246, 0.0556599572, 0.262393951, -0.182958364, -0.118844286, -0.163353726, -0.0945671052, 0.11168465, 0.0820354596, 0.0180940349, -0.135421559, 0.185812682, 0.258482575, 0.132772148, -0.0373393223, 0.0624215081, 0.0671000555, -0.261657447, -0.130482182, 0.132579386, -0.190884918, 0.041321177, -0.197137892, 0.0326368958, 0.256414056, 0.0671977028, 0.0115289818, 0.0246465355, -0.0270507559, -0.182449952, -0.0699588656, -0.153745219, -0.16926384, 0.0633526966, 0.0229592621, 0.164385095, -0.111254871, 0.0148687335, -0.0871399641, -0.30644083, 0.0704381168, -0.302938342, 0.163136542, -0.163225174, 0.161171958, -0.241714865, -0.0642526448, 0.153364688, 0.102497257, 0.14832598, -0.117911123, -0.22630614, 0.182896242, -0.0571457483, 0.146639496, -0.0514917709, -0.141151905, -0.192691699, 0.0471394546, 0.0913215056, -0.152800024, 0.0426181071, -0.0565117002, 0.00609446457, -0.193988711, -0.0499040708, 0.0436979197, 0.0999253839, -0.0795054361, -0.103425018, -0.209491357, 0.197339267, 0.11044497, 0.204888374, -0.320532471, -0.126293123, 0.151542276, -0.174009621, 0.0993844345, -0.000349115813, -0.281020701, 0.00936588086, 0.0860493854, 0.220661372, 0.170487523, 0.238573328, 0.0244113728, -0.0152693167, 0.200015113, 0.0352645107, -0.237889886, -0.116291612, -0.0838106349, -0.0905120596, 0.218899921, -0.127314493, 0.0822635666, 0.138225093, 0.0179952085, -0.15195632, 0.124049164, 0.092439875, -0.1056609, -0.0491449945, -0.0414935164, -0.141843528, -0.0563498996, -0.0736364797, 0.0624214932, -0.0850778669, 0.17593126, -0.0441847481, -0.155779913, -0.0650813878, 0.0375658721, 0.133375734, 0.0923169106, -0.0893951133, 0.0897832513, 0.0213206448, 0.239664406, -0.148517206, -0.030231189, -0.0527165271, 0.22417976, 0.169856504, 0.296273053, -0.212572232, -0.20888643, -0.016295081, 0.101754785, -0.0549197085, 0.211681917, 0.218397483, 0.18634066, 0.126820177, 0.0505925268, -0.0614112951, 0.0752623454, -0.10380286, 0.0540275797, -0.204340652, 0.145865679, -0.0346987806, 0.065127641, 0.0127901398, 0.199785799, 0.177719668, -0.183774799, 0.0209528748, 0.103368029, 0.0971299931, -0.127705738, -0.212714925, -0.0891776234, 0.15857552, -0.190184981, 0.00605630968, 0.0196366478, -0.153378323, -0.0976148546, 0.0536283739, 0.178155646, -0.0522708073, 0.243760437, -0.256778598, 0.159023032, -0.0108456258, 0.0449721664, 0.00447948091, 0.155550942, 0.0962128639, 0.0743119419, -0.123430736, 0.212962896, 0.0239776131, 0.0913750753, -0.13022694, 0.214200482, -0.0275251269, -0.0230850372, 0.0584084429, -0.137045443, -0.149423778, 0.293362677, -0.231559619, -0.155231133, -0.0807164013, -0.0462920144, -0.117076352, -0.108108059, -0.204536229, -0.0108255595, -0.013456245, 0.264667422, 0.0911884233, -0.181063846, 0.191370711, -0.0283466205, -0.1479083, -0.164247975, 0.191607475, -0.103012457, 0.110606916, -0.000815605745, 0.158466443, 0.00851375796, -0.0969890356, 0.126110435, 0.155427545, 0.189703301, 0.0150730461, -0.182569697, 0.241557285, -0.0367574021, 0.17438066, -0.0277641099, 0.151728004, -0.208000898, -0.134433463, 0.107581556, 0.0131943412, 0.128248185, 0.139681146, 0.026148105, 0.241393596, -0.106327146, 0.0285313632, -0.00392851001, 0.26787442, -0.0786702111, -0.0199960638, 0.0751241669, -0.177954569, 0.179708481, 0.260549545, 0.161560953, 0.0470447503, 0.120685622, 0.140657887, -0.123638831, 0.194805682, -0.0563831925, -0.209175766, 0.0824169368, 0.0606862344, -0.171402454, 0.193776771, -0.00800510868, -0.0670984313, 0.0924971923, -0.101887502, -0.0226375572, 0.240748838, -0.0621666946, 0.0973561406, 0.04852999, 0.183064163, 0.26137805, -0.259445339, -0.0423310697, 0.238807201, -0.159126639, -0.260159343, 0.0155518148, 0.139621124, -0.185930684, -0.167278677, 0.153316975, -0.0289743431, -0.0626375005, 0.120228775, -0.138989061, -0.15610528, -0.122687519, -0.145005405, -0.122514747, 0.0639393106, 0.118220925, -0.0740523934, 0.304092497, 0.0344584249, -0.123333976, -0.0309291482, -0.156307325, -0.0993042886, 0.122875266, -0.0432663597, -0.168591157, -0.281338513, -0.043137081, -0.117354706, 0.134987041, -0.14579919, 0.0790656805, 0.0152693419, 0.286864221, -0.135996044, -0.00733812153, 0.0475724824, 0.292973101, 0.00887088105, 0.112235606, 0.157097444, 0.224297404, 0.0614821911, -0.20666416, -0.00968252309, -0.184044868, 0.114056982, 0.0753099993, 0.0102361599, 0.244052678, -0.207539141, 0.0548489466, -0.167633072, -0.0237612631, -0.231893212, -0.0243409649, 0.164452314, 0.0128334379, 0.0672746599, -0.118385501, 0.0196032487, 0.00372122228, -0.0901152939, 0.0240558926, 0.0934285447, -0.0222456753, -0.185950816, -0.170683146, 0.072074756, -0.0274260845, 0.0501453765, 0.0197149329, -0.166320279, 0.123482324, 0.123843014, -0.109266885, -0.013747978, -0.00779475272, 0.155238539, -0.182944626, -0.0116707738, -0.00189979863, -0.0371467322, 0.000649258494, -0.0684414059, -0.0617489815, -0.0876107141, -0.171610132, 0.113506228, -0.188258782, -0.0664495453, 0.0116472142, 0.115066245, 0.213201389, -0.188051775, 0.157321677, -0.17768763, 0.117324159, -0.163545921, 0.210153237, 0.166902661, 0.0325763598, 0.208137721, -0.00108235527, 0.174134597, -0.0782251731, 0.148419902, -0.0446081758, 0.062131986, -0.0802285075, -0.0112878159, 0.191592947, 0.154550329, -0.130775481, -0.0966541022, -0.0837484226, 0.198908642, -0.100747377, -0.00711986143, -0.105124243, -0.116811574, 0.00965594593, 0.01702323, -0.0357450061, 0.217188969, 0.241389364, 0.112407587, 0.156611636, 0.155096814, -0.192019671, 0.244446054, 0.195701391, 0.22498773, 0.226725683, -0.0261454489, 0.0961467847, -0.160606489, 0.142043069, -0.0130630685, 0.0523964949, -0.0840317458, -0.149799123, 0.100000717, -0.198448598, -0.169559553, -0.146289423, -0.0743390396, -0.0182770509, -0.201591939, -0.0772255585, 0.104011148, 0.153238833, 0.190954477, -0.107943065, 0.0712087154, 0.0700664073, 0.113094702, 0.199309185, -0.158572003, -0.0452618487, 0.223115429, -0.11665412, 0.200311944, 0.272724211, 0.21544452, 0.18986252, 0.0543463267, -0.0146445958, -0.0732405484, 0.0544527434, -0.071323432, 0.0412523821, 0.15092124, -0.044222407, 0.0139736934, -0.206451863, -0.169845477, -0.117359452, 0.0564284809, -0.107622862, 0.056094747, 0.0175767932, 0.0678091124, 0.205945954, -0.199567676, -0.131202608, 0.116727181, 0.00307112304, -0.0610344894, 0.304451853, 0.246360987, 0.00679735234, -0.0727391765, 0.105304509, 0.0813725963, -0.0503737293, -0.0423749015, -0.0600213148, -0.0395135209, 0.242647633, -0.0567225255, -0.0953626633, -0.000300093001, 0.0312304609, 0.173153102, 0.0520930588, -0.304377019, 0.0964622498, -0.0814322978, -0.0572857037, -0.124899499, 0.173855051, -0.126501203, -0.0713063776, -0.0373672135, 0.150735512, -0.237116978, -0.139013276, -0.218322858, 0.0921640545, -0.0520263836, 0.257865846, -0.151795939, -0.120246775, -0.108947575, 0.280953765, -0.112184592, -0.0690225884, 0.128942892, -0.00621310109, 0.150983855, 0.265627414, -0.0148573527, -0.00638692081, -0.270087361, 0.0936407074, 0.119968422, -0.168551922, 0.065900743, 0.163260669, -0.0762269944, 0.121191658, -0.227582991, 0.0563046262, -0.14453648, -0.247026324, -0.198427394, 0.146938384, 0.0399760678, -0.00455863774, -0.00801403075, -0.00471097231, 0.129436374, -0.00785559881, -0.23967573, 0.160759911, -0.217170179, 0.059673205, 0.0550655685, -0.0963633731, 0.0493823029, 0.0798566714, 0.109029189, 0.020367872, 0.135246068, -0.113844417, 0.00287559745, -0.209072962, -0.197916552, -0.180231661, 0.101901092, 0.214207754, -0.00789650623, -0.106650531, -0.126928777, -0.0627369136, 0.0654484034, -0.0819197819, 0.29193005, -0.0248275623, -0.0557257682, -0.00748233451, 0.180867657, -0.0344851837, -0.250930518, -0.104754284, 0.147129387, -0.188409835, 0.169326276, -0.160357788, 0.169476837, 0.0106401676, -0.0722912773, 0.22912693, 0.229926616, -0.278435051, -0.00473464234, 0.0555630922, 0.17146723, -0.117122836, -0.0767989457, 0.0572060272, 0.142129436, 0.00657555461, -0.0285110623, -0.260344118, 0.0989044905, -0.105224997, -0.225994274, -0.282512605, -0.132227853, -0.23164551, -0.126432598, -0.175983578, 0.207563102, 0.20213519, 0.116067044, -0.129871324, -0.0641780123, -0.197573081, 0.0170770157, 0.0416710302, 0.237090498, 0.0815810338, 0.199073792, 0.0989497602, 0.170951322, 0.192848817, 0.02512151, 0.0494165868, -0.0813700259, 0.143076003, 0.136122361, 0.175064206, -0.161730811, 0.182675511, 0.0577683002, 0.12183997, 0.0470225997, -0.231185332, 0.0169506967, -0.119522803, 0.0683735013, 0.0920851454, -0.217990443, 0.0190431885, 0.203925014, -0.207395673, -0.0615044907, 0.0312225744, -0.073792249, -0.229524866, 0.155897632, -0.162459046, 0.0172525812, 0.136289224, -0.111660883, 0.237077177, -0.178375512, 0.175627097, -0.0281897094, 0.0541172661, -0.109059267, -0.14404507, -0.124059416, 0.0811684206, -0.0470161177, -0.066804871, -0.0850931481, 0.0434931368, 0.1373014, 0.259490013, -0.0881389454, -0.0493104868, -0.19704245, 0.16196382, -0.13053143, -0.111271337, -0.0854118466, 0.224985242, 0.127444759, 0.0727540329, -0.0320677198, -0.0183699485, 0.00351795973, 0.164765865, 0.13210772, 0.049928043, 0.0186676942, 0.0988922641, -0.131334722, 0.177617058, -0.170443878, 0.0973633751, 0.00504548103, -0.0171984043, 0.187171161, 0.0827463046, -0.157445848, -0.204074711, -0.245190218, 0.245169774, -0.0603508018, 0.17393136, -0.0305710733, 0.0401617177, 0.147684678, -0.0304231029, -0.152545437, 0.0501171015, -0.233973876, 0.136166081, 0.188226268, 0.0445944853, 0.0289832689, -0.202041328, -0.174103916, 0.131884769, -0.201908588, 0.221570641, -0.0861945599, 0.176828861, -0.188249394, 0.09324269, 0.094032906, -0.15741083, 0.0183089897, -0.025142502, -0.185235664, -0.105590858, 0.126755387, 0.0810155272, 0.0908192694, 0.257951409, -0.157443106, 0.205290884, -0.0489252396, -0.0989102721, 0.0708614588, 0.0386378206, 0.201516673, 0.0292547792, -0.0833374709, 0.132945493, 0.156132996, 0.00765515072, -0.190696836, 0.0847563595, -0.130459666, -0.174606368, 0.186493203, -0.185741857, 0.0914283767, -0.200763315, 0.0963705927, -0.164442599, -0.120197445, 0.0842603222, -0.187861234, 0.0992910936, -0.0723259225, 0.131771117, 0.0294709411, -0.0707816929, 0.15362066, 0.111908376, 0.078812331, 0.0535888821, 0.0507810563, 0.131110504, 0.179611921, 0.026744267, -0.0871720165, 0.0355067551, 0.118356422, -0.204518527, 0.0498766974, -0.0372236706, -0.00990310404, 0.10396497, -0.00883602072, -0.177933022, 0.0129285334, -0.12813133, 0.0643947497, -0.0221159253, -0.078253977, -0.156190872, 0.0223176498, -0.0749285966, 0.160610095, 0.0397448465, -0.144857541, 0.210528627, -0.177495837, 0.170002475, -0.0258958396, -0.113389783, 0.109926522, 0.195601434, -0.0548773855, -0.149894163, 0.148451984, 0.0346607901, 0.140283972, -0.00360311568, -0.102635242, -0.0503319688, 0.0162678473, -0.0676407441, -0.11571575, 0.112506241, -0.118930839, -0.151946649, 0.0985130519, -0.1923296, -0.0602569394, -0.037379276, -0.193716258, -0.0948935449, -0.020577101, -0.179147139, -0.195478693, 0.123371579, -0.00464495225, 0.0504263602, -0.0386064462, -0.0517891161, -0.169164538, 0.11771892, -0.0632881671, 0.125877112, 0.192654654, -0.0948174372, 0.0738299266, 0.126855522, -0.118285932, -0.0321045406, 0.0178604145, -0.0212341771, 0.148154989, 0.130340979, -0.0704322532, 0.0328871049, -0.227042913, 0.239740446, -0.0955699533, 0.114672013, -0.0708279312, 0.10800238, -0.109282725, 0.142058045, 0.105162479, -0.051887475, -0.0467856638, 0.123139441, -0.106748275, -0.175780401, -0.127217188, -0.181122348, -0.0676865727, 0.117284544, -0.0273130462, 0.0963890329, 0.00385483191, -0.177152038, -0.191867977, 0.077240102, 0.124747507, 0.0890129358, -0.0591309927, -0.121862456, -0.19205831, 0.122563228, 0.176135257, -0.177255824, 0.0381551534, 0.0424975604, -0.185359091, -0.188019961, 0.114714131, 0.161240518, -0.119956791, -0.00404445827, -0.0148509219, 0.0826404542, -0.0528445691, 0.145070598, -0.0415300168, 0.185449079, 0.0144401034, -0.0457542241, 0.121085688, 0.159310594, 0.197267592, 0.0817764252, 0.119335428, 0.0792978927, -0.137601241, -0.0160116367, -0.16096127, 0.0202337243, -0.0156570133, 0.17746596, -0.0477557518, -0.057627324, 0.165322959, -0.147759885, -0.088363573, -0.183882236, 0.216872111, -0.120255038, -0.0487861186, -0.0615872554, 0.126300633, -0.0990248471, 0.0368622988, 0.223582864, 0.0624831654, 0.010734871, -0.116444357, -0.203225613, -0.127781093, -0.166673332, 0.157802746, -0.0282158162, -0.109729975, -0.0391220339, -0.124125309, 0.0324856862, -0.175051495, -0.0247840639, 0.0936974436, -0.00736786192, 0.155662224, 0.157572389, 0.0846097469, 0.0808747634, -0.029931752, 0.130156875, -0.194955394, 0.0540007949, 0.297759801, -0.15280652, 0.0210758597, 0.0932299495, -0.167536736, 0.285581648, -0.0180603843, -0.179686129, 0.204945594, 0.189112514, 0.165582985, 0.143395647, -0.126252934, 0.0896839723, -0.298827648, 0.064478986, 0.000745264464, -0.16088663, -0.174918249, 0.0957706571, 0.0120447576, 0.119768813, 0.0807619318, 0.0893344283, -0.25136587, 0.127414092, 0.207855508, 0.0846856162, 0.0175084565, -0.10128703, 0.101297647, 0.208785698, 0.138138175, 0.0138534503, 0.0905889496, 0.13177821, 0.18886824, -0.0161923002, 0.189213589, -0.0682863444, -0.166542068, -0.00136115553, 0.0997680947, -0.0653852895, 0.146990359, 0.181544811, 0.115617692, 0.298607945, -0.0134123974, 0.145018026, -0.29561004, -0.124093696, -0.210322186, 0.137198851, 0.0914252549, -0.0175533239, 0.192823961, 0.183647707, -0.144407481, 0.0237307549, 0.175023243, 0.116533205, -0.010630399, 0.0754853338, -0.0653730035, 0.114706591, -0.159099877, -0.0851648599, -0.1207624, -0.0410666317, -0.172199935, -0.145232454, 0.16999276, -0.146817982, -0.0389965475, -0.0854866505, 0.0712565035, -0.00583642721, -0.197309196, -0.0306858718, -0.151972204, 0.0138290226, 0.201786533, -0.033470422, 0.111182824, 0.0868683606, -0.118202969, 0.0617301315, 0.132822946, -0.154013336, -0.00978311896, -0.161551476, -0.193557248, 0.0101869851, -0.126305878, 0.158561811, 0.00379236042, -0.0607737899, -0.0138211846, -0.158382684, -0.0691986978, 0.133874074, -0.201073974, -0.119042397, -0.0212140232, 0.0352598876, -0.0136535764, -0.0176571012, 0.210377857, -0.197992519, 0.0080832541, -0.00235559046, 0.095504269, -0.209513187, -0.215412378, 0.168746248, -0.215368554, -0.0952431932, -0.0601882786, -0.128752172, 0.113622233, -0.215524599, 0.201375023, -0.107492052, 0.0754652768, -0.0948438123, -0.121238068, 0.149828091, 0.161296472, -0.0535617173, 0.0448756069, 0.215061948, -0.0858141333, -0.104567416, -0.13317892, -0.180668265, 0.157652691, 0.000676110387, 0.0542567819, 0.103542104, -0.160294861, 0.0630884916, -0.0210512578, 0.0308071226, -0.108765341, 0.105836019, -0.0544864237, -0.0361126959, 0.0175312012, -0.0544892699, 0.165185824, -0.0246543884, -0.0384053588, -0.0629663616, -0.165999919, 0.0924038738, -0.0472313017, 0.178175375, 0.147123411, -0.0634953082, 0.212211952, -0.035074994, -0.0309012234, -0.0756640583, -0.0832019448, 0.14364703, 0.0768184513, 0.132498935, 0.117131457, -0.0801562518, 0.181623742, 0.19624342, -0.197934449, 0.181445286, 0.10837917, 0.126055077, 0.0945705026, -0.0554487109, -0.180778623, -0.118354313, 0.110690013, -0.15024513, -0.193064138, -0.171204776, 0.0157593787, 0.100202553, 0.214262843, -0.148953438, -0.11341837, -0.0936558172, 0.0606097542, -0.0733776987, 0.20756118, 0.0454133786, 0.211113855, 0.263197571, 0.0173376407, 0.0348490179, -0.0670863166, -0.0259215664, -0.220633924, 0.167376027, 0.30080685, 0.152899742, 0.100315377, 0.0216483381, 0.0153267374, -0.0821862444, -0.022511309, 0.110671572, -0.197649375, -0.243930042, -0.0089917779, -0.16742897, 0.25845921, 0.0806541368, -0.0169763733, -0.150612444, 0.0804499462, 0.147269264, -0.123657018, -0.101714112, 0.0392946117, 0.235302284, 0.129554257, 0.20972079, 0.00137448253, -0.160698906, 0.0453142338, 0.0750062764, -0.044447802, -0.0454354547, -0.0594326332, 0.0154880593, -0.135283649, 0.156637296, -0.0949086621, -0.204240441, 0.199247792, 0.0847830772, 0.0778177977, 0.262001753, -0.0237951018, 0.254970968, -0.103296667, 0.1293993, -0.211035922, 0.103326999, 0.000826618809, -0.0683762655, 0.156546369, -0.012880085, -0.0566472597, 0.105513714, 0.0323817059, -0.180392623, -0.0829131231, 0.275576562, -0.119350486, -0.256336868, 0.0225851666, -0.0718415678, -0.032045424, 0.157612577, 0.295247853, -0.161926433, 0.0551234297, -0.200971603, -0.149542153, -0.112447798, -0.188605458, -0.10279642, -0.185480207, 0.186702803, 0.203769177, -0.0506769307, 0.340962738, 0.0492642671, 0.00382401654, -0.295713395, 0.0791265443, 0.145609438, -0.118261933, -0.0462953039, -0.26303187, -0.167325541, 0.229171544, 0.125606567, 0.0196683183, -0.0821758062, -0.172154814, 0.134631366, 0.105954275, 0.0713844672, 0.066780068, 0.0916744471, 0.325054318, 0.134490564, -0.18094638, 0.0252105873, -0.154933974, -0.00310963392, 0.0248205513, 0.126237467, 0.014732969, -0.103780881, -0.19062826, -0.0709873661, -0.0277325865, -0.0735364705, 0.133878663, 0.0306869727, 0.197213531, 0.217959478, 0.0710183606, 0.18170689, 0.21944575, 0.0610789806, -0.116570912, 0.12491186, 0.0503248312, -0.110214539, -0.0159544032, 0.232890576, -0.0456155278, 0.00884607527, 0.187331676, 0.21877192, 0.204476058, -0.115975544, 0.0187843088, -0.09255445, -0.29152, 0.0851894468, 0.0949364305, 0.262373477, -0.0559873134, -0.0886857882, -0.107428819, 0.175252438, -0.181784943, 0.248689443, 0.0079609314, -0.155982539, -0.247614115, 0.197390601, 0.0732584447, 0.0571540222, -0.153867841, -0.185098931, -0.225856975, 0.151971042, -0.17325078, 0.166293293, 0.21347858, 0.137752622, 0.0146298427, 0.165977046, 0.200429872, 0.243356928, -0.0243835449, -0.132510141, -0.170158356, -0.210107028, 0.054322429, -0.0642425045, 0.070434615, 0.00680774171, 0.115169078, -0.0843608603, -0.113310277, -0.250803977, 0.00723329745, -0.320745975, 0.0171446204, 0.0268929899, 0.0155198043, 0.183056667, -0.0546245314, -0.0218649153, -0.107723393, -0.0206710231, -0.0810157731, -0.0866106674, 0.154913038, -0.0283856317, 0.157422259, 0.249080539, 0.197582707, 0.0180592034, -0.0630287081, 0.0954426602, -0.00257873558, 0.197637767, -0.0483088568, -0.205665752, 0.178116858, -0.215542749, 0.0139305266, -0.0284120627, 0.0472723357, 0.114193209, -0.113162771, -0.0734884441, 0.190928593, 0.14512518, -0.179998294, 0.0362271219, 0.0808228552, -0.0790003017, 0.0780607685, 0.0691427216, -0.0794865191, -0.190427512, -0.194445565, -0.117233612, -0.181705579, 0.076732479, -0.0706049204, 0.110384241, 0.109668888, 0.00635866122, -0.120385066, -0.182506919, 0.0288684703, -0.155140281, -0.00705729891, 0.0220523346, -0.0523335524, -0.127393574, -0.226881415, -0.0877430663, 0.141399264, 0.180214092, 0.0126109738, 0.104212426, -0.00757380715, 0.258023709, -0.0758938268, -0.169211, 0.0147744548, 0.0781950727, 0.0368106291, -0.278180361, -0.0971170142, 0.119301975, 0.193576843, 0.134058133, -0.0579313375, -0.0559127405, -0.0187151711, -0.0745572597, 0.0402791612, 0.11351911, 0.110996328, 0.10230045, -0.119222939, -0.0110910339, 0.0194552336, 0.14156279, 0.280852199, -0.166947231, 0.102535248, 0.0493896715, -0.0241324138, -0.176901072, -0.0267906673, 0.252696484, 0.307401866, 0.00364437792, 0.158837378, 0.263545632, 0.0133025851, -0.0667897686, -0.0859481618, 0.145068467, -0.0603770092, -0.0731502622, 0.269838184, -0.245759487, -0.0586617142, -0.0775664076, -0.208350435, 0.0898162201, 0.0956078693, -0.134778693, -0.0955108702, -0.0629637241, 0.164887547, -0.0951353088, -0.0474154986, -0.0317355469, -0.311545223, -0.034149304, -0.133716777, -0.254200995, 0.233857363, -0.221086636, -0.0875458941, 0.144417778, -0.0733914226, -0.0500378273, -0.16867502, 0.108182065, 0.128211737, -0.0357037261, 0.16355747, 0.00208666385, -0.341230929, -0.110794365, -0.192407697, -0.185402006, 0.0158167668, 0.228281468, -0.0576616935, -0.0166208204, 0.231899574, -0.0969194695, 0.176652476, 0.166342959, 0.0320710912, -0.179827735, 0.132767901, 0.0290033314, -0.152132601, -0.181854218, -0.0543435551, -0.147026494, 0.132066295, 0.000380948186, -0.046831917, -0.0122211166, 0.265439212, -0.385553628, 0.19313477, 0.133767381, 0.286021829, -0.22221379, -0.293776661, 0.148888484, -0.181432143, -0.16458258, 0.268145353, -0.204560816, 0.0846042112, -0.109482028, -0.0879192576, -0.147025988, 0.288842827, -0.088969633, -0.0655507073, 0.263407081, 0.133582711, -0.0163365304, 0.110040441, -0.0645436272, 0.0251421444, -0.10840106, 0.179400072, -0.106979035, 0.0695290193, 0.109481424, 0.210353449, -0.0532516129, -0.167095572, 0.0434949584, 0.175142482, -0.0420172065, -0.100425139, 0.165737182, -0.165261269, -0.119268917, 0.142626181, -0.188711599, 0.0471658744, -0.0998743027, 0.108773425, 0.171581998, -0.0881806239, -0.118828684, 0.0752182528, -0.185938254, 0.102960572, -0.00374448881, 0.143556684, -0.157970682, -0.0651584789, 0.126855001, 0.182917491, -0.160805538, 0.123719871, -0.0744021162, 0.213524118, -0.207614541, 0.0227269568, -0.0975663513, 0.0987157747, -0.0909273997, 0.138845056, -0.0999631882, 0.181141108, -0.180883646, 0.150684878, 0.072670795, -0.11002925, -0.120575607, -0.0391260162, -0.0647687092, 0.17848663, 0.0242926795, -0.143397227, 0.181315631, 0.115013622, -0.217152998, -0.016199477, -0.0158816669, -0.124248572, -0.12989518, -0.0339076035, 0.264628232, -0.0808567181, -0.0246815663, -0.0834978744, 0.161822602, -0.138402522, -0.00808761735, 0.0439582318, 0.154923141, 0.0127866575, 0.157803074, -0.0195006952, -0.145444661, 0.15624623, 0.213899404, -0.216991454, 0.0774733201, 0.102065235, -0.124791786, -0.207634076, -0.164074779, -0.0574968681, 0.089080818, -0.0694269165, 0.211942866, -0.114976563, 0.214145839, 0.198561743, 0.0715887323, 0.109872617, -0.0963600874, -0.079338029, 0.0805210099, 0.0106852446, 0.191253379, -0.067177996, 0.11775624, -0.110801004, -0.102861449, 0.1769429, -0.223849356, 0.0693205595, 0.145785511, -0.032342162, -0.158411354, -0.00197427161, -0.095368214, -0.188921377, -0.113391459, 0.0368723348, 0.107978091, 0.0824893937, 0.0900589675, -0.041756928, -0.064508982, -0.181163505, -0.171657398, 0.026455136, -0.199689955, 0.0629645661, -0.117474094, -0.15332523, 0.0785275772, -0.111598738, -0.103435583, -0.163627595, -0.00887487829, -0.157007217, 0.00934804231, 0.1409017, -0.000921073661, 0.0372746959, -0.174577355, -0.0164345335, 0.0782096386, -0.0826458782, 0.138327822, 0.0130521106, 0.142504245, -0.0212440453, 0.235662311, 0.292200476, -0.124307498, -0.141203091, 0.104294352, 0.265598536, -0.202951029, -0.31308794, 0.176690981, -0.316680521, 0.308380634, -0.058346685, -0.052924715, -0.068701461, 0.240178868, -0.194287747, 0.128212035, -0.121045195, 0.18089883, -0.0418058485, 0.0846816227, -0.119049914, 0.00999071915, 0.03216362, 0.127670601, -0.200703219, 0.0612659827, -0.307814896, -0.328196347, -0.119040579, -0.175974175, 0.247130468, 0.0949836671, 0.0164293498, -0.0871255696, -0.0288449004, -0.0993912593, 0.0679356381, 0.0571999848, -0.0168665498, 0.173970565, 0.00567579689, 0.206851333, -0.0155466767, 0.116136476, -0.0451772027, 0.0345146023, 0.171833515, -0.14317131, 0.0439632647, 0.0550731719, -0.174111396, 0.249948263, 0.0319778696, -0.08461494, -0.194183409, -0.0776880309, -0.0970808789, 0.0736219287, -0.13262856, -0.0557855815, 0.0211500153, -0.236246914, 0.22175169, 0.162301347, 0.0972244814, -0.176554397, 0.204008728, -0.209684461, -0.18114011, -0.1861417, 0.281658024, -0.00434876187, -0.000967082102, -0.182629734, 0.109987505, -0.0832468048, 0.0613217019, 0.148019463, 0.000290387106, -0.142763898, 0.185766563, -0.0045414567, 0.168641582, -0.156493008, -0.169194326, -0.11528603, -0.0347869396, 0.253748775, 0.0731557384, 0.037423566, 0.162255421, 0.169754088, 0.257631987, 0.165029943, 0.0698102564, 0.0314833559, 0.164437681, -0.128836766, 0.280385345, -0.132313639, 0.0832324475, -0.159102678, -0.190169424, 0.120876521, -0.0708724335, 0.108387083, -0.013849372, -0.173526362, 0.168055281, -0.0783005506, 0.133223042, -0.052906163, -0.16011405, -0.156364277, 0.170717791, -0.135527775, 0.302193105, 0.0370368697, 0.144021943, 0.152141228, 0.072664246, 0.0809864327, -0.0436896682, 0.10182593, 0.0915664807, -0.184139475, 0.280362487, -0.195510402, 0.0830965191, -0.0758729503, 0.223914117, 0.00844487827, 0.00993681513, 0.0982448608, -0.103829846, 0.00631501665, 0.0602077693, -0.229385301, 0.304050446, 0.210445672, -0.0769463331, 0.108615175, -0.0788970515, -0.127578288, 0.214681074, -0.0700043291, 0.166759819, 0.0396312959, -0.144758493, -0.106974468, -0.0965421125, 0.188366085, 0.28905794, -0.125003085, 0.248191193, -0.022866942, 0.301850051, -0.163019001, -0.328558654, -0.0491153672, 0.0805409625, -0.0996451229, 0.256436139, -0.125509635, 0.0881489664, -0.0299049839, -0.272820115, 0.0276542306, 0.072070688, 0.017024979, -0.0835376158, 0.193469211, -0.0293851048, -0.191110089, -0.0412489772, -0.208624303, -0.24148649, -0.205899239, -0.174337134, -0.0175865591, 0.298654824, -0.0985588804, 0.103253216, 0.24924536, 0.205758289, -0.196999446, -0.149646878, -0.143381536, -0.000880725158, -0.0068264748, -0.174360752, 0.249812827, 0.109578051, -0.081599012, 0.113797002, 0.079932496, -0.0615099408, 0.191720381, -0.208634764, 0.150513843, -0.0344681069, 0.218191922, 0.139449969, 0.171120629, 0.1082827, 0.163610205, 0.0875669345, -0.116561994, 0.118207827, 0.0104034245, -0.16478233, -0.0413739011, -0.316277593, -0.0421933122, 0.0120029449, -0.116558015, 0.0348773338, 0.0611173026, -0.145482197, -0.0627405196, -0.182251006, 0.0826851279, -0.0607742444, 0.0268052518, -0.0526164658, -0.0653537959, -0.179316863, 0.105216481, -0.0154515207, -0.155959472, 0.13121824, 0.25053665, 0.213652462, 0.0733022988, 0.0634803474, -0.133813843, -0.0560159571, 0.123325393, 0.169942483, -0.0188645292, -0.146081492, -0.0042090537, -0.152687699, 0.152199179, -0.0402537622, 0.150147647, -0.15232645, -0.101902142, -0.0839850903, -0.278659999, -0.146883801, -0.0142387301, -0.0918006599, 0.198642433, 0.164413884, -0.183536232, -0.0297051743, 0.159891501, -0.122745588, -0.102025181, -0.0521458909, 0.118992224, -0.060556896, 0.195035189, 0.259946346, 0.0685981214, -0.148837596, -0.0323895104, -0.0847889632, 0.182129964, 0.119295359, -0.0368872695, 0.238972053, -0.155852035, 0.167594254, -0.0925863683, 0.0172753409, 0.189614743, 0.162803963, 0.163829163, 0.215808108, 0.0124880038, 0.0426811688, -0.0600209348, 0.0615481213, 0.165346935, 0.0153156063, 0.121975742, -0.175549001, 0.183664352, 0.144022495, 0.0322715566, -0.107829265, 0.0768434852, 0.0050736377, 0.0618446544, 0.153952852, -0.169535995, 0.166753307, -0.186460227, 0.00901123788, -0.0184693541, -0.0857320651, -0.0475749783, 0.00862984639, -0.0971527323, -0.196421653, -0.0968040973, 0.238713965, -0.0107892593, 0.178670123, 0.082849972, -0.067512013, 0.103636593, -0.172591835, 0.162427366, -0.0980086103, 0.103627391, -0.00657122722, 0.196705267, -0.0885492787, -0.21484302, 0.0713789761, 0.00349842641, -0.114411183, 0.00135329366, 0.172899455, -0.0640534312, 0.176380396, 0.129859045, 0.152343497, 0.188691467, -0.0690017864, -0.137624815, 0.0596759468, 0.161572218, 0.030274827, 0.0932867527, -0.0543891117, 0.0914924815, 0.0758234411, 0.189578816, 0.216388658, 0.136622667, -0.224723607, 0.115231387, -0.143994942, -0.0134596284, 0.0285644792, -0.0765158683, -0.0898127109, -0.0216522682, -0.0452857055, -0.180066332, 0.0636309981, -0.136346862, 0.160724685, 0.104276851, -0.0502810515, 0.214406371, 0.00751658203, 0.0742831528, -0.0960830152, -0.103430808, -0.149839222, 0.122873515, -0.199809447, 0.0846741796, 0.0414155461, -0.149651155, 0.0535871387, 0.032020431, 0.00699738273, -0.12234541, -0.0605762973, 0.0471933074, -0.00849266909, 0.0234554689, -0.0544377342, 0.0270179659, 0.172541559, 0.0252916161, 0.0905541778, -0.144034952, 0.00168407825, 0.173910916, -0.0856598467, -0.0220967811, -0.0514697209, 0.0803929046, 0.127755255, 0.171276376, 0.104453139, -0.0212837942, -0.0249362309, -0.358178616, -0.233663827, 0.233707651, 0.256034017, 0.103490725, 0.00574883632, -0.0556842498, 0.131842449, 0.00785240531, 0.0435351245, -0.118263483, -0.150564089, -0.117127106, 0.015985528, 0.088842757, 0.14202477, -0.00392921269, -0.141630784, -0.108435906, 0.150415316, 0.192709893, 0.242879584, -0.187250435, 0.0510517657, 0.229519933, -0.0843288153, 0.0532751195, 0.186514959, 0.0342584439, -0.0914594829, -0.0284124669, 0.141796708, 0.00305303931, -0.0396114551, -0.115827665, -0.12504971, 0.231261835, 0.135242477, -0.0376397893, -0.146970883, 0.233937755, -0.114139147, 0.156069487, 0.179028809, 0.178957433, -0.0414629728, -0.0976045877, 0.0569484569, 0.103674464, -0.089665994, 0.0826087892, -0.105914153, -0.00952274725, 0.185328886, -0.0473689064, 0.171411321, -0.135359928, 0.237343296, -0.293576032, 0.0484540462, 0.0989309847, -0.12313319, 0.21306318, 0.0288836546, 0.0259658769, -0.0176200364, 0.202105507, 0.239969552, 0.125312254, 0.0684467033, -0.189783171, 0.024794735, 0.107969731, 0.17213501, -0.0679843202, -0.176238269, 0.00562783564, 0.198162049, -0.0273213014, -0.229449779, -0.0726197436, -0.146376207, 0.0733661801, -0.122138776, 0.0300521944, 0.000627006986, -0.224758834, -0.219826937, 0.042535685, -0.11363896, 0.0945541859, 0.118705377, 0.0555131733, -0.329797447, 0.0684644952, 0.260578483, -0.0437527634, 0.0811403245, 0.0408508256, 0.15580976, -0.0451794863, 0.0944328681, 0.199969038, 0.0696579441, 0.223595411, -0.0154632749, 0.321737945, 0.251616448, -0.0567427538, 0.035431765, 0.280902177, -0.169113502, -0.231067359, 0.0143873319, 0.0581891723, 0.154215962, 0.0250351746, 0.238159895, 0.128872484, -0.221735775, -0.0697579384, -0.075381659, -0.0484818742, -0.0863361508, 0.123765059, -0.135387972, 0.231054485, -0.0443002544, -0.243541643, 0.151080266, -0.106428668, 0.0855598897, 0.0846331418, -0.0779921785, 0.0547915027, -0.0920602605, 0.0887217745, -0.0030759566, 0.0840683505, -0.0667907745, 0.0150866825, -0.113728702, 0.0240516253, 0.0788644105, 0.0189627409, 0.029980829, 0.182710513, 0.233252287, -0.0950233042, 0.0486974977, 0.0204964131, -0.0657696128, 0.242969364, 0.034332294, -0.123168163, 0.246184021, 0.0397303998, 0.028434189, -0.115440212, 0.0868595541, -0.145101041, 0.0786464363, 0.0524663962, 0.0946072713, -0.160390154, 0.268412858, -0.202053457, 0.170204252, -0.141202495, -0.209169641, -0.0217667911, -0.276255965, -0.208408445, 0.0612591468, 0.18525213, -0.0280163027, 0.0532558374, 0.038261883, -0.111344911, 0.0510275178, 0.137613237, -0.0182486102, 0.022279419, 0.237698808, -0.168505922, -0.0947840884, -0.0860128328, 0.0939792022, 0.0062875296, 0.290792286, -0.178391397, 0.0912785605, -0.071976088, 0.180548236, -0.196116716, -0.154281169, -0.0599976256, 0.261835635, 0.0432700068, 0.244295612, -0.222427472, 0.0652513355, -0.17671591, -0.203425258, -0.131267071, 0.0277503077, -0.261542737, -0.002615412, 0.295612812, 0.0422270782, 0.169738501, -0.136077911, -0.241452679, -0.158954144, 0.0203940291, -0.0218450259, -0.21398285, 0.260178745, 0.0980303138, 0.00973836519, -0.257299483, 0.224123374, 0.0211241115, 0.18352662, -0.064140141, 0.0862681791, -0.163428918, -0.152894586, -0.00333995232, 0.0032048868, -0.0328324623, 0.0929068178, -0.279507995, -0.0916615948, 0.149792582, 0.0819854364, -0.0381851047, -0.0611945577, -0.134679809, 0.0265907645, -0.106183901, -0.0546292849, 0.212225929, 0.155997798, 0.0469628684, 0.0114867613, 0.0375453793, -0.0232304651, 0.201258332, 0.0445280969, -0.108712807, 0.0448913462, -0.0595548563, -0.00239899638, 0.055149626, -0.00122337963, -0.0738636926, -0.081668295, 0.202223718, 0.136749536, -0.227384835, 0.0613598339, -0.115820222, 0.0364864096, 0.0139585184, -0.0280776732, 0.180970713, -0.046631746, 0.0747796074, 0.126691923, -0.0111388853, 0.107929185, -0.0551268123, -0.0529108122, -0.212241918, 0.136584833, 0.155696839, 0.0378725938, -0.151348546, 0.00820482895, 0.0856666714, 0.137337208, 0.147699654, -0.0763601139, -0.0242069904, -0.0654426292, 0.0947293192, 0.0777328461, 0.0894588232, -0.124189667, -0.197469324, 0.18639116, 0.0779219195, 0.141812861, -0.0726427585, -0.194079414, 0.0403500609, 0.0486738719, 0.175959468, -0.0224688575, 0.108159691, 0.110468484, 0.0989225358, -0.0435029604, 0.0932252854, 0.0202672239, -0.0806071311, -0.0692079961, 0.21573095, 0.165748715, 0.0341887586, 0.196531609, -0.106021568, 0.0170011446, 0.0364869945, -0.0480184555, 0.160415426, 0.238614678, 0.0291153304, -0.0692989081, -0.329096109, -0.0360180438, 0.256817967, 0.225853592, -0.224268287, 0.175842762, -0.198225558, 0.0573723502, -0.0511965454, 0.117915072, -0.0368777364, 0.0182616115, -0.00727006095, -0.0168267079, -0.0614160858, 0.156759843, 0.162976161, -0.00199627364, -0.17093797, 0.201199114, -0.194492713, 0.0589784794, 0.0552661046, -0.167786106, 0.140908763, -0.068700999, 0.0502691977, 0.0795648023, 0.0274966806, -0.296720952, -0.163464576, -0.102106683, -0.00985952932, 0.109491237, 0.00823518075, -0.197602898, 0.241903737, 0.0013750908, -0.168662667, -0.123866923, -0.204145133, 0.0930801407, 0.328670114, 0.00163828232, 0.220920488, 0.0642628074, 0.328812987, -0.0748362392, -0.0226152278, 0.000289303658, 0.188728347, -0.0364874303, -0.0651446581, 0.231653139, 0.0857582167, -0.194839388, 0.0351886451, -0.0548176616, 0.0118231382, -0.148435593, 0.0464327261, -0.0904112831, 0.0666049942, -0.209124938, 0.0648437589, 0.182237193, 0.214572534, -0.00191250537, -0.1671011, -0.110546388, -0.154530227, -0.106844932, -0.0305259917, 0.116241798, 0.109203883, 0.142477855, -0.0726438016, 0.0829489529, 0.0612219125, 0.0201825909, -0.131854653, -0.225124791, -0.129626438, -0.0346009545, 0.205493644, -0.123570427, -0.0745602846, -0.187618464, 0.13536644, 0.176973596, 0.234079748, 0.0889393911, -0.0863182768, 0.165225297, 0.137968197, 0.279592723, 0.0361696146, -0.173749968, 0.0601600967, 0.0129619762, 0.208610386, 0.220640108, -0.115378678, 0.0240061432, 0.278004318, -0.0265378393, 0.149464399, -0.303708673, -0.105789356, 0.0307838731, 0.193645462, -0.165561646, -0.0895986408, -0.0594347157, 0.254087687, -0.0558889918, -0.106389455, -0.00137458323, -0.194988936, 0.0805720314, -0.0352395177, 0.194134623, -0.116110273, -0.174519628, 0.0278469343, 0.0595925637, -0.130331695, -0.0923151374, 0.0643297732, -0.177647516, 0.10481973, 0.192607358, -0.141913235, 0.0599878654, -0.154343843, 0.264552563, -0.0673295557, 0.183654264, 0.179233626, 0.00202305615, -0.33549431, -0.156067759, 0.116495214, 0.164007157, -0.0761157051, 0.0759984627, -0.137309909, -0.0688316524, 0.154320285, 0.249968484, -0.219860017, -0.325449139, -0.129957005, -0.326592982, 0.205126315, 0.0471690372, -0.113722183, 0.101460293, -0.132077157, 0.0266415607, 0.00812615175, -0.179480046, 0.162329659, -0.0515648499, 0.315276504, -0.00411519269, -0.02481113, -0.0660336092, 0.20307903, 0.116764992, 0.145217434, 0.231170014, 0.129283935, 0.227875918, 0.335049301, 0.169715032, -0.0661990941, -0.222038403, 0.112036951, 0.118910842, -0.214670569, 0.0934555307, 0.0968824625, -0.150049731, 0.149248824, -0.0754649118, 0.273794323, 0.0952707529, -0.29306978, -0.157772511, 0.135602057, 0.14062117, 0.369418502, -0.0413367189, 0.0816308931, -0.278485179, -0.0156329628, -0.353450298, -0.0292544812, -0.262566298, 0.0992213935, -0.170477495, 0.127993777, 0.165333867, 0.197797731, 0.250114858, 0.104357131, 0.0609139763, -0.390009731, 0.095229812, -0.106860213, -0.1796031, 0.13155356, 0.00892605539, -0.189845622, 0.179488435, -0.129862547, 0.0306370258, 0.000393755792, 0.183470011, 0.201606512, 0.00992667116, 0.138476804, -0.0199141521, -0.0361978561, -0.00738017075, -0.173073292, -0.136918575, -0.221550018, 0.16833882, 0.0337039381, 0.193500176, 0.121161528, -0.0153150447, -0.229320586, -0.162542269, -0.103140332, -0.0991333276, -0.21625343, -0.122940831, -0.0816918612, 0.292686313, -0.126720279, -0.245018229, 0.156526193, 0.231272772, -0.12768504, 0.046446193, -0.135035276, 0.237224385, -0.207771942, -0.165304184, 0.0449262112, -0.16046451, 0.0515512154, 0.0247535985, 0.179941446, 0.141006634, 0.148099631, 0.0461900011, -0.125380158, -0.260761499, -0.0365008488, -0.175376043, 0.173839927, 0.0840524882, 0.150757536, -0.00193478167, 0.134457171, 0.0838706568, 0.19708553, -0.108223915, -0.214755952, -0.180884525, -0.210335225, 0.198198155, -0.0710237324, -0.18349649, -0.10621804, -0.0015054564, -0.0930908322, -0.0695800856, 0.120227791, -0.0628320128, 0.161675051, -0.0369836837, -0.104480736, -0.115745157, 0.113166645, -0.226809382, 0.0440124832, -0.0557170361, -0.00395971676, 0.15534845, 0.116499223, 0.190032437, -0.105497465, -0.26288572, 0.0491223671, -0.219523475, 0.164801389, 0.0884424895, -0.180786639, -0.0025313925, 0.107427284, -0.015959831, 0.280966669, -0.101899825, 0.0844253153, 0.214183345, -0.0680119321, 0.0215379167, -0.215002313, 0.103997082, 0.0602454916, 0.162121207, 0.223211929, 0.0564612225, -0.0155185293, -0.0849888176, 0.0710228682, -0.0188842621, -0.0679497048, 0.228468344, -0.168624103, -0.187010109, -0.0338806175, 0.0473464616, 0.156233341, 0.210370451, -0.162648752, 0.0154813081, 0.0151715912, -0.224204272, 0.162158608, -0.212012723, 0.108205117, 0.120467298, 0.0116960257, 0.0391680412, -0.120638661, -0.0434363931, -0.0632359162, -0.18498835, -0.0534989648, -0.104398511, 0.14394021, -0.0630829409, -0.202434331, -0.221765876, 0.170155361, 0.146729127, 0.136266768, 0.0854845718, 0.00931845978, -0.0396513678, 0.243059888, -0.0143531486, -0.213143229, 0.163626105, 0.228435755, 0.0763803273, 0.294812024, 0.0303754285, 0.0224024169, 0.103866428, -0.0755221769, -0.146329269, 0.187158212, -0.0402141139, 0.215759218, 0.0578194857, 0.00068547955, -0.189536303, -0.157405496, -0.0117263664, -0.171880484, -0.0894706845, -0.195492998, -0.115787826, 0.106829114, -0.0732092932, -0.106249996, 0.0644781068, 0.0493799672, 0.0191225074, 0.199877992, -0.154181615, -0.169715717, -0.202959687, 0.0045042932, -0.139033392, -0.107659563, -0.174030259, -0.0516406633, -0.166010961, 0.136116982, -0.0560865402, -0.116511792, -0.0237821639, -0.0764931142, 0.0603490248, -0.154312968, -0.0190427899, -0.0848358423, -0.120311961, -0.0347254574, 0.0647674352, -0.113835506, -0.177448601, -0.0797593594, 0.234833598, -0.132981062, -0.132999331, -0.0635919347, 0.030990012, 0.17009069, 0.201166883, 0.187781587, -0.203566208, -0.163287312, 0.0935856551, -0.0598677248, 0.152191803, 0.114821628, -0.0730218515, 0.231914148, 0.0966452584, 0.166506305, -0.130623624, -0.0707645714, -0.129302263, 0.119527809, 0.0635081604, -0.112864114, 0.22138299, -0.0632478669, 0.114700712, -0.0792448521, -0.0765444115, -0.119066864, 0.0346016809, 0.303022891, -0.0871448815, -0.158137739, -0.228525937, -0.208690599, 0.171160266, 0.228543878, 0.198012307, 0.0903932974, 0.0979876369, 0.0818847567, -0.337730318, -0.202390894, -0.186501443, 0.1508746, -0.231906936, -0.0942646489, 0.0780744776, 0.00662959693, 0.368186593, 0.0524481647, 0.218401685, -0.0444435291, -0.0281022284, 0.117386088, -0.139238194, 0.344955772, -0.210472822, -0.185517386, 0.0432206802, 0.067795001, 0.18226862, -0.100125775, -0.108723685, 0.313094884, 0.102345057, -0.189623743, 0.119116165, 0.117150754, 0.113522097, -0.0974836648, 0.196477339, -0.299250156, -0.206788749, 0.127461419, -0.136677414, -0.00462659309, -0.082354337, 0.118807323, -0.267264903, -0.107201517, -0.257277042, -0.0105558699, 0.177996054, -0.0946902111, 0.00526810158, -0.0918765366, 0.180687875, -0.256947458, 0.0339876749, -0.0132435262, 0.0372189954, 0.0656750351, 0.123526566, -0.124181502, -0.127795756, 0.133546874, 0.267100155, -0.138555005, 0.112637945, 0.217483208, 0.250305533, -0.221768856, 0.0510481521, -0.0648338422, -0.135197312, 0.163345799, -0.0996528119, -0.295478195, 0.221370354, 0.0090700984, 0.163102254, 0.257673502, 0.0321548171, -0.218750283, -0.0417411365, 0.141176626, 0.0455146618, -0.139999777, -0.210085616, -0.0207382087, 0.159851059, -0.0191368647, 0.0799145848, -0.191577971, 0.222179979, 0.145579785, -0.124980874, 0.00011860668, -0.0531942584, -0.101949774, -0.149084419, 0.150167912, 0.242624894, 0.158585533, 0.0457630903, 0.121281974, 0.12134584, 0.174273595, 0.0234531015, 0.0101215569, 0.261128306, 0.130410358, -0.0646373257, 0.0671577677, 0.204333737, -0.171613261, -0.147265777, -0.0430774093, -0.206877887, 0.0973792225, 0.188770488, 0.0926625952, -0.369100392, -0.169856474, 0.0436665379, 0.0837029666, 0.07298664, 0.0201208107, -0.00663427031, -0.193593293, -0.0612708442, -0.269489616, 0.247763708, -0.0919435471, 0.122422889, 0.0842806175, 0.143494427, -0.040064469, -0.0293035377, 0.205288514, 0.138122469, -0.0655390397, 0.0721975565, 0.0538080819, -0.21350269, 0.121420853, 0.167736843, -0.183765441, 0.140039474, 0.234994337, 0.118522629, -0.0847690701, -0.155740887, -0.0549678095, 0.176273555, 0.12771441, 0.20569995, -0.189131141, 0.246775582, -0.040186435, -0.322248131, 0.00692595076, 0.251584858, -0.213374496, -0.195615217, 0.110311486, 0.259365857, 0.163353637, 0.123199798, -0.0378120169, -0.132168457, -0.146660343, -0.0177994464, -0.246754944, 0.347066194, 0.19430016, -0.0613136515, -0.105118059, 0.0349555612, -0.058653295, -0.0533792377, 0.0502194315, -0.0630996078, 0.0870997682, 0.193092287, -0.131634429, -0.228073478, 0.104649357, -0.0285898186, 0.0438296646, -0.142033562, 0.291676372, 0.0511058569, -0.010557062, -0.192678869, -0.0147832278, 0.333403051, -0.0420459956, -0.100109242, 0.134338498, -0.302299052, 0.0362847596, -0.301566482, -0.108434819, -0.207868457, 0.00391505705, 0.0137217129, -0.121070772, 0.151565805, -0.044486735, 0.304707795, -0.14781113, 0.0983222872, -0.238438904, 0.181199268, 0.0213714615, 0.00745414849, -0.0138446372, 0.086607568, -0.2248061, 0.0525689647, -0.022581771, 0.127698556, -0.00474502984, -0.0635372624, 0.296566814, 0.210853308, 0.133739591, 0.130687475, 0.03697237, 0.292883813, 0.157273754, -0.208699256, 0.103416078, 0.0554397516, -0.113555133, 0.0835159272, -0.1598773, 0.274341464, -0.153718844, -0.307261914, -0.314996988, -0.107934706, -0.287681222, -0.035695672, 0.0989629477, -0.0371217392, 0.142067209, 0.117525682, -0.185213074, 0.203321055, 0.103918776, 0.0360467881, 0.120570228, 0.0285809934, 0.0886411518, -0.0242966563, -0.202274486, -0.201233998, 0.0909243077, 0.000505506992, 0.195792988, -0.0434714705, 0.113136664, -0.0384105146, 0.0505792052, 0.147569552, 0.190747276, 0.0668908209, 0.0549472421, -0.111488663, -0.211737052, 0.180603728, -0.131985426, 0.1968918, -0.140003681, -0.159247667, -0.00467215478, -0.0768030286, 0.0416528136, 0.00666475296, -0.0831374228, 0.155933574, 0.0554835647, 0.0206790417, -0.151442379, -0.115788847, 0.0548514277, 0.0478165597, 0.0842054039, 0.129231438, -0.127966464, 0.147413924, 0.160519347, -0.00875259936, 0.0528210849, -0.0149530768, -0.010312736, 0.0383928567, -0.0103502572, 0.173571721, -0.0675502419, -0.0821278989, 0.116765901, 0.184800014, 0.17291145, -0.153413668, -0.0583886206, -0.122146413, 0.0483285636, 0.214191243, -0.205721736, 0.0823977888, 0.186194047, 0.118455581, -0.149338216, 0.0548166111, -0.0753933787, 0.0112254014, -0.0632569268, -0.144131511, 0.0945755616, 0.0224814937, 0.148579076, -0.0765286684, -0.0323213264, 0.0190389734, -0.107433006, -0.0821404457, -0.154118061, -0.210388929, 0.183495998, 0.0224975739, -0.0916404799, 0.0510140248, -0.0535344146, -0.192821115, -0.0450939275, 0.0833480209, 0.0689259619, 0.0424399003, -0.195493177, -0.108997151, -0.0964532495, -0.0500763245, -0.147860095, 0.0783045068, -0.0543835349, 0.00557268132, -0.0267649665, -0.179763988, -0.0538775064, 0.204667524, 0.0844915882, -0.0702664182, -0.128816217, 0.211553112, -0.20460856, -0.147548541, -0.198193178, 0.192208156, 0.0597049594, -0.144142136, -0.0617672056, -0.0503715128, -0.110759683, 0.0165932272, 0.0270641912, 0.0965968892, 0.150237605, -0.114341743, 0.0793848187, 0.156279072, -0.0775704384, -0.190129012, -0.154963881, 0.216353029, -0.126338452, 0.0519051328, -0.113659844, -0.199669346, 0.0344904214, -0.191059664, 0.102345951, -0.148214802, 0.0581426844, 0.00217875326, -0.0605221391, -0.00890331902, 0.166813642, 0.0926778764, -0.0694191083, -0.0983804986, 0.12547265, -0.14267537, 0.180269465, -0.143098682, -0.13022919, 0.0738431364, -0.163979337, -0.17442669, -0.0242187474, -0.114045739, 0.0767761916, -0.10504967, 0.0503751151, 0.0866678208, 0.00773401279, 0.00430884957, -0.120525025, -0.176838011, -0.0863500014, 0.00866668671, -0.168607041, -0.121515945, 0.14867647, 0.185887799, 0.15785116, 0.140664503, -0.0884601921, 0.0231291223, 0.0829577744, 0.0892267004, -0.197772995, 0.189196065, -0.118800618, 0.0732194334, 0.207739875, -0.103173129, -0.065648064, -0.128727034, -0.110486537, 0.054653123, 0.0793437958, 0.15447484, 0.148488969, 0.120917305, 0.0801374763, -0.129399568, -0.156592786, 0.0600291751, -0.156443983, 0.145239115, -0.0512111932, -0.0894358903, -0.204157606, -0.168812051, -0.108613163, -0.0171637479, -0.105808534, 0.123665437, 0.0821540356, 0.0144526726, -0.142738879, 0.0227865372, 0.0507515483, -0.105444357, 0.155019537, -0.207505211, 0.0971339568, -0.0339849778, -0.0463138744, -0.0321208723, 0.132046655, 0.0198223144, 0.106232792, 0.191176817, 0.00686157215, 0.067138955, -0.145373166, 0.163319066, 0.0499063581, -0.0990407094, -0.197167978, -0.0268944018, 0.145822719, -0.083871156, -0.209732011, 0.157422855, -0.00245159306, -0.0771522969, 0.199315846, -0.149281859, 0.049090676, 0.191661701, 0.158315614, -0.0693620294, -0.0132011902, 0.125350296, -0.0149667272, 0.160916612, 0.11119552, 0.157676488, 0.0098877456, 0.189075068, 0.168989629, -0.173922271, 0.121548429, -0.195168272, 0.202848047, 0.165604517, 0.156058118, 0.0950093716, -0.127327457, -0.111984469, -0.0613512285, 0.0418962389, -0.197636545, -0.114189513, 0.126012728, 0.155268207, 0.0866028816, -0.0889877826, 0.112122208, 0.194389224, 0.112043038, -0.069294557, 0.0346671753, -0.176826715, -0.203006268, -0.150415093, -0.0750610828, -0.0581135936, 0.163826838, -0.029669594, 0.109058082, -0.0119882217, 0.142015621, -0.0904931426, -0.0186770707, -0.0259640589, 0.0281509385, 0.0239989404, 0.116667978, 0.102750033, 0.091286853, -0.0383565463, -0.163616955, 0.187580332, 0.0162753612, -0.0314784348, 0.117369078, 0.0864375383, 0.100502871, -0.148412943, 0.0571034662, -0.0606366396, -0.161042437, -0.0797111019, -0.0348239429, 0.0452777334, 0.0193986744, 0.180022672, -0.00376706664, -0.075681217, 0.213514671, -0.00990024209, 0.188225329, -0.160626784, 0.0900792852, 0.18271482, -0.00601695525, 0.0461863279, -0.120181017, -0.107822776, 0.180234715, 0.100609951, -0.0603300333, -0.159216747, -0.102589242, 0.154994428, -0.0520614609, -0.183861494, -0.0509034172, -0.12675713, -0.0341059603, -0.0555140488, -0.0641053393, 0.0598824546, 0.0111815166, 0.00291509368, 0.17496188, 0.108429745, 0.115839042, 0.134348467, -0.00350385834, -0.282030761, -0.0406435393, 0.0446432419, -0.0427427255, 0.0944782719, -0.0354864225, -0.0111428648, -0.102770053, 0.0271255691, 0.242358834, 0.0536113046, 0.0741038397, -0.2916601, 0.0509373099, 0.0901637748, 0.102783382, -0.287690729, -0.0950423926, 0.0449632443, 0.0110642808, 0.140485168, 0.155553728, 0.257394135, 0.200602695, -0.0335011818, 0.105191864, -0.0773999244, 0.109473541, 0.117318951, 0.0171118602, -0.0794980526, -0.0106161162, -0.0825806633, 0.210200682, 0.049644243, 0.124389246, -0.134129956, 0.107796527, -0.214387313, -0.0956629068, 0.0328465402, -0.0811204761, -0.028460307, -0.128131568, -0.0982517526, -0.0257387385, -0.106076196, 0.0542545803, -0.151404768, 0.124424778, 0.0499416552, -0.177569553, 0.130988628, -0.304376811, -0.19533141, 0.218535423, 0.0927173048, -0.0933397934, -0.0590848438, -0.12533696, -0.182256982, 0.0507504232, 0.350399882, -0.105347395, 0.0997362882, 0.183351919, 0.223954976, 0.0116671519, 0.0770847723, 0.00941148866, -0.0585605204, -0.0564582013, -0.104068607, 0.267437309, 0.0964651331, -0.182642788, -0.189770326, -0.215519488, 0.157907411, -0.131437048, -0.10699293, -0.188718796, 0.0486624055, 0.127689123, -0.248873338, 0.078462258, -0.144253984, 0.129576817, -0.301556379, -0.114970237, 0.173650026, 0.112776645, 0.11526338, 0.115009017, -0.00548774051, 0.154869318, -0.0198779032, -0.162775025, -0.199682802, 0.135350138, 0.00967035349, 0.299527019, 0.218109444, 0.0262131374, -0.115798198, 0.272563934, -0.194497794, 0.143630132, 0.117160715, -0.214732021, 0.268078536, -0.262342006, -0.0561750121, 0.0062987851, 0.0484048985, -0.175266072, -0.0120564355, 0.243626311, -0.0441008434, 0.0145799173, 0.233922571, 0.00730382605, -0.156657904, 0.172205657, 0.221002415, 0.0211234111, -0.0905548707, 0.10886354, 0.118684202, 0.180481613, -0.0196608324, -0.178598583, 0.142019391, -0.0121234935, -0.146662265, 0.0912220255, 0.181317791, -0.16972439, 0.309380949, 0.153544962, 0.038100563, 0.192058325, -0.0871640146, 0.0492480472, 0.0830729306, -0.0759055465, 0.103810854, -0.255007654, 0.197088823, -0.0743090287, -0.21577549, -0.20244053, 0.210097998, 0.0616604239, -0.111432828, 0.184095949, -0.116312213, -0.0247057155, 0.0876967981, 0.109860271, -0.0928253531, -0.133457661, -0.177713558, -0.299925268, -0.0404093228, -0.162057132, -0.108176261, 0.12602371, 0.168155134, -0.0107569452, -0.110608943, 0.0278297774, 0.140921056, 0.112561956, 0.175497711, 0.183747575, -0.212413877, -0.130428985, 0.165591776, -0.0292511694, -0.141024932, -0.0634911358, 0.0630419105, 0.00752701424, -0.0684755668, 0.181002468, -0.102659136, 0.22071445, 0.0109583735, -0.062734507, 0.181735635, 0.184093043, 0.0399840549, 0.036717698, -0.205652788, -0.0349973813, -0.0381838493, -0.201135337, 0.138336897, 0.222890869, 0.204514265, -0.00664423173, 0.196919546, -0.0901932046, 0.0649525076, 0.00495409453, -0.0845536739, 0.0522219203, 0.0688513219, 0.129477873, -0.0250788908, -0.186325192, -0.0678296313, 0.0842106491, 0.105310403, -0.00730011286, 0.223297685, -0.128638223, -0.0857560188, 0.190256432, 0.181896374, 0.164745301, -0.208486781, 0.253901631, 0.205723599, -0.110545166, 0.177340835, 0.0701723173, -0.141629741, 0.0132791987, -0.0979559645, -0.203919381, -0.147979751, -0.0696999133, 0.0551467761, -0.148070619, 0.131242305];
    CONSTANT bias_13 : ARRAY[0..63] OF REAL := [-0.0404071435, 0.0927777886, -0.0413042903, -0.0902542397, -0.0367607661, 0.0712136403, -0.00892876834, -0.0667051747, 0.00637631165, 0.0437391289, -0.0124141583, 0.0894438922, -0.0595212504, 0.0899347588, 0.0368472114, -0.000366137043, -0.0369593501, 0.0098438086, -0.00942459609, 0.0903767124, -0.0075942101, 0.046375595, -0.0592727698, 0.0528409891, -0.0216910169, -0.00787346996, 0.0314517543, 0.0737932697, -0.0810395479, 0.0906123891, 0.0820333436, 0.0979426578, -0.0194323044, -0.0938704684, -0.0664548054, 0.0229378678, -0.0287175067, 0.0409495458, -0.0543716773, 0.0378184244, -0.0231971722, -0.0583018064, -0.064960219, 0.00983823184, -0.0784399733, 0.0101949805, -0.0290268082, 0.0763350129, -0.0110898362, -0.00504951039, 0.0234738979, -0.0619560853, 3.6623473e-07, -0.0102051999, -0.0874569118, 0.0950193256, 0.011268124, 0.0887499079, 0.0580152497, 0.0789389834, -0.0176048651, -0.00555823185, -0.0167076774, -0.0683557615];
    CONSTANT weights_16 : ARRAY[0..191] OF REAL := [-0.204218104, 0.0100585446, 0.124642573, 0.249767885, 0.192972004, -0.114489801, 0.0213469081, -0.192255303, 0.0687296614, -0.116273321, -0.168248311, 0.100407079, -0.0835328773, 0.238771692, -0.1582672, -0.20680669, 0.199099779, -0.355317205, -0.275946528, 0.259559304, -0.152421042, -0.193678349, -0.0476079546, 0.168583572, 0.137155071, -0.424926966, 0.0668462142, 0.121788457, 0.166179895, 0.155418351, -0.239607006, 0.159718022, 0.181392595, 0.012098941, 0.29212448, -0.30051899, -0.042393513, -0.302967817, 0.0276647583, -0.0162179675, -0.0362443365, -0.131818026, 0.0652571768, -0.251479208, -0.163796052, 0.246231601, -0.0993305817, -0.214045271, -0.259664625, 0.121991962, 0.328099579, -0.36496222, 0.286016166, 0.174832657, -0.115100093, 0.240771398, -0.219685465, -0.0312652551, 0.361102194, -0.322652519, 0.172960237, -0.0672435984, -0.196433365, -0.310510099, 0.180873245, -0.229489714, -0.0438734591, -0.0316266902, 0.106365554, -0.354469597, 0.104236148, 0.0969249979, 0.0453101136, 0.189823419, -0.119062148, 0.0151938582, 0.05480076, -0.137107879, 0.231374756, -0.184149876, -0.152093366, 0.298650056, -0.120534711, -0.440170765, -0.291449726, -0.185382351, 0.240590215, 0.0743931085, 0.00839448255, -0.324791044, 0.0127115622, 0.201346219, -0.129334167, 0.217511401, 0.249150231, -0.227794915, -0.152671486, 0.225536987, -0.10112305, -0.260705948, -0.309738696, 0.234022498, 0.247884244, -0.138457581, 0.287121534, 0.107613027, 0.369097799, 0.20829244, -0.189594626, -0.168206543, 0.127910152, 0.117524289, -0.267760575, -0.273475945, -0.0782620981, -0.369871527, 0.318286926, 0.380977005, -0.372844636, -0.159075871, -0.35559544, -0.15261285, 0.021852307, -0.177226037, -0.057486631, 0.270852298, 0.160473123, -0.251653463, 0.100419275, -0.136632696, -0.287902951, -0.344732016, 0.126178026, -0.177843302, 0.339493781, -0.099222295, 0.0892207772, 0.163005397, 0.215954706, -0.0692603961, 0.0789305717, 0.37051788, 0.124587342, -0.095472239, 0.128479376, -0.0207961947, -0.257337809, 0.0661524683, 0.132446691, -0.221712723, -0.32083869, 0.195067048, 0.161428511, -0.336975783, -0.0876864642, 0.283737957, 0.175905675, -0.186329022, -0.0834812075, -0.0544198342, -0.247233495, -0.240931347, -0.316858917, -0.324440151, 0.33110112, 0.302384734, 0.294178426, 0.0780448988, -0.218289346, 0.095910117, 0.0984309539, -0.335624874, 0.34094283, -0.192400947, -0.337153077, 0.305544972, -0.302600533, -0.0743493959, 0.340184033, -0.0958573595, -0.265512377, 0.0674359873, 0.0557227954, -0.208096027, 0.112970375, -0.241400406, -0.123275287, -0.175267965, 0.0384325348, 0.0348930582, -0.135870203, -0.0273135975];
    CONSTANT bias_16 : ARRAY[0..2] OF REAL := [0.0433644801, 0.055319678, -0.0903941169];
END_VAR
